(* IEC 61131-3 sources: ml2plc/examples/models/structured_text (part 6) *)

(* ---- test4_531k.st ---- *)
FUNCTION_BLOCK NeuralNetworkFB

VAR_INPUT
    input_data : ARRAY[0..4] OF REAL;
END_VAR

VAR_OUTPUT
    output_data : ARRAY[0..2] OF REAL;
END_VAR

VAR CONSTANT
    weights_0 : ARRAY[0..2559] OF REAL := [0.006168, -0.007737, -0.004572, -0.003805, -0.081145, -0.022669, -0.040454, -0.017532, -0.025900, -0.064631, -0.047865, -0.007452, -0.080317, 0.042283, 0.000890, -0.064382, -0.009100, -0.011638, -0.047598, -0.005238, 0.002791, -0.005841, -0.060246, -0.016523, -0.014516, -0.002007, -0.014596, -0.018067, 0.025868, 0.006018, -0.015262, -0.018643, -0.003052, 0.012583, -0.056134, 0.000727, -0.037447, -0.016557, -0.037026, -0.016739, -0.030965, -0.044604, -0.004674, -0.071475, 0.008430, -0.054697, 0.000375, 0.079556, -0.010031, -0.040946, -0.032777, -0.007746, -0.021319, -0.012790, -0.047135, -0.089749, 0.014232, 0.001651, -0.023776, 0.034909, -0.031567, -0.041982, 0.035747, -0.039939, -0.017710, 0.002087, -0.028975, -0.017014, 0.012243, -0.012999, -0.019807, -0.044350, 0.018067, -0.069752, 0.001563, -0.005957, -0.004255, -0.000246, -0.075206, -0.042035, -0.012978, -0.036161, -0.007486, -0.039953, -0.050775, -0.010311, -0.028363, -0.017167, -0.033474, -0.011529, -0.009715, -0.016724, -0.065615, 0.021977, 0.009902, -0.036258, -0.007694, 0.001126, -0.018509, 0.036309, -0.008579, -0.014633, -0.052138, -0.042639, -0.052210, -0.021528, -0.017732, -0.081576, -0.008286, 0.005255, -0.036065, -0.015189, -0.074120, -0.017314, -0.025928, 0.000444, -0.013875, 0.020662, -0.034705, -0.007929, -0.053950, -0.012137, 0.003924, 0.038306, -0.033622, -0.008152, -0.007697, -0.002231, -0.047321, -0.068849, -0.014781, 0.004508, -0.070911, -0.011590, -0.005847, 0.034466, -0.049314, -0.054858, -0.120357, -0.022947, -0.045314, -0.014210, -0.011795, -0.027942, 0.004085, -0.047372, -0.050960, 0.020868, 0.007977, -0.037249, -0.039574, -0.058623, -0.080479, -0.019785, -0.043017, -0.044134, 0.001765, -0.015653, -0.023090, 0.017455, -0.043623, -0.057814, -0.025243, -0.048311, -0.009657, -0.077425, -0.045795, -0.026813, -0.032518, -0.053390, -0.006588, -0.063675, -0.066407, -0.033561, -0.019729, -0.040149, -0.013426, -0.000105, 0.018445, 0.011021, -0.035918, -0.016334, -0.050424, -0.018496, -0.003434, 0.034537, -0.002120, -0.037769, -0.010563, -0.056970, -0.021492, 0.004430, 0.038964, -0.040694, -0.064145, -0.055157, 0.039010, 0.005452, -0.020624, 0.023485, 0.006722, -0.008886, 0.010608, -0.069180, -0.045544, -0.005442, -0.116079, -0.024035, -0.061259, -0.022777, -0.005744, 0.004640, -0.035091, -0.041870, -0.030253, -0.044182, 0.013662, -0.113956, -0.027071, -0.015773, -0.026526, -0.070524, -0.007985, -0.011598, -0.077758, -0.045670, -0.048661, -0.014513, -0.013066, -0.015931, -0.015619, 0.002752, -0.020614, 0.010716, 0.002136, -0.078809, -0.036949, -0.007683, -0.004785, -0.004789, -0.027511, -0.009657, -0.049951, -0.008816, -0.020890, -0.008851, 0.024166, -0.053262, -0.020197, -0.017122, -0.089715, 0.003861, -0.042685, 0.017193, -0.013868, 0.002213, 0.020823, -0.021258, -0.026864, 0.002694, -0.029496, -0.053142, 0.038210, -0.007476, -0.006005, -0.020900, -0.014644, -0.038122, -0.021673, -0.001530, -0.002961, -0.058100, -0.002778, -0.000089, 0.000113, -0.026780, -0.094293, 0.008923, 0.000047, 0.001569, -0.030386, -0.009189, 0.015745, -0.066894, -0.028746, -0.048156, -0.030306, -0.006260, -0.040602, 0.006604, 0.011101, -0.031063, -0.006231, 0.002844, -0.009292, -0.029432, -0.065772, -0.100504, -0.038383, 0.013530, -0.043025, -0.055311, -0.036706, -0.001836, -0.033030, 0.001966, 0.003206, -0.047405, -0.065538, -0.016400, -0.012487, -0.044876, -0.009988, -0.026461, -0.107726, -0.001962, 0.014469, -0.013257, -0.035765, -0.038008, 0.019523, -0.028117, -0.046915, -0.067385, -0.016535, 0.002655, -0.062835, -0.037264, -0.012879, -0.006051, -0.006659, -0.030517, -0.016854, -0.013416, -0.029428, -0.056979, 0.002656, 0.019105, -0.015444, -0.034404, 0.006777, -0.023455, 0.009467, -0.029399, 0.021276, 0.008433, -0.017701, -0.089102, -0.008802, -0.072623, -0.041329, -0.025934, -0.044785, -0.014089, -0.001511, -0.016151, -0.027101, 0.001011, -0.028102, -0.021238, -0.027469, 0.002060, 0.001314, -0.064151, -0.056067, -0.020087, 0.013779, -0.019102, -0.020556, -0.018478, -0.014906, -0.043024, -0.009099, -0.015567, 0.018504, 0.008389, -0.026493, -0.034103, -0.008169, -0.011630, -0.061097, -0.001828, -0.036604, -0.090593, -0.003821, 0.004210, -0.175559, 0.019005, 0.004134, -0.017647, 0.037174, -0.033732, -0.053073, 0.022879, -0.012883, -0.023034, -0.038492, -0.011812, -0.017564, 0.009026, -0.036873, -0.057276, -0.006387, -0.012203, -0.006951, -0.021118, -0.031144, 0.034645, 0.045173, 0.000612, -0.024887, -0.032074, -0.003918, -0.026183, -0.027079, 0.029110, -0.011173, 0.000224, -0.027518, -0.042254, -0.012626, -0.033389, 0.002061, 0.001831, -0.054974, -0.019345, -0.095294, -0.030450, -0.085620, -0.009941, -0.045067, 0.000455, -0.037109, -0.013278, -0.000530, 0.028802, -0.033968, 0.017109, -0.049283, 0.000876, -0.003601, -0.020212, -0.006754, -0.006030, -0.082454, -0.071900, -0.014293, -0.005903, -0.046136, -0.014200, 0.014313, -0.030323, -0.013996, -0.011830, -0.005418, -0.002600, -0.024998, 0.006551, -0.007039, -0.071191, -0.094658, -0.055012, -0.022098, -0.030385, -0.070776, -0.013385, 0.019914, -0.029646, -0.028838, 0.009107, -0.008539, 0.020163, -0.012484, -0.028226, -0.017505, -0.028885, -0.013220, -0.068085, -0.039696, -0.076335, -0.006828, 0.017805, 0.011101, -0.014613, -0.005119, -0.036674, -0.070308, -0.006485, -0.070089, -0.026779, -0.003504, 0.000492, -0.036936, -0.058629, -0.073952, -0.041623, 0.007899, 0.007541, -0.010827, -0.033526, -0.036041, -0.004380, -0.034936, -0.000530, -0.004452, 0.024483, -0.019720, 0.004198, -0.024792, -0.006160, 0.022435, -0.045744, 0.010493, -0.004708, -0.039041, -0.022206, 0.058065, -0.058637, 0.029476, -0.009941, 0.031980, 0.027263, 0.028729, -0.018779, 0.035691, -0.000839, 0.011755, -0.013788, -0.033617, -0.047934, 0.016009, -0.061441, -0.043422, -0.014114, 0.013690, -0.000306, 0.062245, -0.065690, 0.013481, 0.013963, -0.018303, -0.023203, 0.051331, -0.046245, -0.051296, 0.000886, 0.029395, -0.048312, 0.020966, 0.018177, 0.009344, 0.030180, -0.006859, 0.066112, -0.006302, 0.049277, -0.022652, 0.012126, -0.001961, 0.006813, -0.031577, -0.006198, 0.035557, -0.002758, 0.014040, -0.024291, 0.004469, 0.000628, -0.026485, -0.029591, -0.003587, -0.007451, -0.046778, 0.001367, -0.075846, 0.031924, 0.018597, -0.030053, -0.047463, -0.042152, -0.016299, -0.002213, -0.026199, 0.036664, -0.034040, 0.052768, 0.005836, -0.043658, -0.053341, 0.001381, 0.043572, 0.020291, 0.073398, 0.037756, -0.005681, 0.026407, 0.033731, -0.048959, 0.012376, 0.030472, 0.008492, 0.005691, -0.006789, -0.018349, 0.075362, -0.022161, -0.079043, -0.009294, -0.000774, -0.039354, -0.042801, -0.035631, -0.030911, 0.004652, 0.057990, 0.022027, 0.018841, -0.019965, -0.067957, 0.066897, 0.019102, 0.001754, -0.046148, 0.019094, 0.008093, 0.003544, -0.008916, -0.002643, -0.064754, -0.038101, -0.035119, -0.033188, -0.015181, 0.042656, 0.017546, -0.013701, -0.012623, 0.008619, -0.031625, -0.024699, 0.012467, 0.006890, -0.010188, -0.063297, -0.006435, -0.041045, -0.000126, -0.081690, 0.012576, 0.000700, 0.010163, 0.004561, -0.029321, -0.003461, 0.025865, -0.006400, -0.045266, -0.024265, 0.033321, -0.117580, -0.014021, -0.009655, 0.045165, 0.045564, 0.007505, 0.004496, 0.050880, -0.012176, -0.041370, -0.088418, -0.017235, -0.067351, 0.056832, 0.069346, 0.035097, 0.089766, -0.014582, 0.079974, -0.006041, -0.014888, -0.035294, 0.013718, -0.018149, 0.068994, 0.017431, -0.039235, -0.042068, -0.007724, 0.022600, -0.003539, -0.040479, -0.017089, 0.017629, -0.026505, 0.039217, -0.011858, -0.075481, -0.028972, -0.019730, 0.006281, 0.010786, 0.018083, -0.008708, -0.015356, -0.085096, -0.019559, 0.044645, -0.007992, -0.028722, -0.061144, 0.001558, -0.022994, -0.016173, -0.049005, 0.003667, 0.112726, 0.041862, -0.021030, 0.062288, 0.077233, 0.000736, 0.061262, -0.008646, -0.055297, 0.012099, 0.047965, 0.002597, 0.065893, -0.097906, 0.014617, 0.033970, -0.035677, -0.003285, 0.040832, -0.010042, -0.019621, 0.053835, 0.019053, 0.053018, -0.010340, -0.002477, -0.028028, -0.023846, -0.013320, 0.021628, -0.001340, -0.059531, 0.026777, 0.017700, -0.019184, -0.000877, -0.024227, -0.001088, 0.005022, 0.015510, 0.017810, -0.000029, -0.041248, -0.079095, 0.023700, -0.012472, -0.018172, 0.088289, -0.014964, -0.000217, 0.003885, 0.018567, -0.009548, -0.028347, -0.018591, 0.043182, 0.052019, -0.001108, 0.042047, -0.122054, 0.027480, -0.064142, 0.004650, 0.014279, 0.031755, 0.011892, -0.034454, -0.020755, 0.044469, 0.005772, -0.040299, -0.012851, -0.035211, 0.067049, -0.121054, -0.007700, -0.005547, 0.036890, -0.033311, 0.084753, 0.026367, 0.048788, 0.030230, 0.053215, -0.027125, 0.004881, 0.040511, -0.032856, -0.096552, 0.040967, 0.015451, -0.027745, -0.007011, 0.053545, -0.033689, 0.045135, -0.094181, 0.004068, -0.005429, 0.053405, -0.060415, 0.000319, -0.053152, -0.047989, 0.013013, 0.025322, 0.038022, -0.018121, 0.006913, -0.011688, -0.025630, -0.022074, -0.002609, -0.055090, -0.008263, -0.019801, 0.052412, -0.026663, -0.017301, 0.017173, 0.033957, 0.015627, -0.086593, 0.023172, 0.037030, 0.011863, -0.022188, -0.019773, -0.021711, -0.003184, -0.020591, -0.008187, 0.000161, -0.062586, -0.038520, -0.027736, -0.020185, -0.023671, -0.078505, 0.014876, 0.047807, 0.023937, -0.005761, -0.002716, 0.037869, -0.004794, -0.012825, 0.035395, -0.029956, -0.008986, -0.067532, -0.016199, -0.048075, 0.001541, -0.014349, 0.015026, 0.044194, 0.018795, -0.081185, -0.046023, 0.046350, -0.000227, 0.021468, -0.011860, -0.017598, -0.030247, 0.011072, -0.012450, 0.014558, -0.016468, 0.017973, 0.042791, 0.007654, 0.054244, -0.019306, -0.016567, -0.043988, 0.037716, -0.026492, 0.012198, 0.063996, 0.013889, -0.013916, 0.094007, -0.047667, -0.043191, 0.023439, -0.041024, 0.037257, 0.084837, -0.053354, -0.023051, -0.060040, -0.024047, -0.032870, 0.011373, -0.070437, 0.025510, 0.029563, -0.028023, -0.056257, -0.032347, 0.015591, -0.013614, -0.107999, -0.058039, 0.008937, 0.051134, -0.010621, -0.012029, -0.002045, -0.045550, 0.019002, -0.029280, -0.058529, 0.012200, 0.032851, -0.062094, -0.023157, 0.001064, -0.019808, 0.071575, -0.014192, 0.044343, -0.055609, 0.082989, 0.021812, 0.008306, 0.008213, 0.029873, 0.023171, 0.013703, 0.011581, 0.001465, 0.019024, 0.034659, -0.039955, -0.003518, -0.039174, -0.037442, -0.031396, 0.025519, -0.005441, -0.020170, -0.007954, -0.027134, -0.044586, -0.015502, 0.003576, -0.002512, -0.010521, -0.075746, -0.045547, 0.002149, -0.045099, -0.017035, -0.007519, 0.057518, 0.028380, 0.018844, -0.000265, 0.033838, -0.016435, -0.009740, -0.000992, 0.001005, -0.013433, -0.014406, -0.010904, 0.000908, -0.031988, -0.011733, -0.060267, 0.058381, 0.004671, 0.003265, 0.045723, 0.000060, 0.022857, -0.053219, -0.032393, -0.054149, -0.009633, 0.084957, -0.031704, 0.048600, -0.073818, 0.012638, -0.070321, -0.003787, 0.053202, 0.059789, 0.035780, -0.047696, -0.005062, 0.019513, 0.003089, 0.002214, -0.000557, 0.022252, -0.037908, -0.063868, -0.048430, -0.021449, -0.005469, -0.020284, -0.013151, -0.002935, 0.024061, -0.027414, -0.060135, 0.019118, 0.010644, -0.020204, 0.043180, 0.011003, -0.026948, -0.029472, 0.006690, -0.014830, 0.034704, 0.002983, -0.000449, -0.033364, -0.002019, 0.023595, 0.048194, -0.002517, 0.015325, -0.055047, 0.006398, -0.026732, -0.063421, -0.051463, 0.022229, -0.007053, 0.003437, 0.036441, 0.011057, -0.010537, 0.053316, 0.047278, -0.088576, -0.051669, 0.003415, -0.010457, 0.003318, 0.020984, -0.032925, 0.000310, -0.075833, -0.005370, 0.004928, -0.045853, -0.068047, 0.009317, -0.003116, 0.016023, 0.046078, -0.004938, 0.018008, -0.052253, -0.035261, -0.061192, -0.006844, 0.017909, -0.005032, -0.035604, 0.038330, -0.007799, 0.001959, -0.082375, -0.057521, 0.002209, -0.036735, 0.029469, 0.046464, 0.023360, 0.054089, 0.000124, -0.098509, -0.034924, -0.008698, -0.014121, -0.009095, 0.054927, -0.035409, 0.033318, -0.013215, -0.028000, -0.009640, 0.005127, 0.002514, -0.058949, -0.031840, 0.024286, 0.037682, -0.032623, 0.014822, 0.004515, -0.022597, -0.047328, -0.013061, -0.004957, -0.000829, -0.032617, 0.008092, -0.006902, -0.011951, -0.011564, 0.012531, 0.004754, -0.014693, 0.020353, 0.019861, 0.054645, -0.060680, -0.019404, 0.017570, 0.033163, -0.051124, 0.010038, -0.051300, -0.015827, -0.065831, 0.009685, -0.033803, 0.029050, 0.033958, -0.032388, -0.029221, -0.044903, -0.002951, -0.027556, -0.031074, 0.022902, 0.010975, -0.000864, 0.017581, -0.036060, 0.000276, 0.055463, 0.029811, 0.008004, -0.045528, 0.007951, 0.010881, -0.019921, -0.008701, 0.029887, -0.012379, -0.062134, -0.002077, 0.039846, -0.015407, 0.025720, -0.040064, 0.013837, -0.014882, -0.012172, 0.024249, -0.000815, 0.001816, -0.077496, -0.006953, 0.065075, -0.015756, 0.011041, 0.027465, 0.031528, -0.071741, -0.030240, 0.053134, -0.023077, -0.006604, -0.022893, 0.029625, -0.061120, 0.023706, -0.000936, -0.032921, -0.008114, 0.003939, 0.023346, -0.013129, -0.059646, 0.045903, -0.023942, 0.050939, -0.002942, -0.020111, -0.015744, 0.013710, 0.035260, 0.000029, -0.004535, -0.036242, -0.037386, -0.027829, -0.031840, 0.002574, -0.007554, -0.035839, 0.020656, -0.027891, -0.010452, 0.001935, -0.048956, 0.056025, -0.081554, 0.063599, -0.028470, -0.083353, -0.039516, 0.022740, 0.010384, -0.034174, -0.007442, -0.058151, -0.015351, 0.032128, -0.007490, -0.035707, -0.013821, -0.052297, -0.008232, -0.003910, -0.002278, -0.002002, 0.041686, -0.033565, -0.020172, 0.011638, -0.047561, 0.032903, -0.030198, -0.029194, 0.029884, 0.007434, 0.002506, -0.093412, 0.003442, -0.048978, -0.003672, 0.008821, -0.016854, -0.022693, 0.019834, 0.003447, -0.014566, -0.035371, -0.010202, -0.030048, 0.010019, 0.009586, 0.033665, -0.052329, 0.012042, -0.013713, -0.053064, -0.004914, 0.065243, -0.014380, 0.001766, 0.002737, -0.036723, -0.036644, -0.096545, 0.033883, -0.008006, 0.000931, -0.004996, -0.105254, -0.033430, -0.003654, -0.047162, 0.001697, -0.047309, -0.021566, 0.012178, -0.040513, -0.018042, -0.059251, 0.011468, -0.026371, 0.021869, -0.016537, -0.000474, 0.008068, -0.015187, 0.022844, -0.057641, -0.020614, -0.010191, 0.005121, -0.013429, 0.027562, 0.023835, -0.069291, -0.015122, -0.002747, -0.078974, -0.035144, -0.012528, -0.019010, -0.016324, 0.062985, -0.042301, 0.043749, 0.069579, 0.011530, -0.016713, -0.000731, 0.022784, -0.021786, -0.002233, 0.017447, -0.006153, -0.017514, 0.025534, 0.027752, -0.007414, 0.026801, -0.009000, 0.040284, 0.010169, 0.007577, -0.013006, 0.002903, -0.107397, -0.036827, -0.021993, -0.033773, -0.005145, -0.006365, 0.027436, -0.082875, -0.015922, -0.029948, -0.016043, 0.027308, 0.004923, 0.009969, -0.004351, -0.018375, 0.000664, -0.036814, 0.007848, 0.014095, -0.019357, 0.005650, 0.014980, 0.041914, -0.057784, -0.048502, 0.005255, 0.009340, -0.007252, 0.019865, -0.059517, 0.028774, -0.013038, 0.053348, -0.008614, -0.019005, 0.008522, -0.014930, -0.059443, 0.002173, -0.008524, -0.036694, 0.013195, -0.035339, 0.009507, -0.021153, -0.108459, -0.002806, -0.038649, -0.013854, 0.001382, -0.004942, 0.030240, -0.050536, -0.127641, -0.043994, -0.038555, -0.002474, -0.034832, 0.051688, 0.003858, 0.018911, -0.010615, -0.022812, -0.041967, -0.052411, 0.002677, -0.012954, -0.017153, -0.023283, -0.019843, -0.024961, -0.072991, -0.016500, -0.043703, -0.023475, -0.040668, 0.050983, -0.010791, -0.045946, -0.037954, 0.048402, 0.025119, 0.002440, 0.005653, -0.002502, 0.059590, -0.014535, 0.034528, -0.068574, -0.048264, 0.037087, -0.005935, 0.013869, 0.055370, -0.060236, 0.035561, 0.036965, -0.049284, -0.065174, -0.031417, 0.028118, -0.000721, -0.007135, -0.049212, -0.002982, -0.064442, 0.015377, 0.020929, -0.072578, 0.039138, -0.035400, -0.003530, -0.042568, 0.018827, -0.003496, 0.042349, -0.031215, -0.027957, 0.049278, 0.008354, -0.000546, -0.021296, 0.017299, 0.011847, -0.028922, -0.003541, -0.007659, 0.011905, 0.065311, 0.059542, -0.049007, -0.011449, 0.015553, -0.033130, -0.018639, 0.009950, 0.032141, -0.028848, 0.068738, -0.005494, -0.004502, -0.030848, 0.001772, 0.023285, 0.019241, -0.060901, 0.033557, -0.025315, -0.109076, -0.000548, 0.040990, 0.010826, -0.042109, -0.034424, -0.045023, -0.063789, 0.024868, 0.015001, 0.001163, -0.033712, -0.052648, -0.016266, 0.001274, 0.013955, -0.050313, -0.010176, 0.034576, 0.004616, -0.018953, -0.035623, 0.024527, -0.044255, 0.014509, -0.063285, 0.004416, -0.009160, 0.013336, -0.087228, 0.015343, 0.002086, -0.037559, -0.006652, -0.004271, -0.037680, 0.008953, 0.044458, -0.056017, -0.010455, 0.006135, -0.081046, 0.038880, -0.029584, 0.068916, -0.015243, 0.008562, -0.022434, -0.062339, 0.020589, 0.025935, 0.002090, 0.011453, -0.012045, -0.026340, -0.010421, -0.017118, 0.023078, -0.048666, -0.056073, -0.026423, 0.035808, -0.034026, 0.065977, -0.001679, 0.031959, -0.006526, 0.025844, -0.000980, 0.002246, 0.012930, -0.001139, -0.008721, 0.033522, -0.048647, -0.040169, -0.009701, 0.013569, -0.011153, -0.007777, 0.001426, -0.003487, -0.015966, -0.016842, -0.020404, -0.011884, -0.002042, 0.024870, 0.029681, -0.001799, 0.024583, -0.031010, -0.035852, 0.001699, -0.044035, 0.047594, 0.064107, -0.002716, 0.034184, 0.001073, -0.005203, -0.022102, -0.015703, 0.002247, 0.011254, -0.034985, -0.031385, -0.009637, 0.069561, -0.034012, -0.011237, -0.015109, -0.063899, 0.017169, 0.045481, 0.057430, -0.025430, -0.004783, -0.041361, -0.040798, -0.015842, -0.047996, 0.003322, -0.059076, 0.010305, 0.003273, 0.002631, 0.044407, 0.005079, 0.021253, -0.011607, 0.041114, -0.013865, 0.008588, 0.004921, -0.013600, -0.014643, 0.030441, -0.023050, 0.013847, -0.008933, -0.023550, 0.001001, 0.001016, -0.001820, 0.004475, -0.007551, 0.008457, 0.003246, -0.059475, -0.009358, -0.080363, -0.019096, -0.009395, -0.011684, 0.001092, 0.039147, -0.038988, 0.029579, -0.008820, -0.031082, -0.060658, 0.000651, 0.000825, -0.026070, -0.006354, -0.049676, -0.020702, -0.003012, -0.006391, -0.007444, 0.023275, 0.002955, 0.007902, 0.036258, 0.019251, -0.013756, -0.014383, 0.024339, -0.010544, -0.018283, 0.027118, 0.010669, -0.012802, -0.004819, 0.006033, -0.016694, -0.064134, 0.038288, -0.055878, -0.025146, -0.039060, 0.014958, 0.001991, -0.079096, -0.021012, -0.030163, 0.087878, 0.037328, -0.015318, 0.058822, -0.034177, 0.044470, -0.128140, 0.001406, -0.070954, 0.016894, 0.004603, -0.045666, -0.018139, 0.008610, 0.071770, -0.019468, 0.033419, 0.003130, 0.044825, 0.011587, -0.001095, 0.016766, -0.006245, -0.064439, 0.033407, -0.094713, -0.006409, -0.000119, 0.002618, -0.031029, -0.052071, -0.010173, -0.022700, -0.016307, -0.001930, 0.037094, -0.004913, -0.005293, 0.015431, 0.036442, -0.012428, 0.074049, -0.063375, -0.013886, 0.030770, -0.046108, 0.036323, -0.081006, -0.027172, -0.011284, -0.018333, -0.021334, -0.013070, -0.011830, -0.021084, 0.002423, 0.034048, -0.038911, -0.001053, -0.002545, 0.000026, 0.026737, 0.030784, -0.002281, -0.011285, 0.029163, -0.033121, -0.021412, -0.016520, -0.002251, 0.008773, -0.045886, 0.012279, 0.009255, -0.005824, 0.000048, -0.005718, -0.037088, -0.007778, -0.019037, -0.023370, 0.002763, 0.024722, -0.007766, -0.057903, -0.012214, 0.032384, -0.027996, 0.024596, 0.003802, -0.001651, -0.015866, 0.021212, 0.057682, -0.028116, -0.013073, 0.020292, -0.009352, -0.130909, -0.024060, -0.044775, -0.005629, 0.020706, 0.020607, -0.021389, -0.005816, 0.046837, -0.023419, 0.025185, -0.008048, 0.021869, 0.006025, -0.007184, -0.072714, 0.049448, 0.095942, -0.002258, -0.019363, -0.019018, -0.013612, -0.017024, -0.024008, -0.060706, 0.012546, 0.008040, -0.017750, -0.021085, 0.048197, -0.092418, 0.013575, -0.030068, -0.040348, -0.043340, 0.001834, -0.021993, -0.074695, 0.001109, 0.023855, 0.017737, -0.018748, -0.030487, 0.005170, -0.015220, 0.030898, 0.009196, 0.017739, -0.063993, -0.028491, 0.038864, -0.000904, -0.003439, 0.060044, 0.007750, -0.050293, 0.003916, -0.020393, -0.007651, -0.083702, 0.012657, -0.041159, -0.074699, 0.017662, -0.019135, -0.023496, 0.079346, -0.044665, -0.087241, 0.057253, 0.035364, 0.038074, 0.033843, -0.025855, -0.017310, 0.032125, -0.001813, -0.042987, -0.008234, -0.047822, -0.026193, -0.017293, 0.016534, -0.052416, 0.047058, 0.006139, 0.000373, -0.050032, -0.010969, -0.014620, -0.065381, -0.065984, 0.039695, 0.013624, 0.009117, -0.073527, 0.005184, 0.012362, 0.013532, 0.003368, 0.026692, 0.001673, 0.010429, 0.034464, 0.005765, 0.041395, 0.004109, -0.009537, -0.008939, 0.001889, 0.022877, 0.022266, -0.022098, 0.008824, -0.111495, -0.014949, -0.010727, -0.013789, -0.008899, -0.014824, -0.039584, 0.057751, 0.016652, -0.009886, 0.028283, -0.028595, 0.053852, -0.039075, -0.013941, -0.006656, 0.003033, 0.020083, -0.052063, 0.075551, 0.016607, 0.033015, -0.028914, 0.000990, 0.051002, -0.051270, -0.000054, -0.045118, 0.030804, 0.013392, 0.037767, 0.017876, 0.028166, 0.031678, -0.006061, -0.131450, 0.004390, 0.000658, 0.019391, 0.006017, -0.022607, -0.025737, 0.045831, -0.037299, 0.005095, -0.051780, -0.013996, 0.002758, -0.019142, -0.099079, -0.024694, -0.034577, 0.065943, 0.028580, -0.028417, -0.017952, -0.003284, 0.012914, 0.000251, 0.038695, 0.003972, 0.075688, -0.050465, -0.008991, -0.066909, 0.010379, -0.027695, 0.002838, -0.088827, -0.035800, -0.070370, -0.001824, -0.002680, -0.091314, -0.046202, -0.030486, -0.059511, 0.025657, -0.028113, 0.006912, -0.001720, -0.004071, -0.015952, -0.045470, -0.110590, 0.035917, 0.031153, -0.038135, 0.038639, -0.030943, -0.053098, 0.010134, 0.032735, -0.043683, 0.006105, -0.022744, 0.004303, -0.039438, -0.017385, -0.009131, -0.021856, -0.068681, 0.028034, 0.032798, -0.017536, 0.001738, -0.010315, -0.047463, -0.019801, 0.052497, -0.018893, -0.032553, 0.001899, 0.002888, 0.006082, -0.102064, 0.015060, 0.043289, 0.035894, -0.034930, -0.005025, -0.022740, -0.011462, 0.022725, 0.004670, -0.004176, 0.052536, -0.059373, 0.036484, -0.007752, -0.020044, -0.038795, -0.005262, -0.002371, 0.008118, -0.015251, 0.007129, -0.005574, -0.001835, -0.050144, -0.066125, -0.049709, -0.001914, -0.010255, -0.062357, 0.026160, -0.079928, -0.089573, -0.026023, -0.079924, -0.037929, -0.060248, -0.097622, -0.022256, -0.012138, -0.023413, -0.014130, -0.022373, -0.018968, 0.071716, -0.014322, -0.016340, -0.016211, -0.028133, -0.041122, -0.052809, -0.055714, -0.039074, -0.006132, -0.069915, 0.075339, 0.018775, 0.003201, -0.091950, 0.011198, -0.072222, -0.207902, -0.052503, -0.016103, -0.016584, -0.024159, -0.003789, -0.014732, -0.007769, -0.030552, -0.029373, -0.030021, -0.062975, 0.035173, -0.007464, -0.071709, -0.023191, -0.020199, -0.250547, -0.036404, -0.027666, -0.045544, -0.021928, -0.053373, -0.074033, -0.020565, 0.001989, -0.017748, -0.001127, -0.044066, -0.254895, -0.028499, -0.041015, 0.014959, -0.047935, -0.044798, -0.072543, -0.024991, -0.001973, -0.015223, -0.045056, -0.044002, -0.057141, 0.079430, -0.000973, -0.030142, -0.014362, -0.008963, -0.021617, -0.000343, -0.017941, -0.055189, -0.011911, -0.024881, -0.020193, -0.036285, 0.011153, -0.086658, -0.115129, -0.075860, -0.032126, -0.031356, -0.035758, -0.039777, -0.010603, -0.039971, -0.005003, -0.092777, -0.016766, -0.035017, 0.067210, -0.020347, 0.000180, -0.028031, -0.005414, -0.046689, -0.011603, -0.042978, -0.047190, 0.001767, -0.060300, -0.026369, -0.017898, -0.014198, -0.023047, -0.015757, -0.054736, -0.002798, 0.031703, -0.022449, -0.055319, -0.076581, -0.025874, -0.054651, -0.066918, -0.014431, -0.018167, -0.033554, -0.022343, -0.031144, -0.095778, 0.002187, -0.020380, -0.029201, -0.029436, -0.026996, -0.082483, -0.026350, -0.033960, -0.047994, -0.052323, -0.073925, -0.012077, -0.069418, -0.020239, -0.034885, -0.035901, 0.025073, 0.022686, -0.073895, -0.000864, -0.032177, -0.112699, -0.035631, 0.036357, -0.098355, -0.059297, -0.109314, -0.083866, -0.028674, -0.092170, -0.025738, -0.047006, -0.059676, -0.390116, 0.017218, -0.019471, -0.039703, -0.077019, -0.017879, -0.045720, -0.048082, -0.068037, -0.116513, -0.003322, -0.039939, -0.057380, -0.002844, -0.030937, -0.078279, -0.046431, 0.007851, -0.007846, -0.013517, -0.013672, -0.028053, -0.044630, 0.056186, -0.025563, -0.025391, -0.107007, -0.015789, -0.016769, -0.037651, -0.091252, -0.028524, -0.068835, -0.122871, -0.040803, -0.009011, 0.097818, 0.022286, -0.025307, -0.013694, -0.049694, -0.025467, -0.009230, -0.036727, -0.087940, -0.003927, -0.015481, -0.043764, -0.053849, -0.031034, -0.030649, -0.014868, -0.045202, -0.069928, -0.034897, 0.002734, -0.063531, -0.007274, -0.006740, -0.020420, -0.006569, -0.037788, 0.001002, -0.035107, 0.035919, -0.036534, -0.022154, 0.006700, -0.033557, -0.043352, -0.005245, -0.044900, -0.032932, -0.028327, -0.025989, -0.006374, -0.000653, -0.039040, -0.028748, -0.032810, -0.013529, -0.022279, -0.020407, -0.136795, -0.092331, -0.019560, -0.042329, -0.042786, -0.002416, -0.004882, 0.079753, -0.049726, -0.001607, -0.077585, -0.032747, 0.027309, -0.289826, -0.050177, 0.007235, -0.087341, 0.013227, 0.091116, 0.005451, 0.021729, -0.028794, -0.035271, 0.002774, -0.028409, -0.024945, 0.011371, -0.004599, -0.022100, -0.008223, 0.000789, 0.011017, -0.054857, -0.019057, -0.087335, -0.035270, 0.021188, -0.044861, 0.062755, -0.042301, -0.047132, -0.020623, -0.039554, -0.031479, -0.085009, 0.004568, 0.076652, -0.026515, -0.028987, -0.029603, -0.053167, -0.003366, -0.027917, -0.070408, -0.022428, -0.018212, 0.016192, -0.034404, 0.002494, -0.018473, -0.011689, -0.007457, -0.071295, -0.044153, -0.021756, -0.074203, -0.057648, -0.028279, -0.031716, -0.249456, -0.073115, 0.005304, 0.073527, -0.010448, 0.019232, -0.013999, -0.077410, 0.010563, -0.113081, -0.030120, -0.004718, -0.032821, -0.018488, 0.040180, -0.013917, -0.057365, -0.013663, -0.034495, -0.029207, 0.004239, -0.055135, -0.025166, -0.013593, -0.017122, -0.017133, -0.028331, -0.121554, -0.087904, -0.169127, -0.007008, -0.001212, -0.044030, -0.024503, -0.019572, -0.058879, -0.025582, -0.016590, -0.026188, -0.021663, -0.059479, -0.015373, -0.087637, -0.014144, 0.068119, -0.030784, 0.017394, 0.008500, -0.018711, -0.002974, -0.023651, -0.007668, -0.044605, -0.037411, -0.003849, -0.036531, 0.008198, -0.038061, -0.126516, -0.002909, -0.042653, -0.078390, -0.007849, -0.082457, 0.015911, -0.021599, -0.006017, -0.012733, -0.039974, 0.024193, -0.060572, 0.003743, -0.053093, -0.017102, -0.024318, -0.111726, -0.037359, -0.009472, -0.041164, -0.042447, -0.057380, -0.024953, -0.053407, -0.055655, -0.014224, -0.009794, 0.044105, 0.013126, -0.041380, -0.044204, 0.004932, -0.018908, -0.017355, -0.245535, -0.026744, -0.064080, -0.029372, -0.007203, -0.023629, -0.063408, 0.023934, -0.014043, -0.005872, -0.037652, -0.043501, -0.010717, -0.012284, -0.006543, -0.119264, -0.021682, -0.170125, -0.049194, 0.040230, -0.008044, -0.046620, -0.006159, 0.013648, -0.019651, -0.045637, -0.058170, 0.080909, 0.006372, -0.005016, -0.000595, 0.006720, 0.005245, -0.042498, -0.014498, 0.000439, 0.002276, -0.062180, -0.015582, 0.004705, 0.016076, 0.013021, -0.084524, -0.017796, -0.039834, -0.017225, -0.025239, -0.023910, 0.027862, -0.093303, -0.048912, -0.084215, -0.013775, -0.031631, -0.018785, 0.030396, -0.040472, -0.039703, -0.015829, -0.000407, -0.031301, -0.052192, -0.026411, -0.171183, -0.004667, -0.018525, 0.002765, -0.014035, -0.068948, -0.039431, -0.021647, -0.028413, -0.013805, 0.013900, -0.012050, -0.126553, -0.052837, 0.015999, -0.044176, -0.037112, -0.008267, -0.018192, -0.071674, -0.060666, -0.097312, -0.059403, -0.087029, -0.005587, -0.005021, 0.011870, -0.006146, 0.010483, -0.052837, 0.003976, 0.004876, 0.002883, -0.024434, -0.077477, 0.030641, -0.019218, -0.035539, 0.013905, 0.031854, 0.002071];
    bias_0 : ARRAY[0..511] OF REAL := [-0.560015, 0.184992, -0.470400, -0.294991, -0.372218, -0.580996, -0.127396, -0.456540, -0.007419, -0.141688, -0.516530, -0.058160, -0.375340, -0.870894, -0.525041, -0.497357, -0.425162, -0.267576, -0.566308, -0.246234, 0.760137, -0.267928, -0.421276, -0.461114, -0.884117, -0.752684, -0.272481, -0.075169, -0.277913, 0.800566, -0.266811, -0.508528, -0.489017, -0.563790, -0.171746, -0.592066, -0.099807, -0.305085, 0.228222, 0.204156, -0.222468, -0.390126, -0.392960, -0.152436, -0.480089, -0.487889, -0.102116, 0.576028, -0.360179, 0.315619, 0.361651, -0.283220, -0.275759, -0.108602, -0.517918, -0.668270, 0.080150, -0.525913, -0.390262, 0.238540, -0.506728, -0.372645, -0.529373, -0.530296, -0.419331, -0.262827, -0.544448, 0.153808, -0.417206, -0.416869, 0.392310, -0.373798, -0.756939, -0.013806, -0.356106, -0.015186, -0.657312, -0.635726, -0.067811, -0.520272, -0.088178, -0.198638, -0.171325, -0.180742, -0.344793, -0.560948, -0.050169, -0.063545, -0.521232, -0.253853, -0.473808, -0.572321, -0.499878, -0.378826, -0.486301, -0.380427, -0.180301, -0.029836, -0.561780, -1.221803, -0.467454, -0.040174, -0.484950, -0.363476, -0.277297, 0.029669, -0.478665, -0.035147, -0.413088, -0.336468, -0.443213, -0.049765, -0.361502, -0.278191, -0.397446, 0.542885, -0.430711, 0.477843, -0.534856, -0.636531, -0.404057, -0.141602, -0.589094, -0.018168, 0.100740, -0.466928, -0.097708, -0.297540, -0.461497, -0.400244, -0.225557, -0.315778, -0.161987, -0.323324, 0.177692, -0.313298, -0.428529, -0.417167, -0.564084, 0.114390, -0.554823, -0.278022, -0.439219, -0.265492, 0.011075, -0.372697, -0.414324, -0.616711, 0.287804, -0.300455, -0.426657, 0.108030, -0.496591, -0.380250, 0.019351, -0.233535, -0.095143, -0.627654, -0.507818, -0.203023, -0.438338, -0.029473, -0.100205, 0.319433, -0.120297, -0.394097, 0.081192, 0.084620, -0.574713, -0.424066, -0.183717, 0.443114, -0.460228, -0.610907, -0.450714, -0.646212, -0.626546, -0.558116, 0.672355, -0.276201, -0.631161, -0.310516, -0.087265, -0.097912, -0.628902, 0.111149, -1.149800, -0.406454, -0.183037, 0.064063, -0.556680, -0.432543, 0.149459, -0.429032, -0.307682, -0.529772, 0.073030, -0.588899, -0.673073, -0.855552, -0.529210, -0.559242, -0.503162, -0.411373, -0.582325, -0.476031, 0.464417, 0.195734, -0.035936, -0.269100, -0.201118, -0.547096, -0.339036, -0.186394, -0.392593, -0.525719, -0.447540, -0.754172, 0.050524, -0.440737, -0.587200, -0.023825, -0.559724, -0.540134, -0.026272, -0.478584, -0.178302, -0.310404, -0.043472, -0.303760, 0.087057, -0.560951, -0.126218, -0.444226, 0.013041, -0.378160, -0.401341, -0.066755, 0.097565, -0.246728, -0.453610, -0.436659, -0.150369, -0.565253, -0.386807, -0.537203, -0.050841, -0.295192, -0.282184, -0.609656, -0.349239, -0.477961, -0.565487, -0.847882, -0.503656, -0.485508, 0.228604, -0.230194, -0.371666, 0.160188, -0.324394, -0.176446, -0.198087, -0.523571, -0.738180, -0.362561, -0.531421, -0.185987, -0.318514, -0.339727, 0.373145, -0.139809, -0.545757, -0.536750, -0.540660, -0.591894, -0.365686, -0.772576, -0.241534, -0.180127, -0.309330, -0.451085, -0.133262, -0.491258, -0.922880, -0.085069, 0.075745, -0.599000, -0.255950, -0.366717, -0.315008, 0.025284, -0.796683, -0.576438, -0.423812, -0.526922, -0.464793, -0.611435, -0.176255, -0.011129, -0.148650, -0.593366, -1.010090, -0.611632, -0.615362, 0.098925, -0.484878, -0.568730, -0.406493, -0.103242, -0.089686, 0.127594, -0.331190, -0.228097, -0.494144, -0.289490, 0.106738, -0.494740, -0.811164, -0.224123, -0.539983, -0.190705, -0.308104, -0.576015, -0.448016, -0.452012, 0.063439, 0.015257, -0.181990, -0.454566, -0.511673, -0.489078, -0.242683, -0.551215, -0.320198, -0.305431, -0.010823, -0.530007, -0.248963, -0.599315, -0.278430, -0.568422, 0.219756, -0.437993, 0.481473, -0.272435, -0.269651, 0.202242, -0.181707, -0.269245, 0.383201, -0.646039, -0.229450, 0.205804, 0.078391, -0.578819, -0.428767, -0.099032, -0.498601, -0.852345, -0.515247, -0.871002, -0.549889, -0.357410, -0.024235, -0.221249, -0.703844, -0.345876, -0.218584, -0.446784, -0.356807, -0.403075, 0.162039, 0.359484, -0.842997, 0.181479, -0.363541, -0.474084, -0.500788, -0.621216, -0.559714, 0.041385, -0.368353, -0.202383, -0.597544, 0.013351, 0.036447, -0.180812, -0.647463, -0.003342, 0.887071, -0.064974, -0.570065, -0.425626, -0.649220, -0.515449, -0.608669, 0.027214, -0.356379, -0.425030, -0.109388, 0.446015, -0.571340, -0.579622, -0.107719, -0.119594, -0.032838, -0.666012, 0.329357, -0.379204, 0.442772, -0.567839, -0.250720, 0.252409, 0.254247, -0.556360, -0.595093, -0.398352, -0.588479, -0.109848, -0.696338, -0.451533, -0.427623, -0.517631, -0.076536, -0.100740, -0.587674, -0.433592, -0.168261, -0.522468, -0.336927, -0.536847, -0.587720, -0.180166, 0.026694, -0.906076, -0.327415, -0.170205, -0.111061, 0.023953, 0.019779, -0.445003, -0.464418, -0.525391, -0.757161, -0.590829, -0.639809, -0.478079, -0.491544, -0.693892, 0.043033, -0.345456, -0.304986, -0.430036, -0.683112, -0.510119, -0.268652, 0.026592, -0.488424, 0.089903, -0.687703, -0.479938, -0.263812, -0.729523, -0.500908, -0.508581, -0.646621, -0.368469, -0.678522, -0.097792, -0.482871, 0.287748, -0.410175, -0.630866, -0.412892, -0.014359, -0.253159, -0.518970, -0.306679, -0.162928, -0.502708, -0.723021, -0.585624, -0.038050, -0.306422, -0.386367, -0.261096, -0.322216, -0.243436, -0.450591, -0.258327, -0.473112, -0.314861, -0.546208, 0.487024, -0.467651, -0.432374, 0.294989, -0.701729, -0.404412, 0.457121, -0.157405, -0.416856, -0.143322, -0.547066, -0.152965, -0.157077, -0.390291, -0.507056, -0.373921, -0.426115, -1.071550];

    weights_1 : ARRAY[0..524287] OF REAL := [-0.033384, -0.029529, -0.002307, -0.065159, -0.029187, -0.063650, -0.017592, 0.007238, 0.087993, -0.013393, -0.032657, -0.027770, 0.025115, 0.008525, -0.039527, -0.057369, -0.025352, -0.038812, -0.061059, 0.028921, -0.036287, 0.002650, -0.005819, 0.022260, 0.010706, 0.017105, 0.022733, -0.102570, 0.048175, -0.065543, 0.042244, -0.001051, -0.005552, 0.001343, -0.132678, -0.084336, 0.023444, 0.044026, 0.006423, -0.002656, -0.035584, -0.011227, -0.018969, -0.118467, -0.076455, -0.008606, 0.038094, -0.070374, 0.028555, 0.027610, -0.009448, 0.019685, -0.124333, -0.049827, -0.077195, -0.056529, 0.012599, -0.009381, 0.023236, -0.004700, -0.095187, -0.027614, -0.016721, -0.042166, 0.026967, -0.001691, 0.168896, -0.045715, -0.077939, 0.018614, -0.005101, -0.049948, -0.086186, -0.070169, 0.003832, -0.060939, -0.058552, -0.003961, 0.025444, 0.039389, -0.016526, 0.027258, 0.057089, -0.003192, 0.038133, -0.103590, 0.044226, -0.036122, -0.014077, -0.072944, -0.070990, -0.015418, 0.025484, -0.126175, -0.014363, 0.001600, -0.006227, 0.025299, 0.023108, -0.017388, -0.064967, -0.032258, 0.059030, 0.027494, -0.043399, 0.041397, -0.048733, -0.125696, 0.080937, -0.005893, -0.060478, 0.024098, -0.059152, -0.067177, -0.024428, -0.035957, 0.037022, 0.043891, 0.072372, -0.013457, -0.059588, -0.048198, 0.001741, -0.015119, 0.067838, 0.029718, 0.007244, 0.034856, -0.126202, 0.020841, -0.018814, 0.008373, 0.025370, -0.008876, -0.166713, -0.021350, -0.010922, -0.026620, 0.007677, 0.017664, -0.021487, -0.014281, -0.068944, -0.000945, 0.006296, -0.090065, -0.070590, 0.038186, -0.092014, -0.025633, -0.067717, 0.052099, 0.003534, 0.056980, -0.031832, -0.060090, -0.079961, 0.048795, -0.048479, 0.017890, 0.036706, 0.054768, 0.039339, -0.000939, -0.090144, 0.016987, -0.139394, -0.082103, -0.043726, -0.038848, -0.062648, 0.009012, -0.028069, 0.002676, -0.151202, -0.023922, -0.014620, 0.000349, -0.040842, -0.030065, 0.001913, 0.013584, 0.027665, 0.023666, -0.034337, -0.007901, 0.020217, -0.045113, 0.014856, -0.063518, -0.025068, 0.097930, -0.106403, -0.069477, 0.057602, 0.059377, 0.052719, -0.047087, -0.084744, 0.052077, 0.053991, -0.009452, 0.053999, 0.023506, -0.057650, -0.039659, -0.058501, -0.008886, 0.146905, -0.033510, 0.038731, -0.094149, 0.072222, 0.033093, -0.011071, -0.012098, 0.006181, 0.044728, -0.111777, -0.038309, 0.030381, 0.096242, -0.040079, -0.030020, 0.029591, -0.101405, 0.022670, -0.080118, 0.004489, -0.090326, -0.068333, -0.058073, 0.017577, 0.004949, -0.036895, -0.091916, -0.095090, -0.032846, -0.030988, -0.011184, -0.076728, -0.055495, -0.063720, 0.004673, 0.043187, 0.015708, -0.021401, -0.025020, 0.034938, -0.081069, -0.117772, 0.000362, 0.020896, 0.042762, 0.059001, 0.019692, -0.051868, -0.004403, -0.001810, -0.016538, -0.005535, -0.020549, 0.033277, -0.023793, -0.050831, -0.070665, -0.004009, -0.007788, -0.049764, -0.015402, -0.170423, 0.093517, -0.043430, -0.029537, 0.068742, 0.054416, 0.020689, -0.060321, 0.019090, -0.018722, -0.070399, -0.101210, -0.027410, -0.048431, 0.026611, 0.012401, -0.046667, -0.046146, -0.089249, -0.095605, 0.025816, 0.029740, 0.043186, -0.006458, -0.021826, -0.020286, -0.041731, -0.029256, -0.083371, -0.027684, -0.043325, -0.090286, 0.040597, -0.067456, -0.058064, -0.015049, 0.043578, -0.052356, -0.000773, 0.032165, -0.052683, 0.045543, 0.024650, -0.031897, -0.052368, 0.023043, 0.023701, -0.049907, -0.019434, 0.037758, -0.006270, 0.066636, 0.042503, 0.007880, -0.024659, -0.013514, -0.066361, -0.053382, 0.004468, -0.129562, 0.100200, -0.030750, -0.087867, -0.021234, 0.054874, -0.090015, -0.041550, 0.005455, -0.090650, 0.047877, 0.022088, 0.023703, 0.038352, 0.044019, 0.029308, -0.023749, -0.036233, -0.016927, -0.029878, -0.063288, 0.026692, -0.016907, -0.055816, 0.030134, -0.012202, -0.082080, 0.059260, -0.058566, 0.034364, -0.073843, -0.127900, 0.042268, 0.020256, -0.057530, -0.035022, 0.000135, -0.032868, -0.032640, 0.021750, -0.034581, -0.018041, -0.070351, -0.057236, -0.005502, -0.007093, 0.037278, -0.004064, -0.009294, 0.016825, 0.019933, 0.008553, 0.012465, -0.025279, -0.052135, -0.033548, 0.058220, -0.061634, 0.015563, -0.051011, -0.023905, -0.049785, -0.019259, 0.041113, 0.051277, 0.028460, 0.055870, -0.023927, -0.113015, -0.012672, -0.000884, 0.050397, -0.013646, -0.092497, -0.055455, 0.036631, 0.084139, 0.009879, 0.048542, -0.099915, 0.030325, -0.007776, -0.011569, -0.053630, -0.068224, 0.017663, 0.058832, 0.071599, 0.012827, 0.056008, -0.021221, 0.043322, -0.071704, 0.006411, 0.035887, -0.073169, -0.010824, 0.020810, -0.015934, -0.095901, -0.114015, -0.026279, -0.049996, -0.020573, 0.051564, -0.072600, 0.012393, 0.015384, -0.062750, -0.008225, 0.027788, -0.009694, 0.030362, 0.027102, 0.079901, 0.007625, -0.148665, -0.032986, 0.032929, 0.015108, -0.007190, -0.009169, -0.042474, 0.063413, 0.016762, 0.025950, 0.036114, 0.036235, -0.049745, -0.028458, -0.058993, -0.061607, -0.032990, 0.002196, 0.052250, -0.005320, 0.095450, -0.093596, -0.055396, -0.051156, -0.095880, -0.064916, 0.016736, -0.004266, -0.052662, -0.061324, -0.016475, -0.058697, -0.033423, -0.085685, -0.042742, -0.012220, 0.026440, -0.034047, -0.007125, -0.034108, 0.000781, -0.040265, 0.020626, -0.058811, 0.039135, -0.007725, 0.022717, -0.002046, 0.012720, -0.085223, 0.030688, -0.067694, -0.016844, -0.014237, 0.037264, -0.025419, 0.080257, -0.024835, -0.017699, -0.016987, 0.059430, 0.191333, -0.044881, -0.078858, -0.040470, -0.002010, -0.117800, -0.049850, -0.001206, -0.000659, 0.031370, 0.014626, -0.068077, -0.017440, -0.075535, 0.048635, -0.028763, -0.038477, -0.065760, -0.033861, -0.024372, 0.043851, 0.024441, 0.072546, -0.004179, 0.016827, 0.047067, -0.027436, 0.091070, 0.071626, -0.041470, -0.018696, -0.020496, 0.039035, 0.067127, 0.149240, 0.010853, 0.054563, 0.033246, 0.032480, 0.031350, -0.034347, -0.011196, -0.023261, -0.013315, -0.053553, -0.017366, 0.031521, -0.014585, -0.009573, 0.092145, -0.039544, -0.032399, 0.015883, -0.058906, -0.112737, -0.084352, 0.105879, -0.026967, -0.015161, 0.050685, -0.013870, 0.021519, 0.019574, 0.039395, -0.021270, 0.019507, -0.067272, 0.008691, 0.080083, -0.071324, -0.019700, 0.076822, 0.094249, -0.093745, 0.023937, 0.020843, -0.044744, -0.047941, -0.023536, 0.061359, -0.060069, 0.016053, -0.023770, 0.006217, -0.069338, -0.025733, -0.040211, 0.034911, -0.029710, -0.013557, -0.022490, -0.093235, -0.041620, -0.001497, 0.057327, -0.001120, 0.053036, 0.005079, -0.016962, -0.048700, 0.114897, 0.050940, -0.092638, -0.040940, -0.182887, 0.005397, -0.012453, 0.014685, 0.055595, 0.004929, 0.019169, -0.097534, -0.079380, 0.004848, -0.215702, 0.004224, 0.048380, -0.027477, 0.050242, -0.044771, -0.058177, -0.057193, -0.026794, -0.058831, -0.024620, 0.076269, 0.035077, -0.041190, -0.047126, 0.091051, 0.022644, 0.029874, -0.049538, 0.070112, 0.026852, -0.007751, 0.049994, -0.007696, -0.002505, -0.016961, -0.118308, -0.009825, 0.054959, -0.012738, 0.079713, -0.138337, -0.096950, -0.006071, -0.016293, -0.086206, -0.032126, 0.022092, -0.091732, -0.039034, -0.061455, 0.009472, 0.042979, -0.095051, 0.021046, 0.036020, -0.044677, -0.074111, -0.135368, 0.025327, 0.002349, -0.077807, -0.004557, 0.047123, -0.105508, -0.100668, 0.014458, -0.058962, -0.055415, -0.063863, -0.075091, 0.062370, -0.035780, -0.031745, -0.037882, -0.057426, -0.154190, -0.078416, -0.012513, 0.035183, 0.019111, -0.004740, -0.003154, 0.129449, -0.072029, 0.035039, 0.020997, -0.043441, -0.019489, -0.027326, 0.078952, -0.052276, -0.060486, -0.033891, -0.068474, -0.024884, -0.017192, 0.015474, -0.139943, -0.026038, -0.055516, -0.059457, -0.028462, -0.000435, -0.062498, 0.095917, -0.028225, -0.062116, -0.028732, 0.043164, -0.009756, -0.021700, 0.020273, -0.010206, 0.059810, 0.002415, -0.060291, 0.014380, -0.154684, 0.036491, -0.133624, -0.028725, 0.111950, 0.010557, 0.039629, -0.019381, -0.042517, 0.018587, 0.009196, -0.072146, 0.000248, 0.035270, 0.047507, -0.024192, -0.036332, -0.119008, -0.026403, 0.082282, -0.051056, -0.059606, -0.056747, -0.046929, -0.011999, -0.069812, 0.007014, -0.045103, 0.062938, 0.029565, -0.073077, -0.081302, -0.138029, -0.025798, -0.020205, -0.040478, 0.064468, -0.003586, 0.072518, 0.026104, -0.018249, 0.000298, -0.019367, -0.002474, 0.003368, -0.080822, 0.014310, -0.002807, -0.009475, -0.036320, -0.054073, -0.105100, 0.122402, 0.027364, -0.038918, 0.065275, -0.042524, 0.073422, 0.048058, -0.017597, -0.029586, -0.011024, -0.082634, -0.043481, -0.038997, -0.002781, 0.005263, -0.037719, 0.019842, -0.000351, -0.061857, 0.028416, -0.046049, 0.039885, 0.045988, 0.039177, 0.038847, -0.102293, 0.010920, -0.023055, 0.009767, 0.072726, -0.052453, -0.146509, -0.009386, -0.076965, 0.059001, -0.024117, 0.027179, -0.025536, -0.084339, 0.038137, 0.013798, -0.045782, -0.051996, -0.029986, -0.057201, 0.009916, -0.012040, -0.033738, -0.027077, 0.018655, -0.003617, -0.084094, -0.053961, 0.038146, -0.033116, 0.057075, -0.019859, -0.065380, 0.016926, -0.066683, 0.009553, -0.051313, -0.066041, -0.019381, 0.035772, 0.072400, 0.000299, -0.006000, -0.002829, -0.005387, 0.011863, 0.013207, 0.002657, 0.074501, 0.027421, 0.038141, -0.026758, -0.039186, 0.056858, 0.019263, -0.122006, -0.046921, 0.069795, -0.056819, -0.173634, 0.009724, 0.093242, 0.041106, 0.050308, 0.005909, -0.039964, -0.051023, 0.020678, -0.011845, -0.065335, -0.006281, -0.048605, -0.022363, 0.050527, -0.055165, -0.035543, 0.036319, -0.025542, 0.027850, -0.034121, 0.072701, 0.006060, 0.003561, -0.040261, -0.037871, -0.010308, 0.042050, -0.065121, -0.060467, 0.014083, -0.012352, 0.025473, 0.004232, -0.031318, -0.020025, -0.050697, -0.068406, -0.023803, 0.015378, -0.043807, 0.017035, 0.180616, -0.094608, -0.025269, 0.037291, -0.010563, -0.017220, -0.032879, -0.014051, 0.004823, -0.020169, -0.005346, -0.030127, 0.060056, -0.044069, 0.069554, 0.148838, -0.016860, 0.002121, 0.003109, -0.056937, -0.026058, -0.030522, -0.012956, 0.003374, 0.005677, -0.089355, 0.000387, 0.031703, 0.000569, -0.049346, -0.033782, -0.139349, 0.037447, -0.058872, -0.048397, 0.013106, 0.074574, -0.007382, -0.060284, 0.033296, -0.010049, 0.050227, -0.006020, -0.046185, -0.011877, -0.001947, -0.003859, -0.060409, -0.030907, 0.066157, -0.019933, -0.019584, -0.047172, 0.103665, 0.041998, -0.053128, -0.060855, 0.037902, -0.044918, -0.025687, -0.055452, -0.138681, -0.029739, -0.050478, -0.032505, -0.034587, 0.052948, -0.087369, 0.075935, -0.056311, 0.059016, -0.031763, 0.042100, 0.033778, 0.035965, -0.012505, 0.072476, -0.022430, -0.001589, -0.008815, -0.062109, 0.041292, -0.101508, -0.029644, -0.093191, -0.007698, 0.036411, 0.042713, 0.001286, -0.019366, -0.005666, 0.044150, -0.002351, -0.032329, 0.050885, 0.051471, -0.064425, -0.036528, 0.007781, 0.051230, -0.114792, -0.071774, 0.015617, -0.010851, -0.114408, -0.031307, 0.014139, -0.018022, 0.000245, -0.049999, -0.041887, 0.027152, -0.058753, -0.059958, -0.056778, 0.042048, -0.021658, 0.020777, -0.038726, 0.006168, -0.076945, -0.203393, -0.009756, -0.091574, -0.068738, -0.006777, -0.045684, 0.171898, -0.059613, -0.072764, -0.075252, -0.089633, 0.043038, -0.043534, 0.009440, -0.067085, -0.012424, -0.027780, -0.027566, 0.005230, 0.042638, 0.036450, -0.121649, -0.101066, 0.024795, -0.075325, 0.029160, 0.006868, -0.048993, -0.018007, -0.005145, 0.029136, -0.060328, 0.168603, -0.027552, -0.050830, 0.075550, -0.139436, -0.073328, 0.027317, 0.007190, 0.013192, -0.025590, 0.032123, -0.022189, 0.009291, 0.023383, -0.049704, -0.004723, -0.063344, 0.066871, 0.007960, 0.069389, -0.077925, -0.121277, -0.098715, -0.108930, -0.056292, 0.064348, -0.029767, -0.037826, -0.045156, -0.068241, -0.036312, -0.037884, -0.019776, -0.000253, -0.012911, -0.039866, -0.037424, -0.040624, -0.134315, 0.042838, -0.121649, -0.024930, 0.014571, 0.097155, -0.043075, 0.038773, 0.035075, 0.080753, 0.026758, 0.011518, -0.027065, 0.044856, -0.075478, 0.019376, -0.020067, -0.042618, -0.067851, -0.095498, 0.056315, -0.074310, -0.006096, -0.009163, -0.009018, -0.017113, 0.004317, 0.100794, 0.056653, -0.076470, -0.085922, -0.047107, 0.044648, -0.027942, -0.005294, -0.008455, 0.035234, -0.033839, 0.074343, -0.008490, -0.125900, 0.017788, -0.012459, -0.043123, 0.058451, -0.029741, -0.010659, -0.019922, 0.022642, -0.031043, -0.006202, -0.036034, 0.011662, -0.046864, -0.062455, -0.080429, -0.046230, -0.117583, -0.027563, -0.139450, 0.051913, 0.019871, -0.036925, 0.004299, -0.013384, -0.078368, -0.053300, 0.007032, -0.089657, -0.088367, -0.030954, -0.034556, -0.102600, 0.010727, -0.103947, 0.057761, 0.158338, -0.091600, -0.025332, -0.059635, -0.070866, 0.007033, 0.069250, -0.063344, 0.023524, -0.050797, 0.027660, -0.056063, -0.063140, -0.076909, 0.096718, -0.023217, 0.049927, 0.029276, 0.055294, -0.010272, 0.055158, -0.053394, 0.026368, -0.078268, -0.116438, -0.033034, 0.132981, -0.034399, 0.018729, 0.064475, -0.113526, 0.018268, -0.084647, -0.102156, -0.032337, 0.063318, 0.004306, -0.097419, -0.027289, -0.077734, -0.010162, -0.069893, -0.059750, -0.130487, -0.050716, 0.019668, -0.015447, -0.023435, 0.039984, -0.029591, -0.073368, -0.097969, -0.094539, -0.124667, 0.027495, 0.043048, -0.028205, -0.006365, 0.040423, 0.000660, -0.096895, -0.003378, 0.080723, -0.038697, 0.006816, 0.014073, -0.065829, -0.093980, -0.066786, -0.011503, -0.044413, -0.034843, -0.131682, -0.059765, 0.113900, -0.063082, -0.016029, 0.099840, 0.036476, 0.076419, 0.059048, -0.141513, 0.005356, 0.011264, -0.043434, -0.017139, -0.056970, -0.071012, -0.079834, -0.075801, -0.043714, -0.104677, 0.082182, 0.014844, 0.047498, -0.037994, 0.103415, -0.100282, -0.009861, -0.039019, -0.013921, -0.124636, -0.060287, -0.136849, 0.018301, 0.039836, -0.008779, 0.035503, 0.046760, 0.092804, 0.002127, 0.023964, -0.041426, -0.034273, -0.041880, -0.011467, 0.046064, -0.016133, 0.017530, 0.005671, 0.025175, -0.040332, 0.020341, 0.035539, -0.102985, 0.029353, 0.001182, 0.050205, 0.014395, 0.103874, -0.024430, 0.035447, -0.060663, -0.021857, -0.027632, -0.065413, 0.076706, -0.041541, -0.009131, 0.037567, -0.034563, -0.067220, 0.009177, -0.049680, 0.006400, -0.078240, -0.010659, -0.043117, -0.007236, -0.120999, -0.023230, 0.008534, -0.042868, 0.122809, -0.001000, -0.027138, -0.069271, 0.030080, -0.027506, -0.033001, 0.046722, -0.007342, -0.041158, -0.018780, -0.155185, -0.063457, -0.045257, -0.142129, 0.010715, -0.017194, -0.025234, 0.079273, 0.045495, -0.070522, -0.031927, 0.012032, 0.041795, 0.019327, 0.036075, -0.011729, -0.144794, 0.081248, -0.013916, -0.163179, 0.023683, 0.074914, 0.087357, -0.101365, -0.042042, -0.022008, 0.035959, -0.043874, -0.047082, -0.072091, 0.043437, -0.057454, -0.001299, -0.035774, -0.069533, -0.054423, -0.060126, 0.037572, -0.054244, -0.020329, 0.006014, -0.060610, -0.018096, -0.007742, 0.011073, -0.033019, -0.023482, -0.103376, -0.070635, 0.008857, -0.079283, -0.051583, 0.021426, -0.028592, -0.077411, -0.100091, 0.004631, -0.014952, -0.100130, -0.027123, -0.090669, -0.058393, -0.043734, -0.094898, 0.131925, -0.005249, 0.084585, -0.135706, -0.060416, -0.064990, -0.000846, 0.003088, 0.132031, 0.002446, 0.055672, -0.016980, 0.024006, -0.035610, -0.022563, 0.042732, 0.012180, -0.111157, 0.008603, -0.068569, 0.013704, 0.096663, 0.011457, -0.024139, -0.016339, -0.100004, 0.012881, -0.100387, -0.037001, -0.028679, -0.003808, 0.045774, 0.034430, -0.083155, 0.094944, 0.009178, -0.045993, -0.030403, 0.000967, -0.068880, 0.078121, -0.026779, -0.053025, 0.035191, -0.064972, -0.148048, -0.013932, -0.013601, -0.000863, 0.046597, -0.110331, -0.119187, -0.006502, -0.171185, -0.069418, 0.055792, 0.039948, 0.017532, -0.038769, -0.066391, -0.013899, -0.066453, -0.072246, 0.027425, -0.073392, -0.058456, -0.055871, -0.028687, 0.040323, -0.060806, 0.060713, -0.006766, -0.061340, -0.066899, -0.097927, -0.096220, -0.091946, -0.036806, 0.003822, -0.050420, -0.040208, -0.057970, -0.111572, 0.000399, -0.125390, 0.020763, -0.015081, -0.063966, 0.032249, 0.026110, 0.056255, 0.028970, -0.045332, 0.030376, -0.074443, 0.013448, -0.099029, -0.025319, -0.065390, -0.109210, -0.038399, 0.039030, -0.083650, 0.054006, -0.032901, 0.061685, -0.022107, 0.011787, -0.097934, 0.009335, -0.036375, -0.169971, -0.046273, 0.023036, -0.037252, 0.001681, -0.116411, -0.102010, -0.137033, -0.005215, -0.027076, -0.001566, -0.010496, -0.018179, -0.132642, 0.008753, 0.036796, -0.056760, -0.095039, 0.025186, -0.026264, -0.135060, 0.026562, 0.055527, -0.021572, -0.041066, -0.062754, -0.082326, -0.053396, -0.005439, -0.054425, -0.067084, -0.006209, -0.017049, -0.066863, -0.013089, -0.074341, 0.006393, 0.021940, 0.006161, -0.022143, 0.018224, -0.006331, -0.038826, -0.174821, -0.072885, 0.013173, -0.060385, -0.091609, -0.037540, -0.027487, 0.011686, -0.074644, 0.058964, 0.089590, 0.012284, -0.099933, -0.010318, -0.123181, -0.026291, 0.043088, -0.031968, -0.004167, -0.061579, 0.008437, 0.039951, 0.094275, -0.021407, -0.050866, -0.082344, 0.033987, -0.068409, 0.041378, -0.075310, -0.119940, 0.010805, -0.006454, 0.005970, -0.038214, 0.065133, -0.110286, 0.022298, 0.024436, -0.036352, -0.018100, -0.035588, -0.138177, -0.086932, 0.007555, -0.126457, -0.071761, -0.058220, -0.077945, -0.123012, -0.005654, -0.077892, -0.001621, -0.073568, -0.013926, -0.058856, -0.044188, -0.003480, 0.045034, -0.015216, -0.045258, -0.096409, -0.048370, 0.003350, -0.028397, -0.076740, 0.029086, -0.006549, -0.014521, 0.072619, 0.028605, -0.001375, -0.044159, -0.036820, -0.066348, 0.011760, 0.025427, -0.048462, 0.049804, -0.021765, 0.049710, -0.049716, -0.069242, -0.015534, 0.003111, -0.079575, 0.002014, -0.132333, -0.018332, -0.188365, -0.063525, 0.014951, -0.056945, 0.018316, -0.085517, -0.068238, -0.064016, 0.035178, 0.002145, 0.033844, -0.069226, -0.006687, -0.045088, 0.000788, 0.043753, -0.030410, -0.021346, -0.064210, -0.074188, -0.102853, -0.088780, -0.007241, 0.011699, -0.000573, -0.039451, -0.028029, -0.167374, -0.019924, -0.091671, -0.038999, 0.113498, -0.087100, -0.028096, 0.010586, -0.056213, -0.043556, -0.061105, -0.101939, -0.081701, -0.063382, 0.025682, 0.039905, 0.018329, 0.009142, -0.032731, 0.018907, -0.005227, -0.064447, -0.029953, -0.064844, -0.019641, 0.118196, -0.011608, -0.018003, -0.098030, 0.038063, -0.081350, -0.021177, -0.061492, -0.077713, 0.014735, -0.056051, -0.017815, -0.038590, -0.011889, -0.111012, -0.045342, 0.066219, -0.028706, -0.113979, -0.078083, -0.007113, -0.000236, 0.062355, -0.042363, -0.067727, -0.009193, 0.004656, -0.071813, -0.030320, 0.016604, 0.024400, -0.201741, 0.002651, 0.051670, -0.092089, -0.047155, 0.027249, -0.056867, -0.039292, 0.025689, -0.012562, 0.002180, 0.022665, -0.020531, -0.059381, -0.058048, -0.039832, -0.051730, 0.054798, -0.010776, 0.028245, -0.039464, -0.043187, -0.077256, -0.088715, 0.064413, 0.003209, -0.040430, -0.072198, -0.004843, -0.101937, 0.006503, -0.105148, 0.054005, 0.002659, -0.027317, -0.013770, -0.045319, -0.025284, 0.012594, -0.010935, -0.169715, -0.073493, -0.045839, -0.153377, 0.055880, 0.052762, -0.014313, -0.020704, -0.094281, 0.109175, -0.042271, -0.046033, -0.019136, -0.010895, -0.007044, -0.033347, -0.063602, -0.090989, -0.131793, -0.088409, -0.057980, -0.063982, 0.040325, -0.035210, 0.035088, 0.055459, -0.071701, -0.118448, -0.101396, -0.109752, 0.040441, -0.070669, 0.065862, -0.061267, -0.015200, -0.057696, -0.106204, -0.075968, 0.054432, -0.108110, -0.063280, -0.147162, -0.082988, 0.013534, -0.124859, -0.089585, 0.048589, -0.036690, -0.076358, 0.099494, -0.000026, -0.069749, -0.071272, -0.045087, -0.016775, 0.072306, -0.017314, 0.029064, 0.032413, 0.052943, -0.013881, 0.047013, -0.119260, -0.059958, -0.037343, -0.015342, -0.025459, 0.034458, -0.029992, -0.002148, -0.017644, -0.066380, -0.041811, 0.025816, 0.008689, -0.127634, 0.036543, 0.034264, -0.122334, -0.059808, -0.117517, -0.052635, -0.073519, -0.055148, 0.081464, 0.049120, 0.004574, -0.090699, 0.081944, -0.029595, -0.023335, 0.068629, -0.102435, 0.011096, -0.012071, 0.008050, 0.028041, 0.029816, -0.042675, -0.015207, 0.147660, -0.086109, 0.001750, -0.012220, -0.131870, -0.046899, -0.054160, -0.019873, -0.031214, -0.032471, 0.009319, -0.040572, 0.007103, 0.017347, 0.062529, -0.039730, 0.025948, -0.067143, -0.014985, -0.127864, -0.059073, -0.069507, 0.015668, -0.058313, -0.001728, -0.102235, -0.092326, -0.079959, 0.008461, 0.041272, -0.038983, -0.068796, -0.111278, -0.043877, 0.025953, -0.033307, 0.016478, -0.041710, 0.003564, -0.104874, -0.021696, -0.053507, -0.059142, -0.060231, -0.014996, -0.039680, -0.077699, -0.085366, 0.002790, -0.041122, 0.028992, -0.063069, 0.015251, 0.082381, 0.022578, 0.014129, 0.034665, -0.014552, -0.019193, 0.080063, -0.000272, 0.039470, 0.029128, 0.064291, -0.043294, -0.080114, 0.010230, 0.054672, -0.066912, -0.052421, 0.082223, 0.003689, -0.100758, 0.043491, -0.034379, 0.017450, -0.058964, 0.015675, -0.051270, 0.098829, 0.078461, -0.022576, -0.071125, -0.027606, -0.016219, -0.045348, -0.031571, -0.094167, -0.045730, 0.014949, -0.086257, -0.014358, 0.029423, -0.001814, 0.016179, -0.005840, -0.146081, 0.057871, 0.003213, -0.034054, -0.037482, -0.055155, -0.080992, -0.040387, -0.035995, -0.043774, -0.033844, 0.042139, -0.019421, -0.050117, 0.003907, -0.067028, -0.015093, -0.012023, -0.009195, 0.076708, -0.045409, -0.047301, -0.014393, 0.027015, -0.020442, 0.021241, -0.092855, -0.062546, 0.069517, 0.020356, 0.032098, -0.044499, -0.005546, -0.059295, -0.028722, -0.034015, 0.015228, -0.032673, 0.024794, -0.068467, 0.117050, -0.054747, -0.063136, -0.034096, -0.083197, -0.039419, -0.136863, -0.024820, -0.046866, -0.076301, 0.005593, -0.075081, 0.050777, -0.055672, 0.039819, 0.019904, 0.048667, -0.060526, -0.036777, 0.010208, 0.018266, -0.072473, -0.012256, -0.016019, -0.064855, -0.090710, -0.054507, 0.012724, -0.014200, -0.033918, -0.064865, -0.147558, -0.051297, -0.033071, -0.067092, -0.022180, -0.024076, -0.073870, -0.052328, 0.069990, 0.030251, -0.090554, 0.020253, 0.040190, 0.013059, 0.015028, -0.025206, 0.085604, -0.100303, -0.086606, 0.015160, 0.003525, -0.059225, -0.047363, -0.024756, -0.034329, -0.024394, -0.068698, -0.022906, 0.043353, -0.060504, -0.038712, -0.057100, 0.137621, 0.046533, 0.037731, -0.018702, 0.036499, 0.052089, -0.005624, 0.010178, -0.063496, -0.032316, -0.053717, -0.066528, 0.008883, 0.050223, 0.039633, -0.038047, -0.062088, 0.018971, -0.064391, 0.035381, -0.044492, 0.094974, -0.079288, -0.112199, 0.013234, 0.006031, -0.088099, 0.000494, 0.056571, -0.070690, 0.016856, 0.014085, 0.049047, -0.035124, -0.095645, -0.003877, -0.020568, -0.001091, -0.038943, 0.002020, -0.000621, -0.023272, -0.159770, -0.009013, -0.030589, 0.020950, 0.155324, 0.007278, -0.072613, 0.063521, 0.009033, -0.116718, -0.076508, -0.031781, -0.073702, 0.045436, -0.005198, -0.034652, 0.013580, 0.005956, -0.013860, -0.001819, -0.024629, -0.007158, 0.060692, 0.138443, 0.027755, -0.099233, -0.033750, 0.025785, -0.016182, -0.019284, 0.083488, -0.022490, -0.064975, -0.113341, 0.022373, 0.209125, -0.008462, -0.052817, 0.044554, -0.042173, 0.010106, 0.013753, 0.005451, 0.045863, 0.057149, -0.101190, 0.020424, 0.003784, 0.035183, 0.053108, 0.049719, 0.002029, 0.098353, 0.049255, 0.059849, 0.006107, 0.007551, -0.021248, -0.057526, -0.059778, -0.139814, 0.017209, -0.007437, 0.044953, -0.079581, 0.035613, 0.015954, 0.038899, -0.057232, -0.044668, 0.095380, 0.006939, 0.098405, -0.078333, 0.003288, -0.090919, -0.066959, -0.031172, 0.106723, -0.043655, -0.062091, 0.059201, -0.042263, 0.074893, 0.027175, 0.034706, -0.127355, -0.050150, -0.094190, -0.072973, 0.054911, 0.029087, -0.057979, 0.068359, -0.062748, 0.053241, 0.068717, 0.014872, -0.060277, 0.032088, 0.034473, -0.037585, -0.070613, -0.017752, 0.037684, 0.111798, 0.095907, 0.077849, -0.073949, 0.099287, 0.077105, 0.013405, 0.032777, -0.050058, 0.024817, -0.065519, 0.022438, -0.065677, -0.118320, 0.098730, -0.034625, -0.094820, 0.112349, -0.050806, -0.034118, -0.069440, 0.035215, -0.053731, 0.018190, 0.014912, -0.005132, 0.010147, -0.005516, 0.019327, -0.039429, -0.025117, -0.025517, 0.079733, -0.125409, -0.055539, -0.073779, -0.057309, 0.012826, 0.037162, -0.028467, -0.104027, 0.039284, 0.042370, 0.042846, 0.023921, -0.066478, -0.038930, -0.029080, 0.040976, 0.012802, -0.007625, -0.018508, -0.025407, 0.066269, -0.005009, -0.018657, 0.120375, -0.009048, -0.137832, 0.076081, -0.069288, 0.028958, -0.110115, 0.018866, 0.122904, -0.022348, 0.036388, 0.031304, -0.072614, -0.009114, -0.113301, -0.050172, 0.078155, 0.000897, 0.043639, 0.026921, -0.156170, 0.045333, -0.032004, -0.010577, -0.005583, -0.025666, -0.069446, -0.022153, 0.095659, -0.106691, -0.058485, 0.319620, 0.028004, -0.012800, 0.016870, -0.012506, -0.002737, 0.075156, 0.059639, -0.090633, 0.014483, -0.013029, -0.002377, -0.021326, 0.000177, 0.135780, -0.050782, 0.048252, -0.026056, -0.009266, -0.020874, 0.009730, 0.041214, 0.040859, 0.036151, 0.001862, 0.034941, -0.037515, -0.058872, 0.018150, 0.172877, -0.006779, -0.063364, -0.036804, -0.027000, -0.090732, 0.049311, 0.079724, -0.041181, 0.093199, 0.031432, 0.011312, -0.099077, -0.081169, 0.017192, -0.031538, -0.031403, -0.005399, 0.097311, -0.068423, 0.045307, -0.088948, -0.081243, -0.029742, -0.012772, -0.054903, -0.018043, 0.010640, -0.075313, -0.088207, -0.042645, 0.012621, -0.209809, 0.034190, -0.047364, 0.069922, -0.044796, -0.064509, 0.004856, 0.053621, 0.023208, 0.047230, -0.027588, -0.048295, 0.038714, 0.033215, 0.026334, 0.065287, 0.023294, -0.141048, 0.031400, -0.000592, -0.035001, -0.013682, 0.022528, -0.037649, -0.060433, -0.045538, -0.012780, 0.012764, -0.004963, 0.035773, -0.031607, -0.007958, 0.010506, 0.040550, -0.062387, -0.085498, -0.023737, 0.019182, -0.032137, -0.025023, -0.017189, -0.050408, -0.087922, 0.015621, -0.003814, 0.082096, -0.046716, -0.095843, -0.067411, 0.034332, 0.080648, -0.056444, 0.056194, 0.033833, 0.026338, 0.088995, 0.077633, -0.067150, 0.035625, 0.013823, 0.004958, 0.010392, 0.077742, -0.007666, 0.020709, 0.053140, -0.069202, 0.002745, 0.049676, -0.027582, 0.044550, 0.015138, -0.051507, 0.015257, -0.003662, -0.005904, -0.012023, 0.048524, 0.008019, -0.007850, -0.051852, 0.011592, 0.104756, 0.145428, -0.135304, 0.063902, 0.043525, 0.004054, 0.012696, -0.071116, -0.005635, 0.113259, -0.081676, -0.044087, 0.049063, -0.027284, -0.056248, -0.010650, 0.093140, 0.013353, 0.050652, -0.050877, -0.051724, -0.090140, -0.057287, 0.008223, 0.052780, -0.011153, -0.052877, 0.114133, -0.011310, -0.059295, 0.076803, -0.038552, 0.025417, -0.057338, 0.006962, -0.064665, -0.130800, 0.042769, -0.006583, 0.028050, -0.072006, 0.088533, -0.059688, 0.040480, 0.053401, 0.016328, -0.066886, -0.038288, 0.031096, -0.000066, -0.112054, 0.148545, 0.057812, 0.059819, 0.030634, -0.038878, 0.028514, -0.094232, -0.027593, -0.042529, 0.027002, 0.007224, -0.007767, -0.119375, -0.022764, -0.040740, 0.062966, 0.015440, 0.070047, 0.029199, 0.062747, -0.027039, 0.030239, -0.041291, -0.127151, 0.015358, 0.039476, -0.056190, -0.008362, 0.085921, 0.027623, -0.103959, 0.092750, -0.022927, 0.193381, -0.024567, -0.029690, 0.001881, 0.015312, -0.108608, 0.007329, 0.025559, 0.018654, 0.031489, -0.023288, 0.002447, 0.016164, -0.028645, 0.011025, 0.024411, -0.071486, -0.069314, -0.069136, -0.012519, -0.092895, -0.062115, 0.057063, 0.071689, -0.027988, -0.045918, 0.019269, -0.092858, 0.059963, 0.082660, 0.003509, -0.070687, 0.032243, 0.030576, -0.020683, 0.016060, -0.047420, 0.031686, 0.012935, -0.016715, -0.052875, -0.061803, -0.040503, -0.031186, -0.053243, -0.016478, -0.051963, 0.040271, 0.089226, -0.097021, -0.002740, 0.037922, -0.000677, 0.095284, 0.110474, -0.015251, -0.000447, 0.022553, -0.000915, -0.054207, -0.034074, -0.033741, 0.024453, -0.021023, 0.018147, -0.009367, 0.096441, 0.008960, -0.042588, 0.061034, -0.060940, -0.058950, 0.031802, -0.087095, 0.092493, -0.069673, 0.033395, 0.087472, 0.006628, 0.027635, -0.035593, -0.049633, -0.108429, -0.075986, 0.038017, 0.008589, 0.006106, 0.049997, -0.015917, -0.006660, 0.004095, 0.012742, 0.055627, 0.033027, 0.028296, -0.051692, 0.073759, 0.004807, -0.080072, 0.049924, 0.061529, 0.078601, -0.042029, -0.002542, -0.047197, -0.001608, 0.054575, -0.033462, -0.018152, -0.002561, -0.043385, 0.057797, -0.063142, -0.065654, 0.011641, -0.081255, 0.007586, 0.067634, 0.004968, 0.011995, -0.033582, -0.086399, 0.094672, -0.021134, -0.052236, -0.072112, -0.052294, 0.069470, -0.007782, -0.039779, 0.032384, -0.071672, -0.033896, 0.012336, 0.026264, -0.010497, 0.105233, 0.056526, 0.076036, -0.051594, -0.008616, -0.026094, -0.003558, 0.012637, -0.095562, 0.065545, -0.065004, 0.047414, -0.073200, 0.069264, -0.018773, -0.020682, 0.057114, -0.062110, 0.023125, -0.017846, 0.122583, -0.046059, 0.105277, -0.035215, 0.034657, 0.050828, 0.073510, -0.050347, -0.019969, -0.069135, -0.051139, -0.036348, -0.026074, 0.037761, -0.085138, 0.015958, -0.007971, 0.063187, -0.026587, 0.048273, -0.034105, -0.062874, -0.017045, 0.041110, 0.045056, -0.004313, -0.053102, -0.027630, -0.060200, 0.118563, -0.020767, -0.035825, 0.006449, 0.014739, -0.056946, -0.068669, -0.061078, -0.090341, 0.030182, 0.056124, 0.174280, 0.005778, -0.006522, 0.002138, -0.066752, -0.001820, -0.025923, -0.039650, -0.043965, 0.026993, -0.070122, -0.048703, 0.083418, -0.067521, -0.057804, -0.026179, 0.048765, -0.043964, -0.026672, 0.117878, 0.121928, 0.005895, -0.075319, 0.026282, 0.057987, 0.018440, -0.072135, -0.056495, 0.028692, 0.049024, -0.016557, -0.009152, 0.053959, -0.070050, -0.051348, -0.040684, -0.015249, -0.039719, 0.003966, 0.083803, 0.137497, 0.179093, -0.018028, -0.040136, 0.018113, -0.042111, 0.000451, -0.069814, 0.028168, -0.068150, -0.049258, 0.026696, 0.022744, -0.015585, -0.067104, -0.084701, -0.040670, -0.053007, -0.044151, 0.014721, 0.034523, -0.072057, -0.093677, -0.037809, -0.118673, -0.053844, -0.112783, 0.044950, -0.048948, 0.048062, 0.028576, -0.074972, -0.015423, -0.013179, -0.065912, -0.005188, -0.000856, 0.013814, 0.016172, -0.033709, 0.028072, -0.057362, 0.012493, -0.053281, 0.081494, -0.075362, 0.072590, -0.039509, 0.000806, -0.051092, 0.047185, 0.018111, -0.055081, 0.008950, 0.000473, 0.023303, -0.078305, -0.060563, 0.064834, -0.024923, 0.029165, -0.014526, 0.015550, -0.022242, -0.048653, -0.015564, 0.012040, 0.038410, 0.000654, 0.027907, -0.048370, -0.049353, 0.028605, 0.018025, -0.024995, 0.081068, -0.002060, -0.112318, 0.073082, -0.001679, -0.067826, 0.012273, 0.012652, -0.027952, -0.028389, 0.051862, 0.000441, 0.027854, 0.016337, -0.010244, 0.007650, -0.007345, -0.077990, -0.051522, -0.032087, -0.023179, -0.071996, 0.036023, 0.022830, -0.066268, 0.040343, -0.045299, -0.071780, -0.006369, 0.027213, 0.009217, -0.018445, -0.035607, 0.014029, -0.170241, -0.005169, -0.029789, 0.085238, -0.024332, -0.051099, 0.000592, 0.051683, 0.069020, -0.034726, -0.030552, 0.042549, 0.068165, -0.051360, 0.001635, -0.030432, 0.053492, -0.038952, -0.057695, -0.097883, -0.001324, -0.018040, -0.058601, -0.011382, -0.054706, -0.053990, 0.017078, -0.018150, 0.068143, 0.071933, 0.014425, -0.055167, -0.021788, -0.021770, -0.067727, 0.053848, -0.056083, -0.029708, -0.046078, 0.090657, -0.038345, 0.000107, 0.004703, -0.001372, -0.044125, 0.004194, -0.127991, 0.015813, -0.076740, -0.057032, 0.047310, 0.103565, 0.020445, 0.120593, -0.034394, -0.062155, 0.012358, 0.061628, 0.113436, -0.043447, 0.048825, -0.049440, -0.054744, 0.023625, 0.063690, 0.035495, 0.074297, -0.015264, 0.000714, -0.068922, 0.067551, -0.079378, 0.011297, 0.074887, 0.062938, -0.111911, -0.028796, -0.085232, -0.032942, 0.033381, -0.014963, -0.114508, -0.104712, 0.009418, -0.131130, -0.036922, 0.027157, -0.042139, 0.028567, -0.017068, -0.081971, 0.038105, -0.013853, 0.048271, -0.036219, -0.062070, -0.107394, 0.004239, -0.111783, -0.123667, -0.018910, -0.028507, -0.065085, -0.028175, -0.038427, -0.089418, 0.002031, -0.045076, 0.064088, 0.019102, -0.033844, -0.035828, -0.079435, 0.019031, -0.054993, 0.139299, -0.009289, -0.002835, -0.069996, 0.018706, -0.044829, -0.059749, -0.079633, -0.038375, 0.118875, -0.067819, -0.040502, 0.026844, -0.095778, 0.057157, -0.031649, -0.064192, 0.007156, -0.040291, -0.031473, 0.059528, 0.075296, -0.034702, -0.006451, -0.041421, 0.127585, -0.027756, -0.026710, -0.056418, 0.019701, 0.034927, -0.072729, -0.036126, -0.018641, 0.016205, -0.006937, -0.047275, 0.004693, -0.020908, 0.016997, -0.112999, 0.003556, 0.024351, 0.098136, 0.041731, 0.036210, -0.028687, -0.031500, -0.030012, -0.020780, 0.061393, -0.045459, -0.005763, -0.068732, -0.093857, 0.058221, 0.028974, 0.035135, -0.064372, 0.023700, 0.038040, 0.007076, -0.018842, -0.037224, -0.036691, 0.037008, -0.108194, -0.022324, -0.087768, -0.044834, -0.035671, 0.114384, 0.033836, -0.034274, 0.116561, -0.104205, 0.043669, -0.018603, -0.028066, -0.135180, 0.074044, -0.030163, -0.077885, 0.045645, -0.033673, 0.024742, 0.122812, 0.066410, -0.113736, -0.050980, 0.072495, -0.008163, 0.026977, 0.068713, -0.026069, 0.055274, -0.025198, -0.012509, -0.082932, -0.022334, -0.058627, -0.061671, 0.118189, -0.066117, -0.164403, -0.002638, -0.000169, 0.058803, 0.037467, 0.027707, 0.040006, -0.055837, 0.023135, -0.057909, 0.010258, -0.099451, -0.103294, -0.041347, -0.053164, -0.046338, -0.019830, -0.002216, -0.024489, -0.014762, -0.033335, 0.075811, -0.023190, -0.095580, 0.060513, -0.087545, -0.038345, 0.059285, -0.059986, 0.049968, -0.094497, -0.015956, 0.018369, 0.025228, 0.019538, 0.019615, 0.008027, -0.015079, -0.005661, -0.151355, 0.082268, -0.014236, 0.009519, -0.026493, 0.025423, 0.009460, -0.033250, -0.006290, 0.064451, 0.016299, -0.032806, -0.155909, 0.034233, -0.082090, -0.084427, -0.015175, 0.012209, -0.096710, -0.083179, -0.009217, -0.029990, -0.191414, 0.017022, 0.005977, -0.079141, -0.012097, -0.076774, 0.003945, 0.066964, -0.043069, -0.100333, -0.026115, 0.009394, 0.032458, 0.027233, 0.051565, -0.024752, -0.042135, -0.019221, -0.039362, 0.051308, 0.048763, 0.012400, -0.069235, 0.022469, 0.040572, 0.104645, -0.043817, 0.022451, 0.005466, -0.139940, -0.047870, 0.021097, 0.094265, 0.045490, -0.057236, 0.011671, -0.071809, -0.044235, 0.026952, -0.016486, -0.007767, -0.006438, 0.050604, -0.067452, -0.164804, 0.018494, -0.112723, -0.072455, 0.049431, 0.014078, 0.010141, 0.021838, -0.135046, 0.050690, 0.081478, -0.076081, -0.047465, -0.028809, -0.076457, 0.047547, -0.029198, -0.036034, 0.014273, -0.094495, -0.045802, 0.030185, -0.050993, -0.026095, -0.047655, -0.072822, 0.020172, -0.060498, 0.001549, 0.038196, 0.006192, -0.101553, 0.043392, -0.035113, -0.067207, 0.003770, -0.005775, -0.059314, -0.058356, -0.018190, -0.029882, -0.145258, -0.013373, -0.068675, -0.025864, -0.058711, -0.078295, -0.058949, -0.039190, 0.050158, -0.035718, -0.048128, 0.045625, -0.083201, 0.049949, 0.103355, -0.039936, -0.026119, 0.053384, 0.016649, -0.079272, 0.003529, 0.085033, 0.034394, 0.040444, -0.080350, -0.022308, 0.065944, 0.027572, -0.039841, 0.042344, 0.047303, -0.048138, 0.023153, -0.003440, 0.011646, 0.049037, -0.037444, -0.075370, 0.011976, -0.066354, -0.061117, 0.000393, 0.053935, 0.001125, 0.052725, 0.040629, -0.065574, 0.035371, -0.080903, -0.057999, -0.064733, 0.024564, -0.142585, -0.053128, -0.004886, -0.071636, -0.080290, 0.006656, 0.065621, 0.041570, 0.067906, -0.035241, 0.084855, -0.043543, -0.084448, -0.019095, 0.022969, 0.017340, -0.003580, -0.008362, 0.052109, -0.122822, -0.103019, 0.021552, -0.061697, 0.059733, 0.011352, 0.081107, 0.038846, 0.030557, -0.005286, -0.025265, 0.082431, -0.018800, -0.004613, 0.018052, -0.007835, 0.084679, -0.017465, -0.095598, 0.041701, 0.042313, 0.009714, -0.016356, -0.005820, 0.070514, 0.044156, -0.057330, -0.041752, 0.023260, -0.152482, 0.001533, -0.057949, 0.021682, 0.050039, -0.032730, 0.097273, -0.030695, -0.123547, 0.021202, -0.090585, -0.046537, 0.031961, 0.006496, 0.050268, -0.007114, -0.046845, -0.055351, -0.025744, 0.106553, 0.005533, -0.008076, -0.065542, -0.087681, -0.087856, -0.080322, 0.069719, -0.040152, -0.010144, -0.134467, -0.068849, 0.016877, -0.028620, -0.058758, -0.051186, -0.095328, -0.003715, -0.075288, 0.018100, -0.054938, -0.071336, -0.020119, -0.159737, -0.056335, -0.187022, 0.019593, 0.063371, 0.099720, -0.227509, 0.021130, 0.030351, -0.037621, -0.034484, -0.011010, -0.032570, 0.003310, 0.065784, 0.044828, -0.048914, -0.043085, 0.070021, 0.093486, -0.013956, -0.122489, 0.041231, 0.020574, -0.006127, -0.106124, -0.089639, 0.082704, -0.051433, -0.050075, -0.113026, -0.072273, 0.010874, -0.065039, -0.043355, 0.018959, -0.173427, -0.063758, 0.088179, -0.107297, 0.051098, -0.019700, 0.019596, -0.008186, 0.021808, -0.058512, -0.044616, -0.033453, -0.041206, 0.014151, -0.048725, 0.001631, -0.018988, 0.088045, -0.018683, 0.077957, -0.066679, 0.020389, 0.049274, 0.062520, -0.100046, -0.106258, -0.029252, -0.047003, 0.014045, -0.144882, -0.041895, -0.068091, -0.072489, 0.039393, 0.010895, -0.077700, -0.007776, -0.011600, -0.002547, -0.016127, 0.047046, -0.147933, 0.025517, -0.083487, -0.032085, -0.039707, -0.025748, 0.034030, -0.023751, -0.047150, 0.046019, 0.030710, -0.034530, 0.001658, 0.038526, -0.039227, -0.025012, -0.017501, 0.002051, 0.057034, -0.009414, -0.047262, -0.068508, -0.024522, -0.011973, 0.097653, 0.024969, -0.047143, 0.008386, -0.057316, 0.007583, 0.028160, -0.069720, 0.135546, -0.082450, 0.038889, -0.037205, -0.041255, 0.013206, 0.020022, -0.013025, -0.039646, 0.025277, -0.062374, 0.014604, -0.035116, 0.042213, -0.069512, -0.155999, -0.068599, -0.021938, 0.033332, -0.030336, -0.075700, -0.057910, -0.061634, -0.083543, 0.102658, -0.042681, -0.048873, 0.024059, -0.021965, -0.065830, 0.013619, -0.087070, -0.057894, 0.000262, 0.002637, -0.071275, -0.015218, -0.040282, -0.038151, -0.029360, 0.058854, -0.076203, -0.074249, 0.037944, -0.058255, -0.069667, 0.014413, 0.039945, 0.040819, -0.035177, 0.078999, -0.015283, -0.115645, -0.037492, 0.015135, -0.033000, 0.102140, -0.003163, 0.007988, -0.042395, 0.019030, 0.082877, -0.042699, -0.030828, 0.020758, 0.007165, -0.089847, 0.056760, -0.011355, -0.077889, -0.026809, -0.103152, 0.096289, -0.033284, 0.073821, 0.012702, -0.014929, -0.067688, 0.171897, -0.040034, 0.024887, -0.041099, -0.000839, -0.044103, 0.027323, -0.024904, -0.100279, -0.008928, 0.060929, 0.010243, 0.116522, 0.010304, 0.036402, -0.011523, -0.018186, -0.079065, 0.060805, -0.073132, 0.022756, -0.017089, -0.062671, -0.018400, -0.030698, 0.038628, -0.062381, -0.080150, 0.011088, -0.071404, 0.099328, -0.031043, -0.025442, -0.028941, 0.035319, 0.075685, 0.141719, -0.118281, -0.042409, 0.084824, -0.007549, -0.069925, -0.057522, -0.104458, -0.058999, -0.060836, -0.005520, 0.037335, 0.009090, 0.013361, 0.065828, 0.015303, -0.067265, -0.006321, 0.033881, -0.110353, -0.083574, -0.049101, -0.070190, -0.008786, 0.006944, 0.043111, 0.008183, -0.150593, -0.041433, -0.065937, 0.045748, 0.033999, 0.005137, -0.031637, -0.000157, -0.040418, 0.111248, -0.017447, -0.040773, 0.028594, -0.020270, -0.019923, -0.071329, -0.036620, -0.031315, -0.057466, 0.042780, -0.033308, 0.009195, 0.122109, -0.000688, 0.038264, 0.020210, -0.089191, -0.099102, -0.007398, -0.072079, -0.079787, 0.023562, -0.032230, -0.054675, 0.043824, -0.087998, 0.012606, -0.015739, -0.002418, 0.045578, 0.008022, -0.112704, 0.005223, 0.032145, -0.120329, 0.054856, -0.060792, -0.025938, -0.012055, -0.018316, 0.024732, -0.008516, 0.023773, 0.059880, 0.055936, 0.058297, -0.065210, -0.018881, -0.040754, -0.083290, -0.050155, -0.129432, 0.081488, -0.053819, -0.034188, 0.094965, 0.002286, 0.001565, 0.075058, 0.023949, -0.162954, -0.041355, 0.004244, 0.049332, -0.027031, 0.019871, 0.047145, -0.065206, -0.126742, 0.042805, 0.015584, -0.051948, 0.149887, -0.081632, -0.054683, 0.026285, -0.033053, -0.024991, -0.011010, 0.052989, 0.056320, 0.027724, -0.049810, -0.073873, -0.060091, -0.025693, -0.051172, 0.036312, 0.000170, 0.019246, -0.165514, 0.088553, 0.111408, -0.010559, -0.068165, 0.043096, -0.103712, -0.060416, 0.025918, -0.034360, -0.022496, -0.059511, -0.016519, -0.065158, 0.046978, 0.043778, -0.082277, -0.082094, -0.067314, -0.028509, -0.051509, 0.000331, 0.037325, -0.067877, -0.094054, -0.050455, 0.052795, 0.000741, -0.066785, 0.071670, -0.150954, -0.049286, -0.046538, -0.056273, -0.053610, -0.072644, -0.074791, -0.085758, 0.018150, 0.024751, -0.053056, -0.050190, -0.107530, -0.027113, -0.067882, -0.108084, -0.071578, -0.077617, -0.089236, -0.060097, 0.053504, -0.015336, 0.022087, -0.020408, -0.037860, -0.047983, 0.060082, -0.039968, 0.068518, 0.066683, -0.125970, 0.015889, -0.003769, -0.080433, -0.051121, 0.017608, -0.023341, -0.065366, -0.124468, -0.096108, -0.017898, -0.119241, 0.004474, -0.100450, -0.035092, 0.089914, 0.050195, -0.070130, -0.050561, -0.002234, -0.024204, 0.060630, -0.041284, -0.049151, -0.062234, -0.038308, 0.038866, -0.032970, 0.001661, 0.078743, -0.052451, -0.041400, -0.014447, 0.065472, -0.075522, -0.093890, -0.017456, 0.037360, -0.038763, -0.080260, -0.006517, -0.006619, 0.046057, 0.157586, -0.014057, -0.015045, -0.013174, -0.077671, -0.009929, -0.098444, -0.008624, -0.011815, -0.055904, 0.126860, 0.023985, -0.103865, -0.112556, -0.066833, 0.082518, -0.048145, -0.039889, 0.007011, -0.041261, -0.007343, -0.032355, 0.068535, 0.041577, -0.069804, 0.085949, -0.046820, 0.012606, 0.019526, -0.062575, 0.024854, -0.026092, -0.002033, -0.032797, 0.075847, -0.054392, -0.005797, 0.059426, -0.018933, -0.089632, 0.009453, 0.123578, 0.011726, -0.036274, -0.008375, -0.076661, -0.025334, 0.039651, -0.038984, -0.009615, 0.044215, 0.023933, 0.038991, 0.033924, -0.053187, -0.066546, -0.030182, -0.085054, 0.078593, 0.009369, -0.001348, -0.036193, 0.052927, 0.023121, -0.079082, 0.009403, -0.074700, -0.063247, -0.078764, -0.032456, -0.054520, -0.015078, -0.060466, -0.024503, -0.038093, -0.069733, -0.125874, 0.016102, 0.004437, -0.043484, -0.028845, -0.023234, -0.004528, 0.061811, -0.002403, -0.046024, 0.003420, 0.000894, -0.029163, -0.022180, -0.162440, -0.094011, -0.024272, -0.132673, -0.063300, 0.091307, -0.027763, 0.006337, -0.090007, -0.016432, 0.136128, -0.058731, -0.114785, 0.092125, -0.011219, 0.005018, 0.040498, 0.001165, -0.023233, -0.038061, 0.016242, -0.106673, -0.092268, -0.063236, -0.000848, -0.046672, 0.027945, -0.245504, -0.024559, 0.044268, 0.000408, 0.030461, 0.032772, -0.100935, -0.075352, -0.046275, 0.017066, -0.070380, -0.117002, 0.019345, 0.141307, -0.009242, -0.067902, -0.090996, 0.026561, 0.066626, 0.007669, -0.041363, -0.005190, 0.091354, 0.001944, -0.020678, -0.008252, -0.071756, -0.069257, -0.001185, 0.068894, 0.035397, -0.121842, 0.010661, 0.007126, 0.008257, -0.066868, -0.136167, -0.071302, -0.067612, -0.029040, -0.143548, 0.014036, -0.148864, -0.018519, -0.034895, -0.033449, 0.064041, -0.068027, 0.025675, -0.062567, -0.038253, -0.059799, 0.033672, -0.014119, -0.028608, -0.106842, 0.087180, 0.057223, 0.010532, 0.160328, -0.038998, 0.023889, -0.098692, -0.048478, 0.010799, -0.075627, -0.070274, 0.077532, -0.011865, -0.006545, 0.077362, -0.048925, -0.119600, -0.015425, -0.031063, 0.108126, -0.021800, 0.032420, -0.000391, -0.083338, -0.026504, 0.096791, -0.172651, 0.055520, -0.131621, -0.049841, -0.099387, 0.066443, -0.056011, -0.000445, 0.017619, -0.064117, 0.082167, 0.037637, -0.003636, -0.026816, -0.025639, 0.009707, 0.034591, 0.024512, -0.008724, -0.049593, -0.022040, -0.079520, -0.083624, -0.026228, -0.013645, -0.104854, -0.153969, 0.051963, 0.013155, 0.002357, -0.030631, -0.069187, -0.008458, 0.010037, -0.159038, 0.118325, 0.040318, 0.112515, -0.073311, -0.071163, -0.028952, 0.004626, -0.018936, 0.009155, 0.025489, 0.018541, -0.125112, -0.031067, -0.109124, 0.013707, -0.014239, -0.003655, 0.022718, 0.042078, -0.012671, -0.044620, -0.049581, -0.031414, -0.030429, 0.130222, 0.071864, -0.121484, 0.083279, -0.012917, -0.061506, -0.076191, -0.044682, -0.030405, -0.038205, 0.053596, 0.011002, -0.091417, -0.002617, 0.006896, 0.045340, 0.063202, -0.018746, -0.023627, 0.101761, 0.034568, -0.003987, 0.095355, -0.021629, 0.121160, 0.032900, 0.090285, -0.127754, 0.104892, -0.026900, 0.026999, 0.065137, -0.020315, -0.093366, -0.030082, 0.003731, 0.002145, -0.021392, 0.039794, -0.016894, 0.043364, -0.124654, 0.034490, -0.084529, -0.015888, -0.010685, 0.069916, -0.074626, -0.022434, -0.024905, -0.095428, -0.103250, -0.035819, -0.075149, -0.036215, -0.006044, -0.118777, 0.053173, 0.038635, -0.063279, 0.035325, -0.002720, 0.037988, 0.004836, -0.172429, 0.034281, 0.008569, -0.046261, 0.038567, 0.047770, 0.104693, -0.032718, 0.113230, -0.003414, -0.071512, -0.090990, 0.016501, -0.023967, -0.029837, -0.014404, -0.035837, 0.031301, -0.005304, -0.080298, -0.011318, -0.012568, -0.052195, -0.066339, -0.022279, -0.068600, 0.068414, 0.008989, 0.004275, 0.034964, -0.047333, -0.006808, 0.026726, -0.007331, 0.048556, 0.024670, -0.040821, 0.013377, -0.076738, 0.007987, -0.005669, -0.028693, -0.011966, 0.037861, -0.129970, 0.004072, -0.041832, 0.041890, 0.054501, -0.037874, -0.057595, 0.014025, -0.117333, -0.078161, 0.013103, -0.042761, -0.054029, -0.012767, 0.040287, -0.084435, -0.027526, -0.067111, 0.037326, 0.003211, -0.011835, 0.110192, 0.007193, 0.015989, -0.117741, -0.095084, -0.069495, -0.064937, 0.067417, -0.007709, -0.116138, 0.133427, -0.040075, -0.068998, -0.094114, 0.017266, 0.080190, 0.081173, 0.032929, -0.001437, -0.000121, -0.145873, -0.061367, -0.005034, -0.047468, 0.026468, -0.062105, -0.033034, -0.005354, -0.036344, -0.057949, -0.052359, 0.006739, 0.003184, 0.012862, -0.043993, -0.085665, -0.009703, -0.076681, 0.010265, -0.034505, -0.062825, 0.003740, -0.008174, -0.073151, -0.073972, -0.001785, 0.048277, -0.011432, -0.036362, -0.066351, -0.114087, -0.027787, -0.074961, -0.105395, -0.056943, -0.091061, -0.027747, 0.012904, -0.059501, -0.004415, -0.085637, -0.058028, -0.060972, 0.001191, 0.016803, -0.014488, -0.009132, 0.053292, -0.040342, -0.057881, 0.044773, -0.003028, 0.023745, -0.045551, -0.008573, -0.016091, -0.037750, -0.052733, 0.010832, 0.037272, -0.049176, 0.035941, -0.016030, -0.037505, 0.004706, -0.117621, -0.024210, 0.000025, -0.004070, -0.082910, 0.013908, -0.005260, 0.001733, -0.161974, -0.004335, -0.037136, 0.005960, -0.016146, 0.108793, 0.042072, 0.048808, -0.051592, 0.120524, -0.035307, -0.048568, -0.021645, -0.101903, -0.068577, -0.050502, 0.027116, -0.019851, -0.099929, 0.132840, 0.014161, 0.003945, 0.016956, -0.039709, -0.022645, 0.051454, 0.023197, 0.009994, -0.037592, 0.024113, -0.076072, 0.053358, -0.100911, -0.038162, -0.072694, -0.005238, 0.008950, 0.017516, 0.033670, 0.020600, -0.075277, 0.216632, 0.007520, -0.086666, 0.053859, 0.068589, 0.043062, 0.060872, 0.030002, -0.043852, -0.213790, -0.010263, 0.014792, -0.031507, 0.016371, 0.037125, -0.093121, -0.025039, 0.079124, -0.017073, -0.050065, -0.081745, -0.056126, 0.036945, 0.029734, -0.001640, 0.025701, 0.110358, 0.051246, -0.032884, -0.131836, -0.056032, 0.060600, -0.062282, 0.037781, 0.093938, -0.042879, -0.022941, -0.040572, 0.031429, -0.042275, 0.015751, 0.061597, 0.103321, 0.036421, -0.129084, 0.085193, 0.042936, 0.067626, 0.093132, -0.035417, 0.021787, 0.028012, 0.001495, -0.090384, -0.010580, -0.049488, -0.027892, -0.122048, 0.010758, 0.031075, 0.014802, -0.040864, 0.020796, 0.007602, 0.182626, 0.022307, -0.038781, -0.061566, -0.054578, 0.037383, 0.088426, -0.051715, -0.015572, -0.066712, -0.021677, -0.069625, -0.036216, -0.133513, -0.114576, -0.013551, -0.034087, -0.092949, -0.043482, 0.078064, 0.031072, 0.007481, 0.034626, -0.063858, 0.076978, -0.005986, 0.014371, -0.017134, -0.038928, -0.051639, 0.023548, 0.036863, 0.049345, 0.044915, 0.100209, -0.057641, -0.013136, -0.051075, 0.048343, 0.045202, -0.019347, -0.023960, -0.065128, -0.093952, 0.013289, 0.026342, -0.006427, -0.024745, -0.020170, -0.039298, -0.112279, -0.083830, -0.025821, -0.067206, -0.016822, -0.061656, 0.056770, 0.065163, -0.128873, -0.087752, -0.031437, 0.004674, -0.027911, -0.056031, 0.061275, -0.072045, -0.082009, 0.107843, 0.007007, 0.022433, 0.000670, 0.030603, -0.050888, -0.015503, 0.024331, 0.000293, -0.071280, -0.057165, -0.034107, -0.017351, -0.006954, -0.106516, -0.041826, -0.028612, -0.010070, -0.057791, -0.055772, -0.041530, -0.087061, -0.059593, -0.027837, -0.026583, -0.003602, 0.013277, -0.044202, -0.035744, -0.067381, 0.060128, -0.011140, 0.021931, -0.063239, -0.091940, 0.001989, -0.065050, -0.038669, -0.048098, -0.016562, -0.017641, -0.003698, 0.026835, -0.204959, -0.069667, -0.027662, -0.030269, 0.021575, -0.112754, -0.014769, 0.060956, 0.022999, 0.005406, -0.088211, -0.066657, 0.001808, -0.114930, 0.069394, -0.102290, 0.031350, -0.014205, 0.005584, 0.022216, -0.040277, -0.034559, -0.029965, -0.043947, -0.011838, -0.032319, -0.024931, -0.077290, -0.103654, 0.015910, 0.008398, 0.098349, -0.041523, 0.037467, -0.049080, 0.094721, 0.031240, 0.014185, -0.092983, -0.063629, -0.052954, 0.065857, 0.020994, -0.014410, 0.010214, 0.083285, 0.024155, 0.004659, 0.036322, -0.041877, 0.007120, -0.019104, -0.011198, -0.069313, 0.020985, -0.015463, 0.026829, 0.006498, 0.007847, -0.004866, -0.002622, -0.052523, -0.052248, -0.057722, 0.079508, -0.013770, 0.001726, 0.029540, 0.016502, 0.136111, -0.005143, 0.123847, -0.070965, 0.004294, 0.011642, 0.000245, -0.056367, -0.047452, -0.102426, -0.049730, -0.078150, -0.040246, 0.005192, -0.088500, -0.083011, 0.026213, 0.014631, -0.041917, -0.067520, 0.022323, -0.068022, 0.005739, -0.007656, 0.025133, 0.031452, 0.009492, -0.038475, -0.013191, -0.010780, 0.018466, 0.010595, -0.002664, 0.023741, -0.107771, 0.028031, 0.041888, -0.071061, -0.072695, -0.011542, -0.083736, -0.075932, -0.016699, -0.007233, -0.020261, 0.091647, 0.008339, 0.018670, -0.052877, 0.003407, -0.048155, -0.000522, 0.031769, 0.003330, -0.010171, 0.052261, -0.040001, -0.054127, 0.082584, 0.054860, 0.071362, -0.049097, -0.101133, -0.028537, 0.044227, -0.009978, 0.052395, -0.055247, 0.044261, -0.064136, 0.023445, 0.048519, -0.045905, 0.010372, -0.010737, 0.027794, 0.036671, 0.025910, -0.028070, -0.015605, -0.051439, -0.057995, 0.043756, -0.067331, -0.045160, 0.008270, -0.058721, -0.028610, 0.031291, -0.021966, -0.035897, -0.065865, -0.018216, -0.051061, -0.022462, 0.061275, -0.101352, -0.122126, 0.065560, -0.085598, -0.007054, -0.073497, 0.077293, -0.016637, -0.000637, -0.015715, -0.033038, -0.077654, -0.052574, 0.040477, -0.028718, -0.063151, -0.077081, -0.019042, 0.001885, 0.029096, 0.023958, 0.020386, -0.026546, 0.028294, 0.119010, 0.052813, 0.006813, -0.152014, -0.095931, 0.017053, -0.049103, -0.057840, -0.042791, -0.025777, -0.009090, 0.096208, -0.019880, -0.009494, 0.016705, -0.031805, -0.001008, 0.000528, -0.057861, -0.001406, -0.064320, -0.082199, 0.049803, 0.001032, -0.093770, 0.135061, -0.199487, -0.053408, 0.111862, -0.093277, 0.045721, -0.028592, -0.123794, -0.011867, -0.000927, -0.025471, 0.021400, 0.008333, -0.037731, -0.133428, 0.037128, -0.069784, -0.054193, 0.027113, -0.025033, 0.020668, -0.055469, 0.003364, 0.010607, -0.035317, 0.053856, -0.065391, -0.058758, 0.058466, -0.030951, -0.019208, -0.070885, 0.027650, -0.060063, -0.063588, 0.030806, -0.018171, -0.089786, 0.000810, -0.028146, 0.006911, -0.089359, -0.091410, -0.040516, -0.114446, 0.118755, -0.077160, -0.052978, -0.066517, 0.109765, -0.022372, -0.070643, 0.045311, 0.016660, 0.027629, 0.084289, 0.108804, -0.052596, 0.012655, 0.000474, 0.262323, 0.107861, 0.035015, -0.009988, -0.014417, -0.004599, -0.027613, -0.015977, 0.068839, -0.013386, 0.118876, 0.096674, 0.034345, -0.057195, -0.034588, -0.009273, 0.038044, 0.042131, 0.033968, -0.023462, 0.058310, -0.042213, -0.021420, 0.094477, -0.019613, 0.059100, 0.001321, 0.082377, -0.053560, 0.012363, -0.006580, 0.023198, 0.009329, -0.080703, -0.052897, -0.021370, 0.027625, 0.055210, 0.034800, -0.063538, -0.000782, 0.022280, -0.040503, -0.048492, -0.007167, 0.065638, -0.064884, -0.064426, 0.115183, -0.018366, -0.044861, 0.000325, 0.004492, -0.107012, 0.167927, -0.069162, 0.013880, -0.015359, -0.074816, 0.002193, -0.009950, -0.014247, -0.085096, -0.057094, 0.033032, 0.097787, 0.034248, -0.092321, -0.054145, 0.047782, -0.066193, 0.002423, -0.119866, -0.146776, -0.047844, -0.097745, -0.007903, -0.039590, -0.109181, -0.020219, 0.003621, 0.010128, -0.055368, 0.041297, -0.014251, 0.117268, 0.038296, 0.053542, -0.053396, -0.057144, -0.044458, 0.023964, 0.004678, -0.066739, -0.045547, -0.059399, -0.111474, 0.013327, -0.010506, 0.019632, -0.055290, -0.042196, -0.015457, 0.070431, -0.043924, 0.010030, 0.073313, 0.004915, 0.004144, -0.076076, -0.110042, -0.119586, 0.004603, -0.046194, -0.048547, -0.059873, -0.008461, -0.047596, 0.024358, 0.025931, -0.068898, -0.068560, -0.066170, -0.022742, 0.006287, 0.029260, 0.024575, -0.079662, -0.062199, -0.038922, 0.034507, -0.089355, -0.117128, -0.024100, -0.029929, -0.037076, 0.007566, 0.015088, -0.100538, 0.171424, -0.150717, -0.045554, -0.021019, -0.010908, -0.052081, 0.047759, -0.079151, -0.035935, 0.064679, 0.042439, -0.027761, -0.001393, 0.045461, 0.000683, -0.020077, -0.093380, -0.052253, 0.026851, -0.058023, 0.046226, -0.003096, 0.001428, -0.059312, -0.055173, 0.029224, -0.034731, 0.015288, 0.035466, -0.089376, -0.023437, 0.060027, 0.017776, 0.100319, -0.009925, 0.068369, -0.046128, -0.003968, 0.075965, 0.003979, -0.042299, -0.005008, -0.012447, -0.111961, 0.018585, -0.022868, -0.106734, -0.075887, 0.002175, -0.055066, 0.150747, -0.027803, -0.130054, -0.153668, -0.033711, -0.108376, -0.047659, -0.061454, 0.039820, -0.054973, 0.098862, -0.017255, 0.064381, -0.023994, -0.016951, 0.021774, -0.036047, 0.024546, 0.004380, -0.093370, 0.002029, 0.046694, -0.021094, -0.021340, -0.182591, -0.086098, -0.011250, 0.065229, -0.047417, 0.012378, -0.077497, -0.013356, -0.038267, 0.136563, -0.086304, -0.029439, -0.056190, -0.039076, 0.000978, 0.092323, 0.137014, -0.008165, -0.051183, -0.026877, -0.065079, 0.039566, 0.077658, -0.041589, -0.045406, 0.001714, -0.115522, -0.057031, -0.011876, -0.018816, 0.027159, -0.045867, -0.029629, 0.014809, -0.056687, 0.048778, -0.063548, -0.010323, -0.071952, -0.013165, -0.069725, -0.049830, -0.049187, 0.003999, -0.101414, -0.064921, -0.064182, 0.029947, 0.009852, -0.123124, 0.000580, -0.046190, -0.016109, -0.076533, 0.014815, 0.010090, -0.082914, 0.010732, 0.042524, 0.070201, 0.004087, 0.039599, 0.048523, -0.046233, -0.003141, 0.029099, -0.104957, -0.107767, 0.053735, -0.041015, -0.062134, -0.099201, -0.031089, 0.038572, -0.031087, -0.051021, -0.042183, -0.014360, -0.031168, -0.046065, 0.005093, -0.039771, -0.091611, -0.006540, -0.057794, 0.039553, 0.071015, 0.121741, 0.018579, 0.042641, 0.032717, -0.040318, -0.042233, -0.003382, 0.068709, -0.107910, -0.046655, -0.022244, 0.001923, -0.023168, 0.015950, -0.073373, -0.066683, 0.014764, -0.005346, -0.008301, -0.035371, -0.038564, -0.131580, -0.037859, -0.030142, -0.028784, -0.018312, -0.043827, -0.100202, 0.114736, -0.077837, 0.010873, 0.012171, 0.002553, 0.087725, 0.047800, 0.033669, -0.029530, -0.018801, -0.028650, 0.039113, -0.090571, -0.002895, 0.049229, -0.042977, -0.105430, -0.067487, 0.044469, -0.021352, -0.078898, -0.003952, 0.023844, 0.052033, -0.023124, 0.053781, -0.013546, 0.008080, 0.030079, -0.015146, -0.060177, -0.036400, -0.095885, -0.044151, -0.072353, 0.054703, -0.024168, -0.011904, -0.069642, 0.051328, 0.029750, 0.049760, -0.046100, -0.065706, 0.134669, -0.010121, -0.042161, 0.005959, -0.054260, 0.063504, -0.083368, -0.186900, -0.037956, 0.047674, -0.018430, -0.074706, -0.029650, -0.015748, 0.032250, -0.038369, 0.049469, -0.051238, -0.013545, 0.006222, 0.113050, -0.035685, -0.080549, -0.031164, 0.038374, 0.059334, 0.004108, -0.022563, 0.006850, 0.056610, 0.035747, -0.050268, 0.091338, -0.015550, 0.037682, -0.021656, -0.098630, 0.026639, -0.035191, -0.018913, -0.004762, 0.051063, -0.087103, -0.016036, 0.064061, -0.065416, -0.056038, -0.066084, -0.001884, -0.028363, -0.044878, -0.002644, -0.064755, -0.001232, -0.059341, -0.010682, -0.001798, -0.096711, -0.017885, -0.047093, -0.018104, -0.046296, -0.062824, -0.010801, -0.094821, -0.025796, -0.079502, -0.103469, -0.062498, 0.043112, -0.078925, -0.049192, -0.015590, 0.018008, 0.070069, 0.031131, -0.007252, 0.034839, -0.000250, -0.006340, -0.070880, -0.013989, 0.010309, -0.148066, 0.044132, 0.050958, 0.022550, -0.099926, 0.100042, 0.026562, -0.084536, 0.028850, 0.036268, -0.083884, 0.013611, -0.095261, -0.033161, -0.040682, 0.025455, 0.011141, 0.034903, -0.061312, -0.110092, -0.008646, 0.048517, -0.097633, 0.011103, -0.043318, -0.034133, -0.008646, 0.078494, -0.068407, 0.017647, 0.006692, 0.018143, 0.019060, 0.048886, -0.040359, -0.018739, -0.114058, 0.019037, -0.046612, -0.042677, -0.101640, -0.001457, -0.075715, -0.050418, -0.052081, -0.033711, -0.026422, -0.009858, 0.004602, 0.016220, -0.006305, 0.025172, 0.002633, -0.006160, 0.099736, -0.061199, -0.018061, -0.079692, -0.042640, 0.055329, -0.020728, -0.049034, -0.101616, -0.025322, -0.142093, 0.017399, -0.019246, -0.026933, -0.047800, 0.015903, -0.045776, -0.031823, 0.043230, -0.000452, -0.003076, -0.006807, 0.056074, -0.055118, -0.054720, -0.067180, 0.040155, 0.040950, -0.042691, 0.064183, -0.014743, -0.016450, -0.012349, 0.007848, -0.059858, -0.023990, 0.021094, -0.031005, -0.085781, 0.018223, 0.005581, 0.008097, 0.022569, -0.063286, -0.028969, -0.026498, -0.029604, -0.092524, 0.052389, -0.000448, -0.108158, -0.014714, -0.032915, -0.096369, 0.039324, -0.046976, -0.092998, -0.070614, 0.022444, -0.065170, -0.054247, -0.041230, -0.050138, 0.043881, -0.016960, 0.054636, -0.053519, 0.098682, -0.083118, 0.008533, -0.056298, 0.047702, -0.057970, -0.096212, 0.014936, -0.075843, 0.009761, 0.000074, -0.019254, -0.062948, -0.026621, -0.011749, -0.023212, -0.031897, -0.007167, -0.019373, -0.103329, 0.050220, -0.005090, 0.038643, 0.002464, -0.040953, -0.009738, 0.079179, 0.013232, 0.016298, 0.045346, 0.010643, -0.070875, -0.048328, -0.023604, -0.094906, -0.042392, -0.004276, 0.018839, 0.013049, 0.012554, -0.008577, 0.019899, -0.094792, -0.019986, -0.076356, -0.034073, -0.049343, 0.081033, 0.014974, 0.032758, -0.013641, -0.027146, 0.012229, -0.028250, -0.095141, 0.028718, 0.083797, 0.015972, 0.038210, -0.039748, -0.103002, 0.021680, -0.026995, 0.018303, -0.016937, 0.001514, -0.060331, -0.016584, 0.021673, 0.013070, 0.030189, 0.018479, -0.087754, 0.032099, 0.021044, 0.021093, 0.114574, -0.030647, -0.109618, 0.025556, 0.019136, -0.083658, -0.005729, -0.076280, -0.045591, 0.059549, 0.023120, -0.029019, -0.066977, 0.023662, -0.018151, -0.025174, 0.035848, -0.045776, 0.044220, -0.059188, 0.033799, 0.063550, -0.024641, 0.009814, 0.037432, -0.059699, -0.029641, -0.074149, -0.025809, -0.030222, -0.012968, 0.027838, -0.007695, 0.022574, -0.021718, 0.057385, 0.046425, -0.050464, -0.109997, -0.074700, -0.046739, 0.046810, 0.001023, -0.084869, -0.050740, 0.012466, -0.120730, -0.047044, 0.011051, -0.029364, -0.077063, -0.017950, -0.055265, 0.020862, -0.022896, -0.114540, -0.038243, 0.052104, -0.009762, -0.045478, -0.033479, 0.035804, -0.017796, 0.010726, -0.093711, -0.063070, 0.047183, -0.032055, 0.022066, -0.041289, 0.004203, 0.036030, -0.016088, 0.010889, -0.043811, -0.048730, -0.029003, -0.045989, -0.024385, -0.022380, 0.044910, -0.058122, -0.061240, -0.031600, -0.022437, -0.018108, -0.022315, -0.076635, -0.089371, -0.030074, -0.060543, 0.047147, -0.086661, -0.006150, -0.067469, -0.018868, 0.018297, -0.082451, 0.064372, -0.043816, -0.018738, 0.003147, 0.027397, -0.040646, 0.000274, -0.038979, -0.008280, 0.030388, 0.003635, -0.017214, 0.034987, -0.118157, -0.018032, -0.022654, -0.031312, 0.044652, -0.069255, -0.030965, 0.034715, -0.075531, -0.017096, 0.033153, 0.004251, -0.011370, 0.059751, -0.025585, 0.051580, 0.028205, 0.002037, 0.010749, -0.006426, -0.049328, 0.051150, -0.008139, -0.043753, -0.009629, -0.083170, 0.070614, -0.041887, -0.033012, 0.015103, 0.042551, 0.017541, 0.003365, -0.066537, -0.065231, -0.115623, -0.057324, 0.011082, -0.048797, -0.071578, -0.068005, -0.007040, 0.006673, -0.043245, -0.000148, -0.063529, -0.053032, -0.043664, -0.008494, 0.057808, -0.043031, 0.088639, -0.005591, 0.076710, -0.071360, 0.021647, -0.002208, 0.055329, -0.058362, 0.024719, -0.022653, -0.075538, -0.038453, 0.006305, -0.014019, 0.060966, -0.034785, 0.012990, -0.008331, 0.038953, -0.031382, -0.018364, -0.041458, 0.009089, -0.077315, 0.061429, 0.040817, -0.049265, -0.002956, -0.061082, -0.022401, 0.041470, -0.018082, 0.051063, 0.005589, -0.025924, -0.111830, 0.007141, 0.004645, -0.099225, 0.037197, -0.006960, -0.074875, -0.052601, -0.019507, -0.052834, -0.045995, -0.003817, -0.044800, -0.030655, -0.053735, -0.044254, 0.035158, 0.045846, -0.040490, -0.085759, -0.020933, 0.048072, -0.027672, -0.036461, -0.045873, -0.031668, 0.005802, 0.008808, 0.011317, -0.025355, 0.026742, -0.000351, 0.012179, 0.046593, -0.010342, -0.008665, 0.027551, 0.007960, -0.126142, -0.044760, 0.017028, 0.004025, 0.041667, -0.069960, -0.066381, -0.036615, 0.015996, -0.017329, -0.061874, 0.013174, -0.027413, -0.021606, -0.026426, -0.066034, 0.043785, -0.021734, -0.013743, -0.030797, -0.023127, -0.171573, 0.025120, -0.031315, 0.061983, -0.055530, -0.026686, 0.043461, 0.061141, -0.102472, -0.113016, 0.003717, -0.020174, -0.018590, -0.073318, 0.032834, 0.027776, 0.033648, 0.001106, 0.050963, -0.012978, -0.035329, -0.079148, -0.007040, 0.026273, -0.033209, -0.005376, 0.042515, 0.008282, -0.012145, -0.044603, -0.047544, 0.014329, -0.023810, -0.025123, 0.052252, 0.008729, -0.020252, 0.014614, 0.020309, 0.042577, 0.026317, 0.014189, 0.044839, -0.022640, -0.033655, -0.026392, 0.039604, -0.032295, -0.025470, -0.046302, 0.052858, 0.016897, 0.056876, -0.043651, 0.074684, 0.020858, -0.063836, -0.133867, -0.001580, 0.077694, -0.081354, 0.035884, -0.022956, -0.014803, -0.043127, 0.016504, -0.008209, 0.018094, -0.008029, -0.055126, 0.062589, 0.010811, -0.003220, -0.040971, 0.019925, -0.059223, 0.073506, -0.002393, 0.036865, -0.138558, -0.063170, 0.045169, 0.052753, 0.008873, 0.010586, -0.017934, -0.113463, -0.064081, -0.008669, 0.035354, 0.046842, -0.034869, 0.008857, -0.016863, 0.015465, -0.060112, -0.058016, 0.005953, -0.036716, -0.077192, 0.026905, -0.019112, -0.008688, 0.016049, -0.080920, -0.095521, -0.039925, -0.014999, 0.004878, -0.087634, 0.006994, 0.057728, -0.099952, -0.049228, -0.009720, -0.064081, 0.129784, -0.068510, -0.021272, -0.013204, -0.030990, 0.033751, 0.009636, 0.008765, -0.070829, -0.019931, 0.042176, 0.031463, -0.026178, -0.001853, -0.088426, -0.071150, -0.061637, 0.005408, 0.025237, 0.008306, -0.111044, -0.005879, -0.044194, -0.126503, 0.001382, -0.050961, -0.050784, -0.112752, -0.044135, -0.042468, 0.039039, 0.026747, -0.068144, -0.044074, 0.069927, -0.089902, 0.062783, -0.055596, -0.014391, -0.007608, 0.016241, 0.021999, 0.031745, 0.032357, 0.019534, 0.052825, 0.071513, -0.022159, -0.008617, 0.022197, -0.017440, 0.051426, 0.064349, -0.092189, -0.046062, -0.058008, -0.047182, 0.000295, -0.004089, -0.047958, -0.071021, 0.080999, 0.015173, 0.035836, 0.018794, 0.161428, 0.023590, -0.030109, -0.035094, -0.053894, -0.017286, 0.010672, 0.035495, -0.064155, -0.106958, -0.056163, -0.072894, 0.012871, -0.024238, 0.080222, -0.072683, 0.089237, -0.005235, -0.011006, -0.061048, -0.107180, -0.058237, -0.014402, -0.107094, 0.078878, -0.034567, 0.048717, -0.073783, -0.124705, 0.016298, -0.027525, -0.008295, -0.004525, -0.030510, -0.024917, 0.068338, 0.023557, -0.074500, 0.072404, 0.000372, -0.044724, -0.124550, 0.051457, 0.040884, 0.010242, -0.036046, 0.030551, -0.043822, -0.050754, -0.055042, -0.036378, -0.059836, -0.097718, -0.029141, 0.032765, -0.011873, 0.049201, -0.108528, -0.039156, 0.016969, -0.071632, -0.055588, -0.005313, -0.018407, -0.060857, 0.046470, -0.041876, -0.003125, 0.055535, -0.000986, 0.031926, 0.012546, 0.029454, -0.075424, -0.007464, -0.028650, -0.017618, -0.005312, -0.025649, -0.071474, -0.102956, -0.013465, 0.048739, -0.055924, 0.005034, -0.048388, -0.027885, 0.074461, -0.071462, -0.004881, 0.060105, -0.031633, -0.009870, 0.121557, 0.029114, -0.050040, -0.051759, -0.052622, 0.003985, -0.016583, -0.098281, -0.114893, -0.030850, -0.039094, 0.026079, -0.006789, -0.030795, -0.022080, -0.042150, -0.057442, -0.008494, 0.006479, 0.022205, 0.023284, -0.066408, 0.018903, 0.000089, -0.011774, 0.045087, -0.057776, 0.068319, -0.074939, 0.004979, 0.023293, 0.011240, 0.019987, -0.103693, 0.138707, 0.056102, -0.012170, -0.026553, -0.020062, 0.017888, 0.016952, 0.005346, -0.061397, -0.008703, -0.121717, 0.040293, 0.035133, 0.035331, -0.012494, 0.000598, -0.116393, -0.022313, 0.017337, -0.063400, 0.004560, 0.006580, 0.023111, -0.052307, -0.021804, 0.047632, -0.039640, -0.002307, 0.029175, -0.045767, 0.095653, -0.024724, 0.002207, 0.012937, 0.009074, 0.044276, 0.048885, 0.060916, -0.037859, -0.050408, -0.044318, 0.000651, -0.074777, -0.019060, -0.034917, -0.044640, 0.013449, 0.005212, 0.063815, -0.007728, -0.017658, 0.094269, -0.009943, -0.009536, -0.035012, -0.130310, 0.047626, -0.044902, 0.016838, -0.093957, -0.050253, -0.011136, 0.034479, 0.009492, 0.040296, -0.010395, 0.027342, -0.033297, -0.018768, -0.041414, 0.060481, -0.050969, 0.055165, 0.027832, -0.002072, 0.011365, 0.043301, 0.035285, -0.031291, -0.041741, 0.018594, -0.042623, 0.081528, 0.014450, 0.014108, -0.070298, -0.076701, 0.070227, -0.063381, -0.020545, -0.045014, -0.026746, 0.056989, -0.038628, 0.010699, 0.032868, -0.105970, 0.044715, -0.069621, -0.024200, 0.010808, 0.046802, 0.021720, 0.019480, -0.065463, -0.006374, -0.078502, -0.119398, -0.054017, -0.022880, -0.157637, -0.027348, 0.015805, 0.126862, -0.040358, -0.058850, -0.019897, 0.048223, 0.038382, -0.020551, 0.031420, 0.018029, 0.015030, -0.023767, -0.013312, 0.128916, 0.040729, 0.016247, 0.074836, 0.044861, -0.137330, 0.033111, -0.106081, 0.023794, -0.055545, 0.001686, -0.124781, 0.026027, 0.005501, 0.004129, -0.017103, -0.035042, -0.032180, -0.003926, 0.075678, -0.053645, -0.107262, -0.003857, 0.016707, 0.018571, 0.030843, 0.000169, -0.025980, -0.072854, -0.027060, 0.037036, -0.144828, -0.068933, -0.024014, -0.038598, -0.082106, 0.010002, -0.141612, 0.012501, -0.063501, 0.023875, -0.013860, -0.039354, -0.127690, -0.017888, 0.128536, -0.047581, -0.010913, -0.094350, -0.023977, 0.023948, -0.021118, -0.104935, 0.020919, -0.024894, 0.005805, -0.027477, -0.084498, 0.032250, 0.037147, -0.092800, 0.053713, -0.171999, -0.020614, 0.037290, 0.026250, 0.095979, -0.074169, 0.051810, -0.068043, 0.035166, -0.079645, -0.100295, 0.033992, -0.048624, -0.031695, -0.005127, 0.083430, 0.004118, 0.036146, 0.037144, -0.048517, -0.085021, -0.029277, -0.159555, -0.039669, -0.024130, -0.028807, -0.022517, -0.013537, -0.054557, 0.133109, -0.000693, 0.035113, -0.178751, -0.066039, -0.032328, -0.044814, 0.062658, 0.027092, 0.002764, 0.022001, -0.057622, 0.085514, -0.065240, 0.000493, 0.048390, -0.009854, -0.067627, -0.023354, -0.028176, 0.032012, -0.107766, 0.000941, -0.038249, 0.063800, 0.008080, -0.046181, -0.010757, -0.052570, -0.026936, 0.004082, 0.081460, 0.021477, 0.063409, 0.027747, -0.077047, 0.060889, -0.158842, 0.005628, -0.023263, 0.018691, -0.091143, 0.010829, -0.050045, -0.037587, -0.100559, 0.006284, 0.008340, -0.021302, -0.052131, -0.047082, -0.025826, 0.026101, -0.069257, -0.163639, 0.011669, 0.002859, 0.077978, -0.013913, -0.063224, -0.003624, 0.029322, -0.078995, 0.118846, -0.051156, 0.043861, -0.072154, 0.065687, -0.017205, 0.006982, 0.032822, 0.007562, -0.051827, -0.057044, 0.027862, 0.010239, -0.020027, -0.025872, 0.121249, 0.080581, -0.000870, -0.079241, -0.056468, 0.111991, -0.001749, -0.083297, -0.074020, 0.058056, 0.060133, 0.065062, 0.136871, -0.017816, -0.009570, -0.013970, -0.034464, -0.099510, -0.006579, -0.022967, 0.059029, 0.035578, -0.027401, 0.168221, -0.163083, 0.017768, -0.018694, 0.065370, -0.003277, -0.052955, 0.100279, 0.158835, -0.053346, -0.029506, -0.008718, 0.021410, 0.070889, -0.060565, 0.031392, -0.050255, -0.042946, 0.067656, 0.030981, -0.015528, 0.030345, 0.100855, -0.031231, 0.019789, -0.092841, -0.019058, -0.037796, -0.102300, -0.056811, 0.036019, -0.007242, -0.005668, 0.000583, -0.133503, -0.090784, 0.111234, -0.062765, -0.090386, -0.102460, -0.045304, 0.024351, 0.131374, -0.026206, 0.037563, -0.029590, -0.082512, -0.046416, 0.061764, -0.015548, -0.075599, -0.018349, 0.005866, -0.091127, 0.031682, -0.023289, -0.049739, -0.020006, -0.089987, 0.031197, 0.030650, -0.023216, 0.092236, -0.079538, 0.021464, -0.016467, -0.084992, 0.002320, -0.096097, 0.042039, -0.039348, 0.067801, -0.085493, -0.059980, -0.031959, -0.110190, -0.040531, -0.066083, 0.079447, -0.061445, -0.033695, -0.045752, -0.058466, -0.009672, -0.003037, -0.095943, -0.088862, -0.033134, 0.096052, -0.042255, 0.075991, -0.036874, -0.084634, -0.039844, -0.077328, -0.108382, -0.136284, -0.016044, -0.034926, 0.022404, 0.026696, -0.091988, 0.110116, 0.033044, -0.180521, 0.012457, -0.033379, -0.064375, -0.155903, -0.006364, 0.034380, 0.001723, 0.035114, 0.099648, 0.033070, 0.003976, 0.064582, -0.005568, 0.014444, -0.006034, -0.028345, -0.039261, -0.091661, -0.157956, 0.043539, -0.001225, -0.022564, 0.026470, -0.050029, -0.033525, -0.072661, 0.018039, 0.029422, -0.011673, -0.034677, -0.024193, -0.021767, -0.001803, -0.120693, 0.073009, 0.045979, -0.083662, -0.231238, 0.073016, 0.122984, -0.068544, -0.046745, -0.016988, -0.052864, 0.001875, 0.109430, 0.036387, -0.017857, -0.120060, 0.011134, -0.133154, 0.073417, 0.052250, -0.065797, 0.044389, -0.052827, 0.036652, 0.051381, 0.087070, -0.015351, -0.035456, 0.038092, -0.046550, -0.014399, -0.016858, 0.063476, 0.019828, 0.065818, -0.022849, -0.050011, -0.015194, -0.011982, -0.146870, 0.066310, -0.000617, -0.017830, -0.014270, -0.075839, 0.061069, -0.047204, 0.021899, 0.024654, 0.035341, 0.062324, 0.012043, -0.108002, -0.073766, -0.075649, -0.026231, -0.058817, -0.026493, -0.134176, -0.043961, -0.168040, -0.042857, -0.021555, -0.102128, -0.066817, 0.023227, -0.071613, -0.082935, -0.010234, 0.037067, -0.003859, -0.090196, 0.056050, 0.015198, 0.086307, -0.005161, -0.008691, -0.179524, 0.000098, 0.000194, 0.051040, 0.009353, 0.055032, -0.059793, -0.024786, 0.031341, -0.022674, -0.037114, -0.075652, -0.026583, 0.124111, 0.039253, -0.052566, -0.074659, 0.025533, -0.053470, 0.045348, 0.023185, -0.001701, -0.100901, -0.198189, -0.113084, -0.100844, -0.269825, -0.005941, -0.166038, -0.124641, 0.028521, 0.010362, 0.091344, 0.043411, 0.072134, -0.069460, -0.017485, -0.063850, 0.039776, -0.153493, 0.029420, -0.024454, -0.061288, -0.062677, 0.044823, -0.021464, -0.041347, -0.009054, 0.018138, 0.007527, 0.028400, -0.023762, -0.124449, 0.000346, -0.020486, -0.034787, -0.005924, -0.059187, 0.004766, -0.063432, -0.006220, -0.048594, -0.109824, 0.066251, -0.009497, 0.007617, -0.025855, -0.031701, 0.019608, -0.011807, -0.118316, 0.028124, -0.101223, 0.092675, -0.069266, 0.084334, 0.019567, -0.125289, 0.009568, 0.071316, 0.042649, -0.015906, -0.032718, -0.006821, 0.124244, 0.029488, -0.079284, 0.006988, -0.034361, 0.081809, 0.077337, -0.040342, 0.083358, 0.014408, 0.007433, -0.000097, -0.079332, -0.033492, -0.043272, 0.017391, -0.081238, 0.044029, 0.021717, 0.012987, 0.090898, -0.015513, -0.068272, 0.042097, -0.017705, 0.117211, -0.199760, -0.069876, 0.030745, -0.098462, 0.003645, 0.011440, -0.076439, -0.019982, -0.009688, -0.033753, -0.023913, 0.041758, -0.075352, 0.030366, 0.069928, -0.037200, 0.035806, 0.020999, 0.011914, 0.045140, -0.017900, -0.014414, -0.050700, 0.022655, 0.046840, -0.069464, 0.040984, 0.056121, 0.076491, 0.006873, -0.119759, 0.008766, -0.146865, -0.119846, -0.080855, 0.043399, -0.075346, -0.100249, 0.010547, 0.067730, 0.055208, 0.017435, -0.037249, 0.022673, 0.010278, -0.066710, -0.019464, -0.036604, 0.061508, -0.144047, -0.026940, -0.120251, 0.011137, 0.057738, -0.032377, 0.029212, -0.067372, -0.010229, -0.000161, -0.028774, 0.018921, 0.013813, -0.126192, -0.129168, 0.060935, -0.004793, -0.024331, -0.014369, 0.040166, -0.161554, -0.029833, -0.009957, -0.073272, 0.008283, -0.098349, 0.005744, 0.010575, -0.090101, 0.047078, -0.075230, -0.090400, 0.000464, -0.088019, -0.036451, -0.004996, 0.127176, 0.020929, -0.038610, 0.011227, 0.022103, -0.049799, -0.060164, -0.030286, -0.023140, -0.036169, 0.004430, 0.008351, 0.010440, -0.009923, 0.002861, 0.068091, -0.049942, 0.008562, 0.032135, 0.008304, -0.068891, 0.066702, -0.049756, -0.038658, -0.065520, -0.047508, 0.068222, -0.106474, 0.054174, -0.105622, -0.007066, 0.042840, -0.068600, 0.054009, 0.052308, -0.088990, 0.067539, -0.033727, -0.015041, -0.187428, 0.031096, 0.010839, 0.036811, 0.025315, -0.038512, 0.107789, -0.100299, -0.038301, -0.040495, 0.183715, -0.077927, 0.031893, -0.073140, 0.011364, -0.041885, -0.005214, -0.050154, -0.014418, -0.074324, 0.031186, -0.009346, 0.028802, -0.105403, -0.059423, -0.079634, -0.027703, -0.059411, -0.064436, 0.025038, 0.001182, -0.039270, -0.051283, -0.044676, -0.024134, 0.010335, -0.059644, -0.031455, -0.035108, 0.093762, 0.079024, -0.050636, 0.003297, 0.064744, -0.012336, -0.015539, 0.044076, 0.006846, 0.033611, -0.030661, -0.070503, -0.024708, -0.100876, -0.057165, 0.074692, 0.034352, 0.027136, -0.018309, -0.075469, -0.068798, -0.037133, 0.016817, 0.051432, -0.042169, -0.045776, -0.068943, -0.024319, 0.011534, 0.067812, 0.002046, 0.008905, -0.110304, -0.013467, -0.059513, 0.039282, 0.027062, -0.070217, -0.249259, -0.075480, 0.057829, -0.045461, 0.081134, 0.036098, -0.051137, -0.059613, 0.017572, 0.009642, 0.023093, -0.089126, 0.138681, -0.092716, 0.106323, 0.026711, 0.111880, 0.045673, -0.074893, -0.057644, -0.078597, -0.026333, -0.047075, -0.118919, 0.023643, -0.079198, 0.018955, -0.101070, 0.088963, -0.027028, -0.083084, -0.138993, 0.052974, 0.034997, -0.040773, 0.073404, -0.020661, 0.044931, 0.038195, 0.000136, 0.014063, -0.004070, 0.011533, 0.058467, 0.039328, -0.099050, -0.042110, 0.048948, -0.076804, -0.044169, 0.034903, -0.058362, 0.044148, -0.004998, -0.014461, -0.029662, -0.000308, -0.053125, -0.096402, -0.028565, -0.011200, 0.006377, -0.041911, 0.102463, -0.005796, -0.004171, -0.051464, 0.056267, -0.058373, -0.061848, -0.034225, -0.025532, -0.062619, 0.037563, 0.077657, 0.074900, 0.002758, -0.093036, -0.029691, -0.010783, 0.023622, 0.054376, 0.080986, -0.024414, 0.000887, 0.070070, -0.045645, 0.022786, -0.052052, 0.115180, 0.010224, 0.015634, -0.090939, 0.036981, -0.044675, 0.132699, -0.031824, 0.068442, -0.026021, 0.072374, -0.034492, 0.104881, -0.052380, 0.033346, -0.058338, -0.063765, -0.102518, 0.020481, -0.031042, 0.025910, -0.054685, 0.005096, -0.031832, 0.023003, 0.005522, 0.009871, -0.020252, -0.092837, -0.011402, -0.033918, -0.065278, 0.030130, 0.018775, -0.015231, -0.015591, -0.021752, -0.078630, -0.047846, -0.015592, -0.007712, -0.012098, -0.093451, -0.036461, -0.049448, -0.153304, -0.117333, -0.050803, 0.112506, -0.006177, 0.007101, 0.080445, -0.027640, -0.071409, -0.016980, 0.028939, 0.043711, -0.050631, -0.083646, 0.158472, -0.009915, -0.079939, -0.026073, -0.060293, 0.065697, -0.051727, 0.122398, -0.022501, -0.052317, 0.087606, -0.008322, -0.030562, -0.066350, -0.059494, 0.165636, 0.017276, 0.098695, -0.063871, -0.040282, 0.022768, -0.072397, 0.043478, -0.095221, -0.085693, -0.024686, 0.045529, -0.118644, -0.055632, 0.005231, 0.028740, 0.002745, -0.020739, -0.079773, -0.119435, 0.045380, -0.037481, -0.045377, -0.088803, -0.006962, 0.016222, 0.047202, 0.000957, 0.047136, -0.020452, -0.058788, -0.162709, 0.026653, 0.003766, -0.009598, -0.054312, -0.019182, -0.050449, -0.128145, -0.076749, -0.005469, -0.040930, 0.063995, 0.043341, -0.178871, -0.006327, -0.004501, -0.004786, 0.033654, -0.063841, -0.078237, -0.079158, -0.063387, 0.118750, 0.026719, 0.053161, -0.013894, 0.037702, 0.016530, -0.021305, 0.019835, -0.072614, -0.036984, 0.030363, -0.006108, 0.044285, 0.045478, 0.040526, -0.002286, -0.013215, -0.035650, 0.004743, -0.031017, 0.103022, 0.011586, 0.018893, 0.073756, -0.009229, -0.037438, 0.126214, -0.116445, -0.030988, 0.060945, -0.121528, -0.066995, 0.072707, 0.045092, 0.057658, -0.003251, 0.000631, 0.041640, -0.030068, -0.028967, -0.016229, -0.013047, -0.005559, 0.047586, -0.001279, 0.030396, -0.067164, -0.090050, 0.005248, 0.005642, -0.096519, 0.066973, 0.001595, 0.061312, 0.016702, -0.026409, -0.000423, 0.055589, -0.063130, 0.001943, -0.048112, -0.076881, 0.071986, -0.002950, -0.015646, -0.107570, 0.001970, 0.024707, -0.016513, -0.030222, -0.074296, 0.002838, 0.116900, -0.061211, -0.058025, -0.097791, -0.058063, -0.018940, -0.152694, -0.062511, -0.039349, -0.025948, -0.013370, 0.001340, -0.072598, 0.019830, -0.167066, 0.060042, -0.015846, 0.104978, -0.009858, -0.024206, 0.030606, 0.045078, -0.102495, 0.012307, -0.081468, 0.015805, -0.032122, 0.035177, -0.054284, 0.087985, 0.032058, 0.029631, 0.045747, -0.040397, -0.099007, -0.011707, 0.002703, -0.043082, 0.030509, 0.023360, 0.032256, -0.060091, 0.014137, 0.004093, 0.063405, -0.028714, -0.067224, 0.012323, 0.000772, -0.046711, -0.037758, -0.007073, -0.040022, 0.015505, -0.064338, 0.017271, 0.030009, 0.026749, -0.038841, -0.003767, -0.019200, 0.009637, -0.099322, 0.069805, -0.005957, 0.061233, 0.016750, -0.043904, -0.026225, -0.115977, -0.044037, 0.014246, -0.057091, -0.033795, -0.010665, -0.005213, -0.000266, -0.061095, -0.021175, 0.017703, -0.002328, 0.034696, 0.070482, 0.014188, -0.015757, -0.031320, 0.042780, -0.028116, -0.140592, -0.068815, -0.013083, -0.016140, -0.002097, -0.021659, -0.003631, -0.039244, 0.017453, -0.076694, 0.030283, 0.052896, -0.057367, -0.059864, -0.050225, 0.019593, -0.001508, -0.060647, -0.067688, 0.027858, 0.040241, -0.027870, -0.043651, 0.000728, 0.001706, -0.017324, 0.037258, 0.005715, -0.082978, -0.009341, -0.018437, 0.034636, -0.007137, -0.012834, -0.086622, -0.029059, -0.045123, 0.033288, -0.067027, 0.003211, -0.070428, -0.095307, 0.047000, 0.047119, 0.022061, -0.029107, 0.002551, -0.049001, 0.007759, 0.000421, -0.041793, -0.035613, -0.016177, -0.046671, -0.044796, 0.008651, -0.057898, 0.047527, -0.047148, -0.012247, -0.098192, -0.002282, -0.047761, 0.029831, 0.019500, 0.002121, -0.161711, 0.044026, -0.113254, -0.053482, 0.061278, -0.066072, -0.031405, -0.078311, 0.039756, -0.066642, 0.018159, -0.026173, 0.000022, 0.043857, -0.035969, 0.003140, 0.003173, 0.019423, -0.023160, -0.040017, -0.036694, 0.003943, -0.007169, 0.046948, -0.088170, -0.048826, 0.037193, -0.007291, -0.014570, 0.030647, 0.050753, -0.042706, 0.039917, -0.063595, 0.039673, -0.020029, 0.006019, -0.034096, -0.000483, -0.065629, 0.053355, 0.008767, 0.010658, -0.042088, 0.054844, 0.003420, 0.053976, 0.059786, -0.013332, 0.001065, -0.028528, -0.061054, -0.000404, 0.031479, 0.012670, -0.017596, 0.084624, 0.023810, -0.026164, 0.036735, 0.001641, 0.021993, -0.061065, 0.057940, 0.001733, -0.016396, -0.100188, -0.026867, -0.019311, -0.055104, 0.045097, -0.013028, 0.039514, 0.006624, -0.049629, 0.070385, 0.008801, -0.053740, -0.013374, -0.009388, 0.019543, -0.032670, -0.048477, -0.049143, 0.051233, 0.021508, -0.012600, 0.046906, 0.058216, 0.045953, 0.014838, -0.023729, -0.046597, 0.001242, -0.040923, -0.003705, -0.046045, -0.029219, 0.006643, -0.016872, 0.003471, -0.027613, 0.021055, 0.118788, -0.039328, -0.012660, 0.046528, 0.017074, -0.032127, -0.065771, 0.043450, 0.021299, -0.062287, 0.027347, 0.017744, -0.051388, -0.057387, -0.001492, 0.019938, -0.058388, -0.032697, -0.041616, 0.040520, -0.026489, 0.040606, 0.071865, -0.011401, -0.043788, 0.038015, -0.018799, -0.080306, -0.014026, -0.032545, -0.030082, -0.056282, -0.038873, -0.095447, 0.003127, -0.009379, -0.022625, -0.028173, -0.034599, -0.052303, 0.016186, -0.111641, -0.035542, 0.027123, 0.066337, -0.003785, -0.063438, -0.048936, -0.019336, -0.036857, -0.007262, -0.037710, -0.070472, 0.003542, -0.001078, -0.063503, -0.055103, 0.021553, -0.057973, 0.033024, 0.016085, -0.069323, -0.024523, -0.041610, 0.022097, -0.063533, -0.098672, -0.050540, 0.056044, -0.017378, 0.097410, -0.034598, -0.086692, 0.010176, 0.045262, 0.005471, -0.020017, 0.003168, -0.041621, -0.026745, -0.080113, 0.065756, 0.032237, 0.052286, 0.124667, 0.004343, -0.059949, -0.075389, -0.081001, 0.000292, 0.020192, -0.055867, 0.036432, 0.006772, 0.114164, -0.074142, -0.052318, 0.077950, -0.021989, -0.053482, -0.030760, -0.019938, -0.024300, 0.000876, -0.027685, -0.023080, -0.088992, 0.002077, -0.046087, 0.040626, 0.036735, -0.011867, -0.004799, 0.033464, -0.020286, -0.011761, -0.037691, -0.039453, -0.044380, 0.053373, -0.009161, -0.081424, -0.064026, -0.086248, -0.074290, 0.023374, 0.035215, -0.012145, -0.011268, -0.034894, 0.046831, -0.089386, 0.024846, 0.003332, 0.003532, -0.024937, -0.035636, -0.056357, 0.021139, 0.023129, -0.024749, -0.012892, -0.032575, -0.106543, 0.058030, -0.087004, -0.075964, -0.090452, 0.007959, 0.104466, -0.017229, -0.036314, -0.027304, -0.073620, -0.000163, 0.017578, -0.047995, -0.026285, 0.007287, 0.014490, 0.068479, -0.049058, -0.008869, 0.030652, -0.021856, -0.095583, -0.064916, -0.023219, 0.013221, 0.049692, 0.062210, 0.079587, 0.008672, -0.003779, 0.035374, -0.038014, -0.027601, 0.033980, 0.050452, -0.087153, 0.046960, -0.018534, 0.025555, -0.013467, -0.112296, 0.051275, -0.027011, 0.044135, -0.013792, -0.011953, -0.085522, -0.037496, -0.044686, 0.053317, -0.021978, -0.004713, -0.012687, 0.044018, -0.072334, -0.065817, 0.028294, 0.006480, -0.019992, 0.006853, 0.010631, -0.028572, -0.002697, -0.022517, -0.036054, -0.112619, -0.000436, 0.073696, -0.006995, 0.002896, 0.031256, -0.041560, 0.010270, -0.061294, 0.020338, -0.044280, 0.032860, -0.029791, -0.053554, -0.048993, -0.031524, -0.060140, 0.004015, 0.012387, -0.056214, -0.009650, 0.017828, -0.072678, 0.003224, 0.040048, 0.016941, -0.008395, -0.126220, 0.020647, -0.036738, 0.043203, -0.096394, 0.115654, 0.043066, -0.036929, -0.041389, 0.007495, -0.011404, -0.056260, -0.042877, 0.007306, 0.051940, 0.025086, -0.041390, -0.056152, 0.012509, -0.043961, -0.021014, -0.063734, -0.036142, 0.046073, -0.067430, 0.008051, 0.000348, -0.006996, -0.038668, 0.030964, -0.014930, 0.011985, 0.063396, -0.057192, 0.047401, -0.091925, 0.041789, 0.031488, 0.013989, -0.024031, -0.015095, -0.063338, -0.044368, 0.060766, -0.046111, 0.023670, -0.143183, 0.025153, -0.081550, 0.048985, 0.000806, 0.022201, -0.066009, 0.056917, 0.035209, -0.012575, -0.040488, -0.078600, -0.036940, -0.009507, -0.025597, 0.085300, 0.026107, -0.029994, -0.036764, -0.021818, -0.033698, -0.026363, -0.004427, -0.017822, -0.030682, 0.075581, 0.014901, -0.053621, 0.003646, -0.034300, 0.033273, -0.094052, 0.013099, -0.061226, -0.061665, -0.044348, -0.004585, -0.015554, 0.024609, 0.016131, 0.057756, -0.088685, -0.006799, 0.082246, 0.046188, -0.012134, -0.062005, 0.005810, -0.052011, -0.028722, -0.063789, -0.043908, -0.021039, -0.021799, 0.054861, -0.063464, -0.092554, -0.015777, -0.060211, -0.078321, 0.050199, -0.050452, 0.042293, -0.021499, 0.001948, 0.022378, -0.055388, -0.072267, -0.026025, -0.000804, 0.023216, -0.054105, -0.017763, 0.041980, -0.043268, -0.034622, -0.057425, 0.027836, -0.023583, 0.018536, -0.013110, -0.043026, -0.019923, 0.014066, 0.033144, 0.003562, -0.060306, -0.028544, 0.096004, -0.034976, -0.031586, -0.076632, -0.001330, 0.034627, -0.070762, 0.052266, -0.010756, -0.070003, -0.060025, -0.030860, -0.076993, -0.044616, -0.035992, -0.036453, -0.033900, 0.033904, 0.030560, -0.150460, -0.098077, -0.057900, -0.060395, 0.025388, 0.066739, 0.039895, 0.027902, 0.054931, -0.049198, -0.032615, -0.033147, 0.057745, -0.035783, 0.011804, -0.059912, -0.028384, -0.000823, -0.005065, -0.039150, -0.048934, -0.061427, -0.056491, -0.052864, -0.063038, -0.052312, -0.062919, 0.040216, -0.015395, -0.000952, 0.045610, 0.020794, 0.081384, -0.060587, -0.049230, -0.068609, 0.005312, -0.036274, 0.087266, -0.046366, -0.045190, -0.008445, -0.075070, -0.015190, 0.029207, -0.064089, -0.037813, 0.009932, -0.087471, -0.050937, -0.049297, 0.021592, -0.038489, -0.041343, -0.021628, -0.104146, -0.043721, -0.053907, -0.078873, -0.046890, -0.004153, 0.006800, -0.010447, -0.001339, 0.021174, -0.079491, 0.015752, -0.044490, -0.061231, -0.043044, -0.001086, -0.032254, -0.011189, 0.028620, 0.002145, -0.143305, -0.058857, 0.000675, -0.045856, -0.045375, -0.027431, -0.007610, -0.050693, -0.027759, -0.001631, -0.049200, 0.012227, 0.002268, -0.002247, -0.027430, -0.023920, 0.015403, 0.083084, 0.009773, 0.055433, 0.005908, 0.049087, -0.030276, -0.027356, 0.025484, -0.004164, 0.004173, -0.082397, 0.043068, -0.030231, -0.019664, -0.086344, -0.047875, 0.006109, 0.031303, -0.009366, -0.018823, 0.039094, -0.013581, -0.069455, 0.032766, 0.018889, -0.043974, 0.039668, -0.051579, 0.000676, 0.070130, -0.065903, -0.046090, 0.002522, 0.019413, -0.076884, 0.038207, 0.054897, 0.010319, 0.072231, 0.055791, -0.104539, 0.013682, -0.042302, -0.051020, -0.027019, -0.048363, 0.016411, 0.004006, 0.099457, -0.008964, -0.002233, 0.017021, -0.078091, -0.006890, -0.086694, -0.072336, -0.086488, -0.060893, -0.035171, -0.071863, -0.022126, 0.010131, 0.116573, 0.016340, -0.103123, 0.029398, -0.016579, -0.022063, 0.012734, -0.069908, -0.049271, 0.007760, -0.016065, 0.020400, -0.046590, 0.025813, 0.034534, 0.081930, -0.033637, -0.127280, -0.024660, -0.056434, -0.042857, 0.045547, -0.005904, -0.070219, 0.001422, -0.083454, 0.053019, -0.010323, -0.040262, 0.001727, -0.020482, -0.062521, -0.026171, -0.066414, -0.061712, 0.045999, 0.003977, -0.010295, 0.055144, 0.020392, -0.028110, -0.057701, -0.049520, -0.074759, -0.080346, -0.041167, -0.018968, -0.104952, 0.030351, -0.064869, 0.034584, 0.038066, 0.001844, 0.080441, -0.036474, 0.053903, -0.016476, -0.003379, 0.038353, 0.005462, -0.035038, -0.087854, -0.069191, -0.021549, -0.121036, -0.003536, 0.017790, 0.006052, 0.004254, -0.025643, -0.085770, 0.007680, 0.012199, 0.027347, 0.006215, 0.093009, -0.013348, -0.009434, -0.016587, 0.016396, 0.065098, -0.015420, -0.011272, 0.033348, -0.030073, 0.002183, 0.038607, -0.019720, -0.007813, -0.031524, -0.029852, -0.036993, -0.067008, 0.004567, -0.020497, -0.080438, 0.012158, 0.021837, -0.038721, -0.043562, 0.054939, 0.017334, 0.031885, 0.027049, 0.026278, -0.094981, -0.049908, 0.023149, 0.025617, 0.037193, -0.061598, -0.005190, -0.055308, 0.042543, 0.035366, -0.055050, -0.056671, -0.060475, -0.029016, -0.053097, 0.050813, -0.032539, 0.033192, -0.040770, 0.003575, -0.016718, 0.093928, -0.058715, -0.029939, 0.025551, -0.056621, -0.027752, -0.049749, 0.003882, -0.091125, 0.064961, 0.022718, -0.030675, 0.084592, -0.015674, 0.019969, 0.027051, 0.119184, 0.065500, 0.041856, 0.003085, -0.050800, 0.021581, -0.021589, -0.000670, -0.008578, -0.018011, 0.089206, 0.008553, 0.012811, -0.043909, -0.086435, -0.109890, 0.039093, -0.078269, 0.012525, 0.040070, 0.009918, -0.038988, -0.032873, -0.064769, -0.083725, 0.012999, 0.043002, 0.026744, -0.031100, -0.014727, 0.015378, 0.026643, 0.042795, -0.009587, -0.067710, -0.055386, -0.058513, 0.043689, 0.024128, 0.008178, 0.079048, 0.024802, -0.010138, 0.007207, 0.042525, -0.063803, -0.030678, 0.012440, -0.008015, -0.034953, 0.011879, 0.036798, -0.006621, 0.026995, 0.044941, -0.078145, -0.038278, -0.002993, -0.029406, -0.032228, 0.048943, -0.059913, -0.069433, 0.025162, -0.025420, -0.044217, 0.008003, -0.033546, -0.025744, -0.003181, 0.027950, -0.044752, 0.054848, 0.015608, -0.101898, -0.080540, -0.126196, -0.071697, -0.003664, 0.035535, -0.053438, 0.012882, 0.042112, 0.013518, -0.045982, -0.078856, 0.048318, -0.025903, -0.012947, -0.095446, 0.019807, 0.017702, -0.035831, -0.029853, -0.005177, -0.074240, 0.098028, -0.023322, 0.050889, -0.101584, 0.021035, -0.043441, -0.006623, 0.014875, 0.042321, -0.154474, 0.039179, 0.000988, 0.004726, -0.028057, -0.045466, -0.015447, -0.047442, -0.058004, -0.097724, 0.009107, -0.002059, -0.051734, -0.149774, 0.116487, -0.062829, 0.041343, 0.042820, 0.069379, -0.063851, -0.038840, -0.077537, -0.045012, -0.099963, 0.002993, 0.038647, 0.000183, -0.052432, -0.018971, -0.042616, -0.082949, -0.006825, -0.033226, -0.122413, -0.030191, -0.151249, 0.017784, -0.031904, -0.181849, -0.049527, 0.066689, 0.022494, -0.007160, 0.049576, 0.002987, 0.010872, 0.044763, 0.090129, -0.070329, -0.028954, 0.034910, 0.059853, -0.080796, -0.040735, -0.015028, -0.068306, 0.024458, 0.175427, 0.051320, 0.060104, 0.024080, 0.005208, -0.041425, -0.064832, 0.006571, -0.047058, -0.009631, -0.013904, 0.022307, -0.044524, -0.062346, -0.036939, -0.104103, -0.090417, 0.019488, 0.024137, 0.010800, -0.027002, -0.066492, 0.085281, -0.056923, -0.027120, 0.007606, -0.106339, 0.003772, -0.048416, 0.018288, -0.025131, -0.048534, 0.037012, -0.004928, -0.054056, 0.030608, 0.018682, -0.073829, -0.035644, 0.033769, 0.110501, -0.044132, -0.011943, -0.020497, -0.014162, 0.048044, 0.012562, 0.056329, -0.057009, 0.033769, -0.029694, -0.027122, 0.038508, -0.069400, 0.039059, -0.017492, -0.042306, 0.060328, 0.007955, -0.044425, -0.025790, -0.021398, -0.044639, 0.068472, -0.064848, -0.094586, -0.050904, -0.128199, -0.035444, -0.018717, 0.018966, -0.038090, -0.158795, -0.052937, -0.118243, -0.056861, 0.022968, -0.091139, -0.159328, 0.040069, -0.026946, -0.060400, -0.039575, -0.009831, 0.019015, -0.101519, -0.010895, -0.034876, -0.016623, -0.060060, -0.037013, 0.001376, -0.052758, -0.067419, 0.021976, -0.032167, 0.054319, -0.058355, -0.066479, -0.016747, -0.054315, 0.022995, 0.006902, 0.025584, 0.013837, 0.029682, 0.121021, -0.075133, -0.012295, -0.055294, -0.021527, -0.078459, 0.016225, -0.190129, 0.000658, -0.069891, 0.026742, -0.041000, -0.073141, -0.077054, -0.022383, 0.077520, -0.060725, 0.047762, -0.044034, -0.040746, 0.003613, 0.052756, -0.061395, 0.122567, -0.078171, -0.050502, -0.081599, 0.062807, -0.043500, -0.078827, -0.015921, -0.120845, -0.018350, 0.007920, 0.032768, -0.068232, -0.047512, -0.093316, -0.013084, -0.105325, -0.028523, 0.044727, -0.105628, -0.032466, 0.025388, -0.053642, -0.067991, -0.045743, -0.010570, -0.019372, -0.026005, -0.005461, 0.045664, -0.018308, -0.003942, -0.063573, 0.039161, -0.065231, -0.052476, 0.026182, 0.000068, -0.088732, -0.046134, -0.002044, 0.017977, -0.057468, 0.007927, -0.004593, -0.038100, 0.012961, -0.005945, -0.232422, 0.004882, 0.025922, -0.046585, -0.065009, -0.007610, 0.060096, 0.015769, -0.088669, 0.121931, -0.041999, -0.000128, -0.031355, -0.039762, -0.021680, -0.200036, -0.012923, -0.056274, -0.054775, -0.004355, -0.224389, 0.014218, -0.005859, -0.006322, 0.002805, -0.064707, 0.041671, 0.016235, 0.148530, -0.034417, 0.006240, -0.092243, -0.003223, 0.074890, -0.050446, -0.069068, -0.004661, 0.015376, 0.043098, 0.035871, 0.002313, 0.123084, 0.069125, -0.014105, -0.035731, 0.011273, -0.015223, 0.024758, -0.025450, -0.077476, 0.024000, -0.030451, -0.164519, -0.017520, -0.048801, -0.076537, -0.057307, -0.083675, 0.034032, -0.062317, -0.065530, -0.058119, -0.052823, 0.011125, -0.000383, 0.055191, 0.011584, -0.042763, 0.182733, -0.058471, 0.068034, -0.040438, 0.051488, -0.034198, -0.005920, -0.060892, -0.092639, 0.036098, 0.012260, -0.146863, 0.040831, 0.023843, -0.046282, 0.002629, 0.035525, -0.020894, -0.065334, 0.091029, -0.053170, -0.021305, -0.125318, -0.158300, 0.010613, -0.031361, 0.046234, 0.055877, -0.139398, -0.071543, -0.019342, 0.037058, -0.033794, -0.057701, -0.067793, 0.053871, -0.066617, -0.050288, 0.042014, 0.002621, -0.023105, -0.113763, -0.028633, -0.068725, 0.028817, 0.001903, -0.048140, -0.038500, -0.020329, -0.022105, 0.005305, -0.033084, -0.052460, 0.040507, -0.077867, 0.081536, -0.059439, -0.037865, -0.076295, 0.103444, 0.063697, 0.010846, -0.005546, -0.088662, -0.071062, 0.023192, -0.022131, -0.049771, -0.000150, 0.011717, -0.054640, -0.037981, 0.069611, -0.084078, 0.038335, 0.075428, -0.054906, -0.046705, -0.120063, -0.005883, -0.040759, -0.075868, -0.055946, 0.003318, -0.086132, -0.163656, 0.059519, -0.057770, -0.098476, 0.017368, 0.085563, 0.018301, -0.217067, -0.139834, -0.082338, -0.019466, 0.021357, 0.026052, 0.017047, -0.036696, 0.018047, -0.067787, -0.010213, 0.031804, 0.092559, 0.002809, -0.013841, -0.056100, -0.029253, 0.055874, 0.043542, -0.051029, 0.138767, -0.047174, -0.011096, 0.013027, 0.046648, -0.135654, -0.035377, 0.143637, 0.019629, -0.029738, 0.007998, 0.045425, 0.044798, 0.000794, -0.085701, -0.056225, 0.033487, -0.061662, -0.129085, -0.040852, 0.006674, 0.035937, -0.088267, 0.002841, -0.052431, 0.010367, -0.063932, 0.066857, 0.002958, 0.065930, 0.055522, -0.083341, 0.000472, 0.057767, -0.121995, -0.023562, 0.045063, 0.135437, -0.004317, -0.016036, -0.037864, -0.017156, -0.058406, 0.019085, -0.051084, -0.033042, 0.045178, -0.054147, -0.024619, -0.131136, -0.035847, -0.072087, -0.043387, -0.096863, -0.005204, -0.018792, 0.021141, -0.046789, 0.033848, -0.025471, 0.014664, 0.080827, 0.086467, 0.036682, -0.010856, 0.020919, -0.079090, -0.100378, -0.031020, -0.007301, -0.015961, 0.039546, 0.055741, 0.033930, -0.122852, 0.014847, 0.043628, -0.084600, -0.137947, -0.050986, -0.043060, 0.003642, -0.084539, -0.075759, 0.002453, -0.026364, -0.093145, -0.082275, 0.084346, -0.047356, -0.051646, -0.173746, -0.073113, -0.098958, -0.116610, -0.059537, -0.066874, 0.048624, 0.023634, 0.013492, -0.100007, -0.023850, -0.057887, -0.055008, -0.068695, -0.125641, -0.091732, -0.019064, 0.026172, -0.066236, 0.041480, 0.039682, 0.053814, 0.009091, 0.064475, -0.058728, 0.035339, -0.041773, -0.011218, 0.005133, 0.004468, -0.064490, -0.078068, 0.031776, 0.062542, 0.000696, -0.007930, 0.018951, -0.071639, -0.060611, -0.077307, 0.022270, 0.064992, -0.026638, -0.017693, 0.060850, -0.039399, -0.028987, -0.121288, -0.112665, 0.065244, -0.057586, 0.064023, -0.001589, -0.030376, 0.014028, -0.035694, -0.011096, -0.111371, -0.016738, -0.129492, -0.030521, -0.007044, -0.048934, -0.050088, -0.032730, -0.125290, -0.064041, 0.090016, 0.042114, -0.098960, -0.070305, -0.089543, -0.126187, -0.009144, -0.050538, 0.011432, 0.002266, 0.085023, -0.084685, -0.054759, -0.029102, -0.006456, -0.048462, -0.003411, -0.077003, -0.067451, 0.061086, -0.090939, -0.163214, -0.004740, -0.044274, 0.011587, 0.043846, -0.016469, -0.078135, 0.017908, -0.068518, -0.075578, -0.003427, -0.051656, -0.070589, -0.004423, -0.017264, -0.012386, 0.059102, -0.013266, -0.080275, -0.089868, 0.041233, -0.031593, -0.052392, -0.037606, -0.027540, -0.217455, -0.089363, -0.086613, 0.030384, 0.029056, -0.118324, -0.074233, -0.033740, 0.035990, 0.054965, -0.103390, -0.000318, 0.065234, 0.017926, 0.063703, 0.032769, -0.003798, -0.055804, 0.051850, -0.136522, -0.105168, 0.023350, -0.068634, 0.002720, -0.095540, 0.070875, -0.152215, -0.052165, 0.020980, -0.012404, 0.154953, 0.007020, 0.021069, -0.104579, 0.025924, 0.013051, -0.061711, -0.108150, -0.099146, 0.021867, 0.015814, -0.057756, -0.055276, -0.017575, -0.049978, 0.063483, -0.071938, -0.073323, 0.027986, 0.036290, 0.019441, 0.007714, -0.053704, 0.031226, -0.001968, -0.000368, -0.008928, 0.021597, 0.052888, 0.047131, -0.030830, 0.004730, -0.027951, -0.028847, 0.000733, 0.027213, 0.003236, -0.039527, 0.024810, -0.045408, -0.056689, -0.002962, 0.013513, -0.016217, 0.049789, 0.016216, 0.028217, -0.103939, -0.035952, 0.064322, 0.004273, 0.021396, -0.057184, -0.036014, -0.082326, -0.047302, -0.068526, 0.036398, -0.024331, -0.059568, -0.072544, 0.016340, -0.002793, -0.149334, -0.015571, -0.125647, 0.074975, -0.064231, 0.045913, -0.024330, -0.064182, 0.005573, 0.010650, -0.059116, 0.029245, -0.022129, -0.052840, 0.038722, -0.093223, -0.024952, -0.039197, -0.045235, -0.032137, -0.026768, 0.069246, -0.021636, 0.063607, -0.007074, -0.134365, 0.078852, 0.089663, -0.085503, 0.069152, -0.049787, 0.012857, -0.191162, -0.008873, -0.010024, 0.030657, -0.033340, -0.032420, -0.136870, 0.045992, -0.063830, -0.007312, 0.024415, -0.018439, -0.004118, -0.084817, -0.067235, -0.096929, -0.063560, 0.000424, -0.094274, -0.000329, -0.041709, 0.032326, 0.003879, 0.037300, -0.070191, 0.010766, -0.045554, -0.036313, -0.039777, -0.133238, -0.053659, 0.002730, -0.052445, 0.014020, -0.100074, 0.029187, 0.011936, -0.033924, -0.038519, -0.016048, 0.021149, -0.056248, -0.108879, 0.047592, -0.145213, -0.035000, 0.021855, 0.011327, 0.006999, -0.066411, -0.003644, -0.093538, 0.151910, -0.011725, -0.006021, 0.037665, -0.014987, -0.001966, 0.036511, -0.141696, 0.016318, -0.049794, -0.000514, -0.051814, 0.002416, -0.004239, 0.020311, -0.002947, -0.001872, -0.005389, -0.027902, -0.064564, -0.048750, -0.016591, 0.077256, -0.003716, 0.030937, -0.015291, 0.116917, 0.082967, -0.026704, 0.093380, -0.005526, -0.052741, 0.021450, -0.029089, -0.053989, -0.045309, -0.029395, -0.107550, 0.012900, 0.042483, -0.052468, 0.004843, -0.054266, 0.009194, -0.099691, -0.077518, -0.027498, 0.051855, 0.002561, 0.066468, 0.088951, 0.003682, 0.012053, -0.033706, -0.079849, -0.131357, -0.020114, 0.058299, 0.015548, -0.030778, -0.013078, 0.052538, 0.021141, -0.051217, -0.062387, -0.010632, 0.124144, -0.010482, -0.013340, 0.014823, 0.008270, -0.049308, -0.071763, 0.025266, 0.025508, -0.032656, 0.069798, -0.091375, -0.028681, -0.013805, -0.036656, 0.094406, -0.084427, 0.001369, -0.137823, -0.014304, 0.036237, -0.075808, -0.034009, 0.007342, -0.047987, -0.047351, -0.226808, 0.036730, 0.037173, -0.050147, -0.048513, -0.093182, -0.024149, 0.055695, 0.024738, 0.002031, -0.026926, -0.010898, -0.138075, 0.055283, -0.025257, 0.049907, -0.006003, -0.062471, -0.065252, -0.011880, -0.105410, -0.015406, -0.001437, -0.042718, 0.045313, 0.009897, -0.016979, 0.024323, 0.080846, -0.037479, -0.022509, 0.040410, -0.128871, 0.011956, -0.006384, -0.037581, -0.011870, 0.079002, 0.014643, 0.069111, -0.040343, -0.060712, 0.036828, -0.071677, -0.049630, -0.026240, 0.021314, 0.030910, -0.053294, 0.019817, -0.163965, -0.075095, -0.069160, -0.007244, 0.035616, -0.059489, -0.080445, 0.026115, -0.050295, 0.059534, 0.030078, 0.052279, -0.075946, -0.065552, -0.038996, 0.016638, -0.032616, 0.059869, -0.148384, -0.019199, 0.093950, -0.050123, -0.115422, -0.060848, -0.020788, 0.011113, -0.067064, 0.105680, 0.129947, -0.035786, -0.084445, -0.019815, -0.060985, 0.089276, -0.070296, 0.010342, 0.015453, 0.066165, -0.012914, 0.084610, -0.006553, 0.003823, -0.023808, -0.086178, -0.082516, -0.032279, -0.039891, -0.001115, -0.002911, 0.059822, -0.040229, 0.026322, 0.064272, -0.010844, 0.087990, -0.083476, -0.008559, -0.018722, 0.018752, 0.094234, -0.058086, -0.064984, -0.060770, -0.033205, -0.024059, 0.278262, -0.005685, 0.106419, -0.006842, 0.032460, -0.024337, 0.095174, 0.007529, -0.058888, -0.078546, -0.074213, 0.006870, 0.006889, -0.029659, -0.165975, 0.049517, -0.057908, -0.073846, -0.064197, 0.007486, 0.030801, -0.038867, -0.076393, 0.074018, -0.120914, -0.042751, -0.070639, 0.077184, 0.017055, -0.009778, -0.038846, -0.091362, 0.000745, -0.138402, -0.115794, -0.065931, 0.046554, -0.174349, -0.049989, -0.067483, -0.013499, -0.031685, -0.038301, 0.039374, -0.081315, -0.035561, -0.094546, 0.007590, -0.018935, 0.037910, -0.042727, -0.029999, 0.001927, 0.027892, 0.045600, 0.028021, -0.013420, -0.016471, -0.092089, 0.063337, -0.156685, 0.015403, -0.051998, -0.061750, -0.133905, 0.077066, -0.056182, -0.007080, -0.092220, -0.114119, -0.030606, 0.079771, -0.052165, -0.043213, -0.002788, -0.021246, -0.010319, -0.095898, -0.038338, -0.041418, 0.046825, -0.040159, -0.034958, 0.014150, -0.040068, 0.063511, 0.069306, -0.012088, -0.063537, -0.027144, 0.028687, -0.067303, -0.026859, -0.015349, -0.092048, 0.019522, -0.000888, -0.082480, -0.034569, -0.060775, 0.026150, 0.028706, -0.086372, -0.047315, -0.157220, -0.060874, 0.068159, -0.029753, -0.039847, 0.019943, -0.014176, 0.018234, 0.019724, -0.124032, -0.047189, 0.004558, 0.004447, -0.051015, 0.030451, -0.028744, -0.071979, -0.116924, -0.062579, -0.056886, -0.067948, -0.019491, 0.005255, -0.014327, -0.044445, -0.022755, -0.075731, 0.074753, -0.111142, -0.064262, -0.041179, 0.009984, -0.110753, -0.029885, 0.042767, -0.015764, -0.035518, 0.086754, 0.059829, 0.006404, 0.088776, -0.066299, 0.011372, -0.040281, 0.033644, -0.015697, -0.094169, 0.033495, -0.157651, 0.041369, -0.111991, -0.012543, 0.027106, -0.060118, 0.000599, -0.065646, -0.134378, 0.016626, -0.051657, -0.034206, -0.133470, -0.048210, 0.017187, -0.103724, -0.139545, -0.087784, -0.066157, 0.053606, 0.001682, -0.003720, -0.047734, 0.026607, 0.053422, 0.003653, -0.029421, -0.053249, -0.042168, -0.014417, -0.097915, 0.044442, 0.018332, -0.139889, -0.027659, -0.066746, -0.014061, -0.042990, -0.161337, 0.098204, -0.118600, -0.052489, -0.052071, 0.090545, -0.023281, 0.037900, 0.031737, 0.057490, -0.072698, -0.128876, -0.012430, -0.038969, -0.119230, -0.018505, 0.079100, 0.041233, -0.008228, -0.006168, -0.007938, -0.035203, -0.041521, -0.158595, -0.032889, -0.072232, -0.095237, -0.039892, 0.057031, -0.050948, -0.074728, -0.050507, 0.049178, 0.003464, -0.056911, 0.008868, -0.083479, -0.054979, -0.038352, -0.041515, 0.036271, -0.113817, -0.035363, 0.059285, -0.035888, 0.038841, 0.006978, 0.024016, 0.079590, -0.029951, 0.044049, 0.016832, -0.179061, -0.046996, -0.040772, -0.030900, -0.033441, -0.002383, 0.016235, 0.014558, 0.024678, -0.122403, -0.035752, 0.023258, -0.099960, -0.098625, -0.159147, 0.091525, -0.081997, 0.041310, 0.059232, -0.055676, -0.073976, 0.099509, -0.106155, -0.021809, -0.047989, 0.006612, -0.015361, -0.020581, -0.071128, -0.006790, 0.002665, -0.081261, -0.184584, 0.018959, -0.026687, -0.102591, -0.111518, -0.079624, -0.034818, -0.000619, -0.076140, 0.027491, -0.026613, -0.066452, 0.008783, 0.006371, -0.003903, -0.087912, -0.224839, -0.022061, -0.203123, -0.139088, 0.076582, -0.065257, -0.057641, 0.056829, 0.040900, 0.081621, 0.060338, -0.167043, -0.153606, 0.028112, -0.009452, -0.126222, -0.061890, -0.006009, -0.097163, -0.074582, -0.011222, -0.059165, -0.065989, -0.007100, -0.116421, -0.032927, -0.072723, -0.129793, 0.036039, -0.032703, -0.065865, -0.065420, 0.020049, -0.039365, -0.058782, -0.019051, -0.067110, -0.010923, -0.062612, 0.016129, 0.038195, -0.126157, -0.000262, 0.099070, -0.048037, 0.042647, -0.079281, 0.005093, -0.003504, 0.022642, -0.006326, -0.024079, -0.075075, -0.164171, 0.001460, -0.034892, 0.039915, -0.078402, -0.021231, -0.082768, -0.061817, -0.104453, -0.046465, -0.135603, 0.064931, -0.002576, 0.022993, 0.028414, 0.000820, -0.113526, 0.006206, 0.022897, -0.133702, -0.038426, 0.061635, 0.010417, -0.038607, 0.022396, -0.029134, -0.037326, 0.032105, -0.032634, -0.162048, 0.003848, 0.027098, 0.015595, 0.008865, -0.142527, 0.035028, -0.037732, -0.042543, 0.005666, -0.007171, 0.001199, -0.049157, 0.073358, -0.033477, 0.013424, -0.011580, 0.013584, -0.008396, -0.019112, 0.068617, -0.046717, -0.063347, -0.022661, -0.047463, 0.039869, -0.088487, 0.077960, -0.029741, -0.111748, -0.047131, 0.017337, -0.145924, -0.086570, 0.025098, -0.070110, 0.042941, 0.018588, 0.006506, -0.009545, 0.019256, 0.007032, 0.041739, 0.043896, 0.061739, -0.119523, -0.064290, -0.045978, -0.066357, 0.056941, -0.202271, -0.035558, 0.017669, -0.026051, -0.023841, -0.029441, -0.015742, -0.069243, -0.077608, -0.071140, -0.035731, 0.010716, -0.067850, -0.012166, -0.081620, -0.037447, -0.037534, -0.018678, -0.084563, 0.046797, -0.020125, -0.035822, -0.012187, -0.043842, -0.025224, -0.049675, 0.005036, -0.090640, -0.102626, -0.057471, -0.046742, 0.007591, 0.002936, -0.020596, -0.004191, -0.062534, 0.010794, -0.059245, -0.028385, -0.042706, 0.042717, -0.033774, -0.008110, -0.019002, -0.026077, -0.052911, 0.004544, -0.103729, -0.075091, -0.009108, 0.034680, 0.061418, 0.000895, -0.058347, -0.067131, 0.071654, 0.033731, 0.023462, 0.031436, 0.040168, 0.015078, -0.071356, -0.157222, 0.010461, -0.120353, -0.050590, 0.023034, 0.035286, 0.046025, -0.018182, 0.008703, -0.000558, -0.084251, -0.082757, 0.032616, 0.079150, -0.057240, -0.066818, 0.036745, -0.089392, 0.081436, -0.170499, 0.051494, 0.061035, 0.003044, 0.025569, -0.011913, -0.068245, -0.150809, 0.005784, -0.004703, 0.028922, -0.136195, -0.152237, 0.073946, -0.003631, 0.001197, -0.076230, 0.083073, 0.016797, -0.054288, -0.038772, -0.078655, 0.049610, 0.014083, -0.146635, -0.041861, -0.086439, -0.018896, 0.019176, -0.002430, 0.076108, 0.005774, -0.022849, -0.059570, -0.008246, -0.012015, -0.019634, -0.124202, -0.065683, -0.016185, 0.021013, -0.086549, 0.000690, -0.023045, -0.084450, 0.006351, -0.095562, 0.023057, 0.002033, -0.045583, 0.001168, 0.000648, -0.085917, -0.050710, 0.030516, 0.015563, -0.059803, 0.007999, 0.008318, 0.046494, 0.007547, 0.005708, 0.022112, -0.158919, -0.017990, 0.011112, -0.131928, -0.030649, -0.027360, 0.058648, -0.049961, -0.030471, 0.028498, -0.124636, 0.011498, -0.078627, 0.020845, -0.055259, 0.013769, -0.022752, -0.135075, -0.135440, -0.028278, -0.057020, 0.025766, -0.028304, 0.006300, -0.166959, -0.104837, 0.033172, -0.110686, -0.051545, -0.045125, -0.113887, -0.092471, -0.035698, -0.101357, -0.052728, -0.127934, -0.053148, -0.098756, -0.058078, 0.006943, -0.018182, 0.006035, 0.003501, -0.045236, -0.036045, 0.059909, 0.040995, -0.050662, -0.106086, 0.079084, -0.033525, 0.015637, -0.028517, -0.097882, 0.019067, -0.060621, 0.013452, -0.060702, -0.013003, -0.050619, -0.053945, 0.030597, 0.062100, -0.111183, -0.042863, 0.001027, -0.021934, -0.060639, -0.075132, -0.021596, -0.028472, -0.078280, -0.104892, -0.114523, 0.050747, -0.056156, 0.056410, -0.022127, -0.039805, -0.047414, 0.001384, 0.024029, 0.010752, -0.117726, 0.029859, -0.019563, -0.006767, 0.008553, 0.068509, -0.016828, 0.111033, -0.048598, -0.027342, 0.077589, -0.042674, 0.009155, 0.064728, 0.065498, -0.044796, -0.030210, 0.036631, -0.039231, 0.065505, -0.012317, 0.028672, 0.049546, -0.018753, -0.048120, 0.004027, -0.033849, -0.051420, -0.074440, 0.068162, -0.056745, -0.055990, -0.027411, -0.028012, 0.047264, 0.041004, -0.010783, 0.081623, -0.123596, 0.031625, 0.056520, -0.001759, -0.004125, 0.103485, -0.074177, 0.065100, -0.058452, -0.087221, -0.049846, 0.035765, -0.033317, -0.067478, 0.020118, -0.034804, -0.010539, -0.076546, 0.013743, -0.040934, 0.002573, 0.020385, -0.077084, -0.063270, 0.003760, -0.055201, 0.019462, 0.015751, -0.074107, 0.059545, -0.022099, -0.024029, 0.050712, -0.041665, 0.033847, -0.089207, 0.001157, 0.078366, -0.090722, -0.082522, -0.081903, -0.020091, -0.066482, -0.073620, -0.041354, 0.041818, 0.039544, -0.044097, -0.170418, -0.036894, -0.050188, -0.062605, -0.080666, 0.002255, -0.065313, 0.022000, -0.077551, -0.156945, -0.059139, 0.017655, -0.041748, -0.089158, -0.066896, -0.025601, -0.000425, -0.051060, 0.006989, 0.030185, -0.029285, -0.052280, -0.028998, -0.011414, -0.040118, -0.030669, -0.095293, 0.018541, -0.039516, -0.131541, 0.060993, -0.097958, -0.026323, -0.006134, -0.033940, -0.039865, -0.069182, 0.006199, 0.046647, 0.000246, -0.093440, -0.009851, -0.011704, 0.013819, -0.045401, -0.024624, -0.111182, -0.080641, -0.059691, 0.046928, -0.010191, -0.065973, -0.074789, 0.000026, -0.037727, -0.022212, -0.005637, 0.024963, -0.038881, -0.077030, -0.006085, 0.055651, 0.062572, 0.099308, -0.053542, 0.059492, 0.009668, -0.013100, -0.078503, 0.020489, -0.108574, 0.009744, -0.160421, -0.082987, -0.022467, -0.005401, -0.089832, -0.014070, 0.023816, -0.061295, 0.035655, -0.004696, -0.157270, -0.061635, -0.021206, 0.001195, -0.097261, 0.006405, -0.112667, -0.046328, 0.012584, 0.050425, -0.059545, -0.046938, -0.002950, 0.040229, -0.077194, 0.049743, -0.068320, -0.078589, -0.047487, 0.082381, -0.075970, 0.061080, -0.060644, 0.000338, -0.067526, 0.040216, 0.097974, 0.022840, -0.064494, -0.081812, 0.010227, -0.033610, 0.048718, -0.163379, -0.076314, -0.105731, 0.008865, -0.064577, -0.012098, -0.077783, 0.032683, -0.009612, -0.043281, -0.025657, -0.065773, -0.099034, -0.093645, -0.015290, 0.028085, -0.010980, -0.038423, 0.000164, -0.149327, -0.024293, -0.102440, -0.061359, -0.023701, 0.068929, 0.008199, 0.013500, 0.061535, 0.001209, -0.003053, -0.012757, -0.164727, -0.017792, 0.171937, -0.024324, -0.049107, 0.052340, -0.053724, -0.089819, 0.021622, -0.069655, -0.065323, -0.059669, 0.020442, -0.024053, 0.006312, -0.120560, 0.002911, 0.003238, 0.036711, -0.065878, 0.061416, -0.018305, -0.069093, -0.058449, -0.031621, 0.127068, 0.047798, -0.057946, -0.123728, -0.056114, -0.041130, 0.019596, -0.019943, -0.007665, -0.051348, -0.120098, -0.165299, -0.131086, -0.076512, -0.052976, -0.101328, -0.017137, 0.028862, -0.009375, -0.027310, -0.152849, -0.061248, -0.100437, -0.085215, -0.016635, -0.067245, -0.009803, -0.039377, -0.127431, -0.011983, 0.058800, -0.047845, -0.009043, -0.038590, -0.059897, -0.076319, 0.046369, -0.008751, -0.067983, -0.063110, -0.010316, -0.065603, -0.073499, 0.004472, -0.020280, 0.088845, -0.094924, 0.113072, 0.003962, -0.005236, -0.051956, 0.039107, -0.086594, 0.097214, -0.026474, -0.083694, -0.104483, -0.033918, 0.061836, -0.032544, 0.080302, -0.035534, -0.022007, -0.030638, 0.019031, -0.001874, 0.013224, -0.064761, -0.026072, 0.039717, -0.027548, -0.054366, -0.142331, -0.075202, 0.039316, -0.069753, -0.033406, -0.079275, -0.002870, -0.056863, 0.017051, 0.007745, -0.021781, -0.071661, 0.114081, -0.041664, 0.067136, -0.023636, -0.066549, -0.007798, 0.075698, -0.050816, -0.048648, 0.037770, 0.016872, -0.010644, -0.060748, -0.083095, -0.082559, 0.001043, 0.027707, 0.020464, -0.014853, -0.052304, 0.037733, 0.001903, 0.053321, -0.129637, -0.037522, 0.008989, -0.113699, -0.059825, -0.073370, -0.091783, -0.056814, 0.039007, -0.027856, 0.041198, 0.036750, -0.001281, -0.060085, -0.015485, -0.006106, 0.037859, -0.117109, -0.115547, 0.003462, -0.045227, -0.027089, -0.050549, 0.036589, 0.073715, 0.032278, -0.024688, -0.063681, -0.073014, -0.053741, 0.016732, 0.030736, 0.039666, 0.050187, 0.008919, 0.172175, -0.054895, -0.026257, -0.069309, 0.063841, -0.095881, 0.019376, -0.024575, -0.015848, -0.005543, -0.005537, 0.013356, 0.032514, -0.033889, 0.087604, -0.045442, -0.000267, -0.046044, 0.026988, 0.078995, -0.048143, 0.034658, -0.045929, 0.014333, -0.066086, 0.003647, -0.029000, -0.054657, -0.004655, -0.144527, -0.037558, -0.031833, 0.001057, 0.024074, -0.012273, 0.019865, -0.075689, -0.009275, 0.063246, 0.054880, -0.037699, 0.005848, 0.014573, 0.043478, -0.087067, -0.026939, -0.024015, 0.022363, 0.114616, -0.105091, -0.038579, -0.024838, -0.043251, -0.026737, 0.075946, 0.001556, 0.025846, -0.015592, 0.090734, 0.094079, -0.029508, 0.048719, 0.187524, -0.060836, -0.111251, -0.011532, 0.018416, 0.007407, -0.098177, -0.011965, 0.129733, -0.038542, -0.075993, -0.053318, -0.069719, -0.059708, 0.033172, 0.031695, -0.069415, -0.003837, -0.125316, -0.058430, -0.001587, -0.027804, -0.037440, 0.018775, 0.010743, 0.103167, 0.084862, 0.031417, 0.092438, 0.091230, -0.018169, -0.003757, 0.048074, 0.031998, 0.043390, 0.087392, 0.015090, -0.007443, 0.078233, -0.005062, 0.039848, 0.063396, 0.117857, -0.000336, -0.030651, 0.055883, -0.079466, -0.058142, -0.007021, -0.017507, -0.110123, -0.101229, 0.014396, 0.013210, 0.032471, 0.058148, 0.017084, -0.003777, 0.067445, -0.130959, 0.038507, -0.018601, -0.028033, -0.023600, -0.028410, 0.047432, 0.023978, -0.032875, 0.007250, -0.113574, -0.016912, -0.084128, 0.125087, 0.013255, -0.074959, -0.065274, -0.107822, 0.004441, -0.073150, -0.018362, -0.062987, -0.137551, 0.042976, -0.117339, 0.001929, -0.002652, -0.051060, -0.124186, 0.118188, 0.039705, 0.034035, 0.074070, -0.052410, -0.030332, -0.059038, 0.051383, -0.018467, 0.004619, 0.075569, -0.080549, -0.100474, -0.033989, 0.155249, 0.049169, -0.046561, -0.030994, -0.022939, -0.061224, 0.084849, -0.041890, -0.095398, 0.080065, 0.045781, -0.022136, 0.014442, -0.083769, 0.072351, -0.052373, -0.009537, -0.000937, 0.034931, 0.053113, -0.038438, 0.059969, -0.003288, 0.050499, 0.047206, -0.039967, -0.067900, -0.036470, 0.024889, 0.013617, 0.049884, -0.023836, -0.043435, 0.030812, -0.031617, -0.049461, -0.117434, -0.001555, -0.055334, 0.003703, 0.011836, -0.097658, 0.075854, -0.098197, -0.042106, 0.120428, 0.097578, 0.096113, -0.096599, -0.050028, -0.024085, 0.020926, 0.070506, 0.010028, -0.029928, 0.040909, 0.090365, 0.118063, 0.061454, -0.025315, -0.038057, -0.010337, 0.041307, 0.029023, 0.008817, 0.063500, 0.051261, 0.014975, 0.029487, -0.046092, -0.065368, -0.046407, -0.115080, 0.014329, 0.012184, -0.016543, -0.047010, -0.026838, -0.013452, -0.018105, -0.054088, -0.052318, -0.001117, -0.004915, -0.097368, 0.029686, 0.009192, 0.000451, -0.093834, 0.027660, 0.037287, -0.028877, -0.046064, -0.131003, 0.012027, -0.060362, -0.011458, 0.037385, 0.003656, -0.083786, 0.009312, 0.067797, 0.009321, -0.052920, -0.062035, -0.111021, -0.061103, -0.013720, 0.002159, -0.065789, -0.069429, 0.093862, -0.022112, -0.052190, -0.023974, 0.037267, -0.007319, -0.014662, 0.012456, 0.064721, -0.119949, 0.051835, 0.086928, -0.053819, 0.149962, -0.048775, 0.007997, 0.013534, 0.156885, -0.170497, 0.002833, 0.076239, 0.018147, 0.016530, 0.117818, 0.086042, -0.026094, -0.071025, -0.019798, 0.016523, -0.094094, 0.058682, 0.042721, 0.016972, -0.030888, -0.005256, 0.010551, -0.071423, -0.010902, 0.047919, -0.008069, -0.081009, 0.098000, -0.025148, -0.004419, -0.083520, 0.001434, -0.027758, -0.001123, -0.036835, -0.010435, -0.078143, 0.038236, -0.122006, 0.057770, -0.001644, -0.027489, -0.035571, -0.079109, 0.057221, -0.072837, 0.089843, 0.004096, 0.070115, -0.041653, -0.005939, -0.050753, 0.023852, -0.037359, -0.040775, 0.032013, -0.036376, 0.100982, -0.077058, 0.017141, 0.033145, 0.131450, -0.047127, -0.046959, -0.090013, 0.009621, -0.030532, -0.043546, -0.114703, -0.056767, 0.046679, 0.019221, -0.020404, -0.019810, 0.034085, 0.023351, -0.002025, 0.028667, 0.067506, -0.057562, -0.065125, -0.028081, 0.032363, -0.073061, 0.003245, -0.037846, -0.029040, -0.004958, -0.004121, -0.059322, 0.007556, -0.006346, 0.008143, 0.047046, -0.088986, -0.003314, 0.027730, 0.038793, -0.006220, -0.054013, 0.054233, 0.016608, 0.064084, -0.004090, 0.026277, 0.024123, 0.029523, -0.058662, 0.092759, -0.109976, -0.122450, 0.052384, -0.063022, 0.048695, 0.043856, -0.026602, 0.003853, 0.045908, 0.075825, -0.002954, 0.029213, -0.013314, -0.109016, -0.054069, 0.000224, 0.005305, 0.040231, 0.069525, -0.031798, -0.037665, -0.019798, 0.006644, 0.021786, -0.145591, -0.142535, -0.054899, 0.018095, -0.002629, -0.029431, 0.010713, -0.008477, -0.031913, 0.007011, -0.036469, 0.065025, 0.078166, -0.018307, -0.034961, 0.026421, 0.061393, 0.076523, -0.031729, 0.099773, -0.027596, 0.027079, 0.051763, 0.002803, 0.042729, -0.043545, 0.052996, 0.015632, -0.015112, -0.028066, 0.025816, -0.038230, 0.027472, 0.035782, 0.017825, -0.018522, -0.014310, -0.022490, -0.037348, -0.004628, -0.100177, -0.073773, -0.094245, 0.009175, -0.060251, -0.010032, 0.049597, -0.044521, -0.008437, 0.053550, -0.104306, 0.000244, -0.024634, 0.043389, -0.026048, 0.049523, -0.008697, -0.035261, 0.098976, -0.056122, -0.003481, -0.019245, 0.062048, -0.021751, 0.064865, -0.008816, 0.040171, 0.047591, -0.004531, 0.038266, 0.080586, -0.030221, -0.040064, -0.040529, -0.000784, -0.096946, 0.077216, -0.063657, 0.017751, 0.134686, 0.047619, 0.070305, 0.026589, 0.072053, -0.021748, 0.039498, -0.055156, -0.004014, -0.095880, -0.061474, 0.005517, 0.060866, -0.013757, -0.031508, -0.032926, -0.002861, -0.027055, 0.044819, 0.022153, 0.014712, 0.087701, -0.025440, -0.093669, 0.055008, 0.083692, -0.066327, -0.077473, -0.183242, -0.009675, 0.096148, -0.021286, 0.011613, -0.016270, 0.045019, -0.057293, 0.024372, -0.074034, -0.171139, 0.047974, -0.015022, -0.043119, 0.032007, -0.058607, -0.020918, -0.024317, -0.004106, 0.077152, 0.143796, -0.037047, 0.037771, -0.038133, 0.036550, -0.027981, -0.033593, -0.079854, -0.054628, 0.014611, -0.060175, 0.005035, -0.049746, 0.046154, -0.081947, -0.018102, -0.024111, -0.129955, -0.140197, -0.000891, -0.064196, 0.001966, 0.015021, 0.029640, 0.067209, 0.017414, -0.065325, 0.020475, -0.064622, -0.058328, 0.010072, -0.012901, 0.024829, -0.085961, -0.059144, -0.110593, 0.038369, 0.025591, 0.009057, -0.019025, -0.033265, -0.091534, -0.018542, -0.060288, 0.038389, 0.008871, 0.050891, 0.067729, -0.027037, -0.041600, -0.055031, -0.013085, 0.163781, 0.087417, -0.062955, 0.056871, -0.119087, 0.054159, -0.062144, 0.008454, 0.039189, -0.105452, 0.044284, -0.104428, -0.009930, -0.011318, -0.046512, 0.107261, 0.042492, -0.042244, -0.042763, 0.038981, 0.071505, -0.130992, -0.042116, -0.096247, 0.008298, 0.030171, 0.009749, 0.100481, -0.035752, 0.074876, -0.034251, 0.068342, -0.038720, -0.003483, 0.002622, -0.045871, 0.070540, -0.054998, 0.051730, 0.068801, -0.093079, -0.009162, -0.053759, 0.023823, -0.006129, -0.105805, 0.012414, -0.028083, -0.068917, -0.024308, -0.036598, -0.014207, 0.017207, -0.067944, 0.034053, -0.016536, -0.107869, 0.009410, -0.070516, 0.030974, 0.042175, -0.052713, -0.069743, -0.057731, -0.019052, 0.012854, -0.011637, -0.086250, 0.070714, 0.063172, -0.078886, -0.031358, 0.014030, -0.064157, 0.030434, -0.054754, 0.038014, -0.086412, -0.008764, -0.044746, -0.030149, -0.083100, 0.018718, 0.016435, 0.170275, 0.016560, -0.034273, 0.103311, 0.046473, 0.029819, 0.030363, -0.069681, -0.110110, -0.048612, 0.012075, -0.042229, -0.055573, -0.113199, 0.075860, 0.011471, -0.007487, 0.044859, -0.054662, -0.030458, 0.039249, -0.029501, 0.025460, 0.019573, -0.027498, 0.145292, -0.158519, 0.012333, 0.085784, -0.043058, 0.030167, 0.046246, 0.106067, -0.009571, 0.109184, 0.056804, 0.000695, 0.015573, -0.073866, 0.051490, 0.103161, -0.038529, -0.078125, 0.030111, -0.093969, -0.009283, 0.029429, 0.052618, 0.057573, -0.040101, -0.033688, 0.000479, 0.050177, -0.015015, 0.013574, 0.022442, -0.070652, 0.017641, 0.051614, 0.087536, 0.002109, -0.023734, -0.011002, -0.025727, -0.056891, 0.023115, 0.026763, -0.041672, 0.008180, 0.100762, -0.016911, 0.020496, 0.010249, 0.016788, -0.045226, -0.064929, -0.016844, -0.036222, 0.060006, 0.017893, -0.061746, 0.076592, -0.106543, -0.000816, 0.007786, -0.000637, -0.005984, -0.083504, -0.059783, 0.034223, -0.017969, -0.056680, 0.066590, 0.017292, -0.155445, 0.048634, -0.002162, 0.065664, 0.019937, -0.086705, 0.147846, 0.162007, -0.024699, 0.085586, -0.033015, 0.071020, 0.000654, -0.109814, -0.104047, -0.043339, -0.036674, 0.051627, -0.001582, 0.046440, 0.025471, 0.023292, -0.052025, 0.063270, -0.038811, -0.085403, 0.025992, -0.052591, -0.076600, 0.006240, 0.057920, -0.126277, 0.008287, -0.020574, 0.071182, -0.047315, -0.089828, -0.051777, 0.030366, -0.004426, -0.057616, 0.062457, -0.023555, 0.019959, -0.017557, -0.033393, -0.063478, 0.017003, 0.096321, -0.069544, -0.026311, 0.045935, -0.026704, -0.043545, -0.038991, 0.024604, 0.005437, -0.023109, 0.026503, -0.127182, -0.045306, -0.017780, -0.120331, 0.070852, 0.003508, -0.086801, 0.003614, 0.016213, -0.044690, 0.005219, 0.059890, -0.027852, 0.021139, -0.008256, 0.079135, 0.018373, 0.041946, -0.018481, 0.002897, -0.086430, -0.060223, -0.058269, -0.038447, 0.037373, 0.056589, -0.126437, -0.057405, 0.032396, -0.032886, -0.018151, -0.054668, 0.114224, 0.021132, 0.034434, -0.125189, 0.243827, 0.053414, 0.078176, 0.009319, -0.071217, 0.094667, -0.007816, 0.010350, 0.024979, 0.070739, -0.037638, -0.008927, -0.096353, -0.012805, 0.030190, 0.009645, 0.049595, -0.023006, -0.002372, -0.060632, -0.059725, -0.078984, -0.087111, 0.154110, -0.076726, 0.040237, 0.026439, -0.078753, 0.035894, -0.027932, -0.041641, -0.019395, 0.020372, -0.027509, -0.029412, -0.019078, -0.089281, -0.039656, -0.045635, 0.037435, 0.056155, -0.025501, 0.053771, 0.011546, -0.035667, 0.038696, -0.050052, -0.120335, 0.010260, -0.082842, 0.075564, -0.009088, 0.034540, 0.133171, 0.017599, -0.025469, 0.063289, -0.028287, 0.001648, -0.006785, 0.018499, -0.019089, 0.013518, -0.013023, 0.020486, -0.016619, 0.046474, -0.059426, -0.035097, -0.060563, -0.050413, 0.036688, -0.036206, -0.002013, -0.019850, -0.044408, -0.101966, 0.016316, -0.042788, -0.043650, 0.059198, -0.024527, -0.056292, 0.009257, -0.006454, -0.070230, 0.080873, 0.026516, -0.028025, -0.054269, 0.119218, -0.048033, -0.070130, 0.015630, 0.038630, -0.025584, -0.020850, -0.030868, -0.033672, 0.053855, 0.013750, -0.019989, 0.092078, -0.068259, 0.032215, -0.088640, -0.009335, 0.020479, -0.009325, -0.016641, 0.110796, 0.018799, 0.060676, -0.002628, -0.080404, -0.057773, 0.094708, 0.054717, -0.044807, 0.013051, -0.060115, 0.015699, -0.071078, -0.049482, 0.037747, 0.037956, -0.014053, 0.018345, -0.005476, -0.027037, -0.035293, 0.023910, 0.012280, 0.057265, 0.035398, -0.081915, 0.052466, -0.075831, 0.010355, 0.128896, -0.004663, -0.039108, -0.064687, 0.186117, 0.010645, 0.001225, -0.089573, 0.050314, -0.064496, -0.051947, 0.003274, 0.025480, -0.007971, -0.100192, -0.078770, 0.014308, -0.035221, 0.072281, 0.012416, -0.097197, -0.105134, -0.034327, 0.010407, 0.137865, 0.000913, 0.013011, 0.017414, -0.103406, 0.047999, -0.072891, -0.056444, -0.049117, -0.062750, 0.016929, -0.071049, 0.036876, -0.052982, -0.117703, 0.021172, -0.054409, -0.116204, 0.017462, -0.005203, -0.021831, -0.028800, 0.159629, -0.054014, -0.008481, -0.042786, 0.028015, -0.073311, -0.005856, -0.072910, 0.084935, 0.014203, -0.000433, 0.046285, -0.104665, 0.002284, -0.000451, 0.029055, -0.081488, 0.067192, 0.039387, -0.020910, -0.007397, 0.018549, -0.028573, -0.009808, -0.019600, 0.045427, -0.134135, 0.005064, 0.007491, 0.162472, 0.036817, 0.036745, -0.077328, 0.025237, 0.116128, -0.005984, 0.017528, 0.021177, 0.034414, -0.077642, 0.093566, -0.049495, 0.093162, 0.045405, 0.053370, -0.039412, 0.056263, 0.007425, -0.056310, -0.038532, -0.170054, -0.019957, -0.030060, -0.052435, 0.025954, -0.057537, 0.017958, -0.045756, -0.075031, -0.064543, 0.014740, -0.121049, -0.034408, -0.078869, -0.020430, -0.137145, -0.047518, -0.175439, -0.020774, -0.168842, -0.077191, 0.030857, -0.019752, 0.026531, 0.056643, -0.027826, 0.029694, 0.041408, -0.054516, -0.037241, 0.017748, 0.009566, -0.084209, -0.118781, -0.047136, 0.034169, 0.023954, 0.029859, 0.023140, 0.051549, 0.026428, -0.077100, 0.006092, 0.156817, 0.043188, -0.067365, 0.005020, -0.029928, 0.057524, -0.043924, -0.062467, 0.096657, -0.038457, -0.111439, 0.019867, -0.041029, -0.079376, -0.075211, -0.074082, -0.174673, -0.047626, -0.074363, -0.019009, 0.011914, 0.038541, -0.018770, -0.121183, -0.030366, -0.052415, -0.055691, -0.076561, -0.072333, -0.051627, 0.023924, 0.000385, 0.071957, 0.005478, 0.054491, -0.049936, -0.020801, -0.055238, 0.061395, -0.017721, -0.015554, 0.146095, -0.012124, -0.109653, -0.004235, -0.055587, -0.034569, 0.027850, -0.034418, -0.163447, -0.003012, -0.059988, -0.004968, -0.077853, -0.010664, 0.009992, -0.027376, 0.017786, -0.096826, -0.078841, -0.027509, -0.044754, -0.016052, -0.018816, 0.006669, -0.038630, -0.060857, 0.056659, -0.045895, -0.010547, 0.047951, 0.041279, -0.051164, 0.031486, 0.037555, 0.046660, -0.085604, -0.016008, -0.038800, -0.093229, -0.094397, -0.048918, -0.001721, 0.088164, -0.049931, 0.087454, 0.005526, -0.067818, -0.093775, -0.017549, -0.007463, -0.012019, -0.023411, 0.117044, 0.048841, -0.061431, 0.062019, 0.104087, 0.003792, -0.032473, 0.034750, 0.001593, -0.099032, -0.088172, 0.005374, 0.101695, 0.093685, -0.016310, 0.014544, 0.063110, -0.000071, -0.038737, -0.032683, 0.033043, 0.035541, -0.066582, 0.104641, 0.049232, 0.014256, 0.079007, -0.036011, -0.065079, 0.136759, 0.085705, -0.051735, 0.081325, -0.074287, -0.027315, -0.052200, 0.039475, -0.061936, -0.027476, 0.026581, 0.063870, -0.035944, -0.005161, -0.019064, -0.086000, -0.018726, -0.042036, -0.063566, 0.034107, -0.018801, -0.063559, 0.071234, -0.082221, 0.045028, -0.033690, -0.071904, -0.090374, 0.013909, -0.067229, -0.094497, -0.045292, -0.033990, 0.013700, 0.011629, -0.028934, 0.019268, -0.117532, 0.036666, -0.142682, -0.022882, -0.065220, 0.035372, -0.005708, -0.015557, -0.063271, -0.044613, -0.010627, 0.022100, -0.056825, 0.064478, -0.053655, 0.093549, -0.011790, -0.092653, -0.025379, -0.045265, 0.024492, -0.078872, 0.079377, -0.023541, 0.027541, -0.001891, -0.014740, 0.015057, 0.022545, 0.027287, 0.005068, -0.043049, 0.012542, -0.086257, 0.019450, -0.102064, -0.032825, -0.042036, -0.130426, -0.060313, 0.019011, 0.147943, 0.008487, 0.076847, 0.037193, -0.143966, -0.005861, -0.005338, -0.011189, -0.007087, -0.136298, -0.098666, -0.007582, 0.101722, -0.036827, -0.026571, -0.038736, 0.014786, 0.090874, 0.002290, 0.028952, -0.091890, 0.011003, 0.014792, -0.018748, -0.017158, -0.027128, -0.085904, -0.124395, 0.017534, -0.053669, 0.012739, 0.071635, 0.062934, 0.049525, -0.098805, 0.014848, -0.026074, -0.052081, -0.016094, 0.017462, -0.026173, -0.055697, 0.098997, -0.017040, -0.113925, -0.082061, -0.084840, -0.112875, -0.070653, 0.002922, -0.169840, 0.053049, -0.064823, -0.098381, 0.229519, -0.107305, 0.053731, 0.103908, 0.001705, 0.085582, -0.006275, -0.126322, 0.206810, -0.069939, -0.072699, -0.087337, 0.041976, -0.066433, -0.057096, -0.064997, -0.009406, 0.006730, -0.046888, 0.048327, 0.038702, -0.080289, -0.020044, -0.049433, 0.011548, -0.013219, 0.034254, -0.105100, -0.008022, -0.099952, -0.017590, 0.050330, -0.096068, -0.025034, 0.013697, 0.016633, -0.031302, 0.018391, -0.037686, 0.041205, -0.006614, -0.072029, -0.066952, -0.032902, -0.086474, -0.001376, -0.004646, -0.110189, 0.050511, -0.033095, 0.044399, -0.047902, -0.056005, -0.083275, -0.060320, 0.016337, -0.049838, -0.003793, 0.185140, 0.061569, 0.016299, -0.018860, 0.037894, 0.012908, -0.116964, -0.043450, -0.044097, 0.038862, -0.029839, -0.120455, -0.013102, -0.031561, -0.166935, 0.074533, -0.044920, -0.049670, 0.004990, -0.010419, 0.069527, -0.049949, 0.065966, 0.001975, 0.168903, -0.061422, -0.018551, -0.026563, -0.134013, -0.014292, -0.066634, 0.115808, 0.065745, 0.168351, 0.090401, 0.006143, -0.018427, -0.087555, 0.010989, -0.151731, 0.094288, 0.041557, -0.023768, 0.013104, 0.084554, 0.001795, -0.040061, 0.051273, -0.008989, 0.022976, -0.036620, -0.040565, -0.003523, -0.096093, -0.019841, -0.068969, -0.027688, -0.026197, 0.012908, -0.043808, -0.162728, 0.011925, 0.062368, 0.124308, 0.028168, -0.030250, 0.171782, 0.038885, -0.124274, -0.083352, -0.028960, 0.056862, -0.022699, -0.138169, -0.064438, -0.051982, -0.060283, -0.073628, 0.030151, 0.016391, 0.017199, -0.009055, 0.138803, 0.005123, -0.033754, -0.021934, 0.023624, 0.102019, 0.082972, -0.037537, 0.013272, -0.081548, -0.020747, 0.058473, -0.008166, -0.100178, -0.005966, -0.001769, 0.014233, 0.010889, 0.003855, 0.016598, -0.036223, -0.023408, 0.237172, 0.082398, -0.133443, 0.025383, -0.023134, 0.004650, -0.100660, -0.009963, -0.145921, -0.025180, -0.001691, 0.176258, -0.005804, 0.044509, -0.003961, -0.020199, -0.001075, -0.028667, -0.136844, -0.019362, -0.109156, 0.070511, 0.044116, -0.016501, 0.047122, -0.134526, -0.050452, -0.029917, -0.089644, 0.022953, 0.018844, -0.016096, -0.015290, -0.002717, -0.048386, 0.008210, -0.012667, 0.031517, 0.067263, 0.000964, 0.042467, 0.021234, -0.038648, -0.039946, -0.092823, -0.128995, 0.042691, 0.109180, 0.063604, 0.001919, -0.126425, 0.023697, 0.026501, 0.028951, -0.103560, 0.048749, -0.099734, -0.071197, -0.021136, -0.073330, -0.091160, 0.069180, 0.001762, -0.028768, -0.008020, -0.091729, -0.070641, -0.087841, 0.003568, -0.045997, 0.013024, -0.125454, -0.109000, 0.041865, -0.009116, 0.057426, 0.100077, 0.103703, -0.021654, 0.058314, -0.030165, -0.102972, -0.102135, -0.009441, -0.038225, 0.005980, 0.025408, -0.001653, 0.028154, -0.037762, -0.023304, -0.018735, -0.052642, -0.013909, 0.009902, -0.005414, -0.060055, 0.024542, 0.050213, 0.097210, 0.001732, -0.027514, -0.041719, 0.090195, -0.029900, 0.098730, 0.121559, 0.017486, 0.028860, -0.087361, 0.066674, -0.069504, -0.047936, -0.110219, -0.013678, -0.068923, 0.032159, -0.013202, 0.038434, -0.065102, -0.009576, -0.010012, -0.052373, -0.040730, 0.070485, -0.041140, 0.028641, 0.022333, -0.064176, 0.004484, -0.055443, -0.045099, -0.061381, -0.110319, -0.012661, 0.058432, -0.001983, 0.090161, -0.017781, -0.057648, -0.036841, 0.004362, -0.015231, 0.012867, -0.040440, -0.072468, -0.134548, 0.010922, -0.071758, 0.024467, -0.091269, -0.061734, 0.140857, -0.047988, -0.036488, -0.051407, -0.015311, 0.020583, 0.038150, 0.029020, -0.090891, -0.046302, 0.029365, 0.005414, -0.051164, -0.007649, -0.013174, 0.126146, -0.122645, -0.056437, -0.082976, -0.080884, 0.052630, 0.016894, 0.010428, 0.004770, -0.073359, 0.016080, -0.085842, 0.158179, -0.060789, -0.009179, -0.042830, -0.067575, -0.047351, 0.019170, -0.020914, 0.013991, -0.087695, -0.025252, 0.011354, -0.086145, 0.025737, -0.003495, -0.056050, -0.012206, 0.005948, -0.000269, -0.097526, -0.015201, -0.004458, 0.001050, -0.106419, -0.082869, 0.130719, 0.063950, -0.065131, -0.038914, 0.034395, 0.028035, -0.091724, 0.033485, -0.020572, -0.012938, -0.011324, -0.102896, 0.039078, -0.010945, -0.036062, 0.028836, 0.038130, -0.120370, 0.018080, -0.025580, 0.024539, -0.021558, -0.029840, 0.016534, -0.096605, -0.013386, 0.080909, 0.087435, 0.000478, -0.084671, 0.189163, -0.026793, -0.055844, -0.055332, 0.027590, -0.006068, -0.024192, -0.065977, 0.020072, -0.071251, -0.076482, 0.038408, 0.037832, 0.015962, -0.002668, 0.050972, -0.013873, -0.064260, -0.070067, -0.057761, -0.034016, 0.039043, 0.032199, -0.001318, 0.010228, -0.001791, -0.101754, -0.007464, 0.035290, 0.024250, 0.023859, -0.006410, -0.141738, -0.006683, 0.005228, 0.102941, -0.023655, 0.023273, -0.069818, 0.021492, -0.121291, 0.000194, 0.075342, 0.024628, -0.058736, -0.004953, -0.024844, -0.094340, -0.005107, 0.031009, 0.045265, -0.007688, -0.087007, -0.051305, 0.015813, -0.063835, -0.052001, 0.013344, 0.021219, -0.055284, -0.102924, -0.082654, 0.045253, -0.047945, -0.042641, -0.127326, 0.035671, -0.037309, -0.078377, -0.045683, -0.010240, -0.011893, -0.061290, -0.019507, -0.026735, 0.093017, -0.054615, -0.044993, -0.018066, -0.132559, 0.036840, -0.038491, -0.045981, -0.103635, 0.031923, -0.087205, -0.015756, -0.093348, -0.060666, 0.011880, -0.010533, 0.094029, 0.056666, -0.009638, 0.060112, 0.066183, 0.056536, -0.029024, 0.018682, 0.040591, 0.064773, 0.034021, -0.065847, -0.000848, 0.167674, 0.007495, 0.024995, -0.019991, -0.016751, -0.091200, 0.029027, -0.077894, 0.026523, -0.068537, 0.030475, -0.046916, 0.024915, 0.008678, 0.010919, -0.071181, -0.012905, -0.045404, 0.059051, 0.011151, 0.008697, 0.000355, -0.044795, 0.006641, -0.107496, 0.077240, 0.052092, -0.017411, -0.035295, -0.048999, -0.046596, -0.137468, 0.027462, -0.064983, -0.086993, -0.042303, -0.063232, -0.026153, 0.009067, -0.010192, -0.113680, -0.089125, -0.143921, 0.068682, 0.047953, 0.016469, 0.033361, -0.112991, 0.013105, -0.016169, -0.098037, 0.011135, 0.108329, -0.069980, -0.032161, -0.004935, 0.038807, -0.047160, -0.009981, -0.013487, 0.032119, -0.018227, -0.039907, -0.000303, -0.068395, 0.064878, 0.085550, 0.041910, -0.038753, -0.004238, 0.049152, -0.005470, 0.060471, -0.015206, -0.071733, -0.011000, -0.013151, -0.080331, 0.019906, 0.010134, 0.025987, -0.017836, -0.008357, -0.069210, 0.046278, -0.040963, -0.100230, 0.010886, -0.049204, -0.037730, -0.002588, 0.038056, -0.120194, -0.026480, -0.087144, 0.014957, -0.059549, 0.059274, 0.029341, -0.020645, 0.001789, 0.005164, -0.008975, 0.024450, 0.017187, -0.046697, -0.166564, -0.001693, 0.054229, -0.049910, -0.036636, -0.004285, 0.057146, 0.047682, 0.018106, -0.008734, 0.045876, -0.077805, -0.031028, -0.007013, -0.058388, -0.028529, -0.030942, 0.006311, 0.027522, -0.056357, -0.050698, 0.012848, -0.000048, -0.027402, 0.046213, -0.073681, -0.085868, 0.023357, -0.101768, 0.060881, -0.042491, -0.012127, -0.007764, -0.090207, 0.030305, -0.036792, -0.000402, 0.008241, -0.135309, 0.078174, 0.011609, -0.028792, 0.046646, -0.118021, -0.011929, -0.037460, -0.020678, 0.013546, 0.024834, -0.029548, -0.094506, -0.075332, 0.014088, -0.041078, 0.022379, -0.034980, -0.026511, -0.007545, -0.064964, -0.024212, 0.026493, 0.007862, 0.049846, 0.028451, -0.039067, -0.007538, -0.122420, 0.087515, -0.034855, -0.143478, -0.090053, -0.022124, -0.072403, -0.088095, 0.033617, -0.022820, -0.051650, -0.173583, 0.018156, -0.057306, 0.038194, -0.063582, -0.041391, 0.064103, -0.065246, -0.079222, -0.061086, -0.000445, -0.060324, -0.044783, 0.058473, -0.053262, -0.038699, -0.014055, -0.082389, 0.034723, -0.068618, 0.025234, 0.030987, 0.056631, 0.020258, -0.049805, -0.006980, -0.025751, -0.062401, 0.137149, -0.035626, -0.045608, -0.063709, -0.025631, 0.043579, -0.148308, -0.076807, 0.062374, -0.090846, -0.020181, -0.041041, -0.053782, -0.071728, -0.075655, -0.102180, 0.023409, 0.035376, 0.089600, -0.022536, 0.052631, 0.081817, 0.115836, 0.055265, -0.065571, 0.003168, -0.048209, -0.057151, -0.014840, -0.044651, 0.004026, -0.017924, -0.048464, 0.024664, -0.039699, -0.005078, -0.126151, -0.024545, 0.001693, -0.135530, -0.082884, 0.087829, 0.022866, -0.047318, -0.054954, 0.006474, -0.054169, -0.039594, -0.009402, -0.024540, 0.082813, 0.006668, -0.024615, -0.113064, -0.065548, 0.037903, -0.014137, -0.005066, 0.009425, 0.179209, -0.143263, -0.005053, 0.055770, -0.080200, -0.069862, -0.019893, -0.074709, -0.059603, 0.011813, -0.053983, -0.011295, -0.008667, -0.068729, -0.036386, -0.124842, -0.005873, -0.137511, -0.094075, -0.014565, 0.009841, -0.021862, -0.084456, -0.056429, -0.001492, -0.015630, -0.013846, -0.075099, -0.185449, -0.006466, -0.132401, 0.021306, -0.078908, 0.046499, -0.015181, -0.028524, 0.042449, 0.024540, 0.012543, -0.094996, -0.090774, -0.122903, 0.087959, -0.042698, -0.008407, -0.080687, -0.064993, -0.059581, -0.066843, -0.010724, 0.001056, -0.017199, 0.012045, -0.054750, -0.043568, -0.046272, -0.001593, 0.019364, -0.089088, 0.086657, 0.006471, 0.068404, -0.055084, -0.020432, 0.034184, 0.012588, -0.032504, -0.095171, 0.025688, 0.100513, 0.001329, -0.085837, -0.037096, 0.062078, -0.008902, 0.053627, -0.104491, 0.021878, -0.012543, -0.098318, 0.003579, 0.072648, 0.012998, 0.097650, -0.030901, -0.058844, 0.017878, -0.054276, 0.021646, -0.113162, -0.140063, -0.054487, 0.110916, -0.094747, -0.102110, 0.046669, -0.087482, -0.041803, -0.024611, -0.054625, -0.039353, -0.035381, -0.090376, 0.002248, -0.099418, 0.124216, 0.048089, 0.077599, -0.080490, 0.086385, -0.058209, 0.053222, -0.063634, -0.050988, -0.004811, -0.039399, 0.121079, 0.087359, -0.051793, -0.055468, -0.010621, -0.023792, 0.017792, 0.040856, -0.073055, -0.154155, -0.115582, -0.075320, 0.031559, -0.063734, -0.127295, 0.000731, 0.026805, -0.064747, -0.063488, -0.033623, -0.089532, 0.060535, 0.089261, -0.044621, -0.096297, -0.110110, 0.022107, 0.026342, -0.116596, 0.013049, -0.060717, 0.002003, -0.017428, 0.165348, -0.076974, -0.001400, -0.015800, -0.030224, -0.058570, -0.007272, -0.098678, 0.007151, 0.060704, -0.042748, -0.164016, -0.066703, 0.012404, -0.003382, 0.031831, 0.024437, -0.039950, -0.035138, 0.133119, -0.053958, 0.144570, 0.014905, -0.022932, 0.054601, 0.021173, -0.060931, -0.137118, 0.041872, -0.060303, 0.071439, 0.018452, -0.062224, 0.004597, -0.131247, -0.128480, -0.000669, -0.063224, -0.004326, 0.016111, 0.032925, 0.009129, -0.080584, -0.049154, -0.038263, -0.026584, -0.018199, -0.013113, -0.035950, 0.066460, 0.009206, -0.027241, 0.060532, -0.022074, -0.027247, 0.062292, -0.024472, -0.024321, -0.107323, -0.019402, -0.061333, 0.126974, 0.177132, 0.084461, 0.029819, -0.021509, 0.004707, -0.036017, -0.008029, -0.013960, 0.009247, -0.068670, -0.028283, 0.094941, -0.017512, 0.022058, -0.197555, -0.040684, -0.049030, -0.125430, -0.155303, 0.049388, 0.026448, 0.019315, -0.024434, -0.123324, 0.063186, -0.035896, -0.056541, 0.211590, -0.084532, -0.008515, -0.118111, -0.094283, 0.043101, -0.070513, -0.075465, -0.020645, 0.026580, -0.045913, -0.085835, -0.016316, -0.015076, 0.017666, -0.042573, 0.180241, -0.016758, -0.014532, 0.026672, -0.029880, -0.054528, -0.123472, 0.027690, 0.169849, -0.074389, -0.025194, -0.018333, -0.064891, 0.005422, -0.020301, 0.091842, -0.056576, -0.014926, -0.080051, 0.007934, -0.011588, -0.051593, -0.021243, -0.098679, -0.094729, 0.009951, 0.049252, -0.023713, -0.042003, 0.099629, 0.002289, -0.016961, -0.105695, -0.006184, -0.112218, -0.021532, 0.030921, 0.022818, -0.076167, -0.056062, 0.045409, 0.033381, 0.077168, -0.069687, -0.055336, -0.054239, -0.089094, -0.051825, 0.044157, -0.090067, 0.032336, -0.015835, -0.099624, -0.111301, -0.015995, -0.069890, -0.054951, -0.022280, -0.039202, -0.096657, -0.038123, -0.014453, -0.045897, 0.031325, 0.011410, 0.028024, -0.010506, -0.056831, -0.047890, -0.053601, -0.086217, 0.044459, -0.055718, 0.003945, -0.098866, 0.027436, 0.010198, -0.025111, -0.156521, -0.051656, -0.054433, -0.108117, -0.017872, 0.057969, 0.071885, -0.093266, -0.009351, 0.115561, 0.067799, -0.050731, -0.098244, 0.070373, 0.006794, -0.017112, 0.054750, -0.087942, -0.133421, -0.123539, -0.018527, -0.058143, -0.066502, 0.133005, -0.067803, 0.028066, -0.051728, -0.033747, -0.024666, 0.070185, 0.025638, -0.103510, 0.087354, -0.047193, 0.001738, 0.060987, -0.093385, -0.051606, 0.006850, -0.078226, 0.052589, 0.017577, -0.053063, -0.050290, -0.065934, -0.012093, -0.062689, -0.005243, 0.020933, 0.031810, -0.074972, -0.128248, -0.017490, -0.028863, 0.090482, -0.033333, 0.058303, -0.063815, -0.040613, 0.046108, 0.032658, 0.019335, -0.041876, -0.052066, 0.032006, -0.024690, 0.082688, -0.017214, 0.004844, -0.007334, -0.043003, 0.063300, -0.007531, -0.004549, 0.026502, -0.014250, 0.015944, -0.049141, -0.033138, -0.050438, -0.145756, -0.066163, 0.043814, 0.015170, -0.001682, -0.095093, -0.039044, -0.054514, -0.101847, -0.121882, 0.018371, -0.018529, -0.022400, -0.099507, -0.032229, 0.026589, -0.035004, 0.011905, -0.046324, -0.161131, 0.019983, -0.006836, -0.098129, -0.012796, -0.038357, 0.018093, 0.013599, -0.016967, 0.014571, -0.029862, 0.024030, -0.024289, 0.001180, 0.028333, -0.029856, -0.068924, 0.013857, -0.070068, 0.021125, -0.031461, 0.011364, -0.049537, 0.022268, 0.025494, -0.111916, -0.013410, -0.007978, 0.050555, -0.069954, -0.030416, 0.022519, -0.094122, -0.052196, -0.096099, -0.004223, -0.090119, -0.023014, -0.011168, -0.018270, 0.025888, -0.073157, -0.108030, 0.030615, -0.052347, -0.009208, 0.001170, 0.069353, -0.038029, -0.002650, -0.084435, 0.213744, -0.009082, -0.178888, 0.013943, 0.012953, -0.041535, 0.106462, -0.056254, -0.016709, 0.002540, 0.045781, -0.013292, -0.007782, -0.060433, -0.104022, -0.034432, 0.081337, 0.004776, 0.027992, -0.067430, 0.024372, -0.038314, 0.077729, -0.012181, 0.071913, -0.149097, -0.005562, -0.070064, -0.063484, 0.053483, -0.106564, -0.083413, -0.144449, 0.028837, -0.097644, 0.041319, -0.027501, -0.086536, -0.028334, -0.067867, -0.169576, -0.060115, 0.074511, 0.087909, -0.086242, -0.124022, 0.076463, -0.117157, -0.011728, -0.143629, 0.011288, -0.028524, 0.084156, 0.006395, -0.010083, -0.035838, -0.031967, -0.104782, -0.015724, -0.033531, 0.025057, -0.130828, 0.004164, -0.054386, -0.021847, 0.044830, -0.075812, -0.023048, -0.067997, 0.063208, -0.014682, -0.087019, 0.007533, -0.061076, 0.015013, -0.039114, -0.026515, 0.028293, -0.060270, 0.000305, 0.014429, -0.050458, -0.051775, 0.071617, -0.087357, -0.001004, -0.060608, -0.029294, -0.143875, -0.049020, 0.009300, 0.144264, -0.031889, -0.107501, -0.030006, 0.003705, -0.036864, 0.024918, -0.073046, -0.073167, -0.018553, -0.037381, 0.037951, -0.054481, -0.002876, -0.091495, -0.036228, -0.048821, 0.038195, -0.062353, 0.034391, 0.020340, 0.004659, -0.205908, -0.031057, 0.083592, 0.031841, -0.095310, 0.018868, -0.018223, 0.074927, 0.031850, 0.022411, 0.036103, -0.006614, -0.110875, -0.134144, -0.041734, -0.018866, 0.029912, 0.036585, 0.070918, -0.069343, -0.018852, 0.038298, 0.022923, -0.018434, 0.079021, -0.036741, -0.011987, -0.089643, 0.023902, -0.059121, 0.006052, -0.007910, -0.017143, -0.055789, -0.030073, -0.096726, -0.015557, -0.054090, -0.051685, 0.051907, -0.003247, -0.004879, 0.077167, -0.071760, -0.113854, -0.008343, 0.058408, 0.041699, 0.050096, -0.147810, -0.009057, -0.085391, -0.061400, -0.008296, 0.081788, -0.124717, 0.000904, -0.034957, -0.077846, 0.028270, -0.040323, -0.080425, 0.021025, 0.015710, -0.172054, 0.029374, -0.091544, -0.009115, -0.070840, 0.045067, 0.121600, 0.028324, -0.018973, 0.018332, -0.015369, 0.009158, -0.047959, -0.007169, -0.076165, 0.042704, -0.015309, 0.003440, -0.070394, -0.102132, -0.120468, 0.023919, -0.038404, -0.033070, -0.099533, -0.032381, -0.033083, -0.117310, 0.102606, -0.048639, -0.056748, -0.066873, 0.012669, 0.076358, 0.004758, 0.049093, -0.030926, -0.036232, -0.057554, -0.112518, -0.019907, 0.031896, 0.019689, -0.057923, 0.024274, 0.034324, -0.006374, -0.096502, -0.047274, -0.026688, -0.088654, -0.090484, 0.014328, -0.037169, 0.026552, 0.030344, -0.071901, -0.050709, 0.012976, -0.008651, -0.068875, -0.123792, 0.063328, -0.044369, -0.060010, 0.055907, -0.016273, -0.073661, 0.025953, -0.096120, 0.017266, 0.016730, -0.075339, 0.008264, -0.063276, -0.037991, 0.133919, 0.029753, -0.124343, -0.028381, -0.021317, -0.021241, 0.026460, -0.060694, -0.033380, -0.055625, -0.012722, -0.020365, 0.043288, 0.085431, 0.051273, -0.153984, 0.028586, -0.008793, 0.006677, -0.027446, -0.074853, 0.013321, -0.101695, 0.040226, 0.012006, 0.060834, -0.053428, -0.001795, -0.067351, 0.059663, -0.014659, -0.115016, -0.053304, -0.026165, 0.107789, -0.002691, -0.048512, -0.079575, 0.013888, -0.033217, -0.023843, -0.027292, -0.096240, 0.037049, -0.002041, -0.172241, -0.067455, 0.006712, -0.165693, -0.069426, -0.001251, -0.012426, -0.038016, 0.024274, 0.032739, -0.124760, -0.051795, -0.044742, 0.071834, -0.017945, 0.007171, -0.049961, 0.034770, -0.085781, -0.002622, -0.017546, -0.105112, -0.051796, -0.026796, -0.058614, -0.065457, -0.055185, 0.085640, -0.016906, -0.029192, -0.018320, 0.056174, 0.070045, -0.034212, -0.083622, -0.038983, -0.080653, -0.012551, 0.009874, -0.020235, 0.007249, -0.080056, -0.039306, 0.004099, -0.051454, -0.048789, -0.018999, 0.001458, -0.106350, -0.091034, -0.048281, -0.092889, 0.017851, -0.042972, -0.036046, -0.012266, -0.007316, -0.032924, -0.013513, -0.050214, 0.110446, -0.026669, 0.040863, -0.046572, 0.006436, 0.018127, -0.064446, 0.044304, 0.035645, -0.062293, -0.107471, -0.138818, -0.061337, 0.015928, 0.025443, 0.039740, 0.114887, 0.008117, 0.036122, -0.025301, -0.077497, -0.021271, 0.022079, 0.034484, 0.035138, 0.056259, 0.146208, -0.103004, -0.010521, -0.008575, -0.066713, -0.088965, 0.039003, -0.047152, -0.011313, 0.045844, -0.043924, -0.045294, -0.084612, -0.055115, -0.016229, -0.021248, -0.125738, -0.087528, -0.037317, -0.040958, -0.061772, 0.008557, 0.057528, -0.032905, -0.008931, -0.007657, -0.014948, -0.042810, -0.158084, -0.056831, 0.029111, -0.090792, 0.037700, -0.043224, -0.005761, -0.209370, -0.085824, 0.031636, -0.071765, -0.065437, -0.023203, -0.145496, -0.100779, -0.048231, -0.148674, -0.016117, -0.039603, -0.029179, -0.031952, -0.061693, -0.159332, 0.035535, -0.033847, 0.025534, -0.174962, -0.125322, -0.087609, -0.014352, -0.116667, -0.025129, -0.019006, -0.039892, -0.084463, -0.047300, -0.058276, -0.059128, -0.203886, -0.111419, -0.137832, -0.086681, -0.101767, -0.161353, -0.018328, -0.009659, 0.007047, -0.088073, 0.008282, -0.018048, -0.245370, 0.035129, -0.133155, -0.010034, 0.023269, -0.036182, -0.048637, -0.038938, -0.008552, -0.033351, -0.055468, -0.109042, -0.108458, -0.064878, -0.012619, -0.032324, -0.038976, -0.115428, -0.182211, -0.094827, -0.088490, -0.080803, -0.165246, -0.092151, -0.076843, 0.027688, -0.029162, -0.061247, -0.072496, -0.032633, 0.110880, -0.063078, -0.013393, 0.027804, -0.069980, -0.034091, -0.177057, -0.030813, -0.054427, 0.058193, -0.018920, -0.035328, -0.065070, -0.172277, -0.005126, -0.081939, -0.112268, -0.066598, -0.208891, -0.138833, 0.003752, 0.049492, -0.090846, 0.016607, -0.046585, -0.164962, -0.030506, -0.017720, -0.071374, 0.023751, -0.103067, -0.031485, -0.072418, -0.043321, -0.039308, -0.153890, -0.036551, -0.012544, -0.111863, -0.067786, -0.089347, 0.060617, -0.033279, -0.000436, 0.006073, -0.075750, -0.071336, 0.043553, -0.095716, -0.108946, -0.073641, -0.120635, -0.125765, -0.084420, 0.016853, -0.089974, 0.021896, 0.002522, -0.044302, -0.014901, -0.063089, -0.133309, -0.075516, -0.043251, -0.106286, -0.171561, -0.161765, -0.141905, -0.047315, -0.031777, -0.088404, 0.025822, 0.163576, 0.053963, -0.073547, -0.038048, -0.075287, -0.014624, -0.064737, -0.085448, 0.008778, -0.040584, -0.085630, -0.047506, -0.069015, -0.117019, -0.092444, -0.201737, -0.045213, 0.073659, -0.039256, -0.175659, -0.141447, -0.026636, -0.034901, -0.027968, 0.099361, 0.044039, -0.075240, 0.010707, -0.010987, -0.115600, 0.006527, 0.034030, -0.089081, -0.023504, -0.021482, 0.095422, -0.012023, -0.001788, -0.142362, -0.019562, -0.025772, -0.024087, 0.030200, -0.107878, -0.066266, -0.077744, -0.036340, 0.065946, 0.107864, -0.082102, 0.008693, -0.043693, -0.159851, -0.066588, 0.084492, -0.024684, -0.113186, -0.127687, -0.010208, -0.023524, -0.067588, -0.037945, 0.023384, -0.061008, -0.051942, -0.166109, 0.032743, 0.012024, -0.089604, -0.157976, -0.047705, 0.054792, -0.168049, -0.146617, -0.107231, 0.003393, 0.044934, -0.048409, -0.044923, -0.087669, -0.131299, -0.011635, -0.028346, -0.059192, -0.077819, -0.001099, -0.082403, -0.026223, -0.146489, 0.178994, -0.153092, -0.125173, -0.113443, -0.042372, 0.040847, -0.181624, 0.014775, 0.019987, 0.012798, -0.056445, 0.019974, -0.025646, -0.013878, -0.009154, 0.009350, -0.090035, -0.052815, -0.115124, -0.013319, -0.003437, 0.019020, -0.028021, -0.085844, -0.048718, -0.048492, -0.036349, -0.153669, -0.052451, -0.125855, -0.051294, -0.088019, -0.132761, -0.009827, -0.246647, 0.004497, -0.069964, -0.035354, 0.028620, -0.181949, 0.006223, -0.056517, -0.034173, -0.077606, -0.126402, 0.077607, -0.017441, 0.061277, -0.165571, 0.006561, -0.000892, -0.107725, -0.053631, 0.004944, -0.107774, -0.024766, -0.102415, -0.127855, 0.027178, -0.038053, 0.027231, -0.051874, -0.050565, -0.020743, -0.010114, -0.200283, -0.093337, -0.081682, -0.013754, 0.025329, -0.062426, -0.026942, -0.022150, 0.018053, -0.057145, -0.118962, -0.051719, -0.035679, -0.115943, 0.003789, -0.211673, -0.072409, -0.076953, -0.022083, -0.062983, -0.032755, -0.098904, -0.087043, 0.004886, -0.069703, -0.185815, -0.113261, -0.060028, -0.076744, -0.111120, 0.010800, -0.029740, -0.023253, -0.113491, 0.000355, -0.010826, -0.059702, -0.008936, -0.076669, -0.081532, -0.008119, -0.019947, -0.052895, -0.000997, 0.063649, 0.010410, -0.115233, -0.008057, -0.058694, -0.062951, -0.081221, -0.010684, -0.085168, 0.000979, -0.084798, 0.063879, -0.003000, -0.025171, -0.025162, 0.002724, -0.052466, -0.098647, -0.026523, -0.042235, -0.027131, -0.016302, -0.013635, -0.036741, -0.030274, -0.013606, -0.102609, 0.007596, -0.033718, -0.146994, -0.093962, -0.142667, 0.079682, -0.157051, 0.006001, -0.049866, -0.119402, -0.066794, 0.010516, -0.070314, -0.095902, -0.023994, 0.060429, -0.030665, -0.057536, -0.084487, -0.006518, -0.103935, -0.062918, -0.044240, 0.034821, -0.141520, -0.055618, -0.073659, -0.010398, -0.170778, -0.125629, -0.026685, -0.064068, -0.026568, -0.078954, -0.079195, -0.096539, -0.027852, -0.061934, -0.105703, -0.045912, -0.108691, -0.110657, -0.054543, -0.017747, -0.216223, -0.149401, -0.124464, -0.058056, -0.097142, 0.055057, 0.008135, 0.029501, -0.094037, -0.085134, -0.118367, 0.007843, 0.020667, -0.001630, 0.037465, -0.057812, -0.043586, 0.032555, -0.057792, -0.014121, -0.099622, -0.200644, -0.084510, -0.114172, 0.000382, -0.012982, 0.005003, 0.023311, -0.133390, -0.041958, -0.086457, 0.007214, -0.019054, 0.094048, -0.184797, 0.000050, -0.043742, -0.011707, -0.088901, 0.066541, -0.026683, -0.025367, -0.120825, -0.091161, -0.052867, -0.084970, -0.098094, -0.084255, -0.035833, -0.140957, 0.026427, -0.138799, -0.118388, -0.016066, -0.173466, -0.151373, -0.099596, -0.011891, -0.008740, -0.091997, -0.036254, -0.044546, -0.069135, -0.085739, -0.084239, 0.006861, 0.022495, 0.026337, -0.104039, -0.161903, -0.117404, -0.039597, 0.001049, -0.136875, -0.135920, -0.029940, -0.119159, -0.005292, 0.023008, -0.146342, -0.035463, -0.029318, -0.095407, -0.005398, -0.031166, 0.007362, -0.116555, 0.035973, -0.012450, -0.051088, 0.002083, -0.075127, -0.092994, -0.065522, -0.082204, -0.146040, -0.095068, -0.163277, -0.094476, -0.092181, -0.102164, -0.002334, -0.065445, -0.100839, -0.046088, -0.094895, -0.159662, -0.016941, -0.043809, 0.134827, 0.010811, -0.118066, -0.034293, 0.045290, -0.066673, 0.066131, -0.127938, -0.217097, -0.083879, -0.077857, -0.005547, -0.101144, -0.124539, -0.161578, -0.108288, -0.147682, 0.027775, -0.128170, -0.086496, 0.062574, -0.000376, -0.023132, -0.027709, 0.035136, -0.089415, -0.021606, 0.025409, 0.153340, -0.042275, 0.014746, -0.016939, -0.166732, -0.092430, -0.033060, -0.161774, -0.110677, 0.049415, 0.035932, -0.024147, -0.054017, -0.129748, -0.040417, 0.019039, -0.084035, -0.076554, -0.038126, 0.035142, -0.154385, -0.021507, 0.032876, -0.074000, -0.190339, -0.045349, -0.068609, -0.024944, -0.197532, -0.014149, 0.069382, 0.093305, -0.096608, -0.149966, -0.084281, -0.085309, -0.205292, 0.013253, -0.016653, -0.204211, 0.082902, -0.074303, -0.002598, -0.046499, -0.086374, 0.005176, 0.035704, -0.106288, -0.052987, -0.047082, 0.022856, -0.044798, -0.116190, 0.037538, 0.033612, -0.111097, -0.055967, 0.037794, -0.178211, 0.121803, 0.050526, -0.024156, 0.004380, 0.003529, -0.044022, -0.056026, 0.013409, -0.072937, -0.023775, -0.032553, -0.013852, 0.007434, 0.095568, -0.052453, -0.085973, -0.049698, -0.005846, 0.001939, -0.199516, 0.067290, 0.002542, 0.000504, 0.017101, -0.141081, -0.004449, -0.063687, -0.094958, -0.221397, -0.086699, -0.037953, -0.242561, -0.051157, -0.041071, -0.106959, -0.083489, -0.031896, -0.049437, -0.052780, 0.081506, 0.001303, -0.037710, -0.117156, -0.010215, 0.034364, 0.013451, -0.058846, -0.093316, -0.030052, 0.042126, -0.007410, -0.104087, -0.100107, -0.116361, -0.031977, -0.007226, -0.063154, -0.026301, -0.052014, -0.030013, -0.118520, -0.117907, 0.027108, -0.026005, -0.078199, -0.064114, -0.067012, -0.047456, -0.039830, -0.059997, 0.058316, 0.021449, 0.020906, -0.065907, -0.096774, 0.153980, -0.052239, -0.158122, -0.136904, -0.026429, -0.146755, -0.145207, -0.105189, -0.009569, 0.108928, -0.178993, -0.046388, -0.051182, -0.053076, -0.008432, -0.037712, -0.050719, -0.125388, 0.019143, -0.083396, -0.043638, 0.036488, -0.065429, -0.042308, -0.071716, 0.018200, -0.073629, -0.126902, -0.019973, 0.013280, -0.104949, -0.037153, -0.041859, -0.065925, -0.000353, -0.018098, -0.025898, -0.142619, -0.051541, -0.024688, -0.060343, -0.065543, -0.016462, -0.144331, 0.097699, 0.003501, -0.203914, 0.025759, 0.009597, -0.063433, -0.019153, -0.067753, -0.046517, -0.039235, -0.064540, 0.001982, -0.154586, 0.032236, -0.139497, -0.057073, -0.042069, 0.109552, -0.039474, -0.020640, 0.030880, -0.132713, -0.097189, -0.029872, -0.097033, -0.044187, -0.093056, -0.221692, -0.051384, -0.023593, -0.022237, -0.027680, -0.003745, -0.124211, -0.131082, -0.112231, -0.087151, 0.024080, 0.015287, -0.079637, 0.019080, 0.106745, -0.047391, -0.039821, 0.065244, -0.037343, 0.086339, -0.107950, -0.124391, 0.019368, -0.118527, -0.075613, 0.026635, -0.015533, -0.148433, -0.076053, 0.026691, -0.047917, -0.131902, -0.152862, -0.034359, -0.049656, 0.054030, -0.092144, -0.045984, -0.095613, 0.065045, -0.015860, -0.054613, -0.021254, -0.031909, -0.088644, -0.150466, -0.086626, 0.096268, -0.051271, -0.047503, -0.010284, 0.026641, -0.109454, -0.029591, -0.108317, -0.018548, -0.032064, -0.032951, -0.042267, -0.029570, -0.108059, -0.125773, -0.043264, -0.053185, -0.025101, 0.024776, 0.027814, 0.010568, -0.018159, -0.037867, 0.070675, -0.082574, -0.082369, -0.011769, -0.003869, -0.069218, -0.045187, -0.105767, -0.078764, -0.119452, -0.057554, -0.141438, -0.048273, -0.005213, -0.016798, -0.021938, -0.054040, 0.087878, -0.053901, -0.024790, -0.074424, 0.090631, 0.077045, -0.122400, -0.045959, -0.080233, -0.023143, -0.008183, -0.073557, -0.058598, -0.067926, -0.068388, 0.046757, -0.091531, -0.014196, -0.072239, -0.021033, -0.106184, -0.101024, 0.100434, -0.041483, -0.099013, -0.064348, -0.061941, -0.105166, -0.036530, -0.170511, -0.056255, -0.082629, -0.103072, -0.001394, -0.077696, -0.031428, 0.010446, -0.036178, -0.076783, -0.103649, -0.046125, -0.064725, -0.131065, 0.054568, -0.121273, -0.108667, -0.218766, -0.015360, -0.091838, -0.022640, -0.166454, -0.031972, -0.071677, -0.127613, -0.025813, -0.065088, -0.099905, -0.078769, -0.029354, -0.059183, -0.100114, -0.042001, -0.096547, -0.035173, -0.033742, -0.033331, -0.007285, 0.013001, -0.172178, -0.124228, 0.062100, -0.068335, -0.001411, -0.000125, -0.166186, -0.002691, -0.167646, -0.015025, 0.039517, 0.029772, 0.051999, 0.016960, 0.027776, -0.048324, -0.174539, -0.054685, -0.016646, -0.100795, -0.102224, -0.069448, -0.000672, -0.112477, 0.000417, -0.123200, -0.079899, 0.010367, -0.130529, -0.037480, -0.068628, -0.092778, 0.004991, -0.064954, -0.098490, -0.033082, 0.084744, -0.040155, -0.132629, -0.080317, -0.012260, -0.078556, -0.047073, -0.055818, -0.099587, -0.033711, -0.083771, -0.094077, 0.061040, -0.046483, -0.012626, -0.088664, -0.080059, 0.046589, -0.024667, -0.008335, -0.115507, -0.039395, 0.029258, -0.110191, 0.062231, 0.102726, -0.080197, -0.103777, 0.067900, -0.114527, -0.005452, -0.018142, -0.071094, 0.044465, -0.119966, -0.090982, 0.107903, -0.131276, -0.028668, -0.048195, -0.051495, -0.096204, -0.222264, -0.003413, -0.048116, -0.045163, -0.019517, -0.048619, -0.104349, -0.008027, 0.037445, 0.019432, -0.102617, 0.049305, -0.078750, -0.081285, -0.104679, -0.131023, -0.064440, -0.037233, -0.109053, -0.070462, 0.015392, -0.010736, -0.105064, -0.192057, -0.011876, 0.051546, -0.072154, -0.007075, -0.034723, 0.072292, 0.054770, 0.058266, 0.018172, 0.134702, -0.091277, 0.034348, -0.018793, -0.009712, -0.014507, 0.012826, 0.001215, 0.022018, -0.017945, -0.017820, -0.082098, -0.054103, 0.016053, -0.122183, -0.027454, 0.050278, 0.000099, -0.004873, -0.037382, -0.089941, -0.066073, 0.048811, 0.033902, 0.004819, -0.029068, -0.088840, -0.083674, 0.031415, -0.059567, -0.101560, -0.068575, -0.007159, 0.051948, -0.105216, 0.052279, -0.068241, -0.076601, 0.054391, -0.076561, -0.049803, -0.104286, 0.016913, 0.049502, -0.093043, 0.120220, -0.084768, 0.065270, -0.017771, 0.006305, 0.017315, -0.061574, -0.071270, -0.017301, 0.050811, 0.022675, 0.000698, -0.030510, 0.054086, 0.032941, -0.131208, 0.026341, -0.039762, 0.037068, -0.054000, 0.066613, 0.064460, -0.003736, -0.035707, -0.008300, -0.004871, 0.005164, -0.039424, -0.070225, -0.010510, 0.096785, -0.063464, 0.040424, -0.005721, -0.005047, -0.025513, -0.040610, -0.020432, -0.057373, -0.055028, -0.014634, 0.039469, 0.006138, -0.016658, -0.052968, -0.011498, -0.006855, -0.035823, -0.112460, -0.012522, -0.027178, -0.022512, 0.002062, -0.012579, -0.009614, -0.042087, 0.003649, -0.032792, 0.040667, -0.039637, -0.073899, 0.025328, -0.019280, -0.047147, -0.152090, 0.070540, 0.006016, -0.042966, 0.012522, -0.060360, 0.000940, -0.009060, 0.041843, -0.101981, 0.015785, -0.022833, -0.066582, 0.039875, -0.069258, -0.024211, -0.086210, 0.017095, 0.016342, -0.026815, -0.056971, 0.051229, -0.092468, -0.076927, -0.065852, -0.006573, 0.026885, -0.022567, -0.101232, -0.080884, -0.011452, -0.063817, 0.027089, 0.000323, 0.062955, 0.023354, 0.000813, -0.017281, 0.025921, -0.071450, -0.002567, -0.087503, 0.057490, 0.052974, 0.012856, 0.028759, -0.099275, 0.000429, -0.111043, -0.048089, -0.014012, -0.009349, 0.011269, -0.075099, 0.079500, -0.016869, -0.068317, -0.002366, -0.054314, 0.033333, 0.035631, -0.026551, -0.015875, -0.024076, -0.002465, -0.047621, -0.027324, 0.002064, -0.067662, -0.007235, -0.003584, 0.036156, 0.009726, -0.001302, -0.120708, 0.105021, -0.007836, 0.044930, 0.059413, 0.039897, -0.086488, -0.016110, -0.002262, -0.048602, -0.027464, -0.028142, 0.073196, -0.012120, 0.038054, -0.069382, -0.008228, -0.010524, 0.076778, 0.023928, -0.026035, -0.120994, 0.056827, -0.068335, -0.023475, -0.003999, -0.090305, -0.072121, 0.047768, 0.017709, -0.125202, -0.040791, -0.029563, -0.024017, -0.053897, -0.180396, -0.014785, 0.039483, 0.023802, -0.074444, -0.016831, -0.034375, 0.025140, -0.045427, 0.015336, -0.043220, 0.041243, -0.009864, 0.035992, -0.027862, 0.022615, 0.099386, 0.009591, 0.048860, -0.099805, 0.001533, 0.037326, 0.016711, -0.060804, -0.005942, -0.040747, -0.072978, 0.034257, -0.017052, 0.063441, 0.027553, -0.111526, -0.052513, 0.060927, -0.065154, 0.022730, -0.084739, 0.039914, 0.014610, -0.078548, -0.094637, 0.042680, -0.030863, 0.029955, -0.000364, -0.079526, 0.018646, 0.087209, -0.056045, -0.016944, 0.026052, -0.027900, -0.078535, -0.028211, -0.009722, -0.054331, 0.004902, 0.068617, -0.043524, 0.004897, 0.043591, -0.037690, 0.011464, -0.021639, 0.023351, 0.037156, -0.034408, -0.012892, 0.032214, -0.097177, 0.011449, -0.034716, 0.094636, -0.019634, -0.119839, -0.044336, 0.007877, -0.045127, -0.107540, 0.024371, -0.058006, -0.106227, 0.059667, -0.070435, 0.033384, -0.023156, 0.082028, -0.013083, -0.040312, 0.051476, -0.044643, -0.113340, -0.049217, -0.047714, 0.035748, 0.085111, -0.029751, 0.029401, -0.082440, 0.011105, -0.009313, -0.006817, 0.083748, -0.001016, -0.084277, -0.006396, -0.000810, 0.035396, 0.008354, -0.076020, -0.001676, 0.020525, -0.015391, -0.112915, -0.014149, -0.040210, -0.032362, -0.020844, 0.040075, 0.031626, 0.044984, 0.028352, -0.046888, 0.004452, -0.023608, -0.018866, -0.013798, 0.024092, 0.046575, 0.017726, 0.015747, -0.077894, -0.034731, 0.022678, -0.056115, -0.023464, -0.010496, 0.003848, -0.023920, 0.015848, 0.052789, -0.078399, 0.015387, -0.008394, -0.005700, -0.065740, -0.059081, 0.031461, 0.032923, -0.027296, 0.046724, -0.032575, 0.007734, -0.020048, -0.172351, 0.010138, -0.084825, -0.025280, -0.118754, 0.013225, 0.053437, -0.039431, 0.039239, 0.006202, -0.044809, -0.039000, -0.081792, -0.032601, 0.002057, -0.022403, -0.133223, -0.027856, -0.081603, 0.003332, -0.004519, 0.002807, 0.008377, -0.009728, -0.002136, -0.029852, 0.035767, -0.040559, -0.072192, -0.035695, -0.027323, -0.039057, -0.018370, -0.048523, 0.004072, 0.015038, -0.041708, -0.035022, -0.062653, 0.023944, -0.000212, -0.056158, -0.085126, -0.021141, -0.045148, 0.040353, 0.022472, -0.041244, -0.111200, 0.011917, -0.148337, -0.069752, -0.080007, -0.062339, -0.050051, 0.036866, 0.003275, -0.069658, 0.014113, -0.092149, -0.047455, -0.015256, -0.009895, -0.089492, 0.077432, -0.032232, 0.001988, 0.047199, -0.007264, -0.014140, -0.021369, -0.054363, -0.063442, 0.002014, -0.051393, 0.006114, 0.062051, -0.047344, -0.104170, -0.006418, 0.040309, 0.027030, -0.009470, -0.046766, 0.038598, -0.073236, 0.019922, -0.066268, -0.023395, -0.029782, -0.063573, 0.055810, 0.037236, -0.019139, 0.000375, -0.036968, -0.073857, -0.045481, -0.042620, 0.077140, 0.009398, -0.044851, -0.144988, -0.025140, 0.066183, -0.050182, 0.000611, -0.015414, -0.023518, -0.016765, 0.040608, 0.022904, 0.001495, -0.001958, 0.008503, -0.055031, -0.024997, -0.043245, 0.036271, -0.055545, 0.015603, -0.025374, 0.000409, -0.027946, 0.043080, 0.004176, -0.023916, -0.061224, -0.067155, -0.037969, 0.062768, 0.025193, -0.017722, -0.010243, 0.083648, -0.045740, -0.042555, 0.019860, 0.011816, -0.095993, -0.001194, -0.042816, -0.062511, -0.083585, 0.030494, -0.112202, -0.055572, 0.008304, 0.049472, -0.070281, -0.021382, -0.096269, -0.062613, 0.131288, -0.027313, -0.001809, 0.101175, -0.034362, -0.067462, -0.038516, -0.073872, -0.154226, 0.038528, 0.008484, 0.025315, -0.004330, 0.058504, -0.029916, 0.047979, -0.010517, -0.162494, -0.106080, 0.022996, -0.031142, 0.038922, 0.040370, -0.133545, 0.061993, 0.009146, -0.006345, -0.007382, -0.070292, 0.091932, 0.042725, -0.008035, -0.050764, -0.049932, -0.122443, -0.107706, -0.063473, -0.093530, -0.009404, -0.054486, 0.017564, -0.014340, 0.058009, -0.012627, -0.034878, -0.016052, -0.000669, 0.052025, -0.016280, -0.076500, 0.009367, -0.039787, -0.069960, -0.055281, -0.160876, 0.013913, -0.052580, -0.027444, -0.061548, 0.020973, 0.037170, 0.043509, -0.077703, 0.032302, -0.048715, 0.047516, -0.056506, -0.030944, -0.027371, 0.049867, -0.063838, -0.017442, 0.005691, -0.067678, 0.013761, 0.006442, 0.024770, -0.033043, 0.075301, -0.049710, -0.050109, 0.012690, 0.004781, -0.022711, -0.044234, -0.056567, -0.015187, -0.037776, 0.033367, -0.075551, 0.036674, 0.046511, -0.122823, -0.046306, -0.007777, -0.093292, 0.010944, 0.019965, 0.054589, -0.005570, -0.095338, 0.046280, -0.010990, -0.046712, 0.093664, -0.045492, 0.020380, -0.011494, -0.032488, -0.049765, -0.054021, -0.055248, -0.009132, -0.035368, -0.079229, 0.008531, -0.017188, -0.039119, -0.015197, 0.075167, -0.007901, -0.053317, 0.021964, 0.035212, -0.017886, -0.081064, -0.006999, -0.045281, -0.034766, 0.073319, -0.018423, -0.016170, 0.062359, -0.043937, 0.020849, -0.020891, 0.009609, -0.065792, 0.032202, 0.019978, 0.009879, -0.041703, 0.008527, 0.047058, -0.080408, -0.042463, -0.036594, 0.037394, -0.020509, -0.077625, 0.067821, -0.044072, 0.017189, 0.000422, -0.076039, 0.004549, 0.004237, 0.015749, 0.076771, -0.039470, -0.119366, -0.017240, 0.000246, 0.032576, 0.054300, -0.025264, -0.009654, -0.025455, 0.038722, -0.033038, 0.069717, -0.076018, -0.002755, -0.069812, -0.004670, 0.014477, 0.000531, -0.005202, -0.024729, -0.047925, -0.031172, -0.009135, -0.022473, -0.125930, -0.058722, 0.020890, 0.059093, 0.060583, -0.051521, 0.012996, -0.064571, 0.026132, -0.067197, -0.009287, 0.048478, -0.072111, -0.064567, -0.066776, -0.025159, -0.051411, 0.027879, -0.045441, -0.014981, -0.078826, -0.013770, 0.047205, -0.068941, 0.011590, -0.076156, -0.044230, -0.039726, 0.020238, -0.074823, -0.016635, -0.010422, -0.066660, -0.026197, -0.069033, -0.110824, -0.070120, -0.005610, -0.019247, 0.042543, 0.086599, 0.052887, -0.043218, 0.022044, 0.002490, -0.065035, 0.101828, 0.031362, 0.032202, -0.010405, -0.133671, -0.120123, 0.047668, 0.012099, -0.127661, -0.019195, -0.029407, 0.053011, -0.054604, 0.002551, -0.016921, -0.005848, -0.003431, 0.138640, -0.003385, -0.011825, 0.046231, -0.037657, 0.019935, -0.083319, -0.033456, 0.011470, -0.031115, 0.005272, 0.036697, -0.005059, -0.061186, -0.047189, 0.011101, 0.015583, -0.035456, -0.140333, -0.008836, -0.057931, 0.004889, 0.065241, -0.047841, 0.026778, 0.042473, 0.036426, -0.015338, -0.071397, -0.051039, -0.020717, -0.002150, -0.129065, -0.129448, -0.058374, -0.036938, -0.045205, -0.087379, -0.066117, 0.027149, 0.063883, -0.046867, -0.034152, -0.015424, 0.086786, 0.042850, 0.010521, 0.020198, -0.070930, -0.041483, 0.012224, 0.013448, -0.016234, -0.048393, 0.050259, 0.024805, 0.049461, 0.007769, -0.012961, 0.025290, -0.109055, 0.024743, -0.098722, -0.026997, -0.048064, 0.031479, -0.019830, 0.029072, -0.019133, -0.014887, 0.001878, -0.000756, 0.023799, -0.101285, -0.041515, -0.041866, -0.067039, 0.020354, -0.067727, 0.004238, 0.001436, 0.002797, -0.006615, 0.022491, -0.022527, -0.013292, 0.032057, -0.009120, 0.022242, 0.074111, 0.040845, -0.019882, 0.003285, -0.011741, -0.004921, -0.012184, -0.060518, -0.118199, -0.043224, 0.058507, -0.139899, 0.019444, -0.071405, 0.002765, -0.052288, -0.021010, -0.042788, -0.017747, -0.019861, -0.046357, 0.016356, 0.003795, -0.027774, -0.001947, -0.005181, 0.028886, -0.051880, -0.034029, -0.021951, 0.044099, -0.055701, 0.070382, 0.022519, 0.003321, 0.045679, 0.033911, -0.046606, 0.046725, -0.113415, -0.009097, 0.036223, 0.016335, -0.039982, -0.025837, 0.024758, 0.023354, 0.021276, -0.038603, -0.075497, 0.021081, 0.010929, -0.115918, -0.005420, 0.099489, -0.099998, -0.075256, -0.039743, -0.061194, 0.083427, -0.003039, 0.048513, 0.031232, -0.066172, 0.047320, -0.081337, -0.091499, -0.001968, 0.011513, 0.025586, -0.017877, 0.006569, -0.055032, 0.025483, 0.013697, -0.042344, -0.018434, -0.010141, -0.042248, 0.023309, -0.022974, 0.002150, -0.002020, -0.007817, -0.021911, -0.003044, 0.000887, 0.035035, -0.040583, 0.017581, 0.076841, 0.058389, -0.093678, -0.153958, 0.062441, -0.049019, 0.041227, -0.012665, 0.046532, 0.019038, 0.010332, 0.056174, 0.046360, -0.044230, 0.035357, -0.015656, -0.071647, 0.042556, 0.020719, 0.019176, 0.008250, -0.099090, 0.024202, -0.020372, -0.033028, -0.131270, 0.046089, 0.017707, 0.040441, -0.036144, -0.007797, -0.036856, 0.033028, 0.005649, 0.006689, -0.055042, -0.020957, 0.023519, 0.051837, 0.028136, 0.063409, 0.032037, 0.045398, -0.028596, 0.029569, -0.037512, 0.061836, -0.054877, -0.026209, -0.145266, 0.026342, 0.012949, -0.013952, 0.010727, -0.017554, -0.015744, -0.024217, -0.066681, -0.042274, 0.029351, 0.052112, -0.123662, 0.008355, -0.038305, 0.031585, 0.057984, -0.048177, 0.029451, 0.044615, -0.074861, -0.065953, -0.059954, -0.028243, 0.032123, 0.104599, 0.093510, -0.069832, -0.010253, -0.035440, -0.064069, -0.013424, 0.002332, 0.052693, -0.065822, 0.094336, -0.045237, -0.067690, -0.053109, -0.108961, 0.019389, -0.032731, -0.064207, -0.018052, -0.055133, 0.068978, -0.029411, -0.060004, -0.020334, 0.072607, -0.043534, -0.123715, -0.074277, -0.061699, -0.037438, -0.095781, 0.078490, 0.012677, 0.028710, -0.059583, -0.027486, 0.037059, -0.085328, -0.002353, 0.024797, 0.033123, -0.098999, -0.034767, 0.039195, -0.015057, 0.065867, -0.001686, -0.074078, -0.022560, -0.042350, -0.110340, 0.001352, -0.058847, 0.019307, -0.006328, -0.014128, 0.025896, -0.163388, 0.192832, 0.025668, -0.013436, -0.063300, -0.013107, -0.069878, -0.016902, -0.052697, 0.113324, -0.086924, -0.063292, -0.011001, 0.036086, -0.041677, -0.000496, -0.072249, 0.058396, -0.004583, -0.002519, 0.076320, 0.027528, -0.068518, -0.037088, -0.093958, -0.026053, -0.009046, -0.040090, 0.098331, 0.022888, 0.044312, -0.042477, 0.044763, 0.028226, -0.056542, -0.039364, 0.001735, -0.051662, -0.043109, 0.027196, -0.049445, 0.022521, -0.056396, 0.056553, 0.044376, 0.034357, -0.049245, 0.041510, 0.016534, -0.007997, 0.007773, -0.028950, -0.046216, -0.033673, 0.038904, 0.082586, -0.022804, -0.007275, -0.022482, -0.014147, 0.033353, -0.040001, 0.031305, -0.066727, -0.037537, -0.014474, -0.073698, 0.011103, -0.047258, -0.023773, -0.028397, -0.014032, -0.012494, 0.015975, 0.043747, -0.079863, 0.058407, -0.033096, -0.059403, -0.004161, -0.063210, -0.104376, 0.005195, 0.085593, -0.031401, -0.050872, -0.021314, 0.041538, 0.058240, -0.059903, 0.058241, -0.079949, 0.022940, -0.025531, 0.009160, 0.019934, 0.046824, 0.046269, 0.000880, 0.045445, -0.028669, -0.030150, -0.106136, 0.042087, -0.034796, -0.016244, -0.093346, -0.060762, -0.071330, 0.020010, -0.018640, -0.041399, -0.011950, -0.024512, -0.045131, 0.038445, 0.118791, -0.073771, -0.042393, -0.042132, -0.041464, -0.025142, -0.034278, -0.005884, 0.024018, -0.025459, 0.008796, -0.016107, 0.044352, 0.005358, 0.033318, -0.000399, -0.042979, -0.001970, -0.003846, -0.024686, 0.036115, -0.030555, 0.025155, 0.055749, 0.011633, -0.074708, -0.047420, -0.036274, -0.057452, -0.052729, 0.051960, -0.097395, -0.039581, 0.025571, -0.003206, 0.024929, -0.171228, -0.088447, -0.024646, -0.012894, 0.068895, -0.001647, -0.031515, -0.009149, -0.067265, 0.032709, -0.090146, 0.023536, -0.051125, 0.110532, -0.040613, -0.075220, -0.042160, 0.073118, -0.084303, -0.075666, -0.127469, -0.013663, -0.052377, -0.072806, -0.029683, 0.025108, 0.021131, 0.062327, 0.138894, -0.120982, -0.064838, 0.020070, 0.103695, 0.139339, -0.067359, -0.017018, -0.017513, 0.008638, 0.001473, -0.042207, 0.009172, -0.009687, -0.051376, 0.007679, -0.010320, -0.012395, -0.112341, -0.041556, -0.010876, -0.104019, -0.050610, -0.018428, -0.027393, 0.008550, -0.063310, -0.038584, -0.077375, -0.085973, 0.057322, 0.004048, 0.049586, -0.121008, 0.008701, 0.067916, 0.043023, -0.088396, 0.031375, 0.051640, 0.049305, 0.044867, -0.020071, -0.099537, 0.026829, -0.022646, -0.104366, 0.008148, 0.008196, -0.106864, -0.045462, -0.003278, -0.110772, -0.112227, -0.151930, 0.097242, -0.005727, -0.102846, -0.040612, 0.053099, 0.037236, -0.053897, -0.068331, -0.073703, -0.145741, -0.032773, 0.019550, 0.122452, -0.124464, 0.027432, 0.013845, -0.027263, -0.096951, 0.035276, -0.037216, -0.037163, 0.067138, 0.023182, -0.027790, -0.003021, -0.055218, -0.006956, 0.072790, -0.061727, 0.032968, -0.021753, 0.003166, -0.079563, -0.037546, -0.060777, -0.071586, -0.023314, -0.046338, -0.107567, 0.000629, -0.092008, -0.022348, -0.012368, -0.034081, 0.040003, -0.065768, 0.043465, -0.015835, 0.023423, -0.054560, 0.041346, 0.011197, -0.015327, 0.040419, 0.048232, 0.030638, -0.065567, 0.044350, -0.062994, 0.036866, -0.028484, -0.070517, -0.040843, 0.021071, -0.035620, -0.000897, 0.042830, -0.021109, 0.037901, -0.042225, 0.015679, 0.009357, 0.005258, -0.029049, 0.035893, -0.010880, 0.019958, -0.071174, -0.039288, -0.048213, -0.031940, 0.019047, -0.088500, -0.008926, -0.122472, -0.002113, 0.025309, 0.025607, 0.009378, 0.018029, 0.008822, -0.042433, -0.038629, -0.012807, 0.007343, -0.066429, -0.097591, -0.027741, 0.024296, -0.061438, -0.056139, -0.047776, -0.044413, -0.094646, 0.071954, 0.007962, -0.022136, -0.016835, -0.028737, -0.022635, -0.076857, -0.048206, -0.049709, 0.027153, -0.013668, -0.015393, -0.046215, -0.069785, 0.040964, -0.122893, 0.005542, -0.089151, -0.077610, -0.048063, -0.079546, -0.040596, -0.083990, -0.050104, -0.107481, -0.025201, -0.048309, -0.033868, -0.031684, -0.061168, -0.033596, -0.028770, -0.077269, 0.043456, 0.005738, 0.034503, -0.083509, 0.041718, -0.062766, -0.103698, -0.062862, 0.030875, -0.135646, -0.003406, -0.023542, 0.048550, 0.044988, 0.049394, -0.065483, -0.039697, 0.041310, -0.045573, -0.022867, 0.031027, -0.081575, -0.020326, -0.041824, -0.009284, -0.016881, 0.051144, -0.036944, 0.039281, -0.092808, -0.044677, 0.030535, -0.066032, -0.086590, -0.027034, -0.009320, -0.065656, 0.066958, 0.049136, 0.067567, 0.085979, -0.045583, -0.229290, -0.124068, 0.079930, 0.070263, -0.017580, -0.085764, 0.030802, 0.055117, -0.007528, 0.022843, 0.019079, 0.016634, 0.075158, -0.074596, -0.007750, -0.001284, 0.104946, -0.037672, -0.030779, -0.039973, -0.011126, 0.019626, -0.022414, -0.094425, -0.050832, 0.056777, 0.078069, 0.132094, 0.015876, 0.082918, 0.004966, -0.056043, 0.025517, -0.051278, 0.055479, -0.052110, 0.000053, -0.000537, -0.055070, 0.042235, -0.057773, 0.017939, -0.044762, -0.055964, -0.032567, 0.016390, 0.001178, -0.023000, -0.032244, 0.031023, 0.010923, 0.045825, -0.020846, 0.030612, 0.085319, -0.101774, 0.032578, -0.001727, -0.039466, 0.034975, -0.047934, -0.057746, -0.111382, -0.066664, -0.080754, -0.130690, 0.105803, -0.049347, -0.061592, -0.049404, -0.015184, 0.013899, -0.040102, -0.008651, 0.055079, -0.013837, 0.040923, 0.033509, -0.037381, -0.066896, -0.048015, -0.027881, 0.049732, -0.024995, -0.003890, -0.020295, 0.002626, -0.048729, 0.057504, -0.046448, 0.059625, -0.037794, -0.066417, 0.037412, -0.021169, -0.004776, 0.021448, -0.034702, -0.003092, 0.093204, 0.040088, -0.074117, 0.021455, -0.052716, -0.040899, 0.048900, 0.060403, -0.046981, -0.030514, -0.036696, -0.074441, -0.024631, 0.023147, 0.176966, -0.033196, -0.056938, 0.012422, 0.069724, -0.031922, -0.067209, 0.056084, -0.081378, -0.032881, -0.090511, -0.011776, -0.038641, -0.022759, 0.040266, 0.063629, -0.021365, -0.051735, -0.058382, -0.022748, -0.048764, -0.034683, -0.048693, 0.054939, 0.007461, -0.031582, 0.051094, 0.016396, -0.088803, 0.014761, -0.039679, -0.090088, 0.010197, 0.041628, 0.011117, -0.116552, 0.022098, 0.008464, 0.049936, -0.011642, -0.029778, -0.027192, 0.054238, 0.072113, 0.045254, -0.044887, 0.048881, 0.033540, -0.038694, -0.056881, -0.000596, -0.067383, -0.032561, -0.001108, -0.028658, 0.094255, -0.046265, -0.011402, -0.034289, 0.035583, -0.006021, 0.030980, -0.005508, 0.017192, -0.007032, -0.046480, -0.084276, -0.040995, -0.012671, -0.055870, -0.089146, -0.094832, 0.027116, 0.013616, 0.034652, -0.055821, -0.004956, -0.033551, -0.033702, -0.003788, 0.016716, -0.032589, -0.040445, -0.072095, -0.041005, 0.027534, -0.072948, 0.060328, 0.045536, 0.008560, 0.085472, -0.072527, -0.049427, -0.037456, -0.014780, 0.029020, -0.040294, 0.046820, 0.039937, -0.025084, 0.046060, -0.003701, 0.002624, 0.068795, -0.027280, -0.015721, -0.005620, -0.052731, 0.052465, -0.154305, -0.019372, -0.019120, -0.001969, 0.015895, 0.101921, -0.035672, -0.113256, 0.024840, -0.051732, -0.055125, -0.040144, 0.061213, -0.069645, 0.038705, 0.089511, -0.069889, -0.060311, -0.030414, 0.023168, -0.040953, 0.005794, -0.016703, -0.029827, 0.035697, -0.081405, 0.019197, 0.026611, -0.100765, 0.078216, -0.066439, 0.077838, 0.019708, 0.032841, 0.035436, -0.043151, -0.051982, 0.010046, 0.013756, -0.004941, -0.119092, -0.001752, 0.031119, 0.038495, -0.023131, 0.006286, -0.055865, 0.033497, 0.014763, -0.022046, 0.029627, -0.067740, -0.000936, -0.011347, -0.018687, -0.057257, -0.068492, -0.013424, 0.061228, -0.053490, 0.017953, -0.009878, -0.006939, 0.031983, -0.059465, -0.027694, 0.020848, 0.027424, 0.087411, 0.098024, 0.036127, -0.058619, -0.085361, 0.038841, 0.001832, -0.051774, -0.060333, 0.024824, -0.065282, 0.051685, 0.009359, -0.117060, -0.064195, -0.150995, 0.051965, 0.034668, -0.077797, 0.006280, 0.024217, 0.058707, 0.061881, 0.046021, 0.019279, 0.033716, 0.047494, -0.027922, -0.113769, 0.036917, 0.060991, -0.074086, 0.034922, 0.044055, -0.006390, 0.042760, -0.086266, 0.028408, -0.031969, -0.004098, 0.006357, -0.051741, 0.077704, 0.008409, -0.042018, -0.026081, 0.037646, 0.039340, 0.030077, -0.005436, -0.042995, -0.048997, 0.043023, 0.005095, -0.088974, -0.110043, -0.035884, -0.008659, -0.106673, -0.036241, 0.033921, -0.051299, -0.083834, -0.050497, 0.016577, -0.003215, -0.080755, 0.004312, 0.051467, 0.032213, -0.008543, 0.044961, -0.065758, -0.012262, -0.023578, -0.011704, 0.009170, 0.048612, 0.023130, -0.049710, -0.024376, 0.019887, -0.075257, 0.013660, 0.038216, 0.006710, 0.015709, 0.008392, 0.062782, 0.000353, -0.054373, 0.007343, 0.030232, -0.120620, 0.116461, -0.063239, -0.044911, 0.038661, -0.017392, -0.038438, -0.005991, -0.063857, -0.104400, 0.025720, -0.064393, 0.010795, 0.065489, -0.127029, -0.082618, -0.073687, -0.083666, -0.044307, 0.032785, 0.036808, 0.009004, -0.004364, 0.002471, 0.030759, 0.024742, -0.023396, 0.011978, -0.074545, -0.020689, -0.022458, 0.031800, -0.068431, -0.064180, 0.016716, -0.086530, -0.062117, -0.088038, 0.057041, -0.096846, 0.036861, 0.022288, -0.035145, 0.009654, -0.065223, -0.061876, 0.012538, -0.049788, -0.008303, -0.069092, -0.024426, -0.078919, 0.029561, 0.007320, 0.018531, -0.107128, -0.073642, -0.040877, 0.044967, 0.027613, 0.056162, 0.008457, 0.010727, -0.042704, -0.005658, 0.107260, -0.040596, -0.082709, 0.040426, -0.059241, 0.058849, -0.020916, 0.018764, -0.012913, -0.051495, 0.018156, 0.034705, -0.008842, -0.119308, 0.023996, -0.015237, 0.019936, -0.005047, -0.056238, -0.016471, 0.015337, 0.020605, -0.037855, -0.059870, -0.067478, -0.055414, -0.023800, 0.000808, -0.001976, -0.052183, -0.015590, 0.079565, -0.101230, -0.039006, -0.042363, -0.039579, 0.067336, 0.051482, -0.052978, 0.023845, -0.027449, 0.030686, -0.013527, -0.072807, -0.000603, -0.071871, -0.054286, -0.167743, -0.067157, 0.013735, -0.002120, -0.042441, 0.043732, -0.021143, -0.027156, -0.053603, 0.118024, 0.030111, -0.126339, -0.044956, -0.020727, -0.067985, -0.060469, -0.031662, -0.042546, -0.045123, 0.042195, -0.077723, -0.073106, -0.066593, -0.059879, 0.064368, -0.064487, -0.001750, 0.041714, -0.034135, 0.041723, -0.011277, -0.099482, -0.000063, -0.106237, 0.009507, 0.023472, 0.048831, 0.006014, -0.056197, -0.039923, -0.006945, -0.064854, -0.027343, 0.042986, -0.087348, 0.014776, -0.027352, -0.112253, 0.054133, -0.037912, 0.005835, -0.013531, 0.091213, -0.204999, -0.023649, -0.050792, -0.005226, -0.019027, -0.060693, 0.000039, -0.016429, 0.041440, 0.074455, -0.021536, 0.095456, -0.006717, -0.081780, -0.090518, 0.142514, -0.030191, -0.028527, 0.011774, -0.067726, -0.061469, -0.001576, -0.039649, 0.012902, -0.045369, 0.021703, 0.049526, -0.012415, -0.033104, 0.032952, 0.112698, 0.003209, -0.055416, -0.023488, 0.023825, -0.005242, 0.011477, -0.024757, 0.075627, -0.011699, 0.040703, -0.000503, -0.074199, 0.010510, 0.008295, -0.007797, 0.077776, 0.017685, 0.013269, -0.049132, 0.060975, -0.006278, -0.052629, -0.008897, 0.018628, 0.028074, -0.070525, 0.085260, -0.059553, -0.004958, -0.096076, 0.041903, -0.093757, -0.028138, 0.008024, -0.026384, -0.053068, -0.013183, 0.021514, -0.059130, -0.043750, -0.000961, -0.097660, 0.039069, -0.021057, 0.018117, 0.077390, 0.033596, -0.021643, 0.142455, -0.017279, 0.094556, 0.018160, -0.048738, -0.017130, 0.059751, -0.016263, -0.034869, -0.038624, -0.011360, -0.057647, -0.007547, -0.053193, -0.017620, 0.001406, -0.026918, -0.050874, -0.069143, 0.132875, 0.025506, -0.026278, 0.014199, -0.036959, 0.031629, -0.053090, 0.049878, -0.058160, -0.069886, 0.007366, -0.009846, -0.157658, -0.028483, -0.036380, 0.055287, 0.102240, -0.064560, -0.034866, 0.090519, -0.085332, -0.022351, -0.000587, -0.036590, -0.049025, -0.085612, -0.048984, 0.002421, 0.009634, 0.010337, -0.018588, -0.042774, -0.142224, -0.181876, -0.054649, -0.071971, 0.022762, 0.004791, -0.029963, 0.028511, 0.060606, 0.002309, -0.035403, -0.038493, 0.100178, 0.002715, -0.013494, -0.051310, -0.037679, -0.027551, 0.015688, -0.052541, 0.079595, -0.042212, -0.048688, -0.032634, 0.016370, -0.040493, -0.035029, 0.005305, -0.033754, 0.009837, -0.045568, 0.032858, -0.071505, -0.140798, -0.105588, -0.080966, -0.026197, -0.022818, -0.071449, 0.043895, 0.036672, 0.090493, -0.026050, -0.115527, -0.069274, -0.127375, -0.049623, 0.036190, -0.007825, 0.158495, 0.023708, 0.011589, -0.017289, -0.056613, 0.012674, -0.013857, -0.066561, -0.036276, 0.023556, 0.129628, -0.000491, 0.009502, 0.010519, 0.037292, -0.063589, -0.129516, 0.007687, -0.058675, 0.016037, -0.097243, 0.043774, 0.017796, -0.092926, -0.011867, -0.030658, 0.040190, 0.085423, -0.088691, 0.057948, -0.088498, -0.022555, 0.002251, -0.059260, 0.028891, -0.010093, 0.053653, 0.012976, -0.040116, 0.070693, 0.006894, 0.068566, 0.038604, -0.041655, 0.156053, -0.006500, -0.084213, -0.037503, 0.054667, -0.000381, -0.020471, -0.011615, -0.070358, -0.063376, 0.125349, -0.024937, -0.016838, -0.063636, -0.043298, -0.021745, 0.019379, -0.077985, 0.020175, 0.011822, 0.003057, 0.066507, -0.088797, 0.042269, 0.041566, 0.040959, 0.097579, 0.047691, 0.002482, 0.024312, 0.028691, -0.107965, 0.031161, 0.034310, -0.004446, -0.036494, -0.005605, 0.146353, 0.009610, -0.093558, 0.066819, 0.078519, 0.014385, -0.066714, -0.063461, 0.020675, -0.010327, -0.015558, -0.084724, -0.060586, -0.064241, 0.062113, 0.045362, -0.016264, -0.045804, 0.015858, -0.009934, -0.062128, -0.002321, 0.002225, -0.006226, -0.048119, 0.010361, -0.097793, -0.017826, 0.067352, -0.083557, -0.040387, -0.127470, -0.039919, 0.005938, -0.003174, -0.014396, 0.013637, 0.095543, -0.035904, -0.020939, -0.029603, -0.032542, -0.154950, 0.015618, -0.015183, -0.021064, -0.064460, -0.038085, 0.011362, 0.067363, 0.004419, 0.009319, 0.005125, -0.050015, -0.089283, -0.028274, 0.043880, -0.000294, 0.123525, -0.053126, -0.065656, -0.063288, 0.029100, -0.008350, 0.031882, -0.008634, 0.067787, -0.155705, 0.002204, -0.104478, 0.022370, -0.084174, -0.150837, 0.021483, -0.033315, -0.014711, -0.016094, -0.016315, 0.090808, -0.059340, -0.041634, -0.005862, -0.001533, 0.024795, 0.032064, 0.024064, 0.033472, -0.029541, -0.100590, 0.066671, 0.014774, -0.057327, -0.045584, 0.014355, 0.009200, -0.045567, 0.003571, -0.033101, -0.029024, -0.036424, 0.010223, 0.068139, -0.021033, 0.031640, 0.001338, 0.032805, -0.017731, 0.020886, 0.021576, 0.067573, 0.047145, 0.025895, 0.046432, -0.209555, 0.036599, -0.022476, -0.007688, -0.035388, -0.001947, 0.033255, 0.096807, -0.077313, 0.065433, -0.131832, 0.110427, 0.037752, -0.077792, 0.095357, -0.046983, -0.002232, 0.000930, 0.043387, 0.122679, -0.028961, -0.133293, 0.068174, 0.034614, 0.054402, -0.041913, 0.063396, 0.004832, 0.009924, 0.061763, -0.029789, -0.039413, 0.039571, -0.055641, 0.065913, 0.065121, -0.013509, 0.032886, -0.020789, 0.017179, 0.056206, 0.008112, -0.074890, 0.096865, -0.017131, 0.034349, 0.034650, 0.038078, 0.019046, -0.001754, -0.024891, -0.095220, -0.056697, -0.036159, -0.024492, -0.154778, 0.002469, -0.039471, -0.032765, -0.012006, 0.023843, 0.035048, 0.016755, -0.114292, 0.020874, 0.037841, -0.036154, 0.000483, -0.062928, 0.015340, 0.043927, 0.019252, 0.044725, -0.004346, 0.047448, -0.070848, -0.028977, 0.037026, -0.017320, 0.023300, 0.076107, 0.151296, 0.005399, -0.032519, -0.063627, -0.034193, 0.037095, 0.043209, -0.008567, 0.085350, 0.023326, 0.032047, -0.018884, -0.037455, -0.073386, -0.051927, -0.048764, -0.014958, 0.061009, -0.049905, -0.059631, 0.094264, -0.024998, 0.025565, -0.076632, -0.014335, -0.041653, 0.023891, 0.069906, -0.048947, 0.043835, -0.033690, -0.080331, -0.035288, 0.079492, 0.057444, 0.034017, 0.016017, -0.001210, -0.078969, -0.021929, -0.098894, 0.024093, -0.056953, -0.039522, -0.007367, -0.079613, -0.005738, -0.077350, 0.028016, -0.051408, 0.016164, 0.109629, 0.002016, -0.091326, 0.019269, -0.054506, -0.025494, 0.022092, 0.062103, -0.016916, -0.046291, 0.018415, -0.001313, -0.032828, 0.000206, 0.016313, 0.027620, 0.012985, -0.072752, -0.063925, 0.077826, -0.079489, -0.000610, -0.018070, -0.044715, 0.062484, -0.010569, -0.017455, 0.026143, -0.114541, 0.066731, -0.039228, 0.039947, -0.022898, 0.021941, -0.030749, 0.027312, -0.024310, -0.047560, 0.038325, 0.003226, -0.028716, -0.057875, -0.015032, -0.014156, 0.017590, 0.010934, -0.041948, 0.035895, 0.054410, 0.000378, -0.071393, 0.005814, 0.009646, -0.024128, 0.093332, 0.031359, 0.087052, -0.050222, 0.000481, 0.025301, -0.121128, -0.027932, 0.033009, 0.026903, 0.068239, -0.077250, -0.034117, 0.008372, 0.026506, -0.007330, 0.065652, 0.026878, 0.067505, -0.046003, 0.170490, 0.046561, -0.088251, -0.074997, -0.014873, -0.129864, 0.031806, -0.061436, -0.074410, 0.030404, -0.028861, 0.032778, 0.074584, -0.054560, 0.081135, 0.042221, -0.050714, -0.021572, 0.032132, -0.101717, 0.112758, 0.002334, -0.049017, -0.013085, -0.094862, -0.011987, -0.029553, -0.013430, -0.036718, 0.037850, -0.047485, 0.025251, -0.026989, 0.003679, -0.036458, -0.020138, 0.001215, -0.038184, 0.091526, -0.002954, -0.036374, -0.086368, -0.046023, -0.032847, 0.072635, -0.143197, -0.064487, 0.063586, 0.038598, 0.034423, -0.004005, 0.029873, -0.020665, 0.012455, 0.037254, 0.104744, -0.000570, -0.080314, 0.045063, -0.058579, 0.037386, -0.004742, 0.008790, 0.007414, -0.028271, -0.022552, 0.018289, -0.085129, 0.063413, 0.070192, -0.101203, -0.070382, -0.035853, -0.032232, 0.039070, -0.028081, 0.003010, 0.026824, 0.006932, 0.012560, 0.001225, -0.016773, -0.076079, 0.027457, 0.038128, -0.036285, -0.001810, 0.027837, 0.009068, -0.042594, -0.022318, -0.002289, -0.053543, -0.108230, -0.037462, -0.021024, -0.085323, 0.030807, 0.034451, -0.015330, -0.075823, 0.024272, 0.014222, 0.051870, -0.051343, -0.065246, -0.017190, 0.031003, -0.085181, -0.076169, -0.004252, -0.051017, 0.062914, -0.042420, 0.039399, -0.066836, -0.079397, 0.022905, -0.033433, -0.080222, -0.021596, -0.031809, -0.067939, -0.050113, 0.008236, 0.034875, -0.098072, -0.061049, -0.048656, 0.063095, -0.047401, 0.011835, -0.032611, -0.005896, -0.012645, 0.042875, -0.105973, -0.017655, -0.000916, -0.004888, -0.042186, -0.025956, 0.014065, -0.086842, -0.017440, -0.000055, -0.155951, -0.035752, -0.036880, 0.050994, -0.043871, 0.055321, -0.032745, -0.001372, 0.028243, -0.044164, -0.051634, -0.008144, 0.036286, 0.033541, 0.019852, 0.053034, 0.037714, 0.124941, 0.114872, -0.004892, 0.024726, 0.050198, 0.015469, -0.075923, -0.048102, 0.155410, -0.063008, -0.059773, -0.015256, 0.089337, -0.012213, 0.011957, -0.101568, -0.030382, -0.014791, 0.044118, -0.030150, -0.052971, -0.031683, -0.001292, 0.124033, 0.042170, 0.090466, -0.016725, 0.022098, -0.091862, 0.005021, -0.033900, -0.032538, -0.021564, -0.013888, -0.055247, -0.048851, -0.052697, 0.017257, 0.038260, 0.032029, -0.007986, 0.000845, -0.030681, 0.083572, -0.023925, 0.053311, -0.030810, -0.013990, -0.032890, -0.010998, -0.064721, -0.006798, -0.104083, -0.018695, 0.006691, 0.024084, -0.112678, -0.045829, 0.037688, 0.077837, 0.006662, 0.000296, -0.023105, 0.069850, 0.030623, -0.034299, -0.084156, 0.003652, -0.064138, -0.004653, 0.062817, 0.111228, -0.060744, -0.064470, 0.052799, -0.003484, 0.005851, -0.030034, -0.073044, -0.049427, -0.059435, 0.029370, -0.007126, 0.013758, 0.047417, -0.054949, 0.005867, 0.071272, -0.059530, 0.056904, 0.025524, -0.000498, -0.071003, -0.019402, 0.061386, -0.038090, 0.050852, -0.021222, 0.006647, 0.017040, 0.046077, -0.020055, 0.079650, -0.005491, 0.034969, -0.080828, 0.015840, -0.045994, 0.017730, -0.061678, 0.006895, 0.018794, -0.038666, 0.002269, -0.049445, 0.047412, 0.076111, -0.014081, 0.101318, -0.106390, 0.023922, 0.042984, 0.005418, 0.007172, -0.016597, -0.008582, -0.107484, -0.018212, -0.038472, -0.023499, 0.026829, -0.013490, -0.077745, 0.039635, -0.055933, -0.086419, 0.049176, 0.087259, -0.031736, -0.073135, -0.044648, -0.022140, 0.076069, 0.056182, 0.019697, 0.048334, 0.008352, -0.097496, -0.019568, 0.007072, -0.026626, 0.014308, -0.053203, -0.003424, -0.005301, -0.004314, 0.016442, 0.020645, -0.035609, -0.003170, 0.000619, -0.036503, 0.046011, 0.018094, -0.016693, -0.045310, -0.031738, -0.055129, -0.048617, -0.052610, -0.097879, -0.008075, -0.069178, 0.005766, 0.010946, -0.021910, -0.102329, -0.061304, 0.097342, -0.030070, 0.050712, -0.018843, -0.028831, -0.023692, 0.049985, -0.037912, 0.003591, -0.000489, 0.058163, 0.006361, 0.013943, -0.063619, -0.076353, -0.039889, -0.000972, 0.022905, -0.070101, 0.085613, 0.056779, -0.082215, -0.046143, -0.045784, -0.025014, -0.017495, -0.083411, 0.040854, 0.041826, -0.016134, 0.021404, 0.023673, 0.074247, 0.011931, 0.000709, -0.001763, 0.060258, -0.015381, -0.069956, -0.092428, 0.041387, 0.016500, 0.044519, 0.049431, -0.041097, -0.030259, 0.028608, -0.017679, 0.027154, 0.002487, 0.014718, 0.084091, -0.012862, 0.021318, -0.058867, 0.005023, -0.038073, -0.031844, -0.028035, -0.010683, 0.108599, -0.117483, 0.072873, -0.011616, 0.009302, 0.035218, 0.097065, -0.067573, 0.006031, -0.021618, -0.032602, 0.034203, 0.002167, -0.022487, -0.078285, -0.049017, -0.080390, 0.042469, -0.019658, -0.045523, -0.014984, -0.015731, -0.058798, 0.001709, -0.100876, -0.033505, 0.034521, 0.053098, -0.039814, -0.018031, -0.078940, -0.103305, -0.034899, -0.044597, -0.029232, 0.133894, -0.012636, 0.029092, -0.151592, -0.029184, -0.004476, -0.041358, -0.062846, 0.013861, 0.046889, -0.084098, 0.061942, 0.053747, -0.062185, -0.098797, -0.131223, -0.083017, 0.015333, 0.135684, 0.047261, -0.034241, -0.017120, 0.111672, 0.055569, -0.049865, -0.013734, -0.019573, -0.006885, -0.148214, 0.033337, -0.046682, 0.078899, -0.049790, 0.016716, -0.047301, 0.028596, 0.007398, -0.017505, 0.011141, -0.001427, -0.064909, 0.042306, -0.013600, -0.044718, -0.026481, 0.023074, 0.088469, -0.115640, -0.066954, -0.070109, -0.042408, -0.158574, -0.046921, -0.028676, 0.066646, 0.041308, 0.003877, -0.120903, 0.123798, 0.050875, -0.217459, -0.022015, -0.018869, -0.026155, -0.014336, 0.082059, -0.007520, -0.043004, -0.068226, -0.096192, -0.025971, 0.023480, -0.048194, -0.063375, -0.049661, -0.055670, -0.025793, -0.003934, -0.086465, -0.033404, 0.047837, -0.083905, 0.035683, -0.004389, -0.028646, -0.072245, 0.027095, -0.048735, 0.055439, -0.013392, 0.056749, -0.123558, 0.085601, -0.035453, -0.057173, -0.122062, -0.006389, -0.035315, -0.055198, -0.054262, 0.058721, 0.046971, 0.045440, -0.107074, -0.007048, -0.057307, -0.037155, -0.011214, -0.031449, -0.007689, -0.047315, -0.132294, -0.075669, -0.052651, -0.029610, -0.067837, -0.087064, -0.017964, 0.008547, 0.024367, -0.008436, -0.069425, -0.052415, -0.082107, -0.040748, 0.035011, 0.008106, 0.049344, 0.045713, -0.028202, 0.048702, -0.104415, -0.150976, -0.090633, -0.011918, -0.052742, -0.041192, -0.046008, -0.003379, -0.065085, -0.057090, -0.069767, -0.053342, -0.064930, 0.018116, -0.089617, 0.080788, 0.088798, -0.034366, -0.074459, -0.080228, -0.000492, 0.084700, 0.050382, -0.041771, 0.018039, 0.070359, -0.019373, -0.098740, 0.074693, 0.054253, 0.062674, -0.060445, -0.057041, -0.088022, -0.054486, -0.108169, 0.057558, -0.143840, -0.162692, -0.008403, 0.057462, -0.004132, -0.028094, -0.051121, -0.006347, -0.077347, -0.075147, -0.108376, -0.125892, -0.029506, 0.017034, -0.026338, 0.009601, 0.027580, -0.039270, 0.052380, -0.126161, -0.012823, -0.050849, -0.020930, 0.070707, -0.046029, 0.038068, 0.007302, -0.020540, 0.070570, 0.018746, -0.076563, -0.144475, -0.176102, -0.046856, -0.067970, 0.028482, -0.119327, -0.065327, 0.098142, 0.024513, 0.079842, 0.086844, -0.023546, -0.056932, -0.023375, -0.048084, 0.133165, -0.064764, -0.044693, -0.059321, 0.062301, -0.049496, -0.047672, 0.004523, 0.000132, -0.056149, -0.097546, -0.008586, -0.039161, -0.092477, -0.059179, -0.027346, -0.010625, -0.083574, 0.062873, -0.037015, -0.004327, 0.075837, -0.022859, -0.022016, -0.028161, 0.027925, 0.059476, -0.040884, 0.031258, -0.056698, -0.150187, 0.001017, 0.136668, -0.086830, 0.108457, -0.063457, -0.065773, -0.100546, -0.017021, -0.027697, -0.000813, 0.009036, -0.038948, 0.019231, 0.019286, -0.040571, -0.067747, 0.007576, -0.040302, -0.027131, -0.025360, 0.051802, -0.081006, 0.021894, -0.023934, 0.037162, -0.055326, -0.035684, 0.086074, 0.085356, -0.001397, -0.078689, -0.074573, -0.015340, -0.040520, -0.092792, -0.002715, 0.014643, 0.069526, 0.036579, 0.049099, 0.100172, 0.021354, 0.005000, -0.026914, 0.030201, -0.044301, 0.019214, 0.031414, -0.064540, 0.005696, 0.070642, 0.041989, 0.023557, -0.038659, -0.017589, -0.108614, 0.007245, 0.104487, -0.175365, -0.070013, -0.007174, -0.036894, -0.046970, -0.031572, -0.011417, 0.021518, -0.068094, -0.091718, -0.056247, 0.015730, 0.035940, -0.072664, -0.010288, 0.018177, -0.093354, -0.092284, 0.049010, 0.044757, 0.008424, -0.019421, 0.006030, 0.058304, 0.037037, 0.010019, 0.081305, 0.058782, -0.058920, 0.013610, -0.012590, -0.058860, 0.071856, -0.079813, -0.128519, -0.076262, -0.016520, 0.026186, -0.019942, -0.048933, -0.087729, 0.064500, 0.021646, 0.028213, 0.026739, -0.040566, -0.011157, -0.012559, -0.120249, -0.090363, -0.073710, -0.071888, -0.027297, -0.070551, -0.047310, -0.007614, -0.097727, -0.010595, 0.030670, -0.055400, -0.067904, 0.084991, 0.023427, 0.099458, -0.070957, 0.054017, -0.050015, 0.082672, -0.008542, 0.002862, 0.049540, -0.057076, 0.005805, -0.134410, -0.030852, 0.066070, -0.043778, -0.063977, 0.018640, -0.064518, -0.010596, 0.012459, -0.061001, 0.048777, 0.027616, 0.038086, 0.033014, -0.020564, 0.077312, -0.018954, -0.042268, -0.074056, -0.062644, -0.076675, 0.114934, 0.040967, -0.087062, 0.011672, -0.010892, -0.024957, 0.057605, 0.117472, -0.121947, 0.014093, -0.116852, 0.032262, -0.069304, -0.029443, -0.041959, -0.055085, -0.029541, 0.033530, 0.044631, -0.077307, -0.017146, 0.026930, -0.015190, -0.078530, -0.008944, -0.054336, -0.032840, -0.061478, 0.049738, -0.016694, 0.083866, 0.057000, -0.039278, 0.003315, -0.036143, 0.041428, -0.121896, -0.093463, 0.072074, -0.280217, -0.143749, -0.047985, -0.002008, 0.018309, -0.019932, 0.049348, -0.081267, -0.062204, -0.112765, 0.028174, 0.053282, -0.051903, 0.031670, -0.006076, -0.083613, 0.064433, -0.008384, -0.087282, -0.076148, -0.102670, -0.083986, 0.057714, 0.001851, -0.060371, -0.042624, -0.002706, -0.049672, -0.032355, -0.054818, -0.077473, -0.023521, 0.025421, -0.104716, -0.031220, -0.102445, -0.046632, -0.009524, 0.018640, 0.049270, -0.021263, -0.002758, -0.014776, 0.059188, 0.084717, -0.118561, -0.018995, -0.002185, -0.046022, -0.021541, 0.141437, 0.099156, 0.037916, 0.018545, -0.069490, -0.110690, 0.017269, -0.048039, 0.202502, -0.020233, -0.012142, 0.091896, 0.001864, -0.015482, -0.016619, -0.042615, -0.043276, 0.057048, -0.088781, 0.018057, -0.035423, 0.049693, -0.001520, -0.016540, -0.039916, -0.070942, 0.003513, -0.057064, -0.005856, -0.041274, 0.032996, 0.003490, 0.045627, -0.076311, 0.154793, -0.157413, -0.023082, 0.038955, -0.060066, -0.011154, 0.003028, -0.104969, -0.085799, 0.005191, -0.049510, -0.007209, -0.003413, 0.007301, 0.001823, 0.016819, -0.015522, 0.087254, 0.005139, -0.008683, 0.046762, -0.066043, -0.015623, -0.002244, -0.071978, 0.095384, -0.105927, 0.021162, -0.053605, -0.035245, -0.088274, -0.132977, -0.027726, 0.036926, -0.061161, -0.021382, -0.202414, 0.068851, 0.013621, 0.006776, 0.015291, -0.016077, -0.058521, -0.076851, 0.077793, -0.120008, 0.053497, 0.049417, -0.107979, 0.000253, -0.011797, 0.086855, 0.017123, -0.019732, 0.092609, 0.018238, 0.031850, 0.007127, -0.063291, -0.094090, -0.105766, 0.034167, -0.068179, -0.106280, 0.067137, -0.090692, 0.007896, 0.012554, 0.056578, 0.115456, 0.061175, 0.036391, -0.007754, -0.014132, -0.059890, 0.015570, -0.031085, -0.064209, 0.065398, -0.036461, -0.056803, -0.030819, 0.193316, -0.053846, 0.021637, 0.021440, -0.070456, -0.041394, 0.086201, 0.034382, -0.046981, -0.035497, 0.020421, -0.021970, 0.016791, -0.015441, 0.003761, -0.061364, 0.052977, -0.016391, 0.093764, -0.013042, 0.056031, -0.060472, -0.054867, 0.016514, 0.023958, -0.027626, -0.032051, -0.004074, -0.024585, -0.043632, 0.092173, -0.068721, 0.066136, -0.039692, -0.083041, 0.059148, -0.106744, 0.029581, 0.023480, 0.057192, -0.080861, 0.068695, 0.062997, -0.031769, -0.048937, -0.036499, -0.150987, 0.061741, 0.107421, -0.009444, -0.068718, -0.035894, 0.050120, 0.053291, -0.046336, -0.110890, 0.026522, -0.016116, -0.033966, -0.069585, 0.029660, -0.103163, 0.103407, -0.065053, -0.029744, 0.085497, -0.132023, -0.104359, -0.096271, -0.025592, 0.047592, -0.038834, 0.029230, 0.055593, -0.030348, 0.045609, -0.119996, -0.028108, -0.024542, -0.034025, -0.051085, -0.112874, -0.107302, -0.033335, 0.016478, -0.000365, -0.015739, 0.016688, -0.052913, -0.094431, -0.023738, -0.085997, -0.072499, 0.000530, -0.137117, 0.012492, 0.068661, 0.032516, -0.068169, -0.106315, 0.015778, -0.041668, -0.019370, -0.023218, -0.041545, -0.034620, 0.006285, -0.010925, 0.046294, 0.011660, -0.034470, -0.048632, 0.019702, -0.078024, -0.114860, 0.035626, -0.012405, 0.009505, -0.031297, 0.012887, 0.080765, -0.074571, -0.017985, 0.062690, -0.071508, 0.052333, -0.103916, 0.058723, 0.000945, -0.095234, -0.026219, 0.075222, -0.065007, -0.113719, -0.076084, -0.040731, -0.035745, -0.100557, -0.000002, 0.069509, -0.049926, 0.030727, -0.018654, -0.127183, -0.044283, -0.000763, 0.039170, 0.071283, -0.040583, -0.092491, 0.036822, -0.088486, -0.068743, 0.036729, -0.012203, 0.020791, -0.004571, -0.001387, -0.079424, 0.026909, -0.056479, -0.085134, 0.017377, -0.029308, 0.034402, 0.036091, 0.004161, -0.043228, 0.043494, 0.046793, 0.058028, -0.050301, -0.019181, -0.028843, 0.059360, -0.028660, 0.014552, 0.137236, 0.055489, 0.053664, -0.048534, 0.022298, 0.178958, -0.026439, -0.037727, 0.060664, -0.074378, -0.049959, -0.003859, 0.023186, 0.122921, -0.073288, -0.123547, -0.103587, -0.036373, -0.093351, -0.025236, -0.021887, -0.067561, 0.018822, -0.039608, -0.044712, -0.053224, -0.129154, -0.058235, 0.014062, 0.056285, -0.006555, -0.004478, -0.020428, -0.083705, -0.075683, -0.030411, -0.112418, -0.031394, -0.069939, -0.057505, 0.116847, 0.002162, -0.014190, 0.069736, -0.054846, 0.015090, -0.053022, -0.017589, 0.013674, -0.106615, 0.045061, 0.130302, -0.053902, -0.048016, -0.009706, -0.162570, -0.076203, -0.000264, -0.038050, -0.004787, -0.003981, -0.096810, -0.055437, -0.096225, -0.019097, 0.048075, -0.032767, -0.054347, -0.064914, -0.055916, -0.062910, -0.011660, -0.062034, -0.069782, 0.079910, -0.069429, -0.049384, 0.045712, -0.040575, 0.063662, -0.012750, -0.070162, 0.056705, -0.041954, 0.004584, 0.024743, -0.088536, -0.054849, 0.062841, -0.071086, 0.112736, -0.042112, -0.043644, -0.053272, -0.074660, 0.119870, 0.075558, -0.095542, -0.157381, 0.039271, -0.030812, -0.047885, 0.074764, -0.082723, 0.026266, -0.092000, -0.024693, -0.082236, -0.044068, 0.105856, -0.044956, -0.028588, -0.066166, -0.115710, 0.069617, -0.059016, -0.041189, -0.041237, -0.011456, -0.005798, -0.056468, -0.037354, -0.015929, -0.066507, -0.056039, 0.018279, -0.009747, 0.001364, -0.035915, -0.053171, -0.008271, -0.038963, -0.023284, -0.068790, -0.077084, -0.135797, 0.007272, -0.194454, -0.076763, -0.102728, 0.058485, -0.052796, -0.048824, -0.109146, -0.036720, -0.007733, 0.058789, -0.000795, 0.013861, 0.009221, -0.001102, -0.034340, 0.052794, -0.070271, 0.056053, -0.073524, 0.027639, -0.054476, -0.024389, -0.053693, -0.040717, 0.067798, -0.021743, 0.092339, 0.010913, -0.003964, 0.001002, -0.057197, -0.097406, -0.133495, -0.003988, -0.045972, 0.004357, -0.031894, 0.065049, 0.033523, 0.039193, -0.058307, -0.051404, -0.054160, -0.074589, 0.038936, -0.004217, -0.012473, -0.029535, 0.008603, 0.010478, -0.100637, -0.047450, -0.025499, -0.061713, -0.001573, 0.088159, -0.031051, 0.095415, 0.053084, -0.038557, 0.001901, 0.106452, -0.031437, 0.014506, -0.059168, -0.058854, 0.046887, 0.043157, 0.045941, -0.178887, -0.057722, -0.106667, -0.066055, 0.040472, 0.042280, -0.001867, 0.033179, 0.013786, 0.045297, -0.035983, 0.007158, 0.010662, -0.047356, -0.136414, -0.012722, 0.011673, 0.054320, -0.008167, -0.078189, -0.068891, -0.000206, -0.010573, 0.004152, 0.048415, -0.019882, -0.110514, -0.068754, -0.009760, 0.001561, -0.019085, 0.012759, -0.044169, -0.043529, 0.030396, -0.006577, -0.077981, -0.118326, -0.006311, 0.032924, -0.035545, 0.058625, -0.084139, -0.066821, 0.034292, 0.013024, 0.087731, -0.094311, 0.051306, -0.067598, 0.057876, 0.033668, 0.102865, -0.009015, -0.013884, -0.106518, -0.006716, 0.008462, 0.000889, -0.019823, 0.009698, 0.094596, 0.129152, -0.002406, -0.093451, -0.016263, 0.045747, -0.041331, -0.061565, 0.035036, 0.056928, -0.042173, 0.066374, -0.033133, -0.009482, -0.021591, 0.005819, 0.021094, 0.023822, 0.076032, 0.013510, -0.024282, -0.012323, -0.006946, -0.005720, -0.019768, -0.081689, -0.022657, -0.029773, -0.032368, -0.041306, 0.066679, -0.036759, 0.047425, 0.059315, -0.027582, 0.045183, 0.016123, 0.082965, 0.042627, -0.045372, -0.034468, -0.076316, -0.149202, 0.011692, -0.008478, -0.014160, -0.087511, -0.035516, 0.033654, -0.081916, 0.025425, 0.063687, 0.071894, -0.071037, 0.126299, -0.158309, -0.003735, -0.002222, 0.030096, -0.053773, 0.050695, 0.052990, -0.041452, -0.066676, -0.100755, -0.015584, 0.037744, 0.059251, -0.050422, -0.163339, -0.111930, -0.039237, 0.056307, -0.046441, 0.141963, 0.033410, 0.044199, -0.025196, 0.085899, -0.037489, 0.088512, 0.026789, -0.058273, 0.016751, -0.041082, -0.033223, -0.046180, -0.010658, -0.089043, 0.039984, -0.054253, -0.025415, 0.117376, 0.032023, -0.099565, -0.020886, 0.159658, 0.008985, 0.027181, 0.059624, -0.039878, -0.111568, -0.112558, -0.000298, -0.031704, 0.026288, -0.084797, 0.027207, -0.040521, -0.000150, -0.019884, 0.052453, -0.022429, -0.103091, -0.082051, -0.058164, -0.075032, 0.019466, -0.101283, -0.073455, -0.155200, -0.068919, -0.021444, -0.028599, 0.030526, -0.114188, -0.032295, -0.063960, 0.044310, 0.032232, -0.099469, -0.094245, -0.095909, -0.108428, -0.051837, -0.001651, 0.012695, -0.086967, 0.028357, 0.045256, -0.006083, -0.019495, -0.061120, -0.039051, 0.015836, -0.124032, -0.046383, 0.102462, 0.025452, -0.000219, -0.106657, -0.071031, -0.086778, 0.093410, -0.099216, -0.158896, -0.037623, -0.031353, 0.065593, -0.010106, -0.018266, -0.108767, -0.020182, 0.160374, 0.006675, 0.028884, -0.049257, 0.001519, -0.005436, 0.073564, 0.025708, -0.012462, -0.029482, 0.032518, 0.074280, 0.003708, -0.013673, 0.085750, 0.019098, -0.058735, 0.012716, -0.097667, 0.037916, -0.053714, -0.064583, -0.020192, -0.027637, -0.064473, 0.090568, 0.044044, -0.035786, -0.034175, 0.091193, -0.079641, -0.025140, -0.016101, -0.021428, -0.019533, 0.034222, -0.075410, 0.065853, 0.075993, 0.099698, -0.048941, -0.073748, 0.102773, -0.025616, 0.185710, 0.019036, -0.121236, -0.006364, -0.022364, 0.014346, 0.007512, 0.006453, -0.065594, -0.043405, 0.052950, -0.050775, 0.027118, -0.070296, 0.035435, 0.032346, -0.006944, -0.006120, 0.018231, 0.051986, 0.019102, -0.040805, -0.050693, -0.082149, -0.165932, 0.056067, 0.034987, -0.176687, 0.059525, 0.031478, -0.018066, -0.044975, 0.099865, -0.086441, 0.113572, 0.052396, -0.020424, 0.045361, -0.045815, -0.055708, -0.085031, 0.032311, -0.045353, -0.062423, -0.051666, 0.015250, -0.078048, -0.032298, -0.051970, -0.021814, 0.090768, 0.091786, -0.054109, -0.007345, -0.042107, -0.084689, -0.058429, -0.047077, -0.004602, 0.025449, -0.089229, -0.069852, 0.010015, -0.081307, 0.028919, 0.128943, 0.065361, 0.098549, -0.066508, -0.125937, -0.021331, -0.005079, 0.041424, 0.020388, -0.100299, 0.006515, 0.115411, -0.014009, 0.038778, 0.014931, -0.008787, 0.120242, -0.000775, -0.022351, -0.098059, -0.013978, -0.078514, 0.027912, 0.053593, 0.017356, -0.055516, -0.109703, 0.016957, -0.120420, -0.059515, 0.026749, -0.021258, 0.048913, 0.049727, 0.015515, -0.046882, -0.086423, 0.000210, -0.037193, 0.007604, -0.079875, -0.092592, -0.003765, 0.001008, -0.047388, -0.042492, 0.006888, -0.069805, 0.031378, -0.026215, -0.050295, 0.026719, -0.086192, -0.006514, -0.028022, 0.060528, -0.087630, 0.081450, 0.018784, 0.048277, -0.091988, -0.013209, -0.036007, 0.007554, -0.034322, 0.001271, -0.076113, 0.084329, -0.013196, -0.021154, 0.034732, -0.021636, 0.117828, -0.061827, 0.037120, -0.070302, -0.094423, 0.072000, 0.004541, -0.015430, 0.024862, -0.033012, 0.044780, -0.127173, -0.015914, 0.000917, -0.040651, 0.047057, 0.010685, 0.075301, 0.034654, -0.005279, -0.146012, -0.028623, -0.014251, -0.131273, 0.012155, -0.130698, -0.098485, 0.022125, 0.018303, 0.054079, -0.016295, -0.057129, -0.098506, 0.058922, -0.009737, -0.053907, 0.019242, -0.014403, 0.012845, 0.082389, -0.020905, 0.060181, -0.067429, -0.016274, -0.005211, -0.068791, -0.030547, -0.066791, -0.022250, 0.071649, 0.056979, 0.051963, -0.059718, -0.016826, -0.056146, -0.060662, -0.111224, 0.044685, 0.116049, -0.024433, 0.023150, -0.026736, -0.090089, -0.036101, -0.100805, -0.055125, -0.050845, -0.039650, -0.072887, 0.053072, 0.049707, 0.043837, 0.031745, 0.002323, 0.058283, 0.044945, 0.077325, -0.008491, -0.085013, -0.094712, 0.106086, -0.033310, -0.012160, -0.095633, -0.045823, 0.080269, -0.004236, -0.039592, -0.027073, -0.000728, 0.012001, 0.115802, -0.033068, 0.047485, -0.082155, -0.063274, -0.086641, 0.016259, 0.044791, -0.042218, 0.082660, -0.034897, 0.022392, -0.002167, -0.046400, -0.015693, 0.001415, 0.001815, -0.000723, 0.066737, 0.035849, 0.027214, -0.049522, -0.089041, -0.020331, -0.065166, -0.109649, -0.002884, 0.011786, -0.103440, 0.074262, 0.015686, -0.033772, -0.042647, 0.011269, -0.082039, -0.010576, -0.064123, 0.015425, -0.117324, -0.029981, -0.040061, 0.052002, 0.023706, 0.010918, -0.155116, -0.021026, -0.017878, -0.022845, 0.030883, -0.111891, -0.063820, 0.023043, -0.014159, 0.012801, 0.052785, -0.047880, -0.035945, 0.008604, -0.075787, -0.086887, -0.062974, -0.128098, -0.009958, -0.088498, -0.064650, -0.000303, 0.020934, -0.034499, -0.080193, 0.020563, -0.016590, -0.011609, -0.010031, 0.045033, -0.057388, -0.049598, 0.072863, -0.063096, -0.009355, -0.086730, -0.071283, 0.029274, -0.006452, -0.030206, -0.016970, -0.063160, -0.087139, -0.051800, 0.014724, 0.123008, -0.020569, -0.029190, 0.022349, -0.057229, 0.066759, -0.017000, -0.044914, 0.004960, -0.002575, -0.043959, -0.052662, -0.032864, -0.080238, -0.006988, -0.035828, -0.085461, 0.087611, -0.081484, 0.004637, 0.038490, 0.051377, -0.007147, -0.143930, 0.025370, -0.060488, 0.010869, -0.065138, 0.063968, 0.021976, -0.085025, -0.006953, -0.084355, -0.093809, 0.021319, 0.062435, -0.161865, -0.011199, -0.061265, -0.049576, -0.098375, -0.059248, -0.051746, 0.043653, -0.027925, -0.148832, 0.051944, -0.123136, -0.042947, -0.051619, 0.020903, -0.040053, -0.026478, -0.094275, -0.084692, -0.088352, -0.030759, -0.082619, -0.075083, 0.031668, -0.170864, 0.014066, -0.000579, 0.005419, -0.018251, 0.079101, -0.015943, -0.246026, -0.051680, 0.006867, -0.032719, -0.054722, -0.023549, -0.034959, 0.013328, -0.132273, 0.077218, -0.062580, -0.129142, -0.105677, 0.052486, -0.054773, -0.045461, -0.015706, -0.011129, -0.001078, 0.036557, -0.028699, 0.043700, 0.066070, 0.069819, 0.101731, 0.020439, -0.046484, 0.041283, -0.049349, 0.002052, -0.077383, 0.034014, 0.002480, -0.108102, -0.031615, -0.018843, -0.053327, 0.127094, -0.007028, -0.006825, 0.004348, 0.098589, -0.019014, 0.142235, -0.013475, -0.012658, -0.064264, 0.015513, -0.088281, -0.008988, 0.021087, -0.045312, 0.079890, -0.053346, 0.063640, -0.027645, -0.021463, 0.188725, -0.006899, 0.032429, 0.019669, -0.046610, -0.066147, -0.100777, 0.039900, 0.052213, -0.049807, -0.042046, 0.024147, -0.057124, -0.024488, -0.003038, -0.001731, -0.003115, -0.074930, -0.047706, 0.001545, 0.037211, 0.043947, 0.000524, 0.106064, 0.028084, -0.053052, -0.081506, 0.018575, 0.057786, -0.009708, 0.101473, 0.045757, -0.136863, -0.016833, -0.060808, 0.025984, -0.029214, -0.048359, 0.022516, -0.088643, 0.033112, -0.074277, -0.030636, -0.098104, -0.102760, -0.029035, -0.085209, 0.020854, -0.025053, -0.044574, -0.100396, -0.038843, 0.019206, -0.111893, -0.075491, -0.147314, -0.001330, -0.030109, 0.043542, 0.012824, 0.082268, -0.046498, 0.042065, -0.012498, 0.047682, -0.041223, 0.049432, 0.019529, 0.101917, -0.078914, -0.059058, -0.031940, -0.097247, -0.046689, 0.058679, -0.080522, 0.013011, -0.049183, -0.085681, 0.074138, -0.042444, 0.125305, 0.020167, 0.100962, -0.008974, -0.119325, 0.017018, -0.102263, 0.020413, -0.040832, -0.083960, -0.049268, -0.218839, -0.001143, -0.112178, -0.029551, -0.146416, 0.097157, -0.107528, -0.010773, -0.060773, -0.038242, -0.141504, -0.059728, -0.068732, -0.022069, -0.046145, -0.088247, -0.028854, -0.012402, -0.126808, 0.010321, 0.052053, -0.026287, 0.114006, -0.128141, 0.020963, -0.012042, -0.037903, 0.006503, -0.017847, -0.129632, 0.088951, -0.069744, -0.116953, -0.033700, -0.023776, 0.064389, -0.005372, -0.032384, -0.067917, 0.075703, -0.078224, -0.040746, -0.093592, 0.075450, 0.002485, -0.006482, -0.012195, 0.000802, -0.054708, -0.116491, 0.100428, 0.113741, -0.016236, -0.045785, 0.033566, -0.067053, 0.036531, 0.080152, -0.064494, -0.102491, -0.047903, 0.096753, -0.068525, 0.054150, -0.058925, 0.043716, -0.084245, -0.039090, 0.094347, -0.049450, -0.054188, 0.106335, 0.021842, -0.054409, -0.049356, -0.070120, -0.024397, -0.119069, 0.021744, -0.065935, -0.038969, 0.073990, -0.021239, -0.100281, -0.042695, 0.021142, 0.008628, 0.080389, -0.112678, -0.079012, -0.083274, -0.016566, 0.004433, -0.009142, 0.020067, -0.010872, -0.034766, 0.063126, 0.006979, -0.024952, -0.028727, -0.033955, -0.002178, -0.020184, -0.079343, -0.019814, -0.070695, -0.084219, -0.007980, -0.080831, 0.093565, 0.021781, 0.036602, -0.025059, -0.070813, -0.161797, -0.069627, -0.087503, -0.010037, -0.024876, -0.012280, -0.088940, 0.004112, 0.009460, 0.018131, 0.032564, -0.022764, -0.070841, -0.016528, -0.083970, -0.022556, 0.077033, -0.028550, 0.055352, -0.047386, -0.005922, 0.081453, -0.017832, 0.067251, 0.040527, -0.173927, -0.061830, 0.005401, 0.012087, -0.035240, -0.018595, 0.019673, -0.037037, -0.035778, -0.081670, 0.029244, -0.134885, -0.035097, -0.100363, -0.001712, 0.033127, -0.054510, -0.021020, 0.047673, -0.120337, 0.054087, -0.024819, -0.050187, -0.098567, -0.056573, 0.013111, -0.121209, 0.042805, -0.051545, 0.053247, -0.176867, 0.045730, 0.016458, -0.010332, 0.065764, -0.004032, 0.116939, -0.154645, 0.056575, -0.019349, -0.068797, -0.046834, -0.039614, 0.002834, 0.278925, -0.020704, -0.124213, -0.169403, -0.007552, -0.003039, 0.093763, -0.083777, -0.064422, -0.169229, 0.037659, -0.095960, 0.008612, -0.000849, -0.030801, -0.048513, -0.035398, 0.019607, -0.003221, -0.012335, -0.096369, -0.030639, -0.010899, -0.067924, -0.072230, -0.012927, -0.016376, 0.070843, 0.007884, -0.001143, 0.047936, 0.029349, 0.006184, 0.042813, -0.001405, 0.027956, 0.042851, 0.021149, -0.024899, -0.010875, -0.060414, -0.000232, -0.144666, -0.130362, -0.136523, -0.088864, 0.027505, -0.066269, 0.039178, -0.063909, 0.030802, -0.076250, -0.024596, -0.022119, -0.061211, 0.026691, 0.094318, -0.022583, -0.085903, -0.045681, -0.081288, -0.055573, 0.005022, -0.047423, 0.167094, -0.101766, 0.013160, 0.038057, 0.011123, 0.015294, -0.082874, -0.002467, -0.074778, -0.108881, 0.023175, 0.019188, -0.054551, -0.022870, 0.031156, 0.033910, -0.048367, -0.018549, -0.090831, -0.057183, -0.025701, -0.016694, -0.153710, 0.041361, -0.103974, -0.036759, -0.068919, -0.048374, 0.018940, 0.042461, 0.026380, 0.039974, 0.017195, -0.105639, 0.110872, 0.000764, -0.079904, 0.095453, -0.042053, -0.015706, 0.056353, -0.089400, -0.030648, 0.043923, -0.067707, -0.173856, -0.118736, -0.012797, 0.043157, -0.006716, 0.026630, 0.006673, -0.013627, 0.060893, 0.029698, -0.035769, -0.124573, -0.059968, 0.019479, -0.048774, 0.003769, -0.085010, 0.015253, -0.064543, 0.049108, -0.061623, -0.070946, -0.069308, -0.018656, 0.012592, 0.024951, -0.048704, -0.105677, 0.118770, -0.061935, -0.048845, -0.059818, 0.033163, -0.046488, 0.025678, -0.031620, -0.097198, 0.032658, 0.005544, -0.052619, 0.001735, -0.005132, -0.004593, 0.050851, -0.010002, 0.050206, 0.064863, -0.050390, -0.107431, 0.055267, -0.035629, -0.014436, -0.002791, -0.056179, -0.066871, 0.019076, -0.064749, -0.023358, -0.104885, -0.017864, -0.066096, 0.221365, -0.054038, -0.037419, -0.009163, -0.004813, -0.005583, -0.062703, 0.072116, 0.070964, -0.034961, -0.064419, -0.054578, 0.043759, 0.030233, 0.054121, 0.019834, 0.048405, -0.014583, 0.002372, -0.110624, 0.021652, -0.013875, -0.018162, 0.018153, -0.044364, 0.147825, -0.128388, -0.122821, -0.054928, -0.099949, -0.051073, -0.028792, 0.043094, -0.045820, -0.071774, 0.027536, 0.024567, -0.005913, -0.059507, -0.089135, -0.008068, -0.025166, 0.036093, 0.039683, 0.015046, 0.015161, 0.144000, 0.022312, -0.024648, -0.014184, 0.082919, -0.055363, 0.020647, 0.077213, -0.013203, 0.060791, 0.012567, 0.070646, 0.039556, 0.004280, -0.002757, -0.074997, 0.029605, -0.124084, 0.074236, 0.008403, 0.053468, 0.092245, -0.000317, -0.033969, 0.038531, -0.127689, 0.088730, -0.032759, 0.013598, -0.072184, 0.116403, -0.081609, 0.066045, -0.020494, 0.063396, -0.047434, 0.022870, 0.088216, 0.142586, -0.002967, -0.109060, 0.051484, 0.079133, -0.070309, 0.040123, -0.098554, -0.004767, -0.085969, -0.047743, -0.028309, -0.018817, -0.040461, -0.029658, 0.065595, -0.010877, 0.023854, -0.041439, -0.039607, -0.062103, 0.037439, -0.125131, 0.060336, -0.036562, -0.069324, 0.002865, -0.006619, 0.027938, 0.027692, 0.154642, 0.011675, -0.119926, -0.077954, -0.063270, -0.030636, -0.071062, -0.026558, 0.046691, -0.085993, 0.074325, 0.026447, 0.068043, -0.088137, 0.067517, -0.045615, 0.043590, -0.073108, -0.071904, -0.126832, -0.076706, -0.017338, -0.027281, -0.062612, -0.028609, 0.048082, 0.019607, 0.122765, 0.033995, 0.040310, -0.004711, 0.018942, -0.071649, -0.001747, -0.090158, 0.062138, -0.001217, 0.023872, -0.070085, -0.033024, 0.012243, -0.063315, -0.098607, -0.009165, 0.062236, 0.035811, 0.063623, -0.042241, -0.005526, -0.008794, 0.041281, 0.001574, -0.021611, 0.012461, -0.047486, 0.075677, -0.081477, 0.007426, 0.052603, 0.048529, 0.033013, -0.075970, -0.002580, -0.121558, 0.039230, -0.091842, 0.014114, -0.056758, -0.034905, -0.058971, 0.130477, -0.087608, -0.142145, -0.061922, -0.048537, -0.062461, 0.010301, -0.002014, 0.026832, 0.059928, -0.086692, -0.076917, 0.036559, -0.062509, -0.022295, -0.021085, 0.049487, -0.063680, 0.007012, 0.028474, -0.008578, 0.017596, 0.099932, -0.086505, -0.100373, 0.043783, -0.004534, -0.024842, 0.107122, -0.127427, -0.027516, -0.008183, -0.039439, 0.066834, 0.034670, -0.023007, -0.041763, 0.067454, -0.019989, -0.084912, -0.024606, 0.040438, 0.021640, -0.069409, -0.085170, -0.059804, 0.108059, -0.076029, 0.015321, -0.042910, 0.079693, -0.011240, -0.013759, -0.028548, 0.080261, -0.017185, -0.012823, -0.105629, -0.127439, -0.003239, 0.064146, -0.011390, -0.013190, 0.089599, -0.001972, -0.033640, 0.073121, -0.089806, 0.010730, -0.037745, -0.022028, 0.045876, 0.067729, -0.172386, -0.038004, 0.069496, 0.041072, -0.035805, -0.084605, 0.102612, 0.064962, -0.006751, -0.075091, -0.157551, 0.027582, -0.135827, -0.003898, -0.005776, 0.034702, -0.037892, 0.088480, 0.034792, -0.094226, 0.093200, -0.068053, -0.002844, 0.010257, -0.049404, 0.023093, 0.046673, -0.075656, 0.063236, 0.043897, 0.011933, -0.121203, 0.019866, -0.024157, 0.056072, 0.032246, -0.068560, -0.091509, 0.067409, 0.075089, -0.140474, 0.016228, -0.036706, -0.059587, -0.108238, 0.006394, -0.098075, -0.033499, 0.094140, 0.014839, 0.061095, -0.025641, -0.002893, 0.068728, 0.109682, 0.057047, -0.085683, 0.035180, 0.066490, -0.097125, -0.046231, -0.022359, -0.076826, 0.018919, -0.054839, -0.067191, -0.019425, 0.011176, -0.055382, -0.024571, -0.019894, 0.094278, 0.059777, 0.069341, -0.098955, 0.016209, 0.025916, 0.060501, 0.052103, 0.050181, -0.072489, 0.001822, -0.019091, -0.054054, -0.061428, -0.082451, 0.062945, -0.025721, -0.120239, -0.006745, -0.066770, -0.034686, -0.039867, 0.008673, -0.038320, -0.036286, -0.097407, -0.092945, 0.010437, 0.087808, 0.121010, -0.083029, 0.041747, 0.074909, 0.055415, -0.041562, 0.035126, 0.060725, -0.064236, 0.017128, -0.009492, -0.083305, 0.033860, -0.010249, -0.033776, 0.082548, -0.031819, 0.035980, -0.052888, -0.099454, 0.044984, -0.007643, -0.031744, 0.099461, -0.030865, -0.057919, 0.094887, -0.048807, -0.051761, 0.039332, -0.061783, -0.008614, -0.109263, -0.037310, 0.088338, -0.084795, -0.107254, -0.011517, 0.058453, -0.127398, -0.024167, -0.099560, 0.001112, -0.049076, -0.023321, -0.080750, 0.074287, 0.043208, -0.046802, -0.001045, 0.031740, -0.041856, -0.062998, -0.080644, 0.031822, 0.007911, 0.028860, -0.063390, 0.051993, 0.073896, -0.113975, -0.060034, -0.074972, -0.026900, -0.044416, 0.069159, 0.001861, 0.022158, -0.060457, -0.075340, 0.032905, 0.052295, 0.043499, -0.143409, -0.061245, 0.027284, 0.100138, -0.070223, -0.063088, 0.027294, -0.034488, -0.021053, 0.005289, 0.049383, 0.022098, 0.024508, -0.005387, 0.012908, -0.052139, -0.071995, -0.004763, -0.005745, -0.031938, 0.069699, 0.069328, -0.055562, -0.001950, -0.055605, -0.011874, -0.024443, 0.046574, 0.070922, 0.004655, -0.153081, 0.035901, -0.053535, -0.071679, 0.004640, -0.043853, -0.018485, 0.002120, -0.003757, 0.015430, 0.059760, -0.051727, -0.074672, -0.022460, 0.060711, 0.030728, -0.076053, -0.010151, -0.005696, 0.020564, -0.026576, -0.117817, -0.106114, -0.052560, 0.148322, -0.086769, 0.016384, 0.018186, 0.008427, 0.118730, -0.083717, -0.091899, 0.044417, 0.018622, -0.108503, -0.115924, 0.059825, 0.004848, 0.094333, 0.041950, 0.008235, 0.034931, 0.066075, 0.048907, 0.001232, -0.009169, -0.006627, -0.019979, -0.067239, 0.015158, 0.088738, -0.054727, 0.039224, 0.011614, 0.094453, 0.033017, -0.040188, 0.030000, -0.013693, -0.051583, -0.096046, 0.186158, 0.034684, 0.054597, 0.085530, -0.071856, -0.003080, -0.036792, 0.024261, -0.123446, 0.000552, -0.025941, 0.023158, 0.073727, -0.186909, -0.051332, -0.005351, -0.056748, -0.003286, 0.029060, 0.016484, -0.160656, 0.014229, 0.024901, 0.000433, -0.086570, -0.101042, -0.061692, -0.043083, 0.132921, -0.043219, 0.013426, -0.076331, 0.006765, -0.035224, -0.009548, 0.004523, -0.009928, -0.037426, 0.026999, 0.044647, -0.097612, -0.106419, 0.045617, 0.028590, -0.009824, 0.012074, -0.002743, -0.023239, -0.014680, -0.040612, -0.096156, 0.035127, 0.063483, -0.002243, 0.039065, -0.062480, 0.032610, -0.031148, 0.008342, -0.014019, -0.105875, -0.159865, -0.093656, -0.055286, 0.016403, 0.002265, -0.094686, 0.026684, -0.049435, -0.047161, 0.017422, 0.012230, 0.066316, -0.003674, -0.034623, -0.027111, -0.020462, -0.008197, -0.142197, 0.054025, -0.093119, -0.076488, 0.052718, 0.002492, -0.068958, 0.014132, -0.054904, -0.057354, -0.071383, -0.011344, -0.021618, -0.108427, -0.145433, -0.071333, 0.142657, -0.005936, -0.041627, -0.020729, 0.009923, -0.081869, -0.008999, -0.033162, 0.011881, -0.047884, 0.034204, 0.046945, -0.001992, -0.034891, 0.002996, -0.003288, -0.066634, -0.032405, 0.052734, -0.026031, -0.089494, 0.004089, -0.030236, -0.034415, -0.106646, 0.021704, 0.009756, 0.004705, -0.074442, 0.001663, -0.008281, 0.105332, 0.009625, 0.024064, 0.029745, -0.025867, 0.007583, -0.056964, -0.046875, -0.083864, 0.064629, -0.046743, 0.034247, -0.011794, -0.100541, -0.035309, -0.028349, -0.075324, 0.068926, 0.085916, 0.060189, -0.021986, -0.127256, 0.022081, -0.029281, 0.072964, 0.012730, -0.022212, -0.091291, 0.046323, -0.090577, 0.001314, 0.069473, -0.141718, 0.029701, -0.073997, -0.023298, 0.135452, 0.022448, 0.014296, 0.020095, -0.064316, -0.104712, 0.151042, -0.079444, 0.055055, -0.047173, 0.052199, 0.093614, 0.048289, -0.022991, -0.040776, 0.014043, -0.039332, -0.041178, 0.071161, 0.079397, 0.130348, -0.031969, -0.031704, -0.043037, -0.093833, -0.025744, -0.125490, 0.017221, 0.066721, -0.007504, 0.000647, -0.056947, -0.059795, -0.002076, -0.054541, -0.037537, 0.058328, -0.099695, 0.003273, -0.099431, -0.006089, 0.030578, 0.009560, -0.025887, 0.063694, -0.068675, -0.029150, 0.025723, 0.020906, 0.089864, 0.020723, 0.014859, -0.037349, -0.037793, 0.093527, 0.081444, -0.092644, -0.087127, 0.029527, 0.048537, -0.115173, -0.063111, -0.031909, 0.088536, 0.018137, -0.081167, 0.001619, -0.043680, -0.071909, -0.035330, -0.034954, 0.116644, -0.065715, -0.017760, -0.026427, -0.067249, -0.006900, -0.056320, -0.004812, -0.023177, 0.067081, -0.027744, -0.003725, -0.145373, 0.015647, -0.097101, -0.004756, 0.034330, 0.054351, -0.118527, -0.087595, -0.016450, -0.049099, -0.102825, -0.019058, 0.073822, 0.034940, -0.020013, -0.064720, 0.020432, -0.034164, -0.006833, -0.038316, -0.032869, 0.050928, -0.015748, -0.011131, -0.086396, 0.010540, -0.156924, -0.056526, -0.030105, 0.057452, -0.012723, 0.075879, -0.023890, -0.007342, -0.064222, -0.043006, -0.019239, -0.005819, -0.044986, -0.038743, -0.006032, 0.025101, 0.022774, -0.054534, -0.103667, 0.011487, 0.190798, 0.108299, 0.042917, -0.023939, -0.117740, 0.033590, -0.064602, -0.013999, 0.043193, 0.038927, 0.035704, -0.030545, -0.049351, 0.060994, 0.059677, 0.029362, -0.008903, 0.026686, -0.080172, -0.039751, -0.012721, 0.084996, 0.025648, 0.059456, 0.032084, -0.049365, -0.058981, -0.016140, -0.021657, 0.008067, 0.028402, 0.039465, -0.035443, 0.046006, -0.030190, -0.009905, -0.111200, 0.193781, 0.077584, -0.077847, -0.048115, -0.027994, 0.093363, -0.048828, -0.065602, -0.023385, -0.064278, -0.042923, 0.023741, -0.055263, 0.022862, 0.054937, -0.076271, 0.057709, -0.009292, -0.140051, -0.053776, 0.012336, -0.022220, -0.002905, -0.050423, -0.036962, 0.036789, -0.111015, -0.191678, -0.052237, -0.005513, -0.067295, -0.068638, -0.015838, -0.086441, 0.063199, 0.010089, 0.019330, -0.050964, -0.037685, -0.063124, -0.072654, 0.035076, -0.037619, 0.032010, -0.146414, -0.047437, -0.088254, -0.182654, -0.014877, -0.046007, 0.053159, -0.123584, -0.005182, 0.072513, -0.018251, -0.023148, -0.017027, -0.038296, -0.068523, -0.024691, -0.062519, 0.089241, 0.035357, -0.091427, 0.102823, 0.081264, -0.040658, -0.038011, -0.073720, 0.053311, -0.010944, -0.027508, -0.121071, -0.092107, 0.046644, 0.003638, 0.024220, -0.051841, 0.028930, -0.105363, 0.025877, -0.045853, -0.038730, -0.050476, -0.061180, 0.032680, 0.019007, -0.016435, 0.048832, -0.036094, -0.025928, 0.088109, -0.044324, -0.046456, -0.102172, -0.078266, 0.046154, -0.085554, 0.046348, -0.170921, -0.049609, -0.084076, -0.133577, 0.001733, -0.014661, -0.059825, 0.016072, -0.126058, 0.072176, -0.041716, 0.034693, -0.050152, 0.151602, -0.039405, 0.094301, -0.135210, -0.062968, 0.049336, 0.170560, -0.062934, -0.050708, 0.018486, -0.034552, 0.004469, -0.071524, -0.009086, 0.030148, -0.027819, 0.048332, 0.027030, -0.152994, -0.058798, -0.043051, -0.104403, 0.025738, 0.004462, -0.013778, -0.033396, -0.127688, -0.052882, -0.080473, -0.092271, -0.078257, 0.182776, -0.049685, -0.137087, -0.055259, 0.001868, -0.086574, 0.033292, 0.187537, -0.039205, -0.053402, 0.030355, 0.015705, -0.046719, -0.117753, -0.061079, -0.098135, 0.131762, 0.003304, 0.053049, -0.028354, -0.146513, 0.055464, -0.008877, -0.060552, -0.077999, 0.020827, -0.035238, -0.074845, -0.025212, -0.147339, -0.027634, 0.035816, -0.063690, -0.025672, 0.004898, -0.031316, 0.091041, 0.018315, -0.101892, -0.086485, 0.143695, -0.006991, 0.018283, -0.043585, -0.042744, 0.029925, -0.078878, 0.049567, 0.005446, 0.047773, -0.046774, 0.064382, 0.051969, -0.056702, 0.029580, -0.103247, -0.027872, -0.032601, -0.052721, -0.042497, -0.018380, -0.062414, -0.049742, -0.097229, -0.069659, -0.015462, -0.081283, -0.011053, 0.030449, 0.023198, -0.031693, -0.118992, -0.133412, 0.007843, -0.047782, -0.168452, -0.030556, -0.038905, -0.051209, -0.097596, 0.073918, 0.107897, -0.042236, 0.158061, -0.144178, -0.019235, -0.121797, 0.005928, -0.090351, -0.036755, -0.016933, -0.034056, -0.121848, 0.071037, 0.000367, 0.109322, -0.005593, -0.054305, -0.019988, -0.082484, -0.016823, -0.112041, 0.094327, -0.053974, -0.104684, -0.068446, -0.089244, -0.042051, -0.044145, -0.036927, 0.022932, -0.037697, 0.021653, -0.025395, -0.244184, -0.113074, -0.163505, 0.006051, 0.101812, 0.048411, -0.105669, 0.002190, -0.010528, -0.064640, -0.058983, -0.022133, -0.126819, -0.027736, -0.076435, -0.117226, 0.023534, 0.042782, 0.039267, 0.059143, -0.042982, 0.016340, -0.109023, -0.100459, -0.026546, -0.130721, -0.082379, 0.004303, -0.023848, 0.008346, -0.108817, 0.130459, -0.042305, 0.071361, -0.089276, -0.043546, 0.089902, -0.136867, -0.031616, -0.084518, 0.115926, 0.064512, -0.095147, -0.068327, -0.015632, 0.008248, -0.034256, -0.152608, -0.169806, -0.178491, -0.042213, -0.023331, -0.016783, 0.160933, -0.021842, -0.000171, -0.058031, 0.025954, 0.057407, 0.048159, 0.001748, -0.011599, 0.156595, -0.071206, -0.026471, -0.078741, -0.053723, -0.007596, -0.026601, -0.165506, -0.022450, -0.125028, -0.013771, -0.069691, 0.192336, 0.024503, 0.021078, -0.030427, 0.025821, -0.063028, 0.096533, -0.030032, 0.045074, 0.077081, -0.008456, -0.092787, 0.043200, 0.017105, -0.070824, -0.092485, -0.033740, -0.005099, -0.030864, -0.018966, 0.020710, -0.080985, 0.032151, -0.052606, 0.113173, 0.075205, 0.034844, -0.029137, 0.005254, -0.112766, 0.110184, -0.094336, -0.058529, -0.025092, -0.090667, -0.020840, -0.026790, 0.094637, -0.258136, -0.124921, -0.082968, -0.060406, -0.066327, -0.057936, -0.022427, -0.080120, -0.011597, 0.024020, 0.024205, -0.026354, -0.039850, 0.020358, -0.022701, -0.071214, 0.120739, -0.043692, -0.145228, -0.039825, -0.112153, -0.070385, -0.069119, 0.173364, -0.027400, -0.075773, -0.061633, -0.012213, -0.178031, -0.101653, 0.163625, 0.020717, -0.018327, -0.218038, -0.190681, -0.039060, -0.042673, 0.008428, 0.127543, -0.090229, -0.057429, 0.016679, 0.127045, -0.137850, -0.038272, -0.064948, -0.057540, 0.025880, 0.016880, 0.014231, -0.034886, -0.031950, -0.005971, -0.235479, -0.030798, 0.009437, 0.070699, -0.068845, 0.061600, -0.124328, -0.072009, 0.012748, -0.025597, -0.047320, -0.011317, -0.022095, -0.060418, -0.095922, 0.027252, 0.043362, -0.054888, -0.080458, -0.089956, -0.022815, -0.079545, -0.041749, -0.040203, -0.066261, 0.012081, -0.131117, 0.100072, 0.097987, -0.063531, -0.026315, -0.002767, -0.148441, -0.125116, -0.025425, -0.101658, -0.057261, 0.074986, -0.116761, -0.011753, 0.042165, 0.015626, -0.011716, -0.027685, -0.003814, -0.079777, -0.154295, 0.007557, -0.009171, 0.028355, -0.046406, -0.176114, 0.116419, -0.065623, -0.035008, -0.024359, -0.144912, -0.040641, -0.033460, -0.163387, -0.072141, -0.082214, -0.003354, -0.044865, -0.112721, -0.006326, 0.062080, -0.120486, -0.052337, -0.034182, -0.067074, 0.044388, 0.019557, 0.021054, -0.057327, -0.044452, 0.077458, -0.043223, -0.127530, -0.051239, -0.015334, 0.014615, -0.021666, 0.012191, -0.028619, -0.065239, 0.038966, -0.020452, -0.015205, 0.097999, -0.022246, -0.063607, 0.072451, -0.081477, -0.042769, -0.016452, -0.141211, 0.007877, -0.091193, -0.077559, 0.013948, 0.034710, 0.011981, -0.039689, -0.097243, -0.055530, 0.038794, -0.069140, -0.128422, 0.028463, 0.009647, -0.014191, -0.137023, 0.185082, -0.065594, -0.043297, -0.096460, -0.014261, -0.005524, -0.029411, -0.028811, -0.133511, -0.182811, -0.080395, -0.043038, -0.064343, -0.068713, -0.020861, 0.030646, -0.038291, -0.010629, 0.041734, -0.032885, -0.077099, 0.058683, 0.032282, -0.026016, -0.024800, -0.105072, -0.074154, -0.079181, -0.074488, -0.159334, 0.022990, -0.042301, -0.071522, 0.005890, 0.023272, 0.098457, -0.013586, 0.074446, -0.006635, 0.098760, -0.060553, -0.017206, 0.014563, -0.038965, -0.216787, -0.046289, -0.096570, -0.023825, -0.057254, -0.057359, -0.133965, -0.121756, -0.147200, 0.056417, -0.102980, -0.041730, -0.162711, -0.045676, 0.125697, -0.007934, -0.034402, 0.082049, -0.096391, -0.035479, -0.089091, 0.025045, -0.108692, -0.050674, -0.022240, 0.059389, 0.005461, -0.046276, -0.053832, -0.037780, 0.101248, -0.047133, -0.030896, 0.110552, -0.023435, -0.057290, -0.012764, -0.015591, -0.100311, -0.043008, -0.017713, 0.038141, -0.051783, -0.065460, -0.008126, -0.053048, -0.074334, -0.061954, -0.063351, 0.028501, 0.022562, -0.053348, 0.056303, -0.040777, -0.050117, -0.054473, -0.214663, -0.049226, 0.000514, 0.011466, 0.087542, 0.082160, 0.026084, -0.025850, -0.041291, 0.010475, -0.081947, -0.002853, 0.038569, -0.125660, -0.089133, -0.101859, -0.205432, -0.040204, -0.062556, 0.059396, -0.001824, 0.037082, 0.091295, -0.002579, -0.146735, -0.076730, -0.024454, -0.033321, 0.025141, 0.051398, 0.000992, -0.110595, 0.025582, 0.016764, -0.042011, -0.030836, -0.073239, 0.061248, 0.028096, 0.086382, 0.009981, -0.096286, 0.045249, -0.065385, 0.073933, -0.056785, -0.061417, 0.145273, -0.014207, 0.062997, 0.056427, -0.066544, -0.061366, -0.007421, -0.109062, -0.004910, -0.005835, -0.073653, -0.045920, -0.078985, 0.065761, -0.057269, -0.019345, -0.069586, -0.053418, 0.023425, -0.088187, -0.065265, -0.018256, -0.095052, -0.006811, -0.054146, -0.046155, 0.020785, 0.030240, -0.058011, -0.071365, -0.083136, -0.076044, -0.041066, -0.048407, 0.024175, -0.027553, -0.066984, -0.015667, -0.066674, -0.046423, -0.064130, 0.053099, -0.026815, 0.035087, -0.078979, -0.056962, -0.054000, -0.000037, -0.063930, -0.018860, -0.024536, 0.080523, 0.026160, -0.127455, 0.114009, 0.080279, -0.053831, -0.050693, -0.037087, 0.007867, -0.004330, -0.006373, 0.019286, 0.052374, -0.052579, -0.006938, -0.329782, -0.039352, -0.018805, -0.016777, 0.002095, -0.002307, 0.156382, -0.101360, -0.096210, 0.056135, 0.127942, -0.007395, -0.121728, -0.093216, 0.000487, -0.021572, -0.016592, -0.017144, -0.005201, 0.011268, -0.035444, -0.073245, -0.045975, 0.002995, -0.001074, -0.088368, -0.073828, -0.087264, 0.036174, -0.052460, -0.080534, -0.055981, -0.025288, -0.016437, -0.071649, -0.008278, 0.165022, -0.088118, 0.001388, 0.024181, 0.026911, 0.012641, 0.020585, -0.075240, -0.018638, -0.067051, 0.069959, 0.170820, 0.006515, 0.025929, 0.102541, -0.074864, -0.099353, 0.030630, -0.085635, 0.016895, -0.011329, -0.045738, -0.002050, 0.055384, -0.051417, -0.044837, -0.158386, -0.045893, 0.008375, -0.115328, -0.141601, -0.041594, -0.008707, -0.105702, 0.062784, -0.046299, 0.115974, -0.014390, 0.023424, -0.051838, -0.008791, -0.142343, -0.032981, -0.009161, -0.082746, -0.023770, -0.126271, 0.118627, -0.054001, -0.079382, 0.016553, -0.109287, -0.173760, -0.045968, -0.022492, 0.032117, 0.039749, 0.038022, 0.019501, 0.057318, -0.092348, 0.024279, 0.008751, -0.004733, 0.033983, -0.014413, 0.008008, -0.066118, -0.047620, -0.037768, -0.028034, -0.050694, 0.044808, -0.001769, -0.031190, -0.061289, -0.068212, -0.065531, 0.026462, -0.082107, 0.038085, 0.192427, 0.054888, -0.068736, -0.035353, -0.116864, -0.116778, 0.002845, 0.102922, -0.034813, -0.077096, 0.023053, 0.185517, 0.067112, -0.029985, -0.076704, -0.058413, -0.050670, -0.037896, 0.014568, -0.046547, -0.021854, -0.145607, -0.020634, 0.107476, 0.010138, -0.019057, -0.002309, -0.043291, 0.034544, -0.004618, -0.155199, 0.006162, 0.052951, -0.029454, -0.000785, -0.105379, 0.038246, -0.159836, -0.045051, -0.036711, 0.049980, -0.236019, -0.015501, -0.095187, 0.001600, -0.026802, -0.048786, 0.177292, 0.005055, -0.192704, -0.038522, -0.039149, -0.049878, 0.110460, -0.049663, 0.012630, -0.070386, -0.030293, -0.019220, -0.027024, 0.087013, 0.022363, 0.046263, -0.054686, 0.005116, -0.082935, -0.138954, -0.022582, -0.077615, -0.131286, 0.058682, 0.004372, 0.046471, 0.017979, -0.044654, -0.030402, -0.016628, -0.032710, -0.063484, -0.068896, -0.074876, 0.014904, -0.105302, 0.057217, -0.099658, -0.042585, 0.061426, -0.166224, -0.028532, 0.118437, 0.025493, -0.195295, -0.032015, -0.015156, -0.086206, -0.008265, -0.035661, -0.028865, 0.005585, -0.131265, -0.027048, -0.035745, 0.068351, 0.002855, -0.074264, 0.041888, -0.170568, -0.353267, -0.060257, 0.149051, 0.047362, -0.059695, -0.045859, -0.003147, -0.067913, 0.083960, -0.014261, -0.032706, 0.005225, -0.025054, -0.108937, 0.087945, -0.076292, 0.024029, -0.039604, -0.007256, -0.002659, -0.096988, 0.024814, -0.079193, -0.101249, 0.075844, 0.147371, -0.066630, -0.083950, -0.074104, -0.051853, 0.008674, -0.030880, -0.041910, -0.029799, -0.004262, -0.089828, -0.016161, -0.064815, 0.048148, -0.041686, 0.115317, -0.066204, 0.008983, -0.028989, 0.047423, 0.103350, -0.029573, -0.032925, -0.088245, 0.006277, 0.064263, -0.061042, -0.011185, -0.069057, -0.000358, 0.025701, -0.079192, -0.049166, -0.098866, 0.046770, -0.023411, -0.020509, -0.055341, -0.060243, -0.038646, -0.067413, -0.078970, -0.063524, -0.101888, -0.059843, -0.045762, -0.115017, -0.060804, -0.136545, -0.071654, -0.088179, -0.030497, -0.054571, -0.104392, -0.003461, 0.214393, -0.005693, -0.121026, -0.125352, 0.012695, 0.249620, 0.065622, 0.032291, 0.010677, -0.075246, -0.066354, -0.016085, -0.058951, -0.001556, -0.014633, 0.056909, -0.089476, 0.062736, 0.008953, -0.063394, -0.004174, -0.149104, 0.077215, -0.095256, -0.057465, -0.067922, -0.031080, -0.174526, -0.134629, -0.103108, -0.023201, 0.088130, -0.032204, -0.007449, -0.099018, -0.082088, 0.101044, 0.005332, -0.062333, 0.027056, 0.027389, -0.084466, 0.035402, 0.137065, -0.013951, 0.028618, -0.044097, -0.091274, 0.070372, -0.020146, 0.019434, -0.098537, -0.040067, -0.041211, -0.039383, -0.078840, -0.036407, 0.023555, 0.053303, 0.049500, 0.038706, -0.010309, 0.049634, -0.067563, 0.161169, -0.021887, 0.285796, -0.063063, 0.010759, 0.002628, 0.009829, 0.036018, -0.092091, 0.024075, -0.016201, -0.070995, -0.108342, 0.063088, -0.001071, -0.097729, -0.180997, -0.016512, 0.001880, -0.012864, 0.016373, 0.024356, 0.007003, -0.008083, -0.043663, -0.068836, 0.044262, 0.072293, 0.023163, -0.038995, -0.049353, 0.010789, 0.016263, -0.048670, -0.006467, 0.048540, -0.112442, -0.088272, -0.095814, -0.055172, 0.120459, 0.079814, -0.016390, -0.131937, 0.019155, -0.004988, -0.050056, -0.106159, -0.001027, -0.044487, -0.024318, -0.086109, -0.056495, 0.017369, 0.010633, 0.175056, -0.145529, -0.074427, -0.060456, 0.060121, -0.085285, 0.008007, -0.038709, -0.044643, 0.006764, 0.099668, -0.034252, 0.059792, -0.021037, -0.020583, -0.046104, -0.035722, -0.045693, -0.089087, -0.014155, -0.003972, 0.101838, 0.031095, -0.105264, -0.035699, -0.017077, -0.008260, -0.024336, -0.127891, 0.018958, -0.017495, -0.034422, -0.155966, 0.047770, -0.003367, -0.058342, -0.006714, -0.094675, -0.070605, 0.035781, -0.014861, -0.005177, -0.047116, -0.009938, 0.092635, -0.121787, 0.036342, -0.008658, -0.000693, -0.022360, -0.128559, 0.024951, 0.075928, -0.017103, -0.079702, 0.064128, -0.048471, 0.036344, -0.070022, -0.022653, 0.007062, 0.114320, -0.009702, 0.018459, -0.022280, -0.003471, -0.030503, -0.027479, -0.011105, -0.003479, 0.006434, -0.078802, 0.016626, -0.152677, 0.008036, -0.123818, -0.033182, -0.009579, -0.020875, -0.099024, -0.046605, 0.006124, 0.038697, 0.002911, -0.004862, -0.011011, -0.017162, -0.058632, -0.067551, -0.005074, -0.033862, -0.089205, 0.098446, -0.038248, -0.078185, -0.051789, -0.028342, -0.089506, -0.005710, -0.033162, 0.040791, -0.054909, -0.045527, 0.032811, 0.009475, -0.022653, 0.086993, -0.035223, -0.096285, 0.066461, -0.085415, -0.050167, 0.126636, 0.005920, 0.026729, -0.062372, -0.023425, -0.059541, -0.016627, 0.028459, -0.008657, 0.045552, 0.028944, -0.008587, -0.028984, -0.048973, 0.028516, -0.035108, -0.014791, -0.115441, -0.009204, -0.054635, 0.020323, -0.076607, -0.006386, -0.062295, -0.010837, -0.002946, -0.004753, -0.075995, -0.019151, 0.026653, -0.055252, -0.025752, -0.028139, -0.055336, 0.041539, 0.119143, 0.054213, 0.023311, 0.035523, 0.163799, -0.084370, -0.006368, 0.032889, -0.130785, -0.066669, -0.084978, 0.005710, 0.017336, -0.095782, 0.067561, -0.011075, -0.041473, -0.077304, 0.011438, 0.040235, 0.012068, 0.025631, 0.103836, -0.035008, -0.084202, -0.026820, -0.108802, -0.048239, 0.018601, 0.005712, -0.116183, -0.133309, 0.005885, -0.078528, -0.019562, -0.034441, 0.041153, -0.103225, 0.086466, 0.011207, -0.009399, 0.070473, 0.030032, -0.043582, -0.040213, -0.114716, -0.076699, 0.036022, 0.000643, 0.006833, 0.059864, -0.034281, 0.077255, 0.085894, -0.077888, -0.000598, -0.043438, -0.069916, -0.032235, 0.030933, -0.013493, -0.223522, -0.013240, -0.099935, 0.037698, 0.086780, -0.087136, -0.141730, 0.095858, -0.053741, -0.020657, -0.014677, -0.091353, -0.098611, 0.003813, 0.083886, -0.049445, -0.064291, 0.093682, -0.056976, 0.010728, 0.014752, 0.008512, -0.021565, -0.204120, 0.049028, -0.123387, -0.066123, -0.038785, 0.033924, -0.019403, -0.090021, -0.072224, -0.097452, 0.006034, 0.089320, 0.054554, 0.031002, -0.084638, 0.023435, -0.111592, -0.005178, -0.011029, -0.050374, 0.015767, -0.090184, -0.080340, -0.008382, -0.018973, -0.068450, 0.032361, -0.036686, -0.103969, -0.016252, 0.019982, -0.008185, -0.095021, 0.061913, 0.048657, 0.026769, -0.015099, 0.033451, -0.055305, 0.044684, -0.010776, -0.012715, -0.029224, 0.002175, -0.222520, 0.044771, 0.027187, -0.031721, -0.024656, -0.032330, -0.071036, -0.027092, 0.008232, -0.031220, -0.011416, 0.013364, -0.049720, -0.061612, -0.018893, -0.012818, 0.051327, -0.071312, -0.065438, -0.045103, -0.021075, -0.050439, 0.068589, -0.034896, 0.008825, -0.120729, -0.099533, 0.082879, -0.067828, -0.111752, 0.061723, -0.011638, -0.103540, 0.024033, 0.002900, 0.034418, -0.095234, -0.002065, -0.035662, -0.021780, -0.058053, 0.000122, -0.059780, -0.018264, -0.107547, -0.049398, 0.020006, 0.017396, -0.077957, 0.028856, -0.004907, -0.093284, -0.075502, -0.054878, -0.073408, -0.203728, -0.034882, 0.085969, -0.092965, 0.000065, -0.029543, -0.090368, 0.015148, -0.065117, 0.030501, -0.010839, 0.073891, 0.058111, 0.032314, -0.001745, -0.048138, -0.017583, 0.056402, -0.047286, -0.024440, 0.025617, -0.093688, 0.036021, -0.062100, 0.017335, -0.026576, -0.014742, -0.058651, -0.081470, 0.121177, -0.013778, -0.074912, -0.003833, -0.086448, -0.013217, -0.120910, -0.042840, -0.003682, 0.047104, -0.031488, -0.043794, 0.027502, 0.010863, -0.170779, -0.213337, 0.036520, -0.046476, -0.058490, -0.101465, -0.109924, -0.007855, -0.023567, 0.033321, -0.055589, -0.015235, -0.027083, 0.022458, -0.009274, 0.009427, -0.017470, -0.003905, -0.008742, 0.006524, -0.071169, 0.109476, 0.047594, 0.048183, 0.020002, -0.035335, -0.070214, -0.056982, -0.080004, -0.095673, 0.028472, 0.029065, -0.096139, -0.043901, -0.003959, 0.019004, 0.002549, -0.034978, -0.013856, 0.111614, -0.047736, -0.024331, 0.008224, -0.023100, -0.074720, -0.129617, 0.025722, 0.024387, 0.026232, -0.104972, -0.040938, -0.007184, -0.062529, -0.056997, -0.106204, 0.057434, 0.019292, -0.086066, 0.079518, -0.064589, -0.032589, -0.008047, -0.032427, -0.004642, -0.000121, -0.113550, -0.057967, 0.039928, 0.048686, -0.001672, -0.074518, -0.113259, 0.007759, 0.007430, 0.054954, 0.093921, -0.008323, -0.070801, -0.004015, -0.053653, -0.015920, -0.031946, -0.056061, 0.038382, 0.047206, -0.074632, 0.041768, 0.010541, -0.045905, -0.061099, 0.018372, 0.003985, -0.148946, 0.127021, -0.068985, -0.021707, -0.015926, -0.047116, -0.024497, -0.045974, 0.048987, -0.112864, -0.086685, -0.026091, -0.110585, -0.004474, 0.029283, -0.047720, 0.036173, 0.105518, -0.013299, 0.035948, -0.054473, -0.065985, 0.004724, 0.010013, 0.026576, -0.004515, 0.010263, -0.098595, 0.028887, -0.042134, 0.037570, -0.123087, 0.004317, -0.054928, 0.038714, -0.005508, -0.077282, -0.026217, -0.031202, 0.023505, 0.001232, -0.086690, 0.023627, 0.018870, 0.057541, -0.066431, -0.007884, 0.066479, 0.058507, 0.098255, -0.015763, -0.062301, -0.083580, -0.090068, -0.028522, -0.005728, -0.044243, -0.077679, 0.032932, 0.009908, 0.087303, -0.004342, 0.055860, -0.131574, 0.000815, 0.036075, -0.020497, -0.063652, -0.075577, 0.016039, -0.050923, -0.016228, -0.020622, -0.047281, 0.010959, 0.026843, -0.094905, -0.141510, -0.063099, -0.027648, -0.097951, -0.028519, -0.060947, 0.016329, -0.034399, -0.048080, -0.014085, 0.037490, 0.000629, -0.038923, -0.042182, -0.020998, -0.090564, -0.045410, 0.027764, -0.107516, 0.100510, -0.085301, -0.094226, 0.055894, -0.038381, -0.173367, -0.057219, -0.057741, -0.026432, 0.005541, 0.048477, 0.049503, 0.022750, 0.021837, 0.031998, -0.011642, 0.049856, 0.025804, -0.037924, 0.012891, -0.056447, 0.072073, 0.096851, 0.090220, -0.047905, 0.157181, 0.011718, -0.094982, 0.018262, 0.056758, -0.167487, -0.025642, 0.004012, -0.047260, -0.066026, -0.067824, -0.080638, -0.003369, 0.014243, -0.035616, 0.250999, -0.091146, -0.036393, -0.044280, -0.073156, 0.064068, -0.078618, -0.037899, -0.003965, -0.090805, 0.024637, -0.005052, 0.000160, -0.051241, 0.020876, -0.037098, 0.076243, 0.025154, -0.044180, -0.043015, -0.063405, 0.003892, 0.013478, -0.050741, -0.059532, -0.042346, -0.100208, 0.026086, 0.021458, 0.025305, 0.013267, -0.004242, 0.081941, 0.019036, -0.052920, -0.035176, -0.137160, -0.002089, -0.004236, -0.020096, 0.061414, -0.036816, 0.035729, 0.000526, 0.004611, 0.003982, -0.022941, -0.128069, -0.096469, 0.012697, -0.060756, -0.051984, 0.046185, 0.003478, -0.009179, 0.029115, 0.018867, -0.073050, -0.010741, -0.027284, 0.039047, 0.021808, 0.048134, 0.023247, -0.090834, -0.025033, 0.019866, 0.109574, -0.013172, -0.057581, -0.031592, -0.175928, -0.047297, -0.000549, -0.074287, 0.020059, -0.010104, -0.050175, -0.005628, -0.014806, 0.059833, -0.048188, -0.057278, -0.128971, -0.009649, -0.040882, 0.040156, 0.057941, 0.075666, 0.088565, 0.023836, 0.028673, 0.066055, -0.056973, 0.028586, -0.011703, 0.049122, 0.021673, -0.100982, -0.028172, -0.059499, 0.005623, -0.038687, 0.038385, -0.045828, 0.058253, -0.081635, -0.064490, 0.048731, -0.066659, -0.160283, -0.013296, 0.048260, -0.081082, 0.146743, 0.041531, -0.018828, -0.107528, -0.056579, -0.078907, -0.024666, 0.078807, -0.036496, 0.021495, -0.065796, 0.119508, -0.070000, 0.038146, 0.025168, -0.011130, 0.023162, -0.078076, 0.134110, -0.122887, -0.071939, -0.063865, 0.026495, -0.090763, 0.110223, -0.018612, -0.073783, 0.070844, 0.006154, -0.016200, 0.024145, 0.018980, -0.027177, -0.127069, -0.029517, -0.034410, -0.004239, -0.061369, 0.010044, 0.045201, -0.070050, -0.000841, -0.100733, -0.022724, 0.023188, 0.078417, 0.047568, 0.081125, -0.011703, -0.032229, -0.129816, -0.056315, 0.078229, -0.065519, -0.027533, 0.038553, -0.077342, -0.014275, 0.053284, -0.038188, -0.113149, -0.027261, -0.004367, 0.072859, -0.001779, -0.046326, -0.037242, 0.035273, -0.042660, -0.050138, 0.050434, 0.102263, 0.034849, -0.184492, -0.050461, -0.070510, -0.065404, 0.004022, -0.057614, -0.126554, 0.024064, -0.050399, 0.013065, 0.012425, -0.041356, -0.134218, -0.094917, 0.001690, 0.040458, 0.047159, -0.106508, -0.018987, -0.019455, -0.011856, -0.096385, -0.014005, -0.086200, -0.018164, 0.011985, 0.054541, -0.007436, -0.046966, -0.007488, -0.020597, -0.071979, -0.014625, 0.060498, 0.017438, -0.046236, -0.098351, 0.033843, -0.006417, -0.129055, -0.098622, -0.093556, -0.014697, 0.018319, -0.034075, -0.054235, -0.046857, -0.026156, 0.021589, -0.010139, 0.016821, -0.037345, 0.116298, -0.080032, -0.067884, 0.012872, -0.011397, -0.018931, 0.026250, -0.089147, -0.001903, 0.010090, 0.132998, -0.060965, -0.085030, -0.060639, -0.056364, -0.035465, -0.127831, 0.015606, -0.074462, -0.005544, -0.068957, 0.046449, -0.086330, -0.012603, -0.082004, -0.117010, 0.048684, -0.031492, -0.064006, -0.046639, -0.069808, -0.050286, 0.090209, -0.052699, -0.026423, -0.018488, 0.036691, -0.033819, -0.063499, 0.137955, -0.030882, -0.020109, 0.072221, -0.043745, 0.044606, -0.005556, -0.099426, 0.041952, 0.028182, -0.092963, -0.096173, 0.019346, -0.095328, -0.068932, -0.017693, -0.026763, 0.043324, -0.021115, -0.035485, 0.005930, -0.022532, -0.074279, 0.088808, -0.104667, 0.064799, 0.019775, -0.067078, -0.014434, -0.020884, 0.008876, -0.008904, -0.074224, -0.020308, -0.062500, 0.048448, -0.073500, 0.001498, 0.069641, 0.050864, -0.026757, 0.125927, 0.028181, 0.084187, -0.000511, -0.123227, -0.057238, -0.043651, -0.083715, 0.080893, 0.018578, -0.058951, -0.008505, -0.097347, -0.056705, 0.022824, -0.005706, 0.117858, -0.043508, 0.090180, -0.089432, -0.095643, -0.088594, -0.152568, -0.061503, -0.031947, -0.005448, -0.005902, 0.049872, -0.010965, -0.067014, 0.004835, -0.060075, 0.095651, -0.144315, -0.070748, -0.095052, 0.028240, -0.038928, -0.064277, -0.083431, 0.030517, -0.041354, -0.050716, 0.052629, -0.068237, 0.031427, -0.014004, -0.013929, 0.009465, -0.093110, 0.117796, -0.005033, 0.034095, -0.052736, -0.028902, -0.005827, 0.021224, -0.057974, -0.008905, -0.003964, -0.048983, 0.030055, -0.058860, -0.055180, -0.004130, 0.009610, 0.050254, 0.017659, -0.022502, 0.001583, 0.053765, -0.039341, 0.074821, -0.045782, -0.041464, 0.048093, 0.077864, -0.057131, -0.039910, 0.034560, -0.016306, -0.065110, -0.031812, -0.011313, -0.035654, -0.011269, -0.091166, -0.074539, 0.015209, -0.100601, -0.076104, -0.022497, -0.088469, -0.069046, -0.034331, 0.005348, 0.046140, 0.022205, 0.026882, 0.023319, 0.002629, 0.038270, -0.042153, -0.065917, -0.009443, 0.062001, -0.098069, -0.029147, -0.041776, -0.021410, 0.036256, 0.086030, -0.032598, -0.032321, 0.030187, -0.025840, 0.028869, 0.006134, -0.018116, -0.043985, 0.084097, 0.034182, -0.015990, 0.021510, -0.039514, -0.036587, -0.000551, -0.047041, 0.017478, -0.044576, 0.029663, -0.033072, 0.045138, -0.050483, 0.041991, 0.027627, -0.061959, 0.002664, -0.070472, -0.038597, -0.077485, 0.025256, -0.007948, -0.016386, -0.064853, 0.035619, 0.013204, -0.068504, -0.108223, -0.064518, 0.023422, -0.114383, 0.139713, 0.022439, -0.096535, 0.014931, -0.010828, -0.028497, -0.072424, 0.027524, -0.057675, -0.005220, -0.054485, -0.020382, -0.007691, -0.058670, 0.041173, -0.005312, -0.040566, -0.051326, -0.036791, -0.056307, -0.065251, -0.008716, -0.065359, -0.025858, -0.004741, 0.034219, 0.040921, -0.012617, -0.100385, -0.059865, 0.050355, -0.075146, 0.046534, 0.057637, -0.021474, 0.034043, -0.014749, -0.062555, 0.004959, 0.010498, 0.049457, 0.005266, -0.030115, 0.010730, 0.009790, 0.034836, -0.053574, 0.069973, -0.040219, -0.057181, -0.058389, 0.016645, -0.011767, -0.086257, 0.001311, 0.011531, -0.039425, 0.027308, -0.027393, 0.049271, -0.019905, -0.056747, -0.031338, -0.079278, 0.002838, -0.022288, 0.007963, -0.031374, -0.046416, -0.018405, -0.023699, -0.001097, -0.020119, 0.107821, -0.041356, 0.010854, -0.076691, -0.095031, -0.074690, 0.049549, 0.016949, -0.068721, 0.051532, -0.036639, -0.040257, -0.015062, -0.036576, 0.060312, 0.005254, 0.034574, -0.044725, 0.027216, -0.007746, 0.030657, -0.013915, -0.129942, -0.029581, -0.007347, -0.086749, 0.038458, -0.047191, -0.009184, -0.004774, 0.043529, 0.051046, 0.039564, 0.019046, -0.051241, 0.013909, -0.069711, -0.066116, -0.049822, 0.047454, -0.056034, -0.036928, -0.140422, -0.019218, -0.038814, 0.102466, 0.009581, -0.005314, -0.069584, 0.002451, 0.008590, 0.014017, -0.035718, 0.030785, -0.053764, 0.037071, -0.098005, -0.048848, -0.008080, -0.021399, -0.034789, 0.030486, -0.025485, -0.070068, -0.045872, -0.049218, -0.020967, -0.151260, -0.054825, -0.031289, -0.020578, -0.026312, -0.026344, -0.071513, -0.013684, 0.042277, -0.051347, -0.044932, -0.046644, -0.002615, -0.043923, -0.020330, 0.035787, 0.001567, 0.000544, -0.026975, 0.015855, -0.013403, 0.013222, -0.020440, -0.027687, -0.055849, 0.018843, -0.018155, 0.013469, 0.026430, -0.038038, -0.003469, 0.041605, -0.006536, 0.058962, -0.079651, -0.000943, 0.005300, 0.084589, 0.014519, 0.052868, 0.027427, 0.025502, 0.048705, -0.102661, 0.023260, 0.037824, -0.031291, -0.107944, 0.002667, -0.065874, -0.058374, 0.051629, -0.028741, -0.057765, -0.038135, -0.003586, -0.018138, -0.032879, -0.029282, -0.035931, -0.081484, -0.002991, 0.029659, -0.028128, -0.095437, 0.033979, -0.028527, -0.027444, 0.047019, -0.009720, 0.059101, 0.019969, -0.024505, 0.006486, -0.056482, -0.045081, 0.088361, -0.009602, 0.052496, 0.088921, -0.040595, -0.014679, 0.031478, 0.021217, -0.050064, -0.060849, 0.035060, -0.043317, -0.009586, -0.069423, -0.025781, -0.095633, -0.031084, 0.014966, 0.025155, 0.092650, -0.020475, 0.015566, 0.074766, 0.008110, 0.051616, -0.049870, -0.008411, -0.055707, -0.020167, -0.008520, -0.013035, 0.031292, -0.041761, 0.020355, -0.010691, -0.055884, 0.045159, -0.012974, 0.018334, 0.052564, 0.038922, 0.010197, -0.045917, -0.037018, 0.030081, 0.002647, -0.048437, 0.107416, 0.005787, 0.007980, -0.010777, 0.030923, -0.004033, -0.009583, 0.037876, 0.020150, -0.080204, -0.043093, -0.031272, -0.006968, -0.065084, -0.050228, 0.006630, -0.031749, 0.070576, -0.057652, 0.022752, -0.020294, 0.042358, -0.051160, 0.019803, -0.000540, -0.014776, -0.027188, 0.106502, 0.009980, -0.009856, -0.021479, -0.052336, -0.043259, -0.021795, -0.043944, 0.024931, -0.041363, 0.026461, 0.043788, 0.055555, -0.029620, -0.036950, 0.030699, -0.093166, -0.025483, -0.037112, -0.049220, -0.019301, -0.017845, -0.066699, 0.039633, 0.066475, -0.019780, -0.043654, 0.018040, -0.037966, -0.027633, -0.088614, -0.048538, 0.154368, 0.039184, -0.066512, -0.056830, 0.067511, 0.005411, 0.020124, -0.022162, 0.022996, 0.033637, -0.031659, 0.053052, 0.080177, -0.001518, 0.041537, -0.039659, -0.046235, 0.000103, 0.042011, -0.090694, -0.016772, 0.009624, -0.035882, -0.044624, -0.057184, 0.001307, 0.000473, 0.052815, 0.019095, 0.034549, -0.017963, 0.029497, 0.027700, -0.011830, 0.026879, -0.109512, -0.041768, 0.035898, -0.082122, 0.015829, 0.005649, 0.042768, -0.009723, -0.046947, -0.045634, 0.063854, 0.028111, 0.046058, 0.042238, 0.053790, -0.040352, -0.126498, -0.034851, 0.047811, 0.027451, 0.037159, -0.030246, -0.013936, 0.057859, -0.033310, -0.009853, -0.082341, -0.049318, -0.013564, -0.048982, -0.028802, -0.019008, 0.012738, 0.017829, 0.030056, 0.020740, -0.026471, 0.024307, 0.041186, -0.085157, -0.013602, -0.051461, -0.005012, -0.005000, -0.103550, 0.051523, -0.017500, 0.021092, 0.071463, -0.021039, -0.004429, 0.044168, -0.085573, -0.058429, 0.032739, -0.028623, 0.022137, -0.071804, 0.033921, -0.014059, -0.039833, -0.040592, -0.019970, 0.009944, 0.015974, 0.059259, 0.010963, -0.088046, 0.060450, -0.077762, 0.043078, 0.041125, 0.087556, -0.027895, -0.073645, 0.043351, -0.032651, 0.065614, -0.007077, -0.033351, 0.052232, -0.056617, 0.043481, 0.080861, -0.005492, -0.094426, -0.009007, 0.167212, -0.016250, -0.053406, 0.049982, 0.025783, 0.001632, -0.028909, 0.003383, -0.044613, 0.013321, -0.068968, -0.065984, 0.000915, -0.008226, 0.017494, 0.043023, -0.077931, -0.040359, -0.078011, -0.056298, -0.020883, -0.017678, -0.041765, -0.039420, 0.041604, -0.061008, -0.032015, 0.004175, 0.025296, -0.028223, 0.032274, -0.087738, -0.032836, -0.077023, 0.010255, 0.050338, -0.009003, -0.060156, -0.090089, 0.024912, -0.021133, -0.004327, -0.011846, 0.056043, -0.031014, 0.059790, -0.059508, -0.032654, -0.044813, -0.043298, 0.039287, -0.145521, -0.030794, 0.047285, -0.018679, -0.004350, 0.010885, -0.044219, -0.068962, 0.064550, 0.016079, -0.097771, -0.064699, -0.006255, -0.027247, -0.132277, 0.056984, 0.004509, 0.027786, 0.046356, -0.022476, -0.014826, -0.036749, 0.055384, -0.068181, -0.037577, -0.045528, 0.030968, 0.061187, -0.053814, -0.052963, -0.026087, 0.034284, 0.003211, -0.011430, -0.007831, 0.038487, 0.001737, -0.031421, -0.001223, -0.046447, -0.031806, 0.035765, -0.042623, -0.032546, -0.107783, -0.078684, -0.032575, 0.033198, -0.075618, -0.049330, -0.055026, -0.004401, -0.053714, -0.069151, -0.045564, 0.037801, 0.006669, -0.040558, -0.099999, 0.026012, -0.014630, -0.059436, 0.012347, -0.030250, 0.042127, 0.049460, 0.054620, -0.055998, -0.044719, -0.036478, 0.046786, -0.054942, 0.057123, -0.005991, -0.020113, -0.008893, -0.051253, -0.010756, 0.028370, 0.008825, 0.014175, 0.000936, -0.105411, -0.049502, 0.028609, 0.042259, 0.013660, -0.025378, 0.019675, 0.006016, -0.037579, 0.051940, -0.048143, -0.037766, -0.048834, 0.086401, -0.037263, 0.008594, -0.083823, -0.013237, -0.002679, -0.035262, -0.030562, -0.053251, -0.002623, 0.049476, -0.076979, 0.015293, -0.106672, 0.049713, 0.027693, -0.002111, 0.002069, 0.049140, 0.059761, -0.107418, -0.078835, -0.051738, 0.028174, 0.034104, -0.068585, -0.081836, 0.058505, 0.052327, -0.058343, 0.000991, 0.024253, -0.045842, -0.057909, 0.028271, -0.031456, -0.056584, -0.059993, 0.014597, 0.055008, 0.004978, -0.059469, 0.018218, -0.016546, -0.038141, 0.006172, 0.093128, 0.034614, 0.020585, 0.035272, -0.035444, 0.059786, 0.000001, -0.021240, 0.026218, -0.067114, -0.072628, -0.012140, -0.083590, 0.024547, 0.026521, 0.012225, -0.028448, -0.076354, 0.093132, -0.083385, 0.015652, 0.009358, -0.045384, -0.045952, 0.037005, -0.071603, -0.019381, 0.011198, -0.031188, -0.005055, 0.036167, -0.011040, -0.097904, -0.080996, -0.021872, -0.011991, -0.037678, 0.009223, -0.076593, -0.012164, 0.050702, 0.016698, -0.000831, -0.023730, 0.036530, -0.096167, -0.100298, -0.080263, -0.050667, 0.072829, -0.041241, -0.084170, -0.004050, 0.008271, -0.058837, -0.024358, -0.117122, -0.016855, -0.000742, 0.020439, -0.022080, -0.048813, -0.054021, 0.028100, -0.016648, -0.022490, 0.012356, -0.015182, -0.021539, 0.033746, -0.082526, -0.128281, -0.021757, 0.029247, 0.008669, -0.001452, 0.020872, -0.128693, -0.049285, -0.058384, -0.029824, -0.091323, 0.019272, -0.068471, -0.041645, -0.061103, -0.174939, -0.042261, 0.027925, 0.037647, -0.037925, -0.021876, -0.037025, 0.039632, -0.019286, -0.000579, 0.016031, -0.000470, 0.029051, 0.042747, 0.018872, -0.042006, -0.013370, 0.010056, 0.030043, 0.060118, -0.014174, -0.058666, -0.026398, -0.002816, -0.077691, 0.020266, 0.078138, -0.060514, 0.041850, -0.050326, -0.001633, 0.029649, 0.055573, -0.011459, -0.028964, -0.053438, -0.044626, -0.022250, -0.053011, -0.079133, -0.029754, 0.043844, -0.021643, -0.033186, -0.045815, 0.029073, 0.055200, -0.033130, 0.057207, -0.009716, -0.070749, 0.014969, 0.012496, -0.063902, -0.021139, -0.091922, -0.084624, -0.034199, -0.049070, -0.006086, -0.077594, -0.015464, 0.011657, 0.072792, 0.017096, 0.025830, -0.008898, 0.023861, -0.064412, -0.072412, 0.045928, 0.009613, 0.037087, -0.034517, 0.024733, 0.019073, -0.128854, -0.057955, -0.036791, -0.105092, -0.153920, -0.017232, -0.004706, -0.098116, -0.049742, 0.018539, -0.006997, -0.024921, -0.034826, -0.004083, 0.002700, -0.067912, -0.005870, -0.063639, -0.028239, -0.163650, -0.098413, 0.003563, -0.029007, 0.004511, -0.015958, -0.007827, -0.013601, 0.010542, -0.030040, 0.031941, 0.022150, -0.018562, -0.051012, -0.047894, -0.007946, 0.013225, -0.015309, 0.078759, -0.054810, -0.027558, -0.019950, -0.044635, 0.037296, -0.015363, 0.027618, 0.019815, 0.041275, -0.066971, 0.009621, -0.018568, -0.018924, -0.041022, -0.060359, 0.005489, -0.023672, 0.020758, 0.044671, 0.067138, 0.077588, -0.081789, -0.062725, 0.041609, -0.043830, -0.027084, -0.086357, -0.007694, -0.026673, -0.007507, 0.020130, 0.008523, 0.005047, -0.023753, -0.061559, -0.012355, 0.033044, 0.003651, 0.085360, 0.004197, -0.089349, -0.024021, -0.101628, -0.090773, 0.028533, -0.045526, -0.029688, -0.038340, 0.005105, -0.104210, 0.049140, 0.042378, -0.050778, -0.105047, -0.037811, -0.071797, -0.069117, -0.017801, -0.061144, -0.029388, 0.016694, -0.047164, 0.039047, 0.007254, -0.007719, -0.002368, -0.144939, 0.020033, 0.050754, 0.033694, -0.092493, -0.025542, -0.068298, -0.036310, -0.071863, -0.030570, -0.064097, -0.121717, -0.009608, -0.041141, -0.093160, 0.024675, 0.016404, 0.026258, 0.054545, -0.052406, 0.194548, -0.056541, -0.000991, 0.055076, 0.000788, 0.107427, 0.077608, 0.053667, -0.093291, 0.113948, -0.014785, 0.016171, 0.021810, 0.061026, -0.078097, 0.034950, -0.085995, -0.049582, 0.006181, -0.041375, -0.015347, -0.096530, -0.010407, -0.002305, -0.062089, 0.107949, -0.081143, -0.065052, 0.018643, -0.011289, 0.045833, -0.018786, -0.057225, 0.028864, 0.055845, 0.035979, -0.055507, -0.042518, -0.010652, -0.009299, -0.083990, 0.067573, 0.040766, -0.003317, -0.047525, 0.050685, -0.072810, -0.089724, 0.008653, -0.017253, 0.066601, 0.022022, 0.056543, 0.041371, 0.026775, -0.083636, 0.053629, 0.010841, -0.051302, -0.025853, 0.089053, -0.017006, -0.079062, -0.074395, -0.056579, 0.037270, -0.046993, -0.078722, -0.065455, -0.011145, 0.119032, -0.050291, -0.036435, -0.000447, -0.051150, -0.013817, 0.004792, -0.083261, 0.002852, -0.011294, 0.141814, 0.043494, -0.048719, -0.091687, 0.018106, -0.035869, -0.013401, 0.257510, -0.052464, 0.042465, 0.022969, 0.057901, 0.037051, -0.034387, 0.062450, -0.048979, -0.060350, -0.093782, -0.083801, 0.049798, 0.084666, 0.092729, -0.009625, -0.024833, -0.008560, 0.056544, 0.031521, -0.063865, -0.057432, 0.021491, -0.088993, -0.046886, -0.022607, -0.002234, 0.029743, 0.028290, -0.042826, -0.017595, 0.038790, -0.073017, 0.061919, -0.123016, -0.017496, -0.115303, 0.003896, -0.040097, -0.015226, 0.037192, -0.012201, -0.122593, -0.131954, 0.103753, -0.000618, -0.195157, 0.054219, -0.053845, -0.134831, 0.065532, -0.035411, 0.017654, -0.057996, 0.028103, -0.035214, -0.007614, 0.046756, 0.077368, -0.064125, 0.053240, -0.008890, -0.031710, -0.029356, -0.044073, 0.060533, -0.024366, 0.055505, -0.035533, -0.021554, 0.007848, -0.054686, -0.010978, -0.033633, -0.132828, -0.149202, -0.013499, 0.113365, -0.021898, -0.069082, -0.167524, 0.050995, 0.019246, -0.125828, 0.036307, -0.038806, -0.047986, 0.038869, 0.007681, -0.147859, -0.010586, 0.006187, -0.048775, -0.061377, -0.064399, -0.049739, -0.063982, -0.033895, -0.077065, -0.037164, 0.062687, 0.020053, 0.111535, -0.044381, -0.042287, 0.004592, 0.025130, -0.083729, -0.100378, -0.033485, -0.027804, 0.043819, 0.086527, -0.033612, 0.043661, -0.065376, -0.029317, -0.032526, -0.004246, 0.033062, 0.047427, 0.000593, 0.081232, 0.045342, 0.046435, -0.009796, -0.033656, 0.003209, 0.027570, 0.014522, -0.024723, -0.033850, -0.027615, 0.010995, 0.014937, 0.009186, -0.071271, 0.013896, -0.030931, -0.059247, -0.088826, -0.059132, -0.051057, 0.023327, -0.005925, 0.075231, -0.008776, 0.029755, -0.024824, 0.015854, 0.082884, -0.068139, 0.026672, -0.032952, -0.078143, 0.047592, 0.027374, -0.032162, 0.026697, -0.211765, -0.063203, 0.038965, -0.031341, -0.036798, -0.018522, 0.011700, 0.010850, -0.027457, 0.055742, -0.041545, 0.004901, -0.085454, -0.031242, 0.085596, 0.031418, -0.001046, -0.152154, 0.021999, -0.021420, 0.040137, -0.015282, -0.123665, -0.010237, -0.060965, 0.035563, -0.019125, -0.080765, -0.005314, 0.057946, 0.021449, -0.010708, -0.037237, 0.052583, -0.031713, 0.051813, 0.017146, -0.100258, 0.030435, -0.060867, -0.087205, 0.044120, -0.033227, 0.026428, -0.022785, -0.135918, -0.051791, -0.032137, 0.006790, 0.131783, -0.033351, 0.117479, -0.003419, -0.090764, -0.082497, -0.072349, -0.078458, -0.018983, 0.044555, 0.066247, 0.022521, -0.067058, -0.031781, -0.016099, -0.065312, 0.172849, -0.062709, -0.013295, 0.207553, -0.054839, -0.052565, -0.009897, 0.060956, -0.041477, -0.039195, 0.006924, -0.020545, 0.008872, 0.071831, -0.040125, -0.036325, 0.090904, -0.011682, -0.098378, -0.064508, 0.037170, -0.048716, -0.017058, 0.074266, -0.008396, -0.034206, -0.015635, -0.053864, 0.001130, -0.001194, -0.034568, 0.005998, 0.008784, -0.069021, -0.053254, 0.006735, -0.050686, -0.010805, 0.056545, 0.055201, -0.007899, -0.000109, -0.022535, -0.005074, 0.009170, 0.007025, 0.128567, 0.070862, 0.052764, 0.147491, -0.049683, -0.023905, 0.032378, -0.023771, 0.043060, 0.020489, 0.011106, 0.095528, -0.049149, -0.087748, 0.023779, 0.006996, 0.050866, -0.028645, 0.051304, -0.076321, -0.075981, -0.004006, 0.097408, -0.024517, 0.038255, -0.007109, 0.002195, -0.012713, -0.009154, -0.051861, 0.043442, 0.021001, -0.075387, -0.017008, 0.163428, 0.151835, -0.111666, -0.020939, -0.055993, 0.075403, 0.024777, -0.008455, 0.034277, 0.027488, -0.073943, 0.079737, -0.027880, 0.031365, -0.055198, 0.008336, -0.070811, 0.028304, -0.031673, 0.031577, -0.029318, -0.026651, -0.055558, -0.036993, -0.009035, 0.018839, 0.044263, 0.046676, 0.041699, -0.009175, -0.038026, -0.052620, -0.032551, 0.028103, -0.056447, -0.051186, -0.054846, -0.130555, -0.039558, -0.002051, -0.047583, -0.020334, 0.001799, 0.010303, -0.006501, -0.061266, -0.091996, -0.063424, -0.055278, -0.027865, -0.029512, 0.046944, -0.070843, -0.002392, -0.001148, 0.009335, -0.048298, 0.019506, -0.026967, -0.016290, -0.014686, 0.035188, 0.025487, -0.039796, 0.012236, -0.004610, 0.035143, 0.009837, -0.027285, 0.006610, 0.057921, 0.021999, -0.044756, -0.038521, -0.004023, -0.097415, -0.020247, -0.010709, -0.025158, -0.122152, 0.005971, 0.017427, -0.063786, 0.049203, -0.088936, 0.129712, -0.013308, 0.012153, 0.123926, -0.018006, -0.086217, 0.011013, 0.044853, -0.050986, -0.049116, -0.000860, -0.042369, 0.045579, -0.057376, 0.044130, -0.018959, 0.005465, -0.002321, 0.174958, -0.019490, 0.005120, -0.056792, 0.115501, -0.049324, -0.070652, 0.013332, -0.108012, -0.074348, -0.046094, 0.063419, 0.005077, 0.029876, 0.081903, -0.072014, -0.000813, -0.048604, -0.101248, -0.021385, -0.016490, -0.029082, 0.049976, -0.052273, 0.020571, 0.118662, 0.054338, -0.033958, -0.016765, 0.032947, -0.028244, -0.005554, 0.008206, 0.001883, -0.018956, 0.032202, 0.125719, 0.031056, 0.067222, -0.045470, -0.084153, -0.036906, -0.025340, -0.046476, -0.073876, 0.019931, 0.089997, -0.046651, 0.001806, 0.040690, -0.004755, 0.018249, -0.019682, -0.154496, 0.028633, -0.068493, -0.058105, -0.038481, -0.041503, -0.063282, 0.022701, -0.021017, -0.033315, 0.101691, 0.072165, -0.111002, 0.000579, -0.014911, 0.008666, -0.022503, -0.114990, -0.063191, 0.043709, -0.059212, -0.020256, -0.015350, -0.143788, -0.015232, 0.081204, 0.036269, -0.007064, -0.047201, 0.007638, -0.022822, 0.021532, -0.027827, 0.014358, -0.042914, -0.021364, -0.034156, -0.078591, -0.053191, 0.002962, 0.021616, 0.013087, -0.079357, -0.043824, 0.007905, -0.077043, -0.000195, 0.077485, 0.024426, -0.032682, -0.084392, -0.068236, -0.064986, 0.026441, -0.005585, 0.083868, 0.018410, -0.037001, 0.001200, 0.025614, -0.009802, -0.053129, -0.055443, 0.021221, 0.032608, 0.095745, -0.027498, 0.030994, 0.038117, -0.086504, 0.008128, -0.046345, -0.056229, -0.012374, 0.064968, -0.021619, -0.122459, 0.011039, -0.040211, -0.027947, -0.034107, -0.064560, 0.052563, 0.071782, -0.050182, 0.055767, -0.015403, -0.048081, -0.046833, -0.018423, 0.010635, 0.007728, 0.053058, 0.073272, -0.040959, 0.064196, 0.032800, -0.013520, 0.065076, 0.006553, 0.047893, -0.101628, 0.038737, -0.013072, 0.007367, 0.048545, -0.042766, -0.067069, -0.085023, 0.007058, -0.006949, -0.025782, 0.039321, -0.000729, 0.096354, -0.030016, 0.049453, 0.038717, 0.139017, -0.013875, -0.047340, -0.037800, -0.018954, -0.046420, -0.060582, -0.066605, -0.001013, -0.051686, 0.010816, -0.037926, -0.050338, -0.011110, 0.010868, 0.001945, 0.042954, 0.020697, -0.025829, -0.054856, -0.014662, -0.004170, 0.016540, 0.061922, -0.051190, 0.013005, 0.050039, -0.044650, 0.035860, -0.032220, -0.001529, -0.033366, -0.082304, -0.050251, -0.025247, -0.046426, -0.025282, 0.000596, 0.036723, 0.056235, 0.011875, -0.028808, -0.058611, -0.006064, 0.053039, 0.147430, 0.086074, -0.025188, -0.013304, 0.059633, 0.050075, 0.038427, 0.130852, -0.020584, 0.010835, -0.062576, -0.033973, 0.214160, -0.050995, 0.067686, -0.056669, 0.133342, -0.040062, -0.051672, -0.041135, -0.009696, 0.016761, 0.047138, -0.015924, 0.018771, -0.040290, -0.008432, -0.040874, -0.068422, -0.052418, -0.025756, -0.033115, -0.152364, 0.009264, 0.041816, 0.047732, 0.006941, 0.056750, 0.043440, -0.002703, -0.032254, 0.002963, 0.025549, 0.146710, 0.026432, -0.041480, -0.039417, -0.044345, -0.064250, 0.074828, 0.010934, -0.080936, 0.049992, -0.071627, -0.056751, 0.001661, -0.026634, 0.005047, 0.007404, -0.084714, -0.035431, -0.036082, 0.006626, -0.070094, -0.086694, -0.059489, -0.086461, 0.049894, -0.075303, -0.024158, 0.068284, -0.059437, 0.029994, 0.022438, 0.058122, -0.121063, 0.070188, -0.046874, 0.034298, 0.070377, -0.002278, -0.118225, -0.071475, 0.006086, -0.122562, 0.093926, -0.060618, -0.002653, -0.038643, 0.023209, 0.027932, 0.003212, -0.058562, -0.024115, -0.052546, 0.051797, -0.019878, 0.021019, -0.108936, -0.027713, -0.099738, -0.042135, 0.038177, 0.000355, 0.096039, -0.052022, 0.030956, 0.094164, -0.058538, 0.039671, 0.086757, 0.014920, 0.016636, -0.048333, 0.017311, 0.030099, 0.043885, -0.013102, -0.107403, -0.001304, 0.044494, -0.030026, -0.032065, 0.005425, 0.036699, -0.016288, 0.064453, 0.001369, -0.031336, -0.058331, -0.046519, 0.075704, -0.053302, 0.021478, 0.022641, 0.028522, 0.026269, 0.020805, 0.064696, -0.037500, -0.051863, -0.044713, 0.005749, -0.040579, 0.020447, 0.178045, -0.035549, -0.090129, -0.020278, 0.007164, -0.067896, -0.011750, 0.043563, -0.013228, 0.002037, -0.044841, -0.001210, 0.060763, 0.028835, -0.034061, -0.022014, -0.006284, 0.032435, -0.027576, -0.010869, 0.015713, 0.019194, -0.053829, -0.070169, -0.023544, 0.039860, -0.021339, 0.206991, -0.036724, -0.022980, -0.036702, -0.028836, 0.082508, -0.017695, 0.001057, -0.040106, 0.041867, 0.053078, -0.032217, -0.045433, 0.062794, -0.116584, 0.064057, -0.082692, 0.065363, 0.021158, 0.007203, 0.021949, 0.015012, -0.062381, -0.081845, 0.023755, 0.003053, 0.094206, 0.048381, 0.020483, -0.035105, 0.007099, -0.042150, -0.077121, 0.105827, -0.042978, 0.024999, 0.039259, -0.036679, -0.055034, -0.027415, -0.050472, 0.133710, -0.086366, -0.051837, -0.033874, -0.001918, -0.068510, -0.066124, 0.055830, 0.024121, -0.030996, -0.059586, -0.126845, 0.014853, 0.023979, -0.016813, -0.036059, 0.005497, -0.001744, -0.011228, -0.054162, 0.000212, -0.059108, 0.006150, -0.100591, -0.012706, -0.002079, -0.036095, 0.059025, 0.058427, -0.047658, -0.085878, -0.003825, -0.021719, 0.097969, -0.008472, -0.101525, 0.152424, 0.015084, 0.016755, -0.011717, 0.040678, 0.076988, 0.007861, -0.133235, -0.019077, -0.037622, -0.008812, -0.020324, 0.054178, -0.066352, -0.011137, -0.015077, -0.011100, -0.032354, 0.051316, -0.017881, 0.043528, -0.012103, 0.021915, 0.032739, 0.038686, -0.050713, 0.010282, -0.068668, -0.108241, -0.054484, -0.060317, 0.083591, -0.116136, 0.032526, -0.033501, -0.056013, -0.052116, 0.070448, -0.049598, 0.011613, 0.008910, 0.038162, -0.101442, 0.108809, -0.000966, 0.016464, 0.021935, 0.008834, -0.077715, -0.075100, 0.027921, -0.068926, 0.079474, -0.022689, -0.001986, -0.051277, 0.097827, -0.094835, 0.021149, -0.001290, 0.098269, 0.018245, 0.014117, -0.019221, -0.139288, -0.140260, -0.216663, -0.067123, -0.007954, -0.070305, -0.131392, 0.028992, -0.075814, -0.216474, -0.041121, -0.079205, -0.017008, 0.004406, -0.133763, -0.120335, 0.027415, -0.028227, -0.005272, -0.010618, -0.044691, -0.011186, -0.082832, -0.136533, -0.028127, -0.131424, 0.040462, -0.257600, 0.000879, -0.017354, -0.054879, 0.017777, -0.056820, -0.048491, -0.042182, -0.022618, -0.043016, -0.107275, -0.080198, -0.235750, -0.134751, -0.241967, -0.109410, -0.032236, 0.106443, -0.030918, -0.056977, 0.003744, -0.189146, -0.026825, -0.003702, -0.099006, 0.088972, -0.011714, -0.020084, -0.060780, -0.014608, 0.001902, -0.080473, -0.110178, -0.093512, -0.045460, -0.074499, -0.224542, -0.052300, -0.065561, -0.050999, -0.040666, -0.126406, -0.118581, -0.060659, 0.038766, -0.145522, -0.134856, -0.132665, -0.054770, -0.015885, -0.073237, -0.057602, -0.016430, -0.018919, 0.001127, -0.109499, -0.043953, -0.011362, -0.004470, -0.077645, -0.120693, -0.002513, -0.060660, 0.059077, 0.040595, -0.074257, 0.111706, -0.149191, -0.084908, -0.004905, -0.068535, -0.062124, -0.180972, -0.089743, 0.020816, 0.047279, -0.317862, 0.037405, -0.157970, -0.065703, -0.029378, 0.025230, 0.000216, 0.004594, -0.044993, -0.091305, -0.060427, 0.008613, -0.098845, -0.142697, 0.020872, 0.006225, -0.083229, 0.082263, -0.193704, -0.027010, -0.017073, 0.027769, -0.056129, -0.064507, -0.072746, -0.066520, -0.058807, 0.085610, -0.191552, -0.204948, -0.080138, -0.101093, -0.058193, -0.079196, -0.008175, 0.080279, -0.115049, -0.035359, -0.113528, -0.097297, 0.002104, -0.049830, -0.012998, -0.246174, -0.133591, -0.031280, -0.073730, -0.082934, -0.022443, 0.032028, -0.055307, 0.015335, -0.023204, -0.093992, -0.038545, -0.074008, -0.230947, -0.070076, -0.038155, -0.001173, -0.199060, -0.107210, -0.134738, -0.166502, -0.089758, -0.236186, -0.100593, -0.000214, -0.058338, -0.182355, -0.042893, -0.105570, 0.046571, -0.057049, 0.107167, -0.030489, -0.093372, -0.087654, -0.008097, -0.068988, -0.047442, -0.035328, -0.062753, -0.105874, -0.001612, -0.098158, -0.035195, -0.012225, -0.198811, -0.058699, -0.065595, -0.060039, -0.019482, -0.261605, -0.062722, -0.174505, 0.044461, 0.000418, -0.073597, -0.014742, -0.119996, 0.027673, -0.306784, -0.044464, 0.020495, -0.108272, -0.011942, -0.160995, -0.068014, 0.017439, 0.049686, -0.027048, -0.050954, -0.090613, -0.064160, -0.088138, -0.003039, -0.062957, 0.006673, 0.000549, -0.068937, -0.048703, -0.194248, -0.016856, -0.058878, 0.130419, 0.003473, -0.077479, -0.013790, -0.062568, -0.069191, -0.051060, -0.138878, -0.026250, -0.089663, 0.114139, -0.073663, -0.096216, -0.264539, -0.038320, -0.150481, -0.181797, -0.094030, -0.012894, 0.048350, -0.039397, -0.064724, 0.030703, 0.023465, -0.078914, -0.024402, -0.044427, -0.008087, -0.052390, 0.035408, -0.043568, -0.035483, -0.036130, -0.169305, -0.092193, -0.112367, -0.092931, -0.069909, -0.079447, -0.067674, -0.030093, -0.162978, -0.089309, -0.095786, -0.105337, -0.040179, -0.194382, -0.109255, -0.119321, 0.097332, 0.077535, -0.065376, -0.095971, -0.122401, 0.011910, -0.028561, 0.022962, 0.006196, -0.245600, 0.052920, 0.006687, -0.045832, -0.079456, -0.059968, 0.073262, -0.115019, -0.082959, -0.000781, 0.163152, -0.036403, -0.069456, -0.007862, -0.024953, -0.079295, -0.191691, -0.078663, 0.021091, -0.227016, -0.043179, -0.138465, -0.013539, -0.114283, -0.060111, 0.019287, 0.047823, -0.048238, -0.058352, -0.014305, -0.051256, -0.041274, 0.004132, -0.111296, -0.083784, -0.049828, -0.195085, -0.028649, -0.113048, 0.026562, -0.027709, -0.071833, -0.187459, -0.028762, 0.022646, -0.046769, -0.168483, -0.192737, -0.069680, -0.117937, -0.061608, -0.043799, -0.025224, -0.027796, -0.010183, -0.078827, -0.052158, -0.122967, 0.003863, -0.084815, -0.052506, -0.064414, 0.019364, -0.000156, -0.004532, 0.157568, -0.002007, -0.116468, -0.030266, -0.046671, 0.014290, -0.095026, 0.077296, -0.113064, -0.047836, -0.046997, 0.011932, 0.016311, -0.051419, 0.015563, 0.022635, -0.005580, -0.036960, 0.011924, -0.036943, -0.033903, -0.009504, 0.027408, -0.051750, 0.011636, -0.006321, -0.055989, -0.080723, -0.063392, -0.191854, 0.094341, -0.168875, 0.094913, -0.119573, -0.234446, -0.114735, -0.091197, -0.073302, -0.030044, 0.069192, -0.100611, 0.090918, -0.035427, -0.049440, -0.019807, -0.226882, -0.125111, -0.067501, -0.065617, -0.132148, -0.067738, 0.092646, 0.011500, -0.074131, 0.049097, -0.137780, -0.116282, -0.041184, -0.040251, -0.022875, -0.067993, -0.026388, -0.093414, -0.022007, -0.097562, -0.150413, -0.045008, -0.030805, -0.008501, -0.045966, -0.048500, -0.090365, -0.091777, -0.057220, -0.153665, -0.061367, -0.029407, 0.128637, 0.101573, -0.137034, -0.071715, -0.186157, -0.122058, 0.088682, -0.065063, 0.095647, -0.059457, -0.030371, -0.047643, -0.044364, -0.044645, -0.163671, -0.162538, -0.096962, -0.258163, -0.078400, 0.031680, -0.106692, -0.003206, -0.046805, -0.108745, -0.059493, 0.011153, -0.105725, -0.052198, -0.027984, -0.036291, -0.047214, 0.003807, -0.070586, 0.051100, -0.084418, 0.059150, -0.143746, -0.002402, -0.041341, -0.074525, -0.307251, -0.074497, -0.021811, -0.052556, -0.047454, 0.004429, -0.050418, -0.053955, -0.200399, -0.108571, -0.273987, -0.110818, 0.011381, 0.042350, -0.232437, -0.067009, -0.001332, -0.097111, -0.099113, 0.104921, -0.083181, 0.007801, -0.037268, -0.039062, -0.042396, 0.011687, -0.073068, -0.004040, -0.121645, -0.072308, -0.017030, -0.004403, -0.045735, -0.066902, -0.016052, -0.066869, -0.097706, -0.071623, -0.033760, -0.008265, -0.089338, -0.122949, -0.010282, 0.016879, -0.032930, 0.020217, 0.042862, -0.015917, -0.167615, -0.072399, -0.098245, -0.173154, -0.086275, -0.012994, -0.057169, -0.219174, -0.077715, -0.051647, -0.019255, -0.036295, -0.239088, 0.007132, 0.002907, -0.101527, -0.026322, -0.174124, -0.089557, -0.156273, -0.074191, 0.044921, -0.178879, -0.178034, -0.080824, -0.051061, -0.007920, 0.051420, -0.003184, -0.188301, -0.034439, -0.054429, 0.028831, -0.255539, -0.127128, -0.024446, 0.016956, -0.176738, -0.081588, 0.011119, -0.075282, -0.028418, -0.006992, 0.060621, -0.028167, -0.028466, -0.017587, 0.011511, -0.109716, 0.012165, -0.189773, 0.004074, 0.013619, -0.055732, 0.020354, -0.011178, -0.136734, -0.018203, 0.093006, -0.116100, -0.227026, -0.084893, 0.075513, -0.147215, -0.069600, -0.038842, -0.074885, -0.106524, -0.029464, -0.131731, 0.002613, -0.165230, 0.053779, -0.001308, 0.047918, -0.116434, -0.170997, -0.085773, -0.007947, -0.180840, 0.016133, -0.187137, -0.131900, -0.029316, -0.083808, 0.006222, -0.033325, -0.097141, -0.079205, 0.004509, -0.062909, -0.044813, -0.070630, -0.106283, -0.020437, -0.055688, -0.118819, 0.026292, -0.175671, -0.011704, -0.036917, -0.146298, 0.011920, -0.036205, -0.029080, -0.052207, -0.094720, -0.056330, -0.005100, 0.002046, 0.077170, -0.091039, 0.047166, 0.007676, -0.032784, 0.024435, 0.026957, -0.090764, -0.064824, -0.034536, -0.041221, -0.063092, -0.003542, 0.031172, -0.021564, -0.044462, -0.102838, 0.125246, -0.015248, -0.010700, -0.265452, -0.058393, -0.029818, -0.206248, -0.043016, -0.048019, -0.048757, -0.047849, -0.041496, -0.123704, -0.021396, 0.035586, -0.073480, -0.083714, -0.108823, -0.050442, 0.026409, -0.084831, -0.036976, -0.087426, -0.071380, -0.076160, -0.080451, -0.116149, -0.136749, -0.041344, 0.072267, -0.006150, 0.021261, -0.110958, -0.108982, -0.114580, -0.015877, -0.108073, -0.038731, 0.026936, -0.035091, 0.005634, -0.050048, 0.008861, -0.094915, -0.059489, -0.091176, -0.048168, -0.062011, -0.043047, -0.260580, 0.001920, -0.025064, -0.027854, -0.167023, 0.050445, -0.312416, -0.062079, -0.044039, -0.033847, -0.029103, -0.073964, -0.276927, -0.058498, -0.060322, -0.050647, 0.026420, -0.067432, -0.046036, -0.036605, 0.021040, -0.091314, -0.084891, -0.274403, 0.018752, -0.110477, 0.061086, -0.047116, 0.064337, -0.089875, -0.031460, -0.093952, -0.054936, 0.004450, -0.108555, 0.055532, 0.012272, -0.076081, -0.182792, -0.070996, 0.043535, -0.094123, -0.059035, -0.051654, -0.092303, 0.008631, -0.074074, -0.169173, -0.042527, -0.152860, -0.024166, -0.016936, 0.078360, -0.025243, -0.066497, -0.193022, -0.133604, -0.106405, 0.014136, -0.085178, -0.143537, -0.034306, 0.042317, -0.060663, -0.031738, 0.074420, -0.088452, 0.020693, 0.013155, -0.026140, 0.012659, -0.010880, -0.163437, -0.067099, -0.130081, 0.016741, 0.023184, -0.123184, -0.181626, -0.034885, -0.118022, -0.138220, -0.033194, -0.031318, -0.033607, -0.118880, 0.046737, -0.018189, -0.032766, -0.058378, -0.022813, -0.017494, -0.096621, -0.030036, -0.067692, -0.201650, 0.085627, -0.009083, -0.017875, -0.297608, 0.048642, -0.102329, 0.086569, -0.059522, -0.039305, -0.021544, -0.111997, -0.049828, -0.106849, -0.053079, -0.046722, 0.037525, -0.082797, -0.213914, -0.093523, 0.028319, -0.040565, -0.210737, 0.011833, 0.021425, -0.072890, -0.114910, -0.001919, 0.132163, -0.025848, -0.010649, 0.028678, -0.013689, -0.055577, -0.100874, -0.056272, -0.049217, -0.107011, -0.193937, 0.006729, -0.071857, -0.026988, -0.011933, 0.019128, -0.028068, -0.005423, -0.063825, -0.054708, -0.078512, -0.048961, -0.076800, -0.016931, -0.170894, -0.053812, -0.028304, -0.087425, -0.009683, -0.046607, -0.118959, -0.045943, -0.089734, 0.015671, 0.072366, -0.113117, 0.143542, 0.038795, -0.047562, 0.016604, 0.054502, -0.010068, -0.085432, 0.008405, -0.142927, 0.040498, -0.173235, -0.152115, -0.053125, 0.045000, -0.077608, -0.071945, -0.087043, 0.003956, -0.174529, -0.037818, 0.016295, -0.030988, -0.001088, -0.066850, -0.132490, 0.057261, 0.044182, -0.045069, 0.020789, -0.049942, 0.011445, -0.108275, -0.135410, -0.080771, -0.086122, -0.078658, -0.047863, -0.021433, -0.054276, 0.038922, -0.024002, -0.047699, -0.092900, 0.120490, 0.114505, -0.130849, -0.139952, -0.074148, -0.032428, 0.070761, -0.067243, -0.079600, 0.059012, -0.079172, -0.064182, 0.003457, -0.049222, -0.012660, -0.050501, -0.038698, -0.121507, -0.020425, -0.066579, 0.015957, -0.054982, -0.023061, -0.012044, -0.073363, -0.127265, -0.070491, -0.043124, -0.071764, -0.089815, 0.000772, -0.273480, -0.127691, -0.130202, -0.093500, -0.062768, -0.087740, -0.008137, 0.004927, -0.105788, -0.071129, -0.099531, -0.047567, 0.012178, 0.179336, 0.022404, -0.109877, -0.059627, -0.007590, -0.083402, -0.024952, 0.014701, -0.028451, -0.168316, -0.025727, 0.001805, -0.025163, -0.066703, -0.069352, 0.022233, -0.050381, -0.006471, -0.028009, 0.129355, 0.052263, 0.068933, -0.052881, -0.025853, 0.089178, -0.207722, -0.121516, -0.195841, -0.098323, 0.064877, -0.072171, -0.067184, -0.042226, -0.023481, -0.003250, -0.112816, 0.027062, -0.042962, -0.056689, -0.001926, -0.031804, -0.079703, -0.070596, -0.059414, -0.082193, -0.113767, -0.041428, -0.010825, 0.003004, -0.047331, -0.002810, -0.034390, -0.070814, 0.058350, -0.348842, -0.051248, 0.040663, -0.010413, -0.211957, -0.054112, -0.093049, -0.060771, -0.081721, -0.059620, -0.360002, -0.157251, -0.026673, -0.131512, -0.034410, -0.002914, -0.203386, -0.168576, -0.043249, -0.299155, 0.009610, -0.100530, -0.099528, 0.020010, -0.099036, -0.022509, -0.032966, -0.082076, -0.307881, -0.005578, 0.030772, 0.008333, -0.039635, 0.115676, -0.036622, 0.011369, -0.042783, -0.002581, -0.009361, -0.069790, 0.023749, 0.007701, 0.009249, 0.014441, 0.039436, -0.008241, 0.039999, 0.019680, -0.058053, -0.034101, 0.035051, -0.081468, -0.053030, -0.064046, 0.036227, -0.039281, -0.009415, 0.031356, -0.067011, 0.145602, -0.057864, -0.078059, -0.038197, 0.002640, -0.024893, 0.095646, -0.008470, -0.034667, -0.026269, -0.042077, 0.038182, -0.149906, -0.067800, 0.028686, 0.055143, 0.040812, 0.030068, -0.006305, -0.015785, -0.073677, 0.052821, 0.005910, -0.018952, -0.029184, -0.085646, -0.075885, 0.036635, -0.039148, 0.002890, -0.024606, -0.145552, -0.052260, -0.027406, -0.006346, 0.016297, -0.017283, 0.148743, 0.017871, -0.094696, -0.103702, -0.022983, -0.010019, 0.022426, 0.072679, 0.004435, -0.099726, -0.060332, -0.051930, -0.066914, -0.003446, 0.035558, 0.008699, -0.028839, 0.150336, 0.021356, -0.022776, 0.012163, 0.011885, 0.022644, -0.175879, 0.021651, -0.022787, -0.014086, -0.008559, 0.009957, 0.029150, 0.053565, 0.051346, 0.014028, 0.038273, -0.015051, -0.032818, 0.104398, 0.013020, 0.158879, 0.045321, -0.063281, 0.001215, -0.045204, 0.001845, 0.025051, -0.046509, 0.049436, 0.015378, -0.083483, -0.037967, 0.049652, -0.010117, -0.081599, 0.063537, -0.132966, -0.041144, 0.022041, 0.012476, -0.029055, 0.108374, 0.034412, -0.044941, -0.046956, -0.030483, 0.111881, -0.026376, -0.002557, -0.036081, 0.013620, -0.055433, -0.071572, -0.042349, 0.059105, 0.003858, -0.040213, 0.007498, -0.011084, 0.001961, 0.034275, -0.108767, -0.030036, -0.000014, -0.127193, -0.015742, 0.037221, 0.004537, -0.042776, 0.069779, -0.014538, 0.042171, -0.079126, 0.007285, -0.048477, -0.040161, -0.057675, -0.051591, 0.058155, 0.084365, -0.030297, -0.140720, 0.022009, -0.116807, -0.024193, -0.030957, -0.049631, -0.020872, -0.056993, 0.050941, 0.037165, 0.033620, 0.015149, -0.015758, -0.076048, 0.010457, -0.101498, 0.009879, -0.117139, 0.029464, -0.022909, 0.052811, 0.002603, -0.056514, -0.040799, -0.005622, -0.038084, -0.003440, 0.080666, -0.092763, 0.035913, 0.066393, 0.003485, 0.069730, -0.182495, -0.001342, -0.089103, 0.032059, -0.053364, -0.006247, -0.008305, -0.007602, 0.045414, -0.075847, -0.020047, 0.059648, -0.063760, 0.012130, -0.033339, 0.010523, 0.029612, 0.116552, -0.009146, 0.001623, 0.004435, -0.081916, 0.030693, 0.036820, 0.010007, 0.036432, 0.024308, -0.032862, -0.021101, -0.013855, 0.062942, -0.037166, 0.013606, 0.015279, -0.018948, -0.037109, -0.006643, -0.142712, 0.034371, 0.075079, 0.044232, -0.018668, 0.044588, 0.010453, -0.097853, -0.043118, -0.021524, -0.053405, -0.017348, -0.015896, -0.059521, -0.013242, -0.009815, 0.040540, -0.039378, -0.040600, -0.045816, -0.100940, -0.050309, -0.094205, -0.053324, 0.053056, -0.014761, -0.029755, 0.029123, 0.162792, 0.026951, -0.056839, -0.117201, 0.037916, -0.010115, 0.055286, -0.040668, -0.090839, 0.039514, -0.050333, -0.005007, 0.022296, -0.105599, 0.043931, -0.025391, -0.005314, 0.055151, -0.014502, 0.027178, -0.019637, -0.041993, -0.015028, -0.036648, 0.036012, -0.148274, -0.038740, 0.069336, -0.074676, 0.071279, -0.089271, 0.014207, -0.020597, -0.028124, -0.034899, 0.090069, -0.003337, -0.099907, -0.064228, -0.020221, -0.029865, 0.016801, -0.068956, -0.045881, -0.033792, -0.046597, 0.103203, 0.049609, -0.010129, 0.000699, 0.006562, 0.034917, 0.002973, -0.039647, 0.002431, -0.021338, -0.049070, -0.075124, -0.020487, -0.032361, -0.034600, -0.022832, -0.009054, -0.067532, -0.014061, -0.021396, -0.068198, -0.053041, 0.005188, -0.014081, -0.044494, -0.041121, -0.044517, -0.083758, -0.016012, -0.067616, -0.001232, 0.035822, 0.031943, 0.015395, -0.031335, -0.029812, -0.070563, -0.017350, 0.034522, 0.020331, -0.062687, 0.053194, 0.064599, 0.050084, -0.046387, -0.024209, -0.095297, -0.060990, -0.030486, -0.083667, 0.066687, 0.031137, 0.014174, 0.009079, -0.053699, 0.016020, -0.016121, 0.043584, -0.029076, -0.008727, 0.053317, -0.019611, -0.046309, -0.009621, -0.085304, -0.058713, -0.064756, -0.001893, -0.008697, 0.045675, -0.079169, -0.064322, -0.037956, -0.074753, -0.082449, -0.059066, 0.007213, 0.028612, -0.086448, 0.051069, -0.056882, -0.123483, -0.028333, -0.003464, -0.019611, 0.098916, 0.110572, -0.065950, -0.117112, -0.024935, 0.055296, -0.015169, 0.035809, -0.023074, -0.027382, -0.053122, -0.017066, -0.063870, 0.047924, -0.091435, -0.026618, -0.057639, 0.032714, -0.047711, -0.006890, -0.029797, -0.010135, 0.012137, -0.118973, 0.012622, -0.009017, -0.017071, 0.026594, 0.010391, -0.051400, 0.018158, -0.082854, 0.009368, -0.127069, -0.057390, -0.014655, -0.034310, -0.056265, -0.019669, 0.017825, -0.045089, 0.000201, 0.001460, -0.024958, 0.111280, -0.102564, -0.090243, -0.010984, -0.037008, 0.022217, 0.059629, -0.040993, -0.037850, -0.055616, -0.019312, 0.042316, -0.031016, -0.069508, 0.047074, -0.003295, 0.043106, 0.004727, 0.037124, 0.001343, 0.015220, 0.005110, -0.018500, -0.016849, -0.013103, 0.019751, -0.000488, -0.035916, -0.108027, -0.031653, -0.006790, 0.004324, -0.062247, 0.050886, 0.012174, 0.024951, -0.142063, -0.111376, -0.020173, -0.006148, -0.127590, -0.025973, -0.065785, -0.079121, 0.024249, -0.055816, -0.007214, -0.041225, -0.066770, -0.039461, -0.055466, -0.026213, -0.061532, -0.022263, 0.031828, 0.033243, -0.060890, 0.002973, -0.046254, 0.061632, -0.057656, 0.034156, -0.039309, 0.054040, 0.009694, -0.058648, -0.090651, -0.035014, -0.107011, 0.040167, -0.003421, 0.027573, -0.008357, -0.072357, 0.043841, -0.043315, 0.051091, 0.052954, 0.013641, 0.053170, 0.040246, 0.056687, -0.064467, -0.009898, 0.056063, 0.009620, 0.038564, -0.057257, -0.068768, -0.003586, -0.061019, -0.048795, -0.102672, 0.048205, -0.086003, 0.060443, 0.032888, -0.029471, 0.035450, -0.019915, 0.012293, 0.051787, 0.104564, 0.016293, 0.041689, -0.005132, 0.012470, -0.052873, -0.001327, 0.002632, 0.042817, 0.001977, -0.027095, 0.082820, -0.022427, 0.011454, 0.030368, 0.044778, -0.113109, 0.117897, 0.023600, -0.064960, 0.085215, 0.098027, -0.037562, 0.087512, 0.036588, -0.007239, 0.048798, 0.026258, 0.012949, 0.004282, 0.010290, 0.008214, 0.065234, -0.025770, 0.049986, -0.002655, -0.009338, -0.023304, -0.076761, -0.018045, -0.027253, -0.013534, -0.090398, 0.044113, -0.019122, -0.057661, -0.031930, -0.053118, -0.039086, -0.002579, 0.054590, -0.046907, 0.080837, -0.019692, 0.017540, -0.055751, -0.072338, -0.027538, 0.056847, -0.034752, -0.015507, 0.059573, -0.026498, -0.035463, 0.021345, -0.025159, -0.024648, 0.005616, 0.038180, 0.069701, 0.037812, -0.051975, -0.075128, 0.025793, -0.025446, 0.144453, -0.072439, 0.007456, 0.060604, 0.023066, 0.012304, -0.046182, 0.027309, -0.055681, -0.003250, -0.083883, -0.056041, -0.044261, -0.052731, 0.017667, -0.003666, 0.006478, -0.051369, -0.026185, -0.041984, 0.019734, 0.021563, -0.027673, 0.006245, -0.081285, -0.068352, -0.045453, -0.041728, 0.010925, -0.031628, 0.016749, -0.031763, -0.016615, -0.024709, 0.013062, 0.002012, 0.005149, -0.076555, -0.056359, -0.029235, -0.032695, -0.063894, -0.003049, 0.064198, -0.026062, -0.057325, -0.000082, -0.046683, -0.064736, 0.046343, 0.049897, 0.043471, -0.061500, 0.024076, 0.007466, 0.038130, 0.041186, 0.096209, 0.043058, -0.015163, 0.057276, -0.034762, 0.050251, -0.034326, 0.007971, 0.038438, -0.041154, 0.011455, 0.058094, -0.032312, -0.027968, -0.067132, -0.064881, 0.037068, -0.006562, 0.022876, -0.011407, 0.035493, 0.047780, -0.097335, -0.053429, 0.048301, -0.031839, -0.066991, 0.048305, -0.066406, -0.100358, -0.036981, 0.006783, 0.062303, -0.017663, -0.080732, 0.055728, -0.085472, -0.039392, -0.035125, -0.018507, -0.055962, -0.078373, 0.000615, -0.058015, 0.034051, -0.002433, -0.037122, -0.096221, 0.046748, -0.000179, -0.012455, -0.001203, 0.009320, 0.008530, -0.009727, -0.050248, -0.047167, 0.103618, -0.007435, 0.006802, -0.065095, 0.002264, -0.032808, -0.070716, -0.027453, 0.000738, 0.025748, -0.054481, -0.005139, -0.082605, 0.017749, -0.026656, 0.063280, 0.070279, 0.002108, 0.070483, -0.026558, -0.056679, -0.037726, -0.065287, -0.000190, 0.054896, -0.002151, 0.006900, 0.019215, -0.055400, -0.038682, 0.025787, 0.004629, 0.010171, -0.022188, -0.044098, 0.037178, 0.056280, -0.043221, 0.015090, 0.060952, -0.050483, 0.048610, 0.014890, -0.015097, -0.141913, -0.061233, 0.018750, -0.024037, -0.067068, -0.062288, -0.032051, -0.033802, -0.014173, 0.004694, 0.029195, -0.050730, -0.083059, -0.003944, 0.007302, -0.107364, -0.088674, -0.102362, 0.015983, -0.107063, -0.056296, 0.017134, -0.067745, -0.016804, -0.063190, -0.036126, 0.041778, -0.070628, 0.047415, -0.014681, -0.030677, -0.005266, -0.053914, -0.075423, -0.071833, -0.025902, -0.037520, 0.014114, -0.042128, -0.061935, 0.026817, -0.019145, 0.001990, 0.037410, -0.073078, -0.039255, 0.053315, 0.047106, 0.012550, -0.109160, -0.001171, -0.051109, -0.080321, 0.035184, -0.093226, 0.002978, -0.011945, -0.058832, 0.013381, -0.050100, -0.018094, -0.042238, -0.005631, 0.034226, -0.047220, 0.000995, 0.030677, -0.025967, -0.051284, -0.011984, 0.021825, 0.087762, -0.030486, -0.059533, -0.006913, -0.046890, 0.002210, 0.086694, -0.022855, -0.047686, -0.005957, 0.020470, -0.075944, -0.036114, 0.098240, 0.094857, 0.046755, 0.039502, 0.022530, -0.015000, -0.038422, -0.045913, 0.049489, -0.041056, -0.071181, 0.036016, -0.017562, 0.095981, -0.052230, -0.007880, 0.033345, 0.014352, 0.033628, -0.011613, -0.027120, -0.016833, -0.055193, 0.048799, -0.047014, -0.012346, -0.013798, 0.041105, 0.057717, -0.020432, -0.070399, -0.017239, -0.018844, 0.035820, -0.064903, 0.000960, -0.029919, -0.049672, 0.028462, -0.087247, -0.049204, 0.060813, 0.000862, -0.007574, 0.004417, 0.044769, 0.073303, -0.112869, -0.049125, -0.019298, -0.142262, -0.048929, 0.035000, -0.037753, -0.010364, 0.036697, -0.057717, -0.059776, -0.072462, -0.023586, 0.076631, 0.002393, -0.004489, -0.036454, -0.088516, -0.045578, 0.043160, -0.000938, -0.001400, -0.005811, -0.143596, 0.017046, -0.112739, -0.011341, -0.021008, -0.015918, -0.051455, -0.120922, 0.023292, -0.007513, -0.028015, 0.050866, 0.101078, -0.050879, -0.010435, 0.018110, -0.024737, -0.024359, -0.036439, -0.043928, 0.014305, 0.027544, 0.021182, -0.028179, -0.005428, -0.051348, 0.056659, -0.051444, 0.041439, 0.002737, -0.043642, 0.060637, 0.109524, -0.073512, -0.051863, -0.009195, -0.019239, 0.038148, -0.023159, 0.024483, -0.050535, -0.098537, 0.001060, -0.034688, -0.072108, -0.036636, -0.138848, -0.007703, 0.000331, -0.033501, -0.010828, 0.013507, 0.059968, -0.028589, 0.036651, -0.025420, -0.009304, 0.045988, -0.006539, -0.040298, 0.001480, -0.050615, -0.040280, 0.014904, -0.015710, -0.041424, 0.006740, -0.100254, -0.056479, 0.009186, 0.040239, -0.069182, -0.005992, -0.008708, -0.022800, 0.023171, -0.002978, 0.003088, -0.094160, -0.003379, -0.046247, -0.039100, -0.072622, -0.157274, -0.020948, -0.049130, -0.046606, -0.020018, -0.033957, -0.017932, -0.009189, -0.076847, -0.017819, 0.006434, -0.070030, 0.184032, 0.029606, -0.027612, -0.068637, -0.041800, -0.068834, -0.073627, -0.065894, -0.024697, 0.019120, -0.043497, -0.116543, 0.014898, -0.037785, -0.016330, -0.024130, 0.100480, -0.058716, -0.008681, 0.005793, -0.026667, -0.047255, 0.018518, -0.091793, 0.064045, -0.022217, 0.049082, -0.121676, -0.016989, -0.039196, 0.027036, 0.005269, -0.055152, -0.057254, -0.045599, -0.077276, -0.134856, 0.038468, 0.018415, -0.003277, 0.000698, 0.021921, -0.049634, -0.007110, -0.053903, -0.086841, -0.081461, -0.064897, -0.034851, -0.037186, -0.023334, -0.073241, 0.075890, 0.038037, -0.031256, 0.019028, 0.054635, 0.010394, -0.061490, -0.013305, -0.126963, 0.008290, 0.034716, 0.019428, 0.029892, -0.069008, -0.020843, 0.004501, 0.006247, 0.021080, 0.103524, 0.087161, 0.017482, -0.007440, 0.005855, 0.039086, 0.042302, -0.062603, -0.043347, 0.007867, -0.050611, -0.055817, -0.006000, -0.036692, 0.059931, -0.117705, 0.070310, 0.023665, -0.017902, -0.061234, -0.036163, 0.001339, -0.084501, -0.019579, -0.005056, 0.101588, 0.002286, 0.029617, 0.100684, 0.000787, -0.052058, -0.068139, 0.045683, -0.059416, 0.034180, -0.026357, 0.023408, -0.014662, -0.000220, -0.047121, -0.035673, -0.000572, -0.076106, -0.087367, -0.036219, 0.065841, -0.064282, -0.071824, -0.036290, 0.064295, -0.114101, -0.075450, -0.115428, -0.063036, 0.049949, -0.071045, -0.007229, 0.089466, -0.093429, 0.084253, -0.105254, -0.064655, 0.029299, -0.054994, 0.057967, -0.029262, -0.094145, 0.031946, 0.002577, -0.031181, -0.048213, -0.118182, 0.025503, -0.042157, -0.033402, -0.007438, -0.028125, -0.018542, -0.025358, -0.002806, -0.060084, -0.053680, -0.048783, 0.000713, -0.014555, 0.004701, -0.017116, -0.060465, -0.079823, -0.065749, -0.003241, -0.090174, -0.027173, -0.006919, 0.006742, -0.050025, 0.004383, -0.053946, -0.107670, -0.133187, -0.046671, 0.013085, -0.017134, -0.070358, -0.131414, -0.085800, -0.026504, 0.110474, -0.022340, -0.057390, -0.098205, -0.061408, -0.007510, -0.079404, -0.035929, 0.024017, 0.035174, 0.035162, -0.042691, 0.010943, -0.065982, -0.028724, -0.022099, 0.017908, 0.078085, 0.002902, 0.007715, 0.008810, -0.061988, -0.086641, 0.000163, 0.013648, -0.083460, -0.012261, -0.031282, -0.107647, -0.026342, -0.095425, -0.088939, -0.050068, -0.105614, -0.005338, -0.049523, 0.095291, 0.020140, -0.062102, -0.012638, 0.022133, -0.123335, -0.087234, 0.025338, -0.078915, -0.038745, -0.094738, -0.053892, -0.046895, -0.015085, -0.024619, -0.158471, 0.049664, 0.049086, -0.045944, 0.083938, -0.067614, -0.091528, -0.036368, 0.015492, 0.029025, 0.092068, 0.116229, -0.027489, -0.047407, -0.026495, -0.012329, -0.009359, 0.011616, -0.091403, -0.016491, 0.009116, -0.084954, -0.000165, 0.005126, -0.066674, -0.034784, -0.051537, 0.010363, 0.003579, 0.001843, -0.044687, -0.047371, -0.040703, 0.000318, 0.036194, 0.025259, 0.044728, 0.052757, -0.030313, 0.028281, -0.029139, 0.044397, 0.046838, -0.032803, -0.008600, -0.057514, 0.035866, 0.023893, 0.048156, -0.063694, -0.082420, -0.034740, 0.036367, -0.107245, -0.020572, -0.024441, 0.027356, -0.023845, -0.051956, -0.062789, 0.002290, -0.013673, -0.056215, -0.002733, -0.021358, -0.018815, -0.043178, -0.073010, -0.089278, -0.056459, -0.047062, 0.033723, -0.063228, -0.049246, -0.060225, -0.132980, -0.087832, -0.121020, -0.030302, 0.034359, 0.022863, 0.004823, 0.042467, 0.043779, -0.058336, 0.052365, -0.039105, -0.136652, -0.047138, -0.064036, 0.012024, -0.054920, -0.036205, 0.032442, -0.078283, -0.019676, -0.068059, -0.039631, -0.026192, -0.034060, -0.017273, 0.075609, 0.013670, -0.088336, -0.058852, 0.043114, -0.092553, 0.049927, -0.030467, -0.069892, -0.100180, -0.023332, -0.007459, 0.049038, -0.054112, -0.005186, 0.005355, 0.016593, -0.006079, -0.031594, -0.025755, -0.067564, -0.009297, 0.018767, 0.053160, -0.043286, -0.028891, 0.111359, -0.093811, 0.040616, 0.052606, 0.017302, -0.127971, 0.024732, -0.038225, 0.044473, -0.019513, -0.043392, 0.041758, -0.030025, -0.031274, -0.012760, -0.186197, 0.020705, 0.012316, -0.094143, 0.005846, -0.059631, -0.043414, -0.089081, 0.026982, -0.024441, -0.074149, -0.028306, 0.033640, 0.000201, -0.071923, 0.026716, 0.051147, -0.004130, -0.036005, -0.047055, 0.047248, -0.044409, -0.016585, -0.049194, -0.040888, 0.052349, 0.055554, -0.027277, 0.022064, -0.045873, -0.127312, -0.057998, -0.047381, -0.008580, -0.063484, -0.123589, 0.011081, -0.017162, 0.019726, -0.066444, -0.010956, 0.036937, 0.016849, -0.024754, -0.049841, -0.031060, -0.007725, 0.015544, -0.027131, -0.099798, 0.013268, -0.110644, -0.078633, -0.057343, -0.031450, -0.006947, -0.063913, 0.003517, -0.030161, 0.037056, -0.108055, -0.002982, -0.069473, 0.030690, -0.019172, -0.020313, -0.032906, -0.034810, -0.017041, 0.050743, 0.057378, -0.088585, -0.001812, 0.027611, -0.030187, -0.038782, 0.001776, -0.009049, -0.147425, -0.052671, -0.031042, 0.024231, 0.037230, 0.026121, -0.029136, -0.019860, 0.044074, -0.066324, -0.053845, 0.072228, -0.153292, -0.032689, 0.005843, -0.062404, 0.049022, -0.047753, 0.019821, 0.045567, -0.019339, -0.080586, 0.018858, -0.013858, 0.004268, 0.031376, 0.031831, -0.034941, -0.085595, -0.093273, 0.006137, -0.112257, -0.043433, -0.015711, -0.020421, -0.083745, -0.089884, 0.011322, 0.066822, -0.005928, -0.011849, -0.025897, 0.071799, 0.031583, 0.024807, -0.053253, 0.014669, -0.031557, 0.008121, 0.053619, 0.026393, 0.009336, -0.020940, -0.062102, 0.011625, -0.080128, -0.020940, -0.037882, -0.044648, -0.027320, -0.027212, -0.032273, 0.076862, -0.032006, -0.111200, -0.013567, -0.054646, -0.001036, 0.068645, -0.032581, -0.012443, -0.046442, -0.041970, -0.000497, 0.053086, 0.014911, -0.035287, -0.038239, -0.017259, 0.019928, -0.091868, -0.087489, -0.011638, -0.028841, 0.004350, -0.097852, -0.008964, -0.066406, -0.055277, -0.062670, 0.007384, 0.098877, -0.066310, -0.069017, -0.030132, -0.078162, -0.044710, -0.097345, -0.117901, -0.003149, 0.000278, 0.019240, -0.005738, -0.043317, -0.100146, 0.014670, 0.032231, 0.004198, -0.017800, -0.030591, -0.077120, -0.036337, -0.061231, -0.049093, -0.102206, 0.149186, -0.010195, -0.075264, -0.022332, 0.009847, -0.070771, -0.019925, 0.004690, -0.016974, -0.113133, -0.068738, -0.021880, -0.031684, -0.035146, -0.060694, 0.015829, 0.048071, -0.119016, 0.011036, -0.018860, 0.022259, 0.007875, 0.008287, -0.049573, -0.071797, -0.007415, 0.087682, -0.034051, -0.035263, 0.015624, -0.063352, 0.045817, 0.031509, -0.148103, 0.006594, -0.058719, 0.048046, -0.028531, -0.031188, 0.028897, -0.011610, -0.053245, -0.013936, 0.020854, 0.101210, 0.010127, 0.059485, -0.019877, -0.083683, -0.002666, 0.005728, 0.020856, -0.055169, -0.010159, -0.078643, 0.072319, -0.050988, 0.022422, -0.016863, 0.154562, -0.059041, 0.044410, -0.025747, 0.039160, -0.006446, -0.112002, -0.057757, -0.117682, -0.003930, -0.050000, -0.058785, -0.085334, -0.085761, 0.043470, 0.013640, -0.031291, -0.079424, -0.044849, 0.008316, -0.108963, -0.039521, -0.013943, -0.030837, -0.075824, 0.052851, -0.099484, 0.006370, -0.075217, 0.008717, -0.044764, -0.158004, 0.018897, -0.025301, 0.034357, -0.011878, 0.023796, -0.029905, 0.099220, 0.007439, -0.029673, -0.006967, 0.002638, -0.020867, 0.000122, 0.017329, -0.060899, 0.055285, 0.032469, 0.022112, 0.031369, -0.011818, -0.076151, 0.030429, 0.016074, -0.096064, -0.051440, -0.076327, 0.063696, 0.047837, -0.006802, -0.012502, -0.089484, 0.035386, -0.043068, -0.053320, 0.015026, -0.068983, -0.031584, -0.022751, -0.064424, -0.013355, 0.041345, 0.058704, 0.060276, -0.096472, -0.019731, -0.063852, -0.085571, 0.006221, 0.004724, -0.068497, -0.071955, -0.078423, -0.013171, -0.090756, -0.018754, -0.027931, -0.024676, 0.029466, -0.043938, -0.056596, -0.044633, -0.072029, -0.075228, 0.004023, -0.123083, -0.087689, 0.048921, -0.064384, 0.011907, -0.046142, 0.005803, 0.005496, 0.014772, -0.026987, -0.047975, 0.035950, -0.073228, 0.009211, 0.037775, 0.033047, -0.081479, 0.048603, -0.044901, -0.008513, -0.055757, -0.020456, 0.026743, 0.090293, 0.021614, -0.057728, -0.034099, 0.030398, -0.003508, -0.058762, -0.037833, 0.026708, -0.079325, -0.058366, -0.039050, 0.007472, -0.024905, 0.015771, 0.026867, -0.000098, -0.038599, -0.001134, -0.056934, -0.100485, 0.121366, -0.008917, -0.018973, -0.039823, 0.013068, 0.006128, -0.029339, 0.047970, 0.027569, 0.079367, -0.025445, 0.006180, 0.049673, -0.038454, -0.045387, -0.010873, 0.022029, -0.013109, -0.065320, -0.070273, -0.014428, 0.054898, -0.007403, -0.032703, -0.071994, -0.014806, -0.001855, 0.005436, 0.097303, -0.008735, -0.098769, -0.095765, -0.076949, 0.040415, -0.085229, 0.058533, -0.041108, -0.001520, -0.061381, 0.008269, -0.000286, 0.052601, 0.037815, 0.028624, -0.021322, -0.082653, -0.014608, -0.052414, 0.072066, -0.009615, 0.047306, -0.046380, -0.028282, 0.024449, -0.020128, -0.095873, -0.039301, -0.001301, 0.119996, 0.012000, 0.021123, -0.035379, -0.111036, 0.003501, -0.089161, 0.079373, -0.005251, -0.088601, 0.046594, -0.079578, 0.051170, 0.036024, -0.012112, 0.022419, -0.042586, 0.033106, 0.016336, 0.028958, -0.086051, -0.042311, -0.044073, -0.017470, 0.040437, -0.057658, -0.106702, -0.128295, -0.007690, -0.005083, 0.050261, -0.003550, -0.077987, 0.060646, -0.054299, -0.044236, -0.052171, 0.038549, -0.024488, 0.052378, -0.082653, -0.065019, -0.070512, -0.046466, -0.117687, -0.033949, -0.121021, -0.031560, -0.033524, -0.027699, -0.046166, -0.067758, 0.085694, -0.092458, -0.026879, -0.035348, 0.000174, -0.145800, -0.106362, -0.028458, -0.068170, -0.081299, -0.008162, -0.024236, 0.155492, -0.028558, -0.015690, -0.015997, -0.056642, -0.134197, -0.056033, -0.044694, -0.062634, -0.034462, -0.077662, -0.118778, -0.029031, -0.000279, 0.011625, 0.007489, -0.015985, -0.009266, -0.022631, 0.043682, -0.037720, -0.000067, -0.124411, -0.031108, 0.025485, -0.021129, -0.013884, -0.047519, -0.129481, 0.054724, 0.045871, 0.021846, -0.064202, -0.115299, -0.022704, -0.045557, 0.008081, -0.052507, -0.102382, -0.018661, 0.010230, 0.110902, -0.013504, -0.047543, -0.055820, -0.052159, -0.046451, -0.038244, -0.051351, 0.042198, -0.079314, 0.009744, -0.019589, -0.070468, -0.005565, -0.004090, 0.014700, -0.049505, 0.006489, -0.000743, 0.009000, -0.048572, 0.011901, -0.002487, -0.023066, 0.067811, 0.011079, -0.032243, 0.020403, -0.033129, -0.019308, -0.028948, -0.032796, -0.028492, 0.002350, -0.052632, -0.003894, 0.051302, -0.032400, -0.059211, -0.056785, -0.015891, -0.030564, 0.015697, -0.013008, -0.074519, -0.021468, -0.069795, -0.114873, -0.086543, -0.019133, 0.032862, -0.087515, 0.013753, 0.042040, -0.029312, -0.056821, 0.010886, 0.014085, -0.035685, -0.038720, 0.021935, 0.113571, -0.016603, 0.026821, -0.050922, -0.024802, -0.038228, -0.041286, -0.069178, -0.007933, 0.072964, 0.082875, 0.020711, -0.010921, 0.043949, 0.055390, -0.018549, -0.001433, -0.004875, 0.010073, 0.036456, -0.099281, -0.033416, -0.038639, 0.053128, -0.009424, -0.004931, -0.027504, 0.006961, 0.020243, -0.052464, -0.060756, 0.021566, -0.062058, 0.010592, 0.050595, -0.012187, 0.088045, 0.028116, 0.113592, -0.036644, -0.078066, -0.085941, 0.067545, 0.058194, 0.123209, -0.080506, 0.003304, -0.047358, -0.066466, -0.034609, -0.027172, -0.014373, -0.006648, -0.109424, 0.015971, 0.016368, -0.110834, -0.107567, -0.124793, 0.124022, -0.009044, -0.104363, 0.057495, 0.008702, -0.101471, 0.059380, 0.019344, -0.002047, 0.050357, 0.011871, -0.072867, 0.020453, -0.066896, -0.016043, -0.049437, -0.019275, -0.020820, -0.004641, 0.042331, -0.065543, -0.023961, -0.097871, -0.097184, -0.003276, 0.045388, -0.010282, 0.035051, 0.010881, 0.048931, 0.004661, 0.014913, 0.011200, -0.044753, 0.032680, -0.016026, -0.011148, -0.138535, -0.018950, -0.064473, -0.044291, -0.002498, -0.057830, 0.025031, 0.012987, -0.032539, -0.012733, -0.085924, -0.010726, 0.088997, 0.040164, -0.027500, 0.087919, -0.032543, -0.019691, 0.055555, -0.042768, -0.015167, -0.026684, -0.114451, -0.096288, -0.035156, -0.049075, -0.011435, 0.066537, -0.095325, -0.051075, 0.060630, -0.025292, -0.048689, -0.031773, -0.001125, -0.036130, -0.050385, 0.025151, -0.114079, -0.129204, -0.014052, -0.053236, 0.025456, -0.021407, -0.011376, -0.044528, -0.006953, -0.016268, -0.092014, -0.045990, -0.096618, -0.106593, 0.074455, -0.028648, -0.024932, -0.004702, 0.025163, -0.050098, 0.002562, -0.051525, 0.017581, 0.042649, 0.076903, -0.055620, -0.037908, -0.012691, -0.035245, -0.070350, -0.036595, -0.015643, -0.154674, -0.029313, -0.032013, -0.031311, -0.044170, -0.003950, 0.038661, -0.050780, 0.153153, -0.056753, -0.048431, -0.017715, -0.163843, -0.121068, -0.071770, 0.004914, -0.070587, 0.039026, 0.092934, -0.029959, -0.046110, -0.018492, -0.155165, -0.039242, -0.060300, -0.051010, -0.107969, -0.101948, 0.041795, -0.020907, 0.041773, -0.028886, -0.083148, -0.118144, 0.001043, -0.007959, -0.037901, 0.014400, 0.103427, 0.027086, -0.095161, -0.017900, 0.017155, -0.022019, 0.022206, 0.068382, -0.046228, -0.003664, 0.066833, -0.089467, -0.127261, -0.049055, -0.062697, -0.056413, -0.048237, 0.034984, -0.045563, -0.001616, 0.055484, -0.020143, -0.037678, 0.078776, -0.029995, -0.055253, -0.035844, 0.063966, -0.090446, -0.064481, -0.012461, -0.013975, -0.069319, 0.032044, -0.041867, -0.002381, 0.079576, -0.055935, -0.007245, -0.104317, 0.062910, 0.065805, -0.076665, 0.138200, -0.064491, -0.034423, 0.035177, 0.039234, 0.026781, 0.005870, -0.079385, -0.060329, -0.067178, -0.038431, 0.044914, -0.023299, -0.064593, -0.172316, -0.031530, -0.002763, 0.016020, 0.080396, -0.155747, 0.048699, -0.084039, -0.009112, 0.060249, 0.026917, 0.007758, -0.051001, -0.062249, -0.028134, -0.112026, -0.189447, -0.095333, -0.065728, -0.027569, 0.034502, 0.060839, 0.132795, -0.107680, -0.113181, -0.049219, -0.020102, -0.078006, -0.027353, -0.010773, -0.020570, -0.055791, -0.018998, 0.029901, -0.057916, -0.048000, 0.000664, -0.010482, -0.055065, 0.014847, -0.022966, -0.081432, 0.032575, -0.071527, -0.010478, -0.045972, 0.025661, 0.078738, -0.038128, -0.005039, 0.064744, -0.010187, -0.087776, -0.059651, 0.013834, 0.037673, -0.032047, -0.065608, 0.049863, 0.065443, 0.058306, 0.113375, 0.019336, -0.059284, -0.000776, 0.006194, 0.043679, 0.045956, -0.033977, -0.132415, -0.089329, 0.024096, 0.011871, -0.095097, -0.006481, 0.003397, -0.123208, 0.081283, -0.082976, 0.061863, 0.041667, 0.021430, -0.102965, -0.177098, 0.008513, -0.102169, 0.053024, -0.009321, 0.008255, -0.057623, 0.033105, -0.061638, -0.123816, -0.086785, -0.088523, -0.137727, -0.010577, -0.032903, 0.045912, -0.112652, 0.109613, -0.057545, -0.036712, 0.040184, -0.153230, -0.065590, -0.096548, 0.008555, -0.026417, 0.022189, 0.013389, -0.132627, -0.038589, -0.102013, -0.010966, -0.101247, -0.028493, 0.008886, -0.006427, 0.018052, -0.013940, -0.034049, -0.037422, -0.070445, 0.069648, -0.036609, 0.079183, -0.037747, -0.069182, 0.020887, -0.043780, 0.040206, 0.032606, 0.045943, 0.167795, 0.045731, 0.008521, -0.061810, -0.035670, 0.096989, -0.075718, -0.112364, -0.078013, -0.098980, 0.036454, -0.020991, -0.025211, -0.187039, 0.028977, 0.020462, 0.028970, 0.024418, 0.012406, -0.053747, -0.222870, -0.069961, -0.144173, 0.014292, 0.059841, -0.007326, 0.016301, 0.057591, -0.021857, 0.108882, 0.061675, -0.080127, 0.038241, -0.008622, 0.037744, -0.028046, -0.116102, -0.008794, 0.021796, 0.084054, 0.034400, -0.036754, 0.103985, -0.040864, -0.088184, -0.064893, -0.002666, 0.045201, -0.168104, 0.067820, -0.038620, 0.030309, 0.019637, -0.087658, -0.042805, -0.012071, 0.029828, -0.018478, -0.079447, -0.027208, 0.016518, -0.019416, 0.165683, -0.073984, -0.049857, -0.010704, 0.112133, 0.072846, 0.062109, 0.051222, -0.086593, -0.003016, 0.087232, 0.019963, -0.033605, 0.054015, -0.067168, -0.092099, -0.055432, -0.069522, -0.041059, -0.115175, 0.008649, -0.043934, -0.042019, -0.080558, 0.016272, 0.010336, 0.040594, -0.085483, -0.050814, -0.037019, -0.070029, 0.040428, -0.011975, -0.058438, 0.035952, 0.052235, 0.050649, 0.013738, -0.138874, 0.015653, 0.053660, -0.028560, -0.015490, -0.017408, -0.088585, 0.069741, 0.063266, 0.012136, 0.063477, -0.045795, -0.015511, 0.012268, 0.009601, -0.096457, -0.031757, -0.045805, 0.030742, -0.026638, 0.058247, -0.076604, -0.086471, 0.011524, -0.109999, 0.000611, -0.021756, -0.084868, 0.054842, -0.047791, -0.018308, -0.019538, 0.000292, 0.009198, 0.000270, -0.091232, -0.017307, -0.003465, 0.075837, 0.041115, -0.021123, -0.110272, 0.063889, -0.071766, 0.028202, -0.076745, -0.138853, 0.026118, 0.035910, -0.067264, -0.100077, 0.059862, -0.072946, 0.009212, -0.109361, -0.122042, 0.031360, -0.014888, -0.011583, -0.026061, 0.004687, 0.022850, 0.009381, -0.029884, 0.105336, 0.036801, 0.004800, 0.002370, -0.007476, -0.031809, 0.056551, -0.064924, -0.119727, 0.006015, -0.126020, -0.146994, 0.038090, -0.096588, 0.193603, -0.121452, -0.062503, 0.008429, 0.037974, 0.081938, 0.039802, -0.053985, 0.060464, 0.017174, 0.047584, 0.005629, -0.086467, -0.039317, -0.113069, 0.041936, -0.084295, 0.089715, -0.051776, 0.014545, -0.041272, -0.058769, -0.020407, -0.018988, -0.009832, -0.030432, 0.003293, 0.031035, -0.099381, 0.027623, -0.048622, 0.030218, -0.055545, -0.013419, 0.110540, -0.036444, -0.007333, -0.123048, -0.076871, -0.084372, -0.016950, 0.012312, 0.037604, -0.053813, -0.038294, 0.089329, 0.037235, 0.047835, -0.045974, 0.002909, -0.043783, -0.090252, -0.050069, 0.038387, 0.084373, 0.035602, 0.030983, -0.023846, -0.029994, 0.031002, -0.053159, -0.008677, -0.114947, -0.081882, -0.071548, -0.136120, -0.043726, 0.005231, 0.045170, -0.062115, -0.048139, -0.034355, -0.027838, -0.030530, 0.017396, -0.132658, -0.072864, -0.009282, -0.060800, -0.023030, -0.058141, 0.020654, -0.040184, 0.010105, 0.040265, -0.015220, -0.081481, 0.086678, 0.053441, -0.062918, 0.107466, 0.021991, -0.037560, -0.058150, -0.166389, 0.061878, 0.018359, -0.081208, -0.071779, -0.074261, -0.049512, 0.052906, 0.034672, -0.002110, -0.029977, -0.068865, -0.066254, -0.009333, -0.004530, 0.005624, -0.034159, 0.065525, -0.190280, -0.007576, 0.015829, 0.077599, -0.003541, 0.031391, 0.104597, 0.016674, 0.000531, -0.093823, 0.024811, 0.044305, -0.068942, -0.080530, -0.003445, -0.052479, -0.082163, -0.129526, -0.049050, -0.149333, -0.108384, 0.025662, -0.095824, -0.001090, -0.012424, -0.036946, 0.094370, 0.031792, -0.008711, -0.055771, 0.017282, 0.039440, -0.102646, -0.046308, 0.032414, -0.010869, -0.059214, 0.047207, -0.155802, 0.018436, 0.002280, 0.062957, -0.027079, 0.002454, -0.079527, -0.057581, -0.010534, -0.004643, 0.203456, 0.086630, -0.084865, -0.087615, -0.054670, 0.014324, -0.026488, 0.009047, -0.073773, 0.017885, -0.100971, -0.113595, 0.164698, -0.034144, -0.051613, -0.090690, 0.029424, 0.032996, -0.047500, -0.051914, -0.051273, -0.035655, 0.076529, -0.085756, -0.048672, 0.062767, -0.014848, 0.097511, -0.009897, -0.067572, -0.041982, -0.068316, -0.086338, -0.028818, 0.000824, -0.081299, -0.008700, -0.099741, -0.019888, 0.017416, -0.065377, -0.017724, -0.035477, 0.037395, -0.030341, -0.026538, -0.010329, -0.062074, 0.011514, 0.107947, 0.011349, 0.015275, -0.130382, 0.019683, 0.084435, -0.007582, -0.076468, 0.049390, -0.014273, -0.073305, 0.038539, -0.015345, -0.031084, -0.086207, 0.029385, -0.011815, -0.089661, 0.065315, -0.107484, 0.002078, 0.057514, -0.014288, -0.028393, -0.084897, -0.022899, -0.151340, -0.093332, 0.067049, -0.043370, -0.074394, -0.023931, 0.080608, -0.020609, -0.002234, -0.071341, 0.004495, 0.055678, -0.031073, -0.059841, -0.010433, -0.020383, -0.075814, -0.043300, -0.037106, 0.022343, -0.224233, -0.039241, -0.004056, -0.033988, -0.040455, 0.013377, -0.078586, 0.031112, 0.000008, -0.093177, -0.181250, -0.014311, -0.036787, 0.089692, -0.111710, -0.040176, -0.085241, -0.054357, -0.001432, -0.157394, -0.031593, 0.091536, 0.002886, -0.102648, 0.055484, -0.072319, -0.042984, 0.087393, -0.026386, 0.096411, -0.036645, 0.033892, 0.036393, 0.007081, -0.071869, 0.009680, 0.088995, 0.023757, -0.025871, -0.041456, -0.069702, -0.055640, -0.037479, -0.008688, -0.077628, 0.084483, -0.000799, 0.020265, -0.080745, -0.057741, -0.058327, 0.019667, -0.038222, -0.107329, -0.025706, -0.040385, -0.104049, 0.013563, -0.006352, -0.124208, 0.001402, -0.049030, -0.083405, 0.037963, -0.061146, -0.101721, -0.013336, -0.047535, 0.020837, -0.044996, 0.096614, -0.024270, 0.023276, -0.005041, -0.143620, 0.011625, 0.016348, -0.065505, -0.036165, 0.009546, -0.061447, -0.023014, -0.121482, 0.107669, -0.044496, -0.015722, 0.007423, -0.064584, 0.046117, 0.024797, 0.019629, 0.219558, -0.085500, -0.097509, 0.015885, -0.097418, -0.028446, 0.014524, -0.074570, 0.033875, 0.098850, -0.029000, -0.032076, -0.074001, -0.007827, -0.028262, -0.042940, 0.031420, -0.119141, -0.017427, -0.055245, -0.017034, -0.027699, -0.076355, -0.090441, 0.047170, -0.032219, 0.033867, -0.123010, -0.084195, -0.045970, -0.060237, -0.173076, -0.133380, -0.006982, -0.119538, 0.019707, 0.143409, 0.080862, -0.027151, 0.014068, -0.080356, 0.005508, -0.041980, -0.012683, -0.076461, -0.045942, -0.040750, -0.042752, -0.112440, -0.107706, -0.067437, -0.045313, -0.064830, -0.008669, 0.009941, -0.019317, 0.027622, -0.041718, -0.026958, -0.000555, 0.030712, 0.008921, -0.035793, -0.069928, -0.117442, -0.061723, -0.021225, 0.015889, 0.018880, 0.020333, -0.009995, 0.043950, -0.004112, -0.060199, -0.059204, -0.056739, -0.024498, -0.005369, 0.012410, 0.081668, -0.121122, 0.004052, 0.020364, 0.024483, 0.015408, -0.109305, -0.039072, 0.041082, 0.060912, 0.028816, -0.120674, 0.012535, 0.002112, -0.030670, -0.044335, -0.095535, -0.017330, -0.005956, -0.001644, -0.025968, 0.056595, 0.062644, -0.125703, 0.031780, -0.033110, 0.010954, -0.089663, -0.038647, -0.030298, 0.038262, -0.110378, -0.050600, -0.014371, 0.039356, 0.005850, -0.068847, -0.062073, -0.040300, -0.086147, 0.047361, 0.048983, -0.088652, 0.062695, -0.029334, 0.034928, -0.067483, 0.018934, -0.089884, -0.078412, 0.001912, -0.035399, 0.022255, -0.016006, -0.098317, 0.055301, 0.010405, -0.035853, -0.096755, -0.081806, -0.020443, -0.062335, -0.146303, 0.046106, -0.018193, -0.088027, 0.024402, -0.001898, 0.124163, -0.070639, 0.005259, -0.039985, 0.036113, 0.007228, 0.007854, 0.078882, -0.027904, -0.021680, 0.070402, -0.050272, -0.001535, 0.054238, 0.038715, -0.007822, 0.012841, -0.012471, 0.044342, -0.103220, -0.062118, 0.003464, 0.050326, 0.031921, 0.050083, -0.091362, -0.125877, -0.173260, 0.022630, -0.012500, 0.004539, 0.064412, 0.002579, -0.164467, -0.022666, 0.013124, -0.021840, -0.090540, 0.062758, 0.043320, -0.091049, -0.055894, 0.002724, -0.008247, -0.096407, 0.063584, 0.028454, -0.002859, -0.055072, -0.033282, 0.028635, -0.069919, 0.138337, -0.056974, -0.032089, -0.027697, -0.084583, -0.029410, 0.155813, 0.000982, -0.060373, -0.032993, -0.078704, -0.200556, -0.093330, -0.037138, -0.009788, 0.040589, -0.050851, 0.015130, 0.001176, -0.071463, -0.069209, 0.004863, -0.084717, -0.065105, -0.012625, -0.001635, -0.012133, -0.024277, -0.099672, -0.081386, -0.043090, -0.113878, -0.023042, -0.051186, 0.013912, -0.024837, -0.044660, -0.009040, -0.052355, -0.015201, -0.024245, -0.017048, 0.039499, 0.039958, -0.131544, 0.038572, -0.000259, -0.077951, 0.027374, -0.020424, -0.114782, 0.061634, -0.034784, 0.042073, 0.037545, -0.045403, -0.045480, -0.011909, -0.069987, -0.029817, 0.058788, -0.031957, 0.019860, -0.006946, -0.094076, 0.023917, -0.080093, -0.003182, -0.078366, -0.011250, 0.052879, -0.047956, 0.024901, -0.129417, 0.027916, -0.003960, -0.042071, -0.008710, -0.062256, -0.094797, -0.004570, 0.067269, -0.038591, 0.033876, -0.041187, -0.072850, -0.034752, 0.072053, 0.040701, 0.025188, 0.029801, 0.025892, 0.062967, 0.029926, -0.006830, -0.096562, -0.105927, -0.046281, 0.013601, 0.051522, -0.031472, -0.029311, -0.045985, 0.019215, -0.010813, -0.057684, -0.006917, 0.014867, -0.016681, 0.010545, -0.025100, -0.085679, 0.028151, -0.102978, -0.042415, 0.007719, -0.013590, -0.053913, -0.037178, 0.029959, 0.029001, -0.012033, -0.011491, -0.002043, -0.054000, -0.096777, -0.093895, 0.028596, -0.027274, -0.014541, -0.017298, 0.015066, -0.068924, 0.026231, 0.003989, 0.028137, -0.078079, -0.021757, -0.019613, 0.019135, -0.036440, -0.043817, -0.004737, 0.026153, -0.116565, -0.036569, 0.093399, -0.050571, -0.016140, -0.064669, -0.026962, -0.049213, -0.001429, -0.053230, -0.022503, -0.046372, -0.102875, -0.031365, 0.061321, -0.007791, 0.078130, -0.023815, -0.063254, -0.015746, 0.042360, 0.021948, -0.009556, -0.065149, 0.015293, -0.023575, -0.092670, -0.046149, -0.020886, 0.065497, -0.008853, -0.001356, -0.026214, 0.007617, -0.027018, -0.075116, 0.018741, -0.055881, -0.097122, -0.081755, 0.034525, -0.021293, -0.049425, -0.075099, 0.049256, -0.098584, 0.015915, 0.102733, -0.116617, -0.067882, -0.055606, -0.060853, -0.024942, 0.027025, -0.082658, -0.042745, -0.002258, 0.040388, 0.016821, 0.002136, 0.052576, 0.018525, -0.044814, -0.006880, 0.025562, -0.070653, -0.034833, -0.087971, 0.045924, -0.096126, -0.037793, -0.064032, 0.021395, -0.081131, 0.016964, 0.020709, -0.051708, -0.102848, 0.068838, 0.141469, -0.034623, 0.068538, -0.022652, -0.006772, -0.000336, -0.107528, -0.067991, -0.040011, -0.013435, -0.051038, -0.169590, -0.117324, -0.020797, -0.106799, 0.064645, -0.059771, -0.167334, -0.131829, 0.031917, -0.046814, -0.082183, 0.118207, -0.081961, -0.010852, -0.014127, -0.021073, -0.034506, -0.029879, 0.064356, -0.104964, -0.065667, -0.173877, -0.073142, -0.018490, 0.057008, -0.176511, -0.064608, -0.013481, -0.013945, -0.084056, 0.039402, 0.004734, -0.056112, 0.047762, -0.050121, -0.040394, -0.000145, -0.041358, -0.053457, -0.108330, -0.120974, 0.097583, -0.006798, -0.014344, -0.108572, -0.057933, -0.009471, 0.000283, -0.012526, 0.065263, 0.000216, -0.018297, -0.005530, 0.004857, -0.011503, -0.078479, 0.009469, -0.019439, 0.025588, 0.001954, -0.035468, -0.011924, -0.023269, -0.104258, -0.021019, 0.056422, -0.044437, 0.013464, -0.024654, -0.053462, -0.006958, -0.006405, -0.027577, -0.093155, -0.139036, -0.026161, -0.094468, -0.046530, 0.029550, -0.050640, 0.018804, -0.030270, 0.006840, -0.007344, -0.017740, 0.022136, 0.019992, -0.043246, -0.138679, -0.035710, -0.068379, -0.028664, -0.053945, -0.019211, 0.001889, 0.054318, -0.058305, -0.024483, 0.035649, -0.040343, -0.102646, 0.061484, -0.013817, -0.106687, -0.049263, 0.014357, 0.024024, -0.029255, -0.015260, -0.104791, 0.069914, 0.012626, 0.034091, 0.030702, -0.039809, -0.098926, 0.006849, -0.046458, -0.041167, -0.071562, -0.009487, -0.021208, -0.056089, 0.077079, 0.024383, -0.041704, -0.039522, -0.047162, 0.050663, -0.041921, 0.033877, -0.023568, -0.046749, -0.107138, 0.114719, -0.036141, -0.010553, 0.017266, -0.048614, 0.011466, -0.125505, -0.038351, 0.003364, -0.285792, 0.065810, 0.055246, -0.093241, 0.044867, -0.078047, -0.017986, 0.038050, 0.047576, -0.042192, 0.008160, -0.073007, -0.046277, -0.051812, -0.026517, 0.025564, 0.011724, -0.062324, 0.020737, -0.048462, -0.065300, -0.030847, 0.045643, -0.067113, -0.027631, -0.024538, 0.036135, -0.033669, -0.012752, -0.061675, -0.067976, 0.057564, -0.106806, -0.066041, 0.097261, -0.013953, -0.088746, 0.001946, 0.056948, -0.018028, -0.012354, -0.041049, -0.058369, 0.054818, -0.007988, -0.053998, -0.047905, -0.131930, 0.001575, -0.026974, -0.059854, -0.051936, 0.039049, -0.118142, -0.002845, 0.032052, 0.003505, 0.089494, -0.046629, 0.039770, 0.025015, -0.039083, 0.019285, 0.020282, 0.171891, -0.004538, 0.004269, 0.017442, -0.039361, 0.093370, -0.041385, 0.009139, 0.030431, -0.045605, -0.071549, -0.066815, -0.048658, -0.061099, -0.006055, -0.056182, 0.112003, 0.034880, -0.045089, 0.045870, -0.093906, -0.029380, -0.013832, -0.094471, 0.190464, 0.014158, 0.016414, -0.052091, -0.054179, -0.055699, -0.125059, -0.002992, 0.037345, 0.004150, -0.015844, -0.087198, -0.134691, 0.043847, -0.065704, -0.024837, 0.040788, 0.013155, -0.108884, 0.022464, -0.043931, 0.006744, -0.017751, 0.044942, -0.025236, -0.023312, -0.095433, -0.037267, -0.060591, -0.065780, -0.010432, -0.006105, -0.007377, 0.014269, -0.038395, -0.111890, -0.056617, 0.055845, -0.125601, 0.023926, 0.028184, -0.101714, -0.037931, 0.021425, 0.129773, 0.063844, 0.011866, -0.003657, -0.065074, -0.019210, -0.002031, -0.053496, -0.096689, -0.034836, 0.013809, -0.118940, 0.057455, 0.020645, -0.062695, 0.076262, 0.061720, 0.022579, -0.050677, 0.024772, -0.124078, -0.002773, -0.003834, 0.014015, -0.002442, -0.052308, 0.057554, -0.076270, -0.058436, 0.106848, 0.054115, 0.033054, -0.013805, 0.032790, -0.033488, 0.018713, -0.020150, -0.025415, -0.059435, -0.019182, -0.061355, -0.027762, -0.001314, -0.173016, 0.025951, 0.010438, 0.040443, 0.034896, -0.033554, -0.054511, -0.049790, -0.003323, 0.045423, -0.044260, 0.032015, -0.034687, -0.083688, -0.048572, -0.122921, 0.025669, -0.041818, -0.025074, -0.021290, 0.102707, -0.133525, -0.080566, 0.004787, -0.040797, -0.157478, 0.007527, -0.100906, 0.022938, 0.166244, -0.007967, 0.137718, 0.046976, -0.058174, -0.028167, -0.089606, 0.051752, 0.039443, 0.084987, 0.165993, -0.069064, -0.054759, 0.015345, -0.020887, -0.018044, -0.135654, -0.065764, -0.038720, -0.019870, -0.003525, -0.016801, -0.040487, 0.006275, -0.061389, -0.007215, -0.052024, -0.073074, 0.004101, -0.024757, -0.026542, -0.002200, -0.045237, 0.005095, -0.029117, 0.009570, -0.037013, -0.026726, 0.012665, 0.005656, -0.012867, -0.041702, 0.047469, 0.008517, -0.048834, -0.054565, 0.055386, -0.005735, -0.010273, -0.011270, 0.004084, -0.058316, -0.065836, 0.030065, -0.040854, 0.015451, -0.062816, 0.060841, -0.077005, -0.040948, -0.050785, -0.032587, -0.050580, 0.015876, -0.050857, -0.049512, 0.055032, -0.070624, -0.093359, -0.051066, -0.050472, -0.068937, 0.034228, 0.028328, 0.017555, 0.027359, -0.050065, -0.058537, -0.103311, -0.053250, -0.070825, 0.009459, -0.079180, -0.059134, 0.005482, 0.006174, -0.016562, 0.050469, 0.061894, -0.064460, -0.056240, 0.008899, 0.027057, -0.142388, -0.150790, -0.133115, -0.065795, -0.069291, -0.038752, 0.000632, -0.054645, -0.067008, -0.040950, 0.020401, -0.087484, -0.026945, -0.001048, -0.080279, 0.013640, -0.048299, -0.046474, -0.027738, -0.057260, -0.009161, 0.065928, 0.005990, 0.002116, 0.008284, -0.035873, 0.030650, -0.059983, -0.077147, -0.100276, 0.048981, -0.057813, 0.084801, -0.082579, 0.036857, -0.014673, 0.092591, -0.029644, 0.008991, 0.059631, -0.039084, 0.015836, -0.073295, 0.042679, 0.038392, 0.060412, -0.036525, 0.042809, 0.044489, 0.003548, -0.049135, 0.043538, 0.023884, -0.034680, -0.073113, 0.016337, -0.128579, 0.027164, -0.073238, -0.007460, 0.066861, 0.127366, -0.012551, -0.040163, -0.002806, -0.057399, -0.065823, -0.114356, -0.037658, -0.117171, -0.062069, 0.014704, -0.005417, -0.047869, 0.043281, -0.034556, -0.077862, -0.010976, -0.079932, -0.102937, 0.019966, -0.027565, -0.044362, 0.003397, 0.025999, -0.089338, -0.038182, 0.004101, -0.010751, 0.018271, -0.056568, 0.007311, 0.001379, -0.036227, 0.018405, -0.063410, -0.066595, 0.050545, 0.033727, -0.054104, -0.132943, -0.061571, 0.009846, -0.015509, -0.021351, 0.055659, -0.072368, -0.023954, 0.056664, -0.027702, -0.005369, -0.048094, -0.018257, 0.042678, -0.017356, -0.127514, -0.080170, -0.115843, 0.052287, -0.046121, 0.023499, -0.052640, -0.050409, 0.000968, 0.051559, -0.043406, 0.068010, -0.064950, -0.067363, 0.000202, -0.101794, 0.026526, -0.067649, 0.046852, 0.011473, 0.134786, -0.017660, -0.020973, -0.044879, -0.029830, 0.011463, -0.107749, -0.112668, -0.099643, 0.002399, -0.073411, -0.014723, -0.089188, 0.051846, -0.018178, 0.012908, -0.005920, 0.038816, -0.026823, 0.098055, -0.119911, -0.025880, -0.038040, -0.073894, 0.098855, -0.025273, -0.010800, 0.022512, 0.002616, 0.006062, 0.016034, 0.018256, -0.079803, -0.024226, 0.227372, -0.125397, -0.070982, 0.048813, 0.029106, 0.164046, -0.064978, 0.029491, -0.087207, 0.076418, 0.053849, -0.093920, 0.030768, 0.016322, 0.030274, -0.061858, -0.043353, -0.087085, 0.026155, -0.000408, -0.148989, 0.062540, 0.014871, -0.049012, 0.001553, 0.013225, 0.017252, -0.095261, -0.055045, -0.073226, -0.017792, 0.048066, 0.052593, 0.025464, -0.014662, -0.105291, -0.127891, -0.014678, -0.054815, 0.049010, -0.052438, 0.029146, -0.052420, -0.053971, -0.019900, -0.031109, -0.061223, 0.021471, -0.051489, -0.106585, -0.001975, 0.037967, -0.049624, -0.080198, -0.055629, -0.013037, 0.020031, 0.013257, 0.050808, -0.008525, -0.066813, 0.041701, 0.065085, -0.024201, -0.184103, -0.158724, -0.037522, -0.031979, 0.013370, 0.052117, -0.116356, 0.012226, 0.001295, -0.032840, 0.006213, -0.011340, -0.027042, 0.083541, 0.071138, -0.018213, 0.059891, -0.027803, -0.135159, 0.068971, -0.163235, -0.042203, -0.017822, -0.145840, -0.111152, -0.066221, 0.007754, -0.037614, 0.014594, -0.028300, -0.018518, -0.006965, -0.036778, 0.024401, 0.001436, -0.047853, -0.032790, -0.109168, -0.016592, -0.045609, -0.001651, -0.026458, -0.033354, 0.028357, -0.007443, -0.034032, -0.031135, -0.027939, -0.043669, -0.098544, -0.055445, -0.002071, -0.038260, -0.015475, 0.041431, 0.013884, 0.011789, -0.119076, -0.121027, -0.057933, -0.105909, -0.054927, -0.034810, -0.106499, -0.036275, -0.065761, 0.030035, 0.111708, -0.185965, -0.040532, -0.137297, 0.004638, -0.017220, -0.022812, 0.036756, -0.075015, 0.036624, 0.043422, -0.191974, 0.016309, 0.055195, 0.087085, -0.066304, 0.012009, -0.075978, -0.130661, -0.066473, 0.034305, -0.091892, -0.095426, 0.008716, 0.064187, 0.096044, 0.059033, -0.038700, -0.056327, 0.020459, -0.054538, -0.077382, -0.042190, -0.107853, -0.064334, 0.004817, 0.013205, 0.120998, 0.019525, -0.064622, 0.072341, -0.011264, -0.084184, -0.044542, -0.077058, -0.037600, -0.009916, -0.029822, 0.044037, -0.047385, -0.004648, -0.114826, -0.077195, -0.087848, -0.128830, -0.027349, 0.012966, 0.006859, -0.099391, -0.020474, -0.113269, -0.007800, -0.188789, -0.134512, -0.059782, 0.033288, -0.146420, 0.030668, -0.136417, -0.052485, 0.077316, 0.014809, -0.042982, -0.075243, -0.011849, -0.062662, 0.014641, -0.030307, -0.128129, -0.071887, -0.033989, 0.068533, -0.045829, -0.085188, -0.109446, 0.047369, -0.112054, 0.008478, -0.209995, 0.152104, -0.091767, -0.029010, -0.055128, -0.029233, 0.022642, -0.112329, -0.004231, 0.015287, 0.022052, -0.064836, 0.030905, 0.000216, -0.042945, 0.041133, 0.028907, 0.051230, -0.026374, -0.203409, -0.091673, -0.107001, -0.006759, 0.004216, -0.049576, -0.031206, -0.005024, -0.119198, -0.033534, 0.063276, 0.027987, -0.005263, -0.055691, -0.012094, -0.099977, 0.002887, 0.100725, -0.057162, -0.147639, -0.062690, -0.031507, 0.098072, 0.150220, 0.021353, 0.026145, 0.035353, -0.008646, -0.076570, -0.032057, -0.047711, -0.066182, -0.059302, -0.095957, -0.118478, 0.145491, 0.054082, 0.048734, -0.068630, -0.134764, -0.138087, -0.020304, -0.036019, -0.095178, -0.005575, -0.066426, 0.011496, -0.103164, -0.059975, -0.164741, -0.062612, -0.035423, -0.213870, -0.061972, -0.062759, -0.002178, -0.033318, -0.062574, -0.040124, 0.018677, -0.057370, 0.165069, -0.059838, 0.184887, -0.040646, 0.041050, -0.014279, -0.139462, -0.117726, -0.030898, -0.092441, -0.081233, -0.016168, -0.060292, -0.004028, -0.025901, -0.044579, -0.089942, 0.037415, -0.160155, -0.098615, -0.181247, 0.048684, -0.072471, 0.027594, -0.070913, -0.057243, 0.123974, 0.027444, -0.004528, -0.116187, -0.106280, -0.058004, -0.109892, -0.067068, -0.047330, 0.092614, 0.014806, -0.173221, 0.041959, -0.061590, 0.128227, 0.012728, -0.142270, -0.084548, -0.051522, -0.088439, -0.024191, -0.005864, 0.026152, -0.117741, -0.019413, -0.110606, -0.085372, -0.001362, 0.067231, -0.042058, -0.086749, 0.044118, -0.081706, -0.072810, 0.030074, -0.055909, -0.003391, -0.001106, -0.043906, -0.187066, -0.100059, -0.091004, -0.108761, 0.143701, 0.058389, 0.062547, -0.071166, 0.003733, 0.002040, -0.039469, 0.046336, -0.073177, 0.014500, -0.012917, -0.060444, -0.102512, -0.054489, -0.146845, -0.066349, -0.011554, -0.063369, 0.006625, -0.063000, -0.107049, -0.076404, -0.131617, -0.076348, 0.038859, -0.044645, -0.052508, -0.010005, -0.048889, 0.050823, 0.050919, -0.027988, -0.128929, -0.100056, -0.092031, -0.083005, -0.069383, 0.074656, -0.035535, 0.008247, -0.211347, -0.054221, -0.023904, -0.076827, -0.117546, -0.149784, -0.015700, 0.097724, -0.099079, -0.021857, -0.089514, -0.108239, -0.025906, -0.070319, 0.015195, 0.006104, -0.090020, -0.099294, 0.030018, -0.124928, -0.071696, -0.071729, -0.039976, -0.019832, -0.035017, -0.069849, -0.059659, -0.057639, 0.176798, -0.071277, -0.047012, -0.139265, -0.115038, -0.146008, -0.132770, -0.064249, 0.075967, -0.018204, -0.066778, -0.078689, 0.047858, -0.067335, -0.057258, -0.048686, -0.064376, 0.049965, -0.039677, -0.031686, -0.000271, -0.006956, -0.057518, -0.190354, -0.041288, 0.034600, 0.116931, -0.017887, -0.114595, 0.041814, -0.076320, -0.082836, -0.025114, -0.041163, -0.092817, -0.137367, -0.006554, -0.107129, 0.024672, -0.018280, -0.087561, -0.053117, -0.099660, 0.090950, -0.221128, 0.028414, -0.076619, -0.074590, 0.021417, -0.000923, -0.037232, 0.036812, -0.111695, -0.117964, -0.043980, 0.022833, -0.018434, -0.013763, -0.045192, -0.065171, -0.111051, -0.010773, -0.106502, 0.018833, 0.020406, -0.014041, 0.011403, 0.070647, -0.066353, -0.039060, -0.022310, 0.003926, -0.078303, -0.033244, -0.023357, 0.017066, -0.138362, 0.006327, -0.119892, -0.360607, -0.016030, -0.058965, -0.156673, -0.122808, -0.077988, 0.031619, -0.047978, -0.112094, -0.033772, 0.065529, -0.080239, -0.110524, -0.039886, 0.024422, 0.016337, -0.022264, -0.027721, -0.075246, -0.027401, -0.042847, -0.137184, -0.119994, 0.082781, 0.043388, -0.049080, 0.023612, -0.074440, -0.124985, -0.064201, -0.094925, -0.132733, -0.098954, 0.027335, -0.064771, -0.009735, 0.078140, -0.071468, -0.089749, 0.012342, -0.235752, -0.033226, -0.076281, -0.133850, 0.054560, -0.027786, 0.007393, -0.086183, -0.057498, -0.026041, -0.075170, -0.129352, -0.193302, -0.085111, -0.028478, -0.106654, -0.017935, 0.169568, -0.024844, 0.130485, -0.056233, -0.110445, 0.016979, -0.012525, -0.059221, 0.060819, -0.123373, -0.109162, -0.093705, -0.104088, 0.072894, -0.058501, -0.093206, -0.059674, -0.047313, -0.082617, -0.071548, -0.150485, 0.040693, -0.063119, -0.073856, 0.153737, 0.062430, -0.107387, -0.048550, -0.068917, -0.092650, 0.007789, 0.035064, -0.138248, -0.026983, 0.157612, 0.023802, -0.096367, -0.051857, -0.085351, 0.064459, 0.021432, -0.044033, -0.067330, 0.175733, -0.116700, 0.048829, -0.023084, -0.034240, -0.103951, -0.016069, -0.074791, -0.049841, 0.014445, -0.038882, -0.053758, -0.119067, -0.000347, -0.055085, -0.055793, 0.056098, -0.076480, 0.191039, -0.000188, -0.173307, -0.071764, 0.057334, -0.120963, -0.083990, -0.061043, -0.059311, 0.010984, -0.057975, -0.085359, -0.040024, 0.039127, -0.073507, 0.055038, 0.013034, 0.119245, -0.013822, -0.083403, 0.021963, -0.010044, 0.000014, 0.008598, 0.020997, -0.011644, 0.084364, 0.052595, -0.048357, -0.022067, 0.016469, -0.012909, 0.036941, -0.047389, 0.127448, 0.060362, -0.028200, -0.046100, -0.112394, -0.122466, -0.009588, -0.016119, -0.032662, -0.098747, 0.045798, -0.040697, 0.005693, -0.028856, -0.080550, 0.148881, 0.026284, -0.044531, -0.079995, -0.098028, -0.195304, -0.046248, -0.128203, -0.001284, -0.004432, 0.050465, 0.004740, 0.012172, 0.052552, -0.075142, -0.172480, -0.070662, -0.085394, 0.105101, 0.031444, -0.149757, -0.024424, -0.036421, 0.066908, -0.079638, -0.032302, -0.065206, 0.085376, -0.042089, -0.011737, 0.026948, -0.086878, -0.051554, -0.019954, 0.065300, -0.060084, -0.054731, 0.000882, -0.049916, 0.019238, 0.030145, -0.047363, 0.074916, -0.131815, -0.033095, 0.076388, -0.116299, -0.006946, -0.050914, 0.020919, -0.066455, -0.003548, -0.045479, -0.012699, -0.140580, 0.065329, 0.018886, 0.002226, -0.082908, -0.105131, -0.199548, -0.085570, -0.108827, -0.032174, 0.138977, 0.008042, -0.023990, 0.072778, -0.075195, -0.053076, -0.064155, 0.154951, -0.013862, 0.087148, -0.071477, -0.143208, -0.020827, -0.079739, 0.013675, 0.008821, 0.010423, 0.024696, -0.104363, 0.032755, -0.024444, -0.149384, -0.006308, -0.009979, -0.026624, -0.063347, -0.238241, 0.003326, 0.060932, 0.007800, -0.058640, 0.004383, 0.175639, 0.065438, -0.016355, -0.064821, 0.064828, 0.031568, 0.009895, -0.230319, -0.068824, -0.011919, 0.014015, 0.033207, -0.042428, -0.087346, -0.136602, -0.067258, 0.006100, 0.173435, 0.019292, -0.067622, -0.097939, -0.059114, -0.087173, -0.024608, 0.076259, -0.018863, 0.018622, 0.035811, -0.103975, -0.092408, -0.113247, -0.106154, -0.083577, -0.048029, -0.063342, 0.096844, -0.071196, -0.017083, -0.076220, -0.187027, -0.005656, -0.116470, -0.238564, 0.083263, -0.172274, -0.054363, -0.035627, -0.011394, -0.069278, -0.015588, 0.085685, 0.011817, -0.122297, -0.095819, 0.076974, -0.102421, -0.010674, 0.075010, -0.048417, -0.085218, 0.032647, -0.041622, -0.108137, -0.042546, -0.122588, -0.013299, 0.033245, -0.006844, -0.043047, -0.148760, -0.013386, -0.114007, -0.011794, -0.143379, -0.061899, -0.181408, 0.017063, 0.083029, -0.128382, 0.041769, 0.040872, 0.057268, 0.024979, -0.101247, -0.006229, 0.016623, 0.022006, -0.103007, -0.074961, -0.055558, 0.163281, -0.055375, -0.032538, -0.059952, -0.010096, -0.104719, -0.102640, 0.077655, 0.117671, 0.009251, -0.005116, -0.036516, -0.037968, 0.004362, 0.007973, -0.145591, -0.029967, 0.020729, -0.072991, 0.240661, -0.101331, -0.145558, 0.035228, 0.027093, -0.074042, -0.080715, -0.060621, -0.140938, 0.013683, -0.042613, -0.050559, -0.074015, -0.058379, -0.042867, -0.032041, -0.061088, -0.058336, -0.084353, 0.002530, -0.109267, 0.036423, -0.043165, -0.028458, -0.059005, -0.061871, 0.022118, 0.053820, -0.152248, -0.055556, -0.043604, -0.019267, -0.138993, 0.113091, -0.058606, -0.100556, -0.032000, 0.069509, 0.051883, -0.068972, -0.025049, -0.012848, 0.058782, 0.046523, 0.027968, -0.133939, 0.111037, 0.060947, -0.108538, -0.073775, -0.128250, 0.034491, -0.139297, 0.044427, -0.026320, -0.158800, 0.032619, -0.041739, -0.137059, 0.043090, -0.018794, -0.005073, 0.070174, 0.003472, -0.049715, -0.036022, -0.095312, 0.035611, -0.183258, 0.030824, -0.084872, -0.094319, 0.004367, -0.053145, -0.080088, -0.165260, -0.014313, 0.096395, 0.028547, -0.081648, -0.027391, 0.086588, -0.133881, -0.130213, -0.068487, 0.135564, -0.105062, -0.288849, -0.083063, -0.064751, -0.029931, -0.028108, 0.107606, 0.034827, 0.053865, -0.005215, -0.071303, -0.204055, -0.060798, 0.084499, -0.115615, -0.043732, -0.074733, -0.036808, 0.037639, -0.011183, -0.042969, -0.089610, -0.055980, -0.133457, -0.093259, -0.053238, -0.211225, -0.013116, -0.085583, -0.095257, -0.051581, 0.020013, -0.088045, 0.059477, 0.018004, -0.023628, -0.051449, -0.071262, 0.027040, 0.007111, 0.098809, 0.014047, 0.125668, 0.037095, 0.043485, -0.031281, -0.123038, -0.032614, -0.048109, -0.114891, -0.034461, 0.042654, -0.117700, -0.085967, -0.122662, -0.043141, -0.151832, 0.036879, 0.051343, -0.033868, -0.061718, -0.003405, -0.097824, -0.070173, -0.051544, -0.080476, 0.003639, 0.077195, 0.008346, -0.056030, -0.202849, -0.054921, -0.037068, -0.047481, -0.091667, 0.043867, 0.156334, -0.041685, -0.146202, -0.111682, 0.032962, 0.101355, -0.060676, 0.027784, -0.075926, -0.008509, -0.042592, -0.115815, -0.100585, 0.008658, 0.030969, 0.029771, -0.036012, 0.068620, -0.135178, -0.108504, -0.034029, -0.021976, 0.005857, 0.007698, -0.135611, -0.087933, -0.111267, -0.092273, 0.050085, -0.018556, -0.018725, -0.003002, -0.078087, -0.046987, -0.026189, -0.136703, 0.021625, -0.125397, -0.110349, 0.094539, 0.100294, 0.061857, 0.067118, -0.169061, -0.034506, -0.058290, 0.153229, -0.001613, -0.077712, -0.082559, 0.015361, 0.021672, -0.111388, -0.022363, -0.061903, -0.034756, -0.016791, -0.000638, -0.083093, 0.049204, 0.008390, -0.049201, 0.055458, -0.156099, -0.080891, -0.045339, 0.022680, -0.131861, -0.191766, 0.042298, 0.004367, -0.221252, -0.040783, -0.043818, -0.097476, -0.013757, 0.075735, 0.156092, -0.148089, -0.105092, -0.018868, -0.094554, 0.053013, 0.092239, 0.007506, 0.013299, -0.008372, -0.078270, 0.031421, 0.064232, 0.035870, 0.132185, -0.068912, 0.015167, -0.046232, -0.035426, 0.065513, -0.155531, -0.033684, -0.009956, -0.057326, 0.008385, 0.015662, -0.103525, -0.066052, 0.150985, 0.000926, -0.075163, -0.067543, -0.082803, 0.106100, -0.094519, 0.020095, 0.060883, -0.054721, -0.000380, -0.070023, -0.037955, 0.025933, 0.076314, -0.148017, -0.032451, -0.017243, -0.114677, 0.048217, -0.058834, -0.003651, -0.036382, -0.035998, 0.027726, 0.028538, -0.092817, 0.029851, -0.061011, -0.057556, -0.078133, 0.086185, 0.001423, 0.041405, -0.024886, -0.052422, -0.040617, -0.055534, -0.144129, 0.131148, 0.169259, 0.007671, 0.054816, -0.083470, -0.015691, -0.084293, -0.038611, -0.097622, -0.052280, -0.016423, -0.006111, -0.148689, -0.010143, 0.006062, -0.093183, -0.165154, -0.052630, 0.022601, -0.008304, 0.015742, -0.076188, 0.016921, -0.033118, 0.005612, -0.062356, 0.031129, -0.104335, -0.058900, 0.039634, -0.039156, 0.050478, -0.142202, -0.076546, -0.066919, -0.073682, -0.018819, -0.056909, 0.073082, -0.015451, 0.084251, -0.055965, -0.033016, -0.016613, -0.009570, 0.029331, -0.071324, 0.076278, -0.050069, 0.001336, -0.160703, 0.103715, -0.144386, -0.055004, -0.026135, -0.022494, -0.126850, -0.039569, -0.055323, -0.043575, -0.056390, -0.026554, -0.030958, 0.011500, -0.019594, 0.012539, 0.060720, -0.015138, -0.007736, -0.099722, -0.030531, 0.058520, -0.022733, -0.069789, 0.011920, -0.032712, -0.071201, 0.005689, -0.149182, -0.060400, -0.025603, 0.009729, -0.149918, 0.046386, -0.042081, -0.093684, -0.006406, 0.000213, -0.037599, -0.066401, -0.047955, -0.162825, 0.109217, -0.018390, 0.042892, -0.072523, -0.095389, -0.185273, -0.034626, -0.042692, -0.060476, -0.059766, 0.022525, -0.074734, 0.133525, -0.076777, 0.083589, -0.041121, -0.064295, -0.046019, -0.135950, -0.006792, -0.064941, -0.035642, 0.026448, -0.057168, -0.012635, 0.047552, 0.000228, -0.217694, -0.042931, -0.065558, -0.106457, 0.080366, 0.022040, -0.037930, 0.080249, -0.057460, -0.106258, 0.129028, -0.086706, 0.002744, -0.004916, -0.072877, -0.009046, -0.116726, -0.043244, -0.126530, -0.028812, 0.083042, -0.101523, -0.000793, 0.061084, 0.055461, -0.004767, -0.028170, 0.038427, -0.018211, -0.097886, -0.079768, -0.141412, 0.014500, 0.019259, 0.034319, -0.028053, 0.091498, 0.141838, -0.014049, 0.123714, 0.054890, -0.001493, 0.033278, -0.031279, -0.143249, -0.039798, -0.016252, -0.002563, 0.003279, 0.026477, 0.020978, -0.084726, -0.000938, -0.113417, -0.070540, -0.038583, -0.106312, 0.009053, 0.016246, 0.009288, 0.050265, -0.049086, -0.013098, -0.094335, 0.015237, -0.118069, -0.014987, 0.040644, -0.064722, -0.068012, -0.006705, -0.053474, 0.020297, -0.015246, -0.082587, -0.029645, -0.081898, 0.036932, -0.063157, -0.105455, -0.001209, 0.090108, 0.113207, 0.032018, -0.013943, 0.071194, -0.098199, 0.020283, -0.104876, -0.007842, 0.021163, -0.012835, 0.031136, 0.033338, 0.028088, -0.058858, -0.093505, -0.038226, -0.048438, 0.044230, -0.038888, -0.069109, -0.021034, -0.154113, 0.033204, 0.043217, 0.060147, 0.027931, -0.035980, -0.083421, -0.017150, -0.074271, -0.004796, 0.032562, 0.020325, -0.078320, -0.048863, 0.008436, -0.005208, 0.004494, -0.084730, -0.053618, -0.052950, 0.019658, 0.022279, -0.107624, -0.071301, 0.038840, 0.013059, -0.033238, -0.104921, 0.012365, 0.006329, -0.031369, -0.098270, -0.028830, -0.010539, -0.049429, -0.088683, 0.098843, -0.026489, -0.004329, 0.059548, -0.031458, -0.020973, -0.013011, -0.130012, -0.063210, -0.021394, -0.073915, 0.009078, 0.033169, -0.077261, 0.046375, 0.006521, -0.018164, -0.005250, 0.023283, -0.043560, -0.066933, 0.037256, -0.119507, -0.042459, -0.055573, -0.030838, -0.015161, -0.095518, -0.123077, 0.043475, -0.021328, -0.005297, -0.087380, -0.007688, 0.116213, -0.012539, -0.066276, -0.008374, -0.024541, -0.064569, 0.016849, 0.011425, -0.032771, 0.027455, -0.058979, -0.062177, 0.000048, -0.022078, -0.047943, 0.000900, -0.015820, -0.004855, -0.062244, -0.087571, 0.040872, -0.016033, -0.016488, -0.086636, 0.115153, -0.028866, -0.058667, 0.096953, -0.004285, -0.014371, -0.004602, 0.006192, 0.008427, -0.067295, -0.088950, -0.047090, -0.013315, 0.016397, -0.021526, -0.051729, -0.010305, -0.040498, -0.003816, -0.008755, 0.037464, -0.055005, 0.062715, -0.047361, -0.071330, -0.094360, 0.029948, 0.076388, 0.023723, 0.044104, -0.158797, -0.044494, -0.027051, -0.024122, 0.068622, -0.048669, 0.000437, -0.087013, -0.093871, -0.139901, -0.062398, 0.000149, -0.008093, -0.038773, -0.003901, -0.029896, 0.037515, 0.024323, 0.004619, -0.056464, -0.068172, -0.033622, -0.054297, -0.083244, 0.045569, -0.011807, -0.098636, -0.069642, -0.039438, -0.000885, -0.042304, 0.034974, -0.060362, -0.030522, 0.019925, -0.036764, 0.032934, 0.069892, -0.002646, -0.012380, -0.064143, -0.132628, -0.015923, -0.225163, -0.009905, -0.035909, 0.047560, -0.006842, -0.097999, -0.068768, 0.011204, -0.018667, -0.154443, -0.024454, 0.038021, 0.019658, -0.041885, -0.031991, 0.022154, -0.068611, -0.007828, -0.054664, -0.086183, 0.029861, -0.086919, -0.028055, -0.129288, 0.011317, -0.101381, -0.087679, -0.055234, -0.052359, 0.038508, -0.067975, -0.049683, -0.049815, -0.049504, -0.088118, -0.070419, -0.066106, -0.065521, -0.064750, 0.009609, 0.003165, 0.028150, -0.049947, -0.064749, -0.070002, 0.038327, 0.038412, -0.076854, 0.086838, 0.034146, -0.001689, -0.066650, -0.038296, -0.121299, -0.037531, -0.047093, -0.046494, -0.086457, 0.033711, -0.043111, 0.022774, -0.061825, -0.018868, -0.014294, -0.005281, 0.034120, -0.025067, -0.013650, -0.080190, -0.018508, -0.059487, 0.005962, 0.111238, 0.041204, -0.115709, 0.094510, -0.059841, -0.097028, -0.093020, -0.003416, -0.046089, 0.010231, 0.020017, 0.029807, -0.095597, -0.074533, -0.062480, -0.028610, -0.078814, -0.002897, 0.028380, -0.077860, -0.011220, -0.032495, -0.007523, -0.028821, 0.021580, -0.022206, -0.082704, -0.098136, -0.083255, -0.041833, -0.013552, 0.073640, -0.063835, -0.051091, 0.005047, -0.014499, -0.005994, -0.126670, 0.062834, -0.054103, -0.057094, 0.046358, -0.140671, 0.036490, 0.038570, -0.004058, -0.046502, -0.039904, 0.015614, -0.008560, 0.014845, 0.008622, 0.034955, -0.047689, -0.097191, -0.093920, -0.104596, 0.021462, -0.069904, 0.102228, -0.016285, -0.124247, -0.115077, -0.086105, -0.019304, -0.043244, -0.032365, -0.099303, -0.059046, -0.103327, -0.063167, -0.039907, -0.073054, 0.045025, -0.023703, -0.021624, 0.051938, 0.047119, 0.055726, 0.110635, -0.035704, -0.114944, -0.072087, -0.092155, -0.083105, -0.077707, -0.033605, -0.085156, -0.088949, -0.131531, -0.067596, -0.083746, -0.061099, -0.082177, 0.022774, -0.003747, -0.027023, -0.035883, 0.006645, -0.137455, -0.019382, 0.018803, -0.004998, -0.055036, -0.041260, 0.002744, -0.053177, 0.055670, -0.055936, -0.089406, 0.023637, -0.048558, -0.015202, 0.056608, 0.021617, -0.048321, 0.074132, 0.022593, -0.006869, 0.110289, -0.052574, 0.021931, 0.003073, -0.120789, -0.056933, -0.018036, 0.048611, -0.052933, 0.002351, -0.053142, -0.101893, -0.024915, 0.072449, -0.020357, -0.053696, -0.092875, -0.119525, -0.069826, -0.013967, -0.070171, 0.052945, -0.047034, -0.062783, -0.129910, -0.041306, -0.118090, -0.061982, -0.052349, -0.052598, 0.008876, -0.048069, -0.037560, -0.072160, -0.038094, -0.110476, 0.078240, -0.059697, 0.018880, -0.035515, -0.139055, -0.014203, -0.084170, -0.125186, -0.041771, 0.055779, -0.195393, 0.035352, -0.046736, -0.035308, 0.000243, 0.010687, 0.029503, -0.110565, -0.006796, -0.033180, -0.027912, 0.078879, -0.005707, -0.039955, -0.085721, -0.013371, 0.017566, -0.116405, 0.075259, -0.081715, 0.046498, -0.083395, 0.001570, -0.050300, 0.025086, 0.010314, -0.056945, -0.103283, -0.077998, -0.030628, -0.025524, 0.038408, -0.087829, 0.044873, -0.033382, 0.106939, -0.169568, -0.117886, -0.014705, -0.007053, -0.009258, -0.058491, 0.038323, 0.001912, -0.036006, -0.129906, -0.013203, -0.036170, -0.065843, -0.100378, -0.077733, -0.122209, -0.095810, -0.048603, -0.062887, -0.064262, -0.140890, -0.106178, -0.036218, -0.058853, -0.098317, -0.014808, -0.107138, -0.028683, 0.087711, -0.007284, -0.109958, -0.063766, 0.036582, -0.001544, 0.060497, -0.063359, -0.032716, -0.165248, -0.029890, 0.074855, -0.051307, -0.125446, -0.079421, -0.140433, 0.043516, 0.017988, -0.080167, -0.108193, -0.097375, -0.032431, 0.027876, -0.046790, -0.037855, -0.007282, -0.041807, -0.027318, -0.022954, -0.038313, -0.067314, -0.000440, -0.036823, -0.020683, 0.101012, 0.030602, 0.016877, -0.051017, -0.049456, -0.016562, 0.034312, -0.010445, 0.010917, -0.003042, -0.035198, -0.067619, -0.142619, -0.041438, -0.150441, 0.060189, -0.146068, -0.005078, -0.062549, 0.112237, 0.096862, -0.008213, -0.094085, -0.080558, -0.210573, 0.011904, 0.038293, -0.130816, 0.014477, 0.010234, 0.057970, 0.004679, 0.058714, -0.045015, -0.021991, 0.042385, 0.038408, -0.023981, -0.027557, -0.096917, 0.036139, 0.031262, -0.013698, 0.041307, -0.075275, 0.129015, 0.080388, -0.010635, 0.016767, -0.101837, -0.012782, -0.060469, 0.058255, -0.026757, -0.031016, -0.082416, -0.095368, 0.013696, -0.091859, 0.051419, -0.122830, -0.009559, 0.076996, -0.058847, -0.026283, 0.043164, 0.030859, -0.043976, -0.010172, 0.061586, -0.038373, -0.016649, -0.069632, 0.017190, 0.018434, 0.120504, -0.009425, -0.124700, -0.142097, -0.149994, -0.047496, -0.104230, 0.003228, 0.032669, -0.094642, 0.094725, -0.001361, 0.000499, -0.046232, -0.090001, -0.030726, -0.082305, 0.038754, -0.038462, -0.007960, -0.114487, -0.039335, 0.103355, 0.059323, 0.025283, 0.019092, -0.064204, 0.016019, 0.012799, -0.003719, 0.109328, 0.025639, 0.002462, 0.058280, -0.053526, -0.045854, 0.069112, 0.017180, 0.029629, -0.076241, -0.009732, -0.072034, -0.045062, -0.060422, 0.038895, -0.020031, -0.130689, -0.029913, -0.034075, 0.015115, -0.032441, -0.073976, 0.041010, -0.060518, 0.034389, -0.006190, -0.094407, -0.011803, 0.027222, -0.038732, 0.020042, -0.111162, -0.077047, 0.093685, -0.050696, 0.028761, -0.081061, -0.090794, -0.006065, -0.014989, -0.080828, -0.037618, -0.032760, -0.037454, -0.102763, -0.037579, -0.009979, -0.058265, -0.003537, 0.041888, -0.023411, -0.089445, 0.049886, -0.013978, -0.058328, -0.077106, 0.056660, -0.013269, -0.034599, -0.023317, -0.115279, -0.012009, 0.005008, -0.038107, -0.044961, -0.011111, 0.091379, -0.061165, 0.007296, -0.007459, 0.027007, 0.041050, 0.041295, -0.079642, -0.013441, -0.005872, -0.002215, -0.023763, 0.017534, -0.046647, 0.003748, -0.085916, -0.016143, 0.028022, -0.040628, -0.022264, -0.024947, -0.022450, -0.088390, -0.036283, 0.086927, 0.039208, -0.018680, -0.093627, -0.098981, 0.023509, -0.083957, -0.036185, -0.083041, -0.009880, -0.000026, -0.025109, -0.056484, -0.097943, 0.049464, -0.026131, 0.089223, -0.089801, 0.028521, 0.011355, -0.095039, 0.012299, 0.090343, -0.031869, -0.030972, -0.064738, 0.026297, -0.080059, -0.030480, -0.108866, -0.049770, -0.004786, 0.047881, 0.022990, -0.060173, -0.085613, -0.021263, 0.037073, -0.044676, -0.086625, -0.028925, -0.066734, -0.059740, -0.065547, 0.051724, -0.023896, -0.167003, -0.024032, 0.046334, -0.127607, 0.088658, -0.058254, -0.038396, 0.006533, 0.043143, -0.037276, -0.031722, 0.041236, -0.045608, -0.026884, 0.005879, 0.044650, 0.017918, -0.063344, 0.028452, -0.018759, -0.006798, -0.102580, -0.055961, -0.048323, 0.007088, -0.066064, 0.047210, -0.048786, -0.028638, -0.020833, -0.018122, -0.101501, -0.032459, 0.027570, -0.074538, -0.021427, -0.097311, -0.014740, -0.004514, 0.122278, 0.008887, -0.022168, -0.038631, -0.072176, -0.036031, -0.065574, -0.087289, -0.043210, 0.026574, 0.061768, 0.029749, 0.049224, 0.027461, -0.020757, 0.040429, -0.014641, -0.034125, -0.058098, -0.073428, -0.015853, -0.082094, 0.026341, -0.119386, -0.047951, 0.007543, 0.031532, -0.030675, -0.000577, -0.055061, -0.109161, -0.035523, 0.024485, 0.031500, 0.019430, -0.015334, -0.043424, -0.078393, -0.143045, 0.041320, -0.017760, 0.008660, 0.038350, -0.002643, -0.002487, -0.013691, 0.037732, -0.019361, 0.075562, -0.071045, -0.000258, -0.052845, -0.036894, -0.096689, -0.075850, -0.040884, 0.070787, 0.011014, -0.072623, 0.011639, 0.004995, -0.049587, -0.024230, 0.049963, -0.078604, -0.034098, -0.055673, -0.108799, 0.001781, -0.023816, -0.069900, -0.078388, 0.004528, 0.000905, -0.104394, 0.010543, -0.002002, -0.066150, -0.011697, -0.063263, 0.043603, -0.012468, -0.039818, -0.083568, -0.037350, 0.005419, -0.047271, -0.027215, 0.048481, -0.042867, 0.119607, -0.004474, 0.029329, 0.029009, -0.015702, -0.099908, -0.096474, -0.010986, 0.003802, 0.008904, 0.036076, -0.062420, 0.000336, 0.020220, -0.062454, -0.000085, -0.070446, -0.063789, 0.043262, -0.013424, -0.122046, -0.074996, -0.121558, 0.006056, 0.054807, 0.054312, 0.062697, -0.030092, -0.037416, -0.043042, -0.028145, -0.058619, 0.005973, 0.026305, -0.072224, -0.032005, 0.073952, -0.024056, 0.035158, -0.005270, -0.079451, 0.055530, 0.028627, -0.028990, 0.027024, -0.049058, 0.045584, 0.013438, -0.032850, -0.052290, 0.007645, -0.037503, -0.052121, -0.141790, -0.021138, -0.074362, -0.017515, 0.078126, 0.016276, -0.019106, -0.003792, 0.005695, -0.057011, 0.054330, 0.016669, -0.068786, -0.016361, -0.081771, -0.056188, -0.031134, -0.060050, 0.066560, -0.026479, -0.053176, 0.014351, -0.016141, -0.022447, 0.029496, -0.031113, 0.023881, 0.062543, -0.131030, -0.003239, 0.017645, 0.026530, 0.031998, -0.034313, 0.046296, -0.132396, -0.019315, -0.070664, -0.063674, -0.007783, -0.050688, 0.026292, -0.074452, -0.072648, -0.049458, -0.009007, -0.018391, -0.045946, -0.056460, -0.052721, -0.008054, -0.013043, 0.010609, -0.140159, -0.079084, -0.085722, 0.011439, -0.030071, 0.014460, 0.009475, -0.031045, 0.053448, 0.019855, 0.055858, -0.018163, -0.048028, 0.007025, -0.045643, -0.010055, -0.078465, 0.003698, 0.079146, 0.054316, 0.072898, -0.066476, -0.044837, -0.111707, -0.096357, -0.076693, -0.030483, -0.067278, -0.073607, 0.016504, -0.062578, -0.018426, -0.140311, -0.020380, 0.053580, -0.092101, 0.043762, 0.047270, 0.013220, -0.035033, -0.004144, 0.021329, 0.001115, 0.016740, -0.039519, -0.030192, -0.031441, 0.009424, 0.046088, -0.001198, -0.008707, 0.003415, -0.071136, 0.062654, -0.007831, -0.066679, 0.002481, 0.001653, -0.089555, 0.020547, -0.083436, -0.056058, -0.083782, 0.025449, -0.020326, -0.039793, 0.042379, -0.006163, 0.013271, 0.041742, 0.031207, 0.039743, -0.042738, -0.050373, 0.012206, -0.057122, -0.032590, 0.024993, 0.044154, -0.038386, -0.093078, -0.054181, -0.019562, 0.001082, -0.093835, -0.012238, -0.030760, -0.039725, 0.035180, -0.063872, -0.043161, -0.005497, 0.027025, -0.015293, 0.027758, 0.053481, 0.003919, 0.017398, -0.030125, -0.004827, 0.016805, -0.070300, -0.072903, -0.003389, -0.004173, -0.016366, -0.000431, 0.052245, 0.036981, -0.050301, -0.034715, -0.009976, 0.079939, 0.052364, -0.060347, 0.009607, 0.056079, -0.098120, 0.067266, -0.074948, -0.065273, -0.060840, -0.010467, -0.010933, -0.053265, 0.035209, 0.032709, 0.015084, 0.072212, -0.000524, 0.015344, -0.016328, 0.010858, -0.009329, 0.031036, -0.084262, 0.042430, -0.054663, -0.063287, 0.001876, 0.031044, -0.095221, 0.106293, -0.055780, -0.059848, 0.016421, -0.009720, 0.002242, -0.016896, 0.009927, -0.028259, 0.079448, -0.049106, -0.016430, -0.060898, 0.053466, -0.046672, -0.015882, 0.073874, 0.077736, 0.043162, 0.007526, -0.059476, 0.000656, -0.046194, 0.054612, 0.002283, 0.029639, -0.021542, -0.133659, -0.066449, 0.009626, -0.116737, 0.074360, -0.027702, -0.127237, -0.048686, 0.106417, 0.124849, 0.018741, -0.055667, -0.020136, 0.043539, -0.035550, 0.030224, -0.005668, 0.057665, 0.010968, -0.034147, -0.029773, -0.082348, 0.028799, 0.022091, 0.007499, -0.001977, 0.011533, 0.024977, -0.002438, -0.057105, -0.089452, -0.065629, 0.056369, -0.031872, 0.021592, 0.036522, -0.083635, -0.126029, -0.060117, -0.007508, -0.062127, -0.028166, -0.013239, -0.063571, -0.017053, -0.024722, -0.065699, -0.050508, -0.036879, -0.033602, -0.071809, -0.011038, 0.016600, 0.010241, -0.011403, 0.049425, 0.032092, -0.023587, -0.044844, 0.023668, -0.166554, -0.055519, 0.002072, -0.017722, -0.034137, 0.050238, -0.021866, -0.002350, -0.027756, 0.028891, -0.033800, -0.074042, 0.030958, -0.025168, 0.070365, -0.045842, -0.050881, -0.082478, 0.070323, -0.033675, 0.065852, -0.010171, -0.031458, -0.097373, -0.000715, 0.062603, 0.004708, 0.075779, -0.051031, 0.004444, -0.062272, -0.035704, 0.037658, -0.071398, 0.013340, -0.017918, -0.030194, -0.139422, 0.024957, 0.024629, 0.018453, -0.023327, -0.088891, -0.055823, 0.058840, -0.073563, -0.010442, -0.038515, -0.086937, 0.074154, 0.002581, -0.029718, -0.064445, -0.009095, -0.056905, 0.039821, 0.012263, -0.074021, 0.010243, -0.053124, -0.009585, 0.086644, -0.070913, -0.006821, 0.078150, -0.008191, 0.048588, -0.020456, -0.034586, 0.101583, -0.068415, -0.015306, -0.041479, -0.056663, -0.008839, -0.063835, -0.047960, 0.025607, -0.034420, -0.017266, 0.014873, -0.049083, 0.072714, -0.072700, -0.047217, 0.035987, -0.032081, 0.002139, -0.063298, -0.101669, -0.048311, -0.009239, -0.029795, 0.100390, -0.112010, -0.064302, 0.022223, -0.009422, -0.015164, -0.035504, -0.036962, -0.061371, -0.111739, -0.042367, -0.036622, -0.030313, -0.019359, 0.060248, -0.008376, 0.052732, 0.047510, 0.001816, -0.032924, -0.087286, 0.021488, -0.012934, -0.044841, -0.025142, -0.012490, -0.011077, 0.078293, 0.026846, -0.043661, 0.010132, 0.017171, -0.008252, 0.049659, -0.065786, 0.103164, -0.042172, 0.000104, -0.053317, 0.020248, -0.001675, 0.007974, -0.063650, 0.051520, 0.001909, -0.116690, -0.033722, -0.114716, 0.023997, -0.107715, -0.012417, -0.046667, -0.090098, 0.018765, -0.128196, -0.035267, 0.054170, -0.009007, 0.055541, -0.017555, -0.053992, 0.032339, -0.050471, -0.042763, 0.040938, -0.030655, -0.051753, -0.037963, -0.019045, 0.014856, 0.013466, -0.079698, 0.042562, -0.012189, -0.047845, -0.002669, 0.006589, 0.027081, 0.006817, -0.077501, 0.090902, -0.109074, -0.071174, 0.026030, -0.019462, -0.021959, -0.031660, -0.041111, -0.042187, 0.025813, 0.115729, 0.001511, 0.020868, -0.017436, 0.001493, -0.071719, -0.001127, -0.014887, -0.036857, 0.006613, -0.000587, 0.003088, -0.056152, 0.024982, -0.087184, 0.043355, -0.056219, -0.075794, -0.031942, -0.013311, 0.025437, -0.020861, -0.017341, 0.022887, 0.045006, -0.003622, -0.007584, -0.066776, -0.111865, 0.028157, -0.009549, -0.004031, -0.005102, -0.007077, -0.018720, -0.014976, 0.051713, 0.022521, 0.010393, 0.025215, -0.047973, -0.064478, -0.018803, 0.007660, -0.059507, 0.098286, 0.041230, -0.004535, -0.010046, -0.027311, -0.011524, -0.026295, -0.044892, -0.052619, 0.005142, 0.014539, -0.050832, 0.061885, -0.062995, -0.016037, -0.093725, -0.006285, 0.030770, -0.015543, -0.041687, -0.089896, 0.009376, -0.026633, -0.110241, -0.049309, -0.009760, -0.067507, 0.041806, -0.054292, -0.008893, -0.108355, -0.156761, 0.007407, -0.035669, -0.048750, -0.032810, 0.019830, -0.036443, 0.022398, 0.045348, -0.033513, -0.000674, -0.026948, 0.012171, -0.098473, 0.001432, -0.036923, 0.048545, -0.022484, 0.015350, 0.022212, -0.044822, 0.020676, -0.050431, 0.040611, 0.073719, -0.058125, -0.058614, -0.061675, -0.056183, -0.097780, -0.052759, 0.016265, -0.064859, -0.125041, -0.021111, -0.135416, 0.036299, -0.105653, -0.007293, -0.025451, 0.054871, -0.056233, -0.069581, 0.041793, -0.066853, -0.098157, -0.039308, 0.029976, 0.001100, -0.038910, 0.018054, -0.051628, -0.052058, -0.033515, -0.091493, -0.048383, -0.121417, 0.015089, 0.002792, -0.069105, -0.030474, -0.056589, 0.008254, 0.010350, -0.009932, 0.004830, -0.096460, 0.035324, -0.063032, -0.029852, -0.001460, 0.060707, -0.065885, -0.039851, -0.025890, 0.004847, 0.019345, -0.103721, 0.042780, -0.033904, 0.042788, -0.060920, 0.014137, -0.024834, -0.072297, -0.009177, -0.032900, -0.006363, 0.021078, -0.007802, -0.053479, -0.063638, -0.138818, -0.028427, 0.041871, -0.060934, 0.016599, 0.007300, -0.052209, -0.070338, -0.035140, -0.133482, -0.000269, -0.009303, -0.059568, -0.117294, 0.072011, 0.054537, -0.044507, -0.123054, -0.004748, 0.026276, 0.026351, 0.046770, 0.016227, -0.034733, 0.015341, 0.078539, -0.099584, -0.031373, 0.034839, 0.009095, 0.042965, -0.061454, -0.073366, -0.012374, -0.061637, 0.017987, 0.004143, -0.030147, 0.010340, -0.052082, 0.021704, 0.011791, 0.012300, -0.017802, -0.017118, -0.013694, 0.035056, -0.074733, 0.019249, -0.078909, 0.014608, -0.009077, 0.027778, 0.034573, 0.009325, -0.057136, -0.012712, -0.040586, -0.005510, -0.055184, -0.033686, -0.025893, -0.046877, -0.071285, 0.026765, -0.057859, 0.004918, -0.019143, -0.019163, 0.034315, 0.021402, -0.067537, 0.037691, -0.087871, -0.027304, -0.013434, -0.026671, 0.056772, -0.009038, -0.053052, 0.045762, -0.078776, 0.023432, 0.133846, -0.100615, 0.050241, 0.011135, -0.020179, 0.024272, 0.075274, -0.040077, 0.022330, 0.029012, 0.026779, -0.107953, 0.010235, 0.051755, -0.050555, -0.025709, 0.059375, 0.000611, -0.087711, -0.017117, -0.060303, -0.016264, -0.089859, -0.070405, 0.006996, -0.012270, -0.019402, -0.070856, -0.069917, 0.041735, 0.008158, -0.060266, -0.074689, -0.075573, -0.023182, -0.016554, 0.023752, -0.024114, -0.052428, -0.061742, -0.074243, -0.180264, 0.076369, 0.012331, 0.017168, -0.092465, -0.054818, -0.062432, -0.011857, -0.089304, 0.051786, -0.041956, -0.075355, -0.056285, 0.021260, 0.002627, -0.074036, -0.032016, -0.031941, 0.069440, 0.027421, -0.106462, -0.089931, -0.029438, -0.048516, -0.040698, 0.043010, -0.033393, -0.016446, -0.059463, 0.009769, -0.064738, -0.077382, 0.033384, 0.021670, -0.063025, -0.042966, -0.039394, 0.024322, 0.038990, -0.008511, -0.146333, 0.018004, 0.051566, -0.046667, -0.044489, -0.107178, -0.086249, 0.058385, 0.004585, -0.022139, 0.019921, 0.028246, -0.038323, -0.043257, -0.038066, 0.059619, -0.010192, 0.068428, -0.045845, -0.021619, 0.013834, -0.080831, 0.010675, 0.071558, -0.021827, -0.022749, 0.031212, -0.027387, -0.067122, 0.016360, 0.046827, -0.092057, -0.061128, -0.035891, -0.000766, 0.005916, -0.132323, -0.115144, -0.010922, 0.044209, -0.032031, -0.045752, 0.115526, -0.063927, 0.012142, 0.007820, -0.064584, -0.021186, 0.003640, -0.005995, -0.020745, -0.119102, -0.055546, -0.022801, 0.046551, -0.017852, -0.039713, 0.112143, -0.021039, -0.020880, -0.060230, 0.029657, -0.003985, 0.000537, -0.080903, 0.105278, -0.129515, 0.085495, -0.043736, -0.012877, -0.016250, 0.100155, -0.070188, -0.009498, 0.010563, -0.010081, -0.022829, -0.044940, 0.035503, -0.025002, 0.002071, -0.081598, -0.039464, -0.032874, -0.053126, -0.016222, 0.031134, -0.001533, -0.004945, -0.004870, -0.006299, -0.009966, -0.019223, -0.001287, -0.030150, -0.011978, 0.015297, -0.002872, 0.042477, -0.039879, -0.062527, -0.091151, -0.075506, 0.081474, -0.081176, 0.001294, -0.110222, -0.045415, 0.055306, 0.022822, -0.014877, -0.078226, -0.074363, -0.045994, -0.078240, -0.080898, 0.033615, -0.048005, 0.039397, -0.050730, -0.036631, -0.031976, -0.175792, -0.060362, -0.012056, -0.022755, -0.061918, -0.028859, -0.099508, -0.015837, -0.033635, -0.056338, -0.017850, -0.075481, -0.036614, 0.003955, 0.000933, -0.093103, 0.017638, -0.019251, 0.000647, -0.002243, -0.093974, -0.001549, -0.041602, -0.018435, -0.001230, -0.011006, -0.012722, -0.053436, -0.036092, -0.012888, 0.005098, -0.033141, -0.021988, -0.062008, -0.005427, -0.077361, -0.071197, 0.032441, 0.031302, -0.065360, -0.029274, -0.002252, -0.061136, -0.067927, 0.046949, 0.077674, 0.026136, -0.036025, -0.028135, 0.079468, 0.014044, 0.033622, -0.039277, 0.004323, 0.000503, 0.017704, -0.061584, 0.104264, 0.074046, -0.013671, -0.054035, 0.015913, -0.000941, -0.046839, 0.014697, 0.001809, -0.026051, -0.075427, -0.031157, -0.013367, -0.007038, -0.043413, -0.015344, 0.000252, -0.007875, 0.033574, 0.004947, 0.021411, 0.024998, 0.003097, 0.059476, 0.068030, -0.044007, -0.123705, 0.003260, 0.133081, -0.095697, 0.021930, 0.026867, -0.042809, -0.083034, 0.000937, -0.019894, -0.041133, -0.010755, -0.002015, -0.031575, -0.072259, -0.076680, 0.024944, 0.021622, 0.017334, -0.041393, -0.027473, -0.045911, 0.004211, -0.055354, -0.062216, -0.062481, 0.033422, 0.003348, 0.067695, -0.052347, 0.127565, -0.079009, 0.022113, 0.024650, -0.009013, 0.074612, 0.023770, -0.050419, -0.080980, -0.105843, -0.058530, 0.023313, 0.066203, -0.040382, 0.002484, -0.050604, -0.029491, -0.094482, -0.055534, 0.108013, -0.004467, 0.072549, 0.039900, 0.023426, 0.038073, -0.041981, -0.038419, -0.045417, -0.028350, -0.085262, 0.045935, -0.049492, -0.019735, -0.039214, -0.076685, 0.094235, -0.007987, 0.042182, 0.046023, 0.032428, -0.014828, 0.018154, 0.033091, 0.026392, -0.101352, -0.143104, -0.038439, -0.009032, 0.082983, 0.037990, -0.002001, -0.006668, 0.014564, 0.026856, -0.068244, 0.023083, -0.107260, 0.011282, -0.055224, -0.069090, -0.055514, -0.034281, -0.033995, 0.023925, 0.106184, -0.025169, -0.005213, -0.065550, -0.029332, -0.075133, 0.051427, 0.088598, -0.073700, -0.026159, 0.013376, -0.004692, 0.072411, -0.032039, -0.067182, 0.212942, 0.030762, 0.024390, 0.029645, -0.001649, 0.010504, -0.039204, 0.036149, -0.042772, 0.029506, -0.063473, 0.084389, 0.003927, -0.090418, 0.008288, 0.040116, -0.031333, -0.057869, -0.007428, -0.021331, 0.009386, 0.024348, -0.083841, -0.058256, -0.073095, 0.004647, -0.006403, 0.032812, -0.011897, 0.146306, 0.034119, -0.015488, -0.061131, -0.001175, 0.119037, -0.047206, 0.005562, 0.032826, 0.053284, -0.039982, -0.057148, 0.000686, -0.113262, -0.009151, -0.055539, -0.041566, 0.047161, -0.049890, -0.069900, 0.111723, -0.066464, -0.060557, -0.045063, 0.003630, 0.014218, -0.008476, -0.042987, -0.013995, -0.050177, -0.052007, 0.005810, -0.043769, 0.066977, 0.075982, -0.016182, -0.071435, -0.016134, -0.047671, 0.085522, 0.042078, -0.047850, 0.051839, -0.004462, 0.041915, 0.048838, -0.062502, 0.021645, 0.024855, 0.035878, -0.069150, -0.130397, 0.033618, -0.033081, -0.138549, -0.056198, -0.044518, 0.004155, 0.049472, 0.034752, -0.027312, -0.038948, 0.000192, 0.052868, -0.008543, -0.015957, -0.008282, -0.089560, 0.004450, 0.004199, -0.048631, 0.033305, 0.110379, -0.052952, 0.016643, 0.058293, 0.020848, -0.018747, -0.090617, -0.056714, -0.022258, 0.057191, 0.012939, 0.059684, -0.048335, 0.003479, 0.046441, 0.068192, -0.004914, -0.011894, -0.152209, -0.012838, -0.055975, -0.002239, -0.062715, 0.023142, -0.019725, -0.000763, 0.051485, 0.006631, -0.006743, -0.106199, -0.071280, -0.085555, -0.020561, -0.031686, 0.051588, -0.046293, 0.077363, -0.017203, 0.078286, 0.001960, -0.075954, -0.063369, -0.041129, 0.055550, -0.047532, 0.001882, -0.004137, 0.039003, 0.045280, 0.000971, -0.016072, 0.125772, 0.041353, 0.018271, 0.089402, -0.018464, -0.036535, -0.053148, 0.004050, -0.027360, 0.024782, 0.031960, -0.004678, 0.000994, -0.049053, 0.051605, 0.030442, -0.044675, -0.071353, -0.014839, -0.035469, -0.051545, -0.006840, 0.019014, -0.146418, 0.039961, 0.063648, 0.041972, 0.017176, -0.077475, -0.022423, -0.019184, -0.034448, 0.000723, -0.051966, 0.085414, -0.055856, -0.060116, -0.032030, 0.049046, -0.002843, -0.059135, -0.099361, -0.030801, -0.019724, -0.032875, -0.001425, -0.040624, 0.000782, 0.050956, -0.013330, 0.015127, 0.028845, 0.035378, 0.084008, -0.041751, -0.008618, 0.030350, 0.009394, -0.001800, -0.005890, 0.012940, 0.140212, -0.093360, -0.061176, -0.005510, -0.008334, 0.010933, -0.068602, -0.063328, -0.019854, 0.029523, -0.021208, -0.090424, -0.087904, 0.026478, -0.034345, -0.068234, 0.026641, -0.116431, -0.026779, -0.043379, 0.058925, 0.030237, -0.031454, -0.006489, -0.062839, -0.039449, -0.018205, 0.027504, -0.047232, -0.041224, -0.012383, 0.020729, -0.064979, -0.066853, -0.093759, -0.048142, 0.016824, 0.019378, 0.016762, -0.013698, -0.018554, -0.019634, -0.034810, 0.075369, 0.000820, 0.105157, 0.021111, -0.056741, 0.021853, 0.057681, 0.021788, -0.027799, 0.001152, 0.011168, 0.003546, 0.068221, -0.034344, -0.037490, -0.027993, -0.011671, 0.000488, -0.012004, 0.031401, 0.003974, 0.041627, -0.077616, 0.024930, 0.037615, -0.006472, 0.036392, -0.013907, -0.033385, 0.002545, -0.018487, -0.020898, -0.125337, -0.030035, 0.025087, 0.005628, -0.113574, -0.057046, -0.043737, -0.055865, -0.009882, -0.079741, 0.047155, -0.008392, -0.087522, -0.050994, -0.029306, -0.008599, -0.021483, 0.008610, -0.021395, -0.003660, -0.030661, 0.056654, 0.007581, -0.010915, 0.036069, 0.056376, 0.037092, -0.039908, -0.051208, 0.025954, 0.045542, -0.008172, 0.066063, -0.015151, -0.096847, 0.034306, -0.012014, -0.036961, 0.016808, 0.030540, 0.020689, -0.008187, 0.028769, -0.007378, -0.053989, -0.131430, -0.042155, -0.084456, -0.052311, -0.077860, -0.013138, 0.038156, -0.052874, -0.028515, -0.098971, -0.074174, 0.004816, -0.003127, 0.035580, -0.011593, -0.061740, 0.097157, 0.000192, -0.002944, -0.015744, 0.009894, -0.069963, 0.187845, -0.135930, 0.000938, -0.051606, -0.057890, -0.006797, 0.048709, 0.020778, -0.061433, -0.093095, 0.045683, 0.058129, -0.035479, 0.032180, 0.026420, 0.036393, -0.118091, -0.006582, -0.009123, 0.035174, -0.096658, 0.108810, -0.010427, 0.085221, -0.010753, -0.013067, -0.056383, -0.017285, 0.074406, 0.024259, 0.053086, 0.001244, -0.080204, 0.038752, -0.051289, -0.028357, -0.014461, 0.024643, -0.072182, -0.062626, 0.050380, -0.077221, 0.006630, 0.036688, 0.033961, 0.102617, -0.057832, -0.036704, -0.080351, 0.000149, -0.008432, 0.083114, -0.033343, -0.006965, 0.038205, 0.008583, -0.049085, -0.037931, 0.002286, 0.034424, -0.057922, -0.054907, -0.037865, -0.036401, 0.003651, 0.036088, -0.043616, -0.114106, -0.072756, -0.018773, 0.010966, -0.001393, -0.002564, -0.015500, -0.065211, -0.027705, 0.069986, 0.035363, -0.044743, -0.014429, 0.009430, -0.046290, 0.027368, 0.067332, -0.086064, -0.045133, -0.046221, -0.033676, -0.013114, -0.024882, 0.014208, -0.045826, -0.020997, -0.028862, 0.045163, -0.027572, 0.023174, 0.058460, 0.006082, -0.046487, 0.067733, -0.007200, 0.012921, -0.063349, -0.003656, 0.031866, 0.033205, -0.030506, -0.022082, 0.118301, 0.033791, -0.058612, -0.104079, -0.020245, -0.028228, -0.042572, 0.013956, -0.055784, 0.007934, -0.019218, 0.030528, 0.013517, 0.024942, -0.017808, 0.012541, -0.029420, -0.034942, 0.046036, -0.084531, -0.015784, 0.065546, -0.039260, -0.088448, 0.023350, -0.079705, 0.004284, -0.034343, -0.007626, -0.010815, 0.109042, -0.045207, -0.013619, -0.075064, 0.047252, 0.066444, 0.049785, -0.041065, -0.004009, -0.049279, -0.076505, -0.052039, 0.034589, -0.095769, -0.085072, -0.040323, 0.054068, -0.058070, -0.038915, -0.020502, -0.074044, 0.019561, -0.003010, 0.056840, 0.043476, -0.032449, 0.001841, 0.112571, -0.068964, -0.022663, -0.061097, -0.037807, -0.066875, -0.037987, 0.061461, 0.029598, -0.093001, -0.053270, -0.041785, -0.052094, 0.036054, -0.018708, -0.031538, -0.093120, -0.107725, 0.036934, 0.045817, -0.093939, 0.015730, 0.008082, -0.021653, -0.082504, -0.101173, -0.039928, -0.037507, 0.017372, -0.053057, -0.002467, -0.047066, -0.006119, -0.024020, 0.013709, -0.061313, 0.042831, -0.071803, -0.040712, -0.006700, 0.100113, -0.069036, 0.019810, 0.048301, -0.005955, -0.029368, 0.042050, -0.076083, -0.042783, -0.032469, -0.037541, 0.056564, -0.006169, 0.039035, 0.017285, 0.038592, 0.001342, -0.041035, -0.044217, -0.017531, -0.026970, -0.061461, -0.053176, -0.019194, -0.095051, -0.031454, 0.005322, -0.060859, -0.056480, -0.024927, -0.009911, 0.051148, -0.042133, 0.030448, 0.042306, -0.063309, 0.011468, -0.072705, 0.047515, -0.027169, -0.004393, -0.055888, -0.014062, -0.018701, 0.068907, -0.052006, -0.051741, 0.004644, -0.151279, -0.063983, -0.006051, 0.050993, -0.033589, 0.092700, 0.011791, 0.044264, 0.054144, 0.038042, -0.032574, -0.013299, -0.058354, -0.081197, -0.039799, 0.040682, -0.071685, 0.062267, -0.080575, -0.002426, 0.071912, 0.108713, 0.001226, -0.073170, -0.015322, 0.031189, -0.087230, -0.038333, 0.046729, 0.016321, -0.015294, 0.029176, -0.055264, 0.016718, 0.044623, -0.048088, -0.004599, 0.024539, -0.047720, -0.066700, -0.002812, 0.014459, -0.008176, -0.012541, -0.017939, -0.071387, -0.062094, -0.050348, -0.054274, -0.038120, -0.035515, 0.034489, 0.014178, 0.077137, 0.042032, 0.029003, 0.053060, -0.001580, 0.066213, -0.020753, -0.045411, -0.075039, 0.007821, -0.080147, 0.009573, -0.010566, -0.073190, 0.012746, -0.005802, -0.022075, 0.009505, -0.023414, 0.024180, -0.007753, -0.035879, -0.055555, -0.054672, -0.014042, -0.033277, 0.082573, -0.040599, -0.079352, -0.048595, 0.021377, -0.054245, -0.075081, -0.040116, 0.003886, -0.027420, -0.026075, -0.006814, -0.116487, -0.024712, -0.060750, 0.026527, -0.064730, -0.074478, -0.004391, 0.014735, -0.036690, 0.046338, -0.021504, 0.036151, 0.022107, -0.003141, -0.033570, -0.143996, -0.041903, -0.078522, -0.005217, -0.042349, 0.032585, 0.026799, 0.007170, 0.011306, -0.053027, 0.046522, -0.086165, -0.008554, -0.037136, 0.067952, 0.089602, -0.078758, 0.067805, -0.041825, -0.017374, 0.063739, 0.012729, -0.055359, -0.013118, -0.035465, -0.025556, -0.060287, 0.043944, -0.035515, 0.051206, -0.010976, 0.033135, -0.107775, -0.041327, 0.025569, -0.038017, -0.056093, -0.059325, -0.080088, 0.080063, -0.104021, -0.005647, -0.015474, 0.011916, -0.077655, -0.061069, -0.083421, -0.083842, -0.028055, -0.025196, 0.016354, -0.068683, 0.023468, 0.044938, -0.035174, -0.021259, 0.048981, -0.056298, -0.008273, 0.044115, -0.062925, -0.122871, -0.038000, -0.062938, -0.033621, -0.071459, -0.005673, -0.029792, -0.084774, -0.027708, -0.052713, -0.022379, -0.012950, -0.004314, 0.004214, 0.037896, 0.050315, -0.042684, -0.111978, -0.015520, -0.015285, -0.016523, -0.090103, 0.041485, 0.028329, 0.089901, 0.014740, 0.005370, -0.074814, 0.047460, -0.021776, -0.069421, -0.012128, 0.020174, -0.013571, -0.047814, -0.045937, -0.007457, 0.012894, -0.056743, -0.055518, 0.029036, 0.030688, -0.060457, 0.034779, 0.030265, -0.032263, 0.043247, -0.069826, -0.056471, 0.001379, 0.054683, -0.049091, -0.064478, -0.039564, -0.078069, 0.086505, -0.070463, -0.007760, 0.009818, -0.012259, -0.054884, -0.091815, 0.097876, 0.057509, -0.112081, 0.049783, -0.004753, 0.024103, -0.027420, 0.025607, -0.119629, -0.059019, -0.029693, -0.049488, -0.087069, 0.042595, 0.029350, 0.003520, -0.007278, -0.002332, 0.039947, -0.040935, -0.016212, 0.040750, -0.002490, 0.007628, 0.039830, -0.008924, 0.041952, -0.089755, -0.012175, -0.013681, 0.018669, -0.022178, 0.041626, 0.035577, -0.038220, -0.111047, 0.093065, -0.016445, -0.020531, 0.035375, -0.000220, -0.060870, -0.049326, 0.026314, 0.037610, -0.073832, -0.014729, -0.023883, -0.003658, -0.063686, -0.079524, -0.057655, 0.027722, -0.087766, -0.099959, -0.049238, -0.009344, -0.012830, 0.010801, -0.107298, -0.034459, -0.058781, 0.012400, 0.073062, 0.007846, -0.023403, 0.022106, -0.049274, -0.150830, -0.037408, 0.012148, -0.020419, 0.005123, -0.070946, -0.058657, -0.089558, 0.003663, -0.069661, 0.072730, -0.054044, -0.018686, -0.024156, -0.045113, -0.079222, -0.010174, 0.068405, 0.051205, 0.007934, 0.010388, -0.040458, 0.034363, -0.013752, -0.061678, 0.001072, -0.016864, -0.099722, 0.024519, 0.027628, -0.003771, -0.028958, 0.018522, -0.028263, -0.046446, -0.057163, -0.064691, 0.057147, -0.104359, 0.113824, -0.097824, -0.000944, -0.074104, -0.018796, -0.048021, -0.117156, -0.011224, -0.068050, 0.104721, 0.039333, 0.009067, 0.032780, -0.058773, 0.041693, 0.044272, -0.037896, -0.033103, 0.018661, 0.095012, -0.041891, -0.039547, -0.058506, 0.037004, -0.040226, -0.057020, -0.015658, -0.120686, 0.037445, -0.078668, -0.018577, 0.014183, -0.058987, 0.032402, -0.070460, -0.034491, -0.065906, -0.048920, -0.045719, -0.016607, -0.052023, -0.016869, -0.072552, -0.056880, -0.037432, -0.063811, -0.080775, -0.081471, 0.032439, 0.034397, -0.010909, 0.057517, -0.062494, 0.068854, -0.023550, -0.032692, -0.080082, -0.039819, -0.015837, -0.015295, 0.025868, -0.061336, 0.004021, 0.065572, 0.012944, -0.020794, -0.006657, 0.003860, 0.020852, -0.005040, -0.012671, 0.044309, -0.055187, -0.016643, 0.030804, 0.015342, -0.090433, -0.026890, -0.023889, -0.026437, -0.002269, 0.019496, 0.046902, -0.000550, -0.014603, 0.077343, -0.036828, -0.043534, -0.064284, -0.064149, -0.010808, 0.034894, -0.083800, -0.055170, 0.025871, 0.038261, -0.020792, -0.006419, -0.009317, 0.067829, -0.010651, -0.022332, 0.027690, 0.014070, -0.023071, 0.053852, 0.071413, -0.019023, -0.014927, 0.076549, -0.073474, 0.010644, -0.076568, -0.003730, -0.024368, -0.061265, -0.045886, -0.033972, 0.013536, -0.008837, -0.022250, -0.073539, -0.044814, -0.029936, -0.045702, -0.001134, -0.025468, 0.068221, -0.080225, -0.110327, -0.053285, -0.042827, 0.020920, -0.026021, -0.007853, -0.040111, -0.076430, -0.069872, 0.025055, 0.095994, -0.014937, 0.078800, 0.003303, 0.003894, -0.138240, -0.037023, -0.052669, 0.032793, 0.011131, -0.059395, -0.027772, -0.030904, -0.024249, 0.046736, -0.045179, 0.000923, 0.031859, -0.030310, 0.045939, -0.065592, 0.022867, 0.014829, -0.042189, -0.093713, -0.054496, -0.087973, -0.037183, 0.045245, -0.061309, -0.046370, -0.037040, 0.029572, -0.034639, 0.088435, -0.086770, -0.033968, -0.059945, -0.060425, 0.032116, -0.013289, 0.008413, -0.005134, 0.007872, 0.004002, 0.002799, -0.026946, -0.021056, -0.030978, -0.055425, -0.055535, 0.001408, -0.053457, -0.026514, 0.005998, 0.020034, -0.074573, -0.058318, -0.067405, -0.045178, 0.037291, -0.031408, -0.037337, -0.065923, -0.086868, -0.043315, -0.082073, 0.014360, -0.037799, -0.064011, -0.059241, -0.005532, -0.110856, 0.019696, 0.022950, -0.109967, -0.057616, 0.014035, 0.021931, -0.017190, -0.022797, 0.068135, 0.012550, 0.054964, -0.002867, -0.053442, -0.056407, 0.007523, 0.054874, -0.059794, -0.000717, -0.020538, -0.062943, -0.026943, -0.030914, 0.001578, 0.025038, -0.081534, -0.041841, 0.000914, -0.040575, 0.041069, 0.030149, -0.047384, 0.070691, -0.046235, -0.069128, -0.014655, 0.025945, 0.005900, 0.021576, 0.014818, -0.017372, -0.085931, 0.008673, -0.127468, -0.018142, -0.035053, 0.005293, -0.063147, -0.050385, -0.016805, 0.002157, 0.012439, -0.025912, 0.019464, 0.140719, 0.044004, -0.032726, 0.008684, -0.019082, 0.008973, -0.067546, -0.050792, 0.007026, 0.071434, -0.030295, 0.032160, -0.002489, -0.010781, -0.030518, 0.046420, 0.009715, 0.046569, -0.064518, 0.035491, -0.049198, -0.026451, -0.075983, -0.016798, -0.098390, 0.028305, 0.008195, -0.057943, -0.084226, -0.047715, 0.043471, -0.041604, -0.101436, -0.007576, -0.061003, -0.040151, -0.079476, 0.035082, 0.013366, -0.073322, -0.078640, 0.027978, -0.127353, -0.029063, -0.039173, -0.054487, -0.023318, -0.023995, -0.017847, 0.016835, -0.068642, 0.077860, -0.081190, -0.045407, -0.050145, 0.018538, -0.045835, -0.006103, -0.004051, -0.002531, 0.007253, -0.020512, -0.019840, -0.028246, -0.023230, 0.013453, 0.030544, -0.006919, 0.006612, -0.067408, -0.042141, -0.056668, -0.001708, -0.020234, -0.050898, -0.027647, 0.117548, -0.023332, 0.066788, -0.068825, -0.032248, -0.036845, -0.053679, -0.072182, 0.020121, -0.029298, -0.041971, -0.057193, 0.032837, 0.026345, 0.070640, -0.013087, -0.077128, 0.058118, 0.033021, -0.065560, -0.077262, 0.044917, 0.007111, -0.030522, 0.053371, 0.039260, 0.056742, -0.076782, -0.051719, -0.027520, -0.072301, 0.027750, 0.022872, 0.005919, 0.032011, -0.002139, 0.018756, 0.011431, -0.053192, 0.046016, -0.037488, -0.064115, -0.033299, 0.054993, -0.063432, -0.004252, -0.029767, 0.059103, 0.016086, -0.059837, -0.033195, 0.012841, 0.000290, 0.083123, 0.017433, -0.031822, -0.029134, -0.045724, -0.016191, 0.078591, 0.033855, 0.043989, 0.063547, -0.055359, -0.022673, 0.001935, -0.047962, 0.022308, 0.015792, 0.049520, 0.038492, -0.016984, -0.015495, -0.121909, 0.016039, -0.088056, 0.000161, -0.070936, -0.025749, 0.032282, -0.062233, -0.037204, -0.017936, -0.077304, -0.006824, -0.055698, -0.032047, -0.063483, -0.037164, 0.036672, 0.030094, 0.027136, 0.088055, 0.137050, -0.055533, 0.014850, 0.016294, 0.006654, 0.015415, -0.018741, 0.084517, 0.111356, -0.023419, 0.009413, -0.045469, -0.080710, 0.035207, -0.033061, 0.015181, -0.038356, 0.029915, 0.011247, 0.099229, -0.030374, 0.018559, -0.034064, 0.053145, -0.085284, 0.030475, -0.024090, -0.067363, 0.031420, -0.032684, 0.053679, 0.024636, -0.104548, -0.040489, 0.036097, 0.055185, -0.009799, -0.066227, 0.004288, -0.015889, -0.059233, -0.073876, 0.039837, -0.105437, -0.088193, -0.103405, 0.030842, 0.051798, -0.015062, 0.014771, 0.017046, 0.052326, -0.026809, 0.033540, -0.013656, -0.022624, -0.025765, 0.047750, -0.052918, 0.021737, -0.000003, 0.041587, -0.020895, -0.048006, 0.039277, -0.009229, -0.044448, 0.010294, -0.041709, 0.050337, -0.039803, -0.012263, -0.073238, -0.072783, 0.049119, 0.032647, 0.017832, -0.064484, -0.038173, -0.043609, 0.002916, -0.010792, -0.036441, -0.056889, -0.077194, -0.052459, 0.051646, 0.043604, -0.007017, -0.037784, -0.051983, -0.049754, 0.033814, -0.054236, -0.067872, -0.051827, 0.064081, -0.054836, 0.134036, -0.092389, -0.042750, -0.033137, 0.043333, -0.029433,